(* IEC 61131-3 sources: ml2plc/benchmarks/st (part 13) *)

    weights_7 : ARRAY[0..191] OF REAL := [0.888088644, -0.123913772, -0.846282899, 1.17783785, -0.767203927, -0.449209094, -0.772179544, -0.308529139, 1.4158355, 1.31052208, -0.610198379, -0.72990191, -1.32865715, 0.598848462, 0.529765189, 0.906202614, 0.0025848723, -0.916793466, 1.49462843, -0.405332565, -0.581331134, -1.24053252, 0.719219387, 0.456818759, 1.07239103, -0.71875602, -0.512277603, -0.771926701, -0.468680173, 1.47650003, 1.16464531, -0.211401775, -0.830097437, -0.592156947, -0.122473739, 1.40973353, -0.256034911, -0.522334278, 1.13457429, -1.07700145, 0.666598201, 0.474731237, -1.27282381, 0.632757485, 0.708201051, -1.10329938, 0.727127552, 0.492805749, -1.15903831, 0.78498143, 0.360979617, -0.812300086, 0.210701555, 0.955269992, 1.52882719, -0.381138951, -0.742695808, -0.274786711, -0.196780428, 1.68793082, 1.54681039, -0.22795254, -0.553849936, -1.26980937, 0.545592904, 0.425203025, 1.34888792, -0.62540859, -0.476311505, 0.380844444, 0.586091816, -1.1150496, -1.01592028, -0.0146602849, 0.895467341, -0.456928283, -0.584338427, 1.16077256, 0.413884312, -0.21048446, -1.16396976, 0.751783848, 0.324061215, -1.49614906, -0.575325549, -0.530140579, 1.41179919, -1.35693932, 0.686669171, 0.656322777, 1.22251678, -0.695291579, -0.740689158, -0.676817656, -0.355217397, 1.59177208, 0.207133874, 0.497951657, -0.983146548, 0.469873518, 0.117614292, -1.43506837, 0.132174373, 0.389537215, -1.14951098, 0.820351005, 0.0726073906, -0.653037608, 1.48673153, -0.487765312, -0.680322826, 0.0507701635, 0.432502806, -0.945631862, -0.42844075, -0.336914688, 1.56399095, 0.778971314, 0.452257246, -1.42628229, -0.471889734, -0.441351414, 1.41961205, 0.00993562955, -0.574463367, 0.549236596, 1.21431422, -0.684745908, -0.146852493, -0.852580428, -0.388104379, 1.43994546, -0.78573972, -0.31785956, 1.49420559, 1.35582078, -0.0897780806, -0.4087421, 0.695370257, 0.364000231, -1.27974713, 0.373800397, 0.482034594, -1.2333101, 1.32530713, -0.490792662, -0.321068794, 0.503972769, 0.0731279776, -1.43025231, -0.400622934, -0.543340862, 1.15907669, 0.280509353, 0.306184769, -1.45866597, 1.17186499, -0.665238976, -0.192673638, -1.03320301, -0.00132938253, 0.908325374, 1.0105319, 0.0897968858, -0.713194191, 0.359024227, 0.363719821, -1.40014493, -0.18309705, -0.547121286, 0.972757518, 0.502420723, -0.138461307, -1.05406582, 1.36639011, -0.532719135, -0.751533031, 0.933193147, -0.895748973, -0.461577773, -0.881112456, -0.282391846, 0.816898346, 1.63772881, -0.375343144, -0.522669077, -0.108508743, -0.35503307, 1.0366466, -0.95520407, -0.139931589, 0.780282736];
    bias_7 : ARRAY[0..2] OF REAL := [0.0118476562, 0.164545983, -0.221493304];

END_VAR

VAR
    (* Merged variables from all regions *)
    buffer_0 : ARRAY[0..63] OF REAL;
    buffer_1 : ARRAY[0..63] OF REAL;
    c_state_0 : ARRAY[0..63] OF REAL;
    c_state_3 : ARRAY[0..63] OF REAL;
    f_gate_0 : ARRAY[0..63] OF REAL;
    f_gate_3 : ARRAY[0..63] OF REAL;
    g_gate_0 : ARRAY[0..63] OF REAL;
    g_gate_3 : ARRAY[0..63] OF REAL;
    h_state_0 : ARRAY[0..63] OF REAL;
    h_state_3 : ARRAY[0..63] OF REAL;
    i_gate_0 : ARRAY[0..63] OF REAL;
    i_gate_3 : ARRAY[0..63] OF REAL;
    o_gate_0 : ARRAY[0..63] OF REAL;
    o_gate_3 : ARRAY[0..63] OF REAL;

    (* Temporary computation variables *)
    i : DINT;
    j : DINT;
    t : DINT;
    sum : REAL;
    (* Computation helpers *)
    max_val : REAL;
    exp_val : REAL;
    exp_sum : REAL;
    (* Spatial loop variables *)
    oc : DINT;
    oh : DINT;
    ow : DINT;
    ic : DINT;
    kh : DINT;
    kw : DINT;
    ih : DINT;
    iw : DINT;
    (* Transpose loop variables *)
    t2_d0 : DINT;
    t2_d1 : DINT;
    t2_d2 : DINT;
END_VAR

(* Forward pass execution *)

(* Region: r0 [ACYCLIC] *)
(* Acyclic Region r0 *)
(* Layer 0: LSTM (hidden_size=64, input_size=1, seq_len=1) *)
(* Generating output: Y *)

(* Initialize states to zero *)
FOR j := 0 TO 63 DO
    h_state_0[j] := 0.0;
    c_state_0[j] := 0.0;
END_FOR;

(* Process 1 timesteps *)
FOR t := 0 TO 0 DO

    (* Input Gate *)
    FOR j := 0 TO 63 DO
        sum := 0.0;
        FOR i := 0 TO 0 DO
            sum := sum + input_data * weights_0_i[j * 1 + i] ;
        END_FOR;
        FOR i := 0 TO 63 DO
            sum := sum + h_state_0[i] * recurrent_0_i[j * 64 + i] ;
        END_FOR;
    sum := sum + bias_0_i[j];
    i_gate_0[j] := 1.0 / (1.0 + EXP(-sum));
    END_FOR;

    (* Forget Gate *)
    FOR j := 0 TO 63 DO
        sum := 0.0;
        FOR i := 0 TO 0 DO
            sum := sum + input_data * weights_0_f[j * 1 + i] ;
        END_FOR;
        FOR i := 0 TO 63 DO
            sum := sum + h_state_0[i] * recurrent_0_f[j * 64 + i] ;
        END_FOR;
    sum := sum + bias_0_f[j];
    f_gate_0[j] := 1.0 / (1.0 + EXP(-sum));
    END_FOR;

    (* Cell Gate *)
    FOR j := 0 TO 63 DO
        sum := 0.0;
        FOR i := 0 TO 0 DO
            sum := sum + input_data * weights_0_g[j * 1 + i] ;
        END_FOR;
        FOR i := 0 TO 63 DO
            sum := sum + h_state_0[i] * recurrent_0_g[j * 64 + i] ;
        END_FOR;
    sum := sum + bias_0_g[j];
    exp_val := EXP(2.0 * sum);
    g_gate_0[j] := (exp_val - 1.0) / (exp_val + 1.0);
    END_FOR;

    (* Output Gate *)
    FOR j := 0 TO 63 DO
        sum := 0.0;
        FOR i := 0 TO 0 DO
            sum := sum + input_data * weights_0_o[j * 1 + i] ;
        END_FOR;
        FOR i := 0 TO 63 DO
            sum := sum + h_state_0[i] * recurrent_0_o[j * 64 + i] ;
        END_FOR;
    sum := sum + bias_0_o[j];
    o_gate_0[j] := 1.0 / (1.0 + EXP(-sum));
    END_FOR;

    (* Cell state: c_t = f_t * c_{t-1} + i_t * g_t *)
    FOR j := 0 TO 63 DO
        c_state_0[j] := f_gate_0[j] * c_state_0[j] + i_gate_0[j] * g_gate_0[j];
    END_FOR;

    (* Hidden state: h_t = o_t * tanh(c_t) *)
    FOR j := 0 TO 63 DO
        exp_val := EXP(2.0 * c_state_0[j]);
        h_state_0[j] := o_gate_0[j] * ((exp_val - 1.0) / (exp_val + 1.0));
    END_FOR;

    (* Y output: Full sequence *)
    FOR j := 0 TO 63 DO
        buffer_0[t * 64 + j] := h_state_0[j];
    END_FOR;
END_FOR;

(* Layer 1: Squeeze *)
FOR i := 0 TO 63 DO
    buffer_1[i] := buffer_0[i];
END_FOR;

(* Layer 2: Transpose perm=(1, 0, 2)  (1, 1, 64) -> (1, 1, 64) *)
FOR t2_d0 := 0 TO 0 DO
    FOR t2_d1 := 0 TO 0 DO
        FOR t2_d2 := 0 TO 63 DO
            buffer_0[t2_d0 * 64 + t2_d1 * 64 + t2_d2] := buffer_1[t2_d1 * 64 + t2_d0 * 64 + t2_d2];
        END_FOR;
    END_FOR;
END_FOR;

(* Layer 3: LSTM (hidden_size=64, input_size=64, seq_len=1) *)
(* Generating output: Y *)

(* Initialize states to zero *)
FOR j := 0 TO 63 DO
    h_state_3[j] := 0.0;
    c_state_3[j] := 0.0;
END_FOR;

(* Process 1 timesteps *)
FOR t := 0 TO 0 DO

    (* Input Gate *)
    FOR j := 0 TO 63 DO
        sum := 0.0;
        FOR i := 0 TO 63 DO
            sum := sum + buffer_0[t * 64 + i] * weights_3_i[j * 64 + i] ;
        END_FOR;
        FOR i := 0 TO 63 DO
            sum := sum + h_state_3[i] * recurrent_3_i[j * 64 + i] ;
        END_FOR;
    sum := sum + bias_3_i[j];
    i_gate_3[j] := 1.0 / (1.0 + EXP(-sum));
    END_FOR;

    (* Forget Gate *)
    FOR j := 0 TO 63 DO
        sum := 0.0;
        FOR i := 0 TO 63 DO
            sum := sum + buffer_0[t * 64 + i] * weights_3_f[j * 64 + i] ;
        END_FOR;
        FOR i := 0 TO 63 DO
            sum := sum + h_state_3[i] * recurrent_3_f[j * 64 + i] ;
        END_FOR;
    sum := sum + bias_3_f[j];
    f_gate_3[j] := 1.0 / (1.0 + EXP(-sum));
    END_FOR;

    (* Cell Gate *)
    FOR j := 0 TO 63 DO
        sum := 0.0;
        FOR i := 0 TO 63 DO
            sum := sum + buffer_0[t * 64 + i] * weights_3_g[j * 64 + i] ;
        END_FOR;
        FOR i := 0 TO 63 DO
            sum := sum + h_state_3[i] * recurrent_3_g[j * 64 + i] ;
        END_FOR;
    sum := sum + bias_3_g[j];
    exp_val := EXP(2.0 * sum);
    g_gate_3[j] := (exp_val - 1.0) / (exp_val + 1.0);
    END_FOR;

    (* Output Gate *)
    FOR j := 0 TO 63 DO
        sum := 0.0;
        FOR i := 0 TO 63 DO
            sum := sum + buffer_0[t * 64 + i] * weights_3_o[j * 64 + i] ;
        END_FOR;
        FOR i := 0 TO 63 DO
            sum := sum + h_state_3[i] * recurrent_3_o[j * 64 + i] ;
        END_FOR;
    sum := sum + bias_3_o[j];
    o_gate_3[j] := 1.0 / (1.0 + EXP(-sum));
    END_FOR;

    (* Cell state: c_t = f_t * c_{t-1} + i_t * g_t *)
    FOR j := 0 TO 63 DO
        c_state_3[j] := f_gate_3[j] * c_state_3[j] + i_gate_3[j] * g_gate_3[j];
    END_FOR;

    (* Hidden state: h_t = o_t * tanh(c_t) *)
    FOR j := 0 TO 63 DO
        exp_val := EXP(2.0 * c_state_3[j]);
        h_state_3[j] := o_gate_3[j] * ((exp_val - 1.0) / (exp_val + 1.0));
    END_FOR;

    (* Y output: Full sequence *)
    FOR j := 0 TO 63 DO
        buffer_1[t * 64 + j] := h_state_3[j];
    END_FOR;
END_FOR;

(* Layer 4: Squeeze *)
FOR i := 0 TO 63 DO
    buffer_0[i] := buffer_1[i];
END_FOR;

(* Layer 5: Slice starts=[0] ends=[1] axes=[0] steps=[1] *)
FOR i := 0 TO 63 DO
    buffer_1[i] := buffer_0[i];
END_FOR;

(* Layer 6: Squeeze *)
FOR i := 0 TO 63 DO
    buffer_0[i] := buffer_1[i];
END_FOR;

(* Layer 7: Fused Linear + SOFTMAX *)
FOR j := 0 TO 2 DO
    sum := 0.0;
    FOR i := 0 TO 63 DO
        sum := sum + buffer_0[i] * weights_7[i * 3 + j];
    END_FOR;
output_data[j] := sum + bias_7[j];
END_FOR;

(* Softmax: find max *)
max_val := output_data[0];
FOR i := 1 TO 2 DO
    IF output_data[i] > max_val THEN
        max_val := output_data[i];
    END_IF;
END_FOR;

(* Softmax: compute exponentials and sum *)
exp_sum := 0.0;
FOR i := 0 TO 2 DO
    output_data[i] := EXP(output_data[i] - max_val);
    exp_sum := exp_sum + output_data[i];
END_FOR;

(* Softmax: normalize *)
FOR i := 0 TO 2 DO
    output_data[i] := output_data[i] / exp_sum;
END_FOR;

END_FUNCTION_BLOCK

(* ---- LSTM3_straton.st ---- *)
FUNCTION_BLOCK LSTM3_FB

    (* Model Inputs/Outputs *)
VAR_INPUT
    input_data : REAL;
END_VAR

VAR_OUTPUT
    output_data : ARRAY[0..2] OF REAL;
END_VAR

VAR
    CONSTANT weights_0_i : ARRAY[0..63] OF REAL := [0.702140272, 0.550907314, 0.840128601, 0.811903298, 0.307846963, 1.12213707, 0.702723861, 0.78549248, 1.03316271, 0.728771746, 0.658028424, 0.580750406, 0.615542233, 0.771269143, 0.595596969, 0.611394525, 0.644692361, 0.114490122, 0.525960624, 0.181024775, 0.43071872, 0.665743828, 0.662614048, 0.347228467, 0.769034982, 0.228199184, 0.700795293, 0.569566727, 0.677138209, 0.73381424, 0.549547136, 0.302287668, 0.169487387, 0.974528968, 0.748925805, 0.776894212, 0.810905218, 0.427933753, 0.884441376, 0.829136014, 0.288695246, 0.795262098, 0.532379746, 0.22446543, 0.771800041, 0.653539002, 0.731219053, 0.170757174, 0.902539074, 0.538231611, 0.51912272, 0.955829144, 0.832288802, 0.900867701, 0.702928185, 0.872188985, 0.894331634, 0.607017815, 0.705278337, 0.333420843, 0.529384255, 0.336027026, 0.648417652, 0.559612393];
    CONSTANT recurrent_0_i : ARRAY[0..4095] OF REAL := [0.0727516413, 0.0621806681, 0.0826341808, -0.0324631631, 0.0780053213, -0.130033791, -0.0319923647, 0.0896927789, 0.130534112, -0.0421945676, -0.0756037533, -0.0922252685, 0.00545726344, 0.0880259946, -0.0772752613, 0.0512711406, 0.0296145584, 0.0135381324, -0.0145865045, 0.0353048369, -0.0163449794, -0.0219417289, 0.00759037118, -0.0415089913, -0.0641311258, 0.0446674526, 0.0170345269, 0.114942849, 0.0462704226, 0.0438979566, 0.130931437, -0.0146956779, -0.0373039432, 0.160181582, 0.0509333275, -0.0090306839, 0.00299992273, -0.010383524, 0.031728372, -0.00710704457, -0.00758532062, -0.0451442599, 0.0935175195, -0.0125704622, 0.0317067243, 0.0606242865, -0.0168152805, 0.00345395319, -0.0898493975, 0.0553060398, -0.0737185553, -0.0635084957, -0.00217968249, -0.0560640506, 0.0309809372, -0.0389013216, -0.0571859553, -0.00478457334, -0.137683779, -0.0206679888, -0.0514972247, 0.0388438366, 0.0153822303, -0.0171498396, 0.00600126432, -0.0851558447, 0.133651495, -0.0185905043, -0.0246904604, 0.0102146799, 0.0566058196, 4.23480524e-05, -0.0203502793, 0.0520644151, -0.0723077804, 0.0706539601, 0.023620028, -0.114415541, -0.077967003, 0.0202202648, -0.0342062041, -0.0991770253, 0.0620289519, -0.039034795, -0.11893864, 0.0454845876, -0.00476856716, -0.124633782, 0.0523016639, -0.0491373278, -0.0463687293, -0.0284624062, -0.0796379447, 0.0411196351, 0.0183950588, -0.0835485458, -0.0130095724, 0.0761168301, 0.110718943, -0.0617460273, -0.105785653, 0.0356864445, 0.0494417138, 0.020865988, -0.0829355121, 0.000668380701, 0.00423853425, -0.117335983, -0.112802789, -0.0873446092, -0.0655066594, -0.0423219949, -0.0786840543, 0.00250472827, -0.110003382, -0.045915883, -0.0603204183, 0.0303344596, 0.0707006305, 0.0354735367, -0.0640057474, 0.0473994985, -0.0212647375, 0.0411032513, -0.0771477968, -0.0166638345, 0.00337213092, -0.0226932354, 0.0456429943, -0.0196843427, 0.0404657125, 0.0254306849, -0.0168858916, -0.100593567, -0.116192296, 0.0310631618, 0.0672013462, 0.114804812, -0.0465652943, -0.00154955732, -0.036767751, -0.0378884897, -0.0250008237, 0.0466526635, -0.0191811118, -0.000101840356, -0.0592753589, 0.172661081, -0.0531607121, 0.00527921086, -0.0125218285, 0.0705138072, 0.020655388, 0.100712925, 0.0040708594, 0.0298366249, -0.00289789634, -0.105439723, -0.00869502686, 0.0765521899, -0.0580295846, 0.0956573263, -0.0131847216, -0.0422052965, -0.00297464058, 0.0503321402, -0.0478489585, 0.0335775577, -0.0301637445, 0.00344321551, 0.0895170718, 0.0310253073, 0.00502613885, 0.0457690544, -0.0207835399, 0.000252262573, -0.00835427362, -0.133433089, -0.0304905064, 0.092546992, 0.0331540592, 0.000841447385, -0.0252766088, -0.0414331928, 0.0101674721, -0.0159507189, 0.00302448263, -0.00964387413, 0.0656525418, -0.157459468, 0.0171210915, 0.10000737, -0.0236126985, 0.0170642994, -0.0294568427, 0.0334513187, -0.0220087394, -0.0428130999, -0.0756321475, 0.0157396775, -0.0132302316, -0.0658647045, 0.0589430034, 0.00988156162, -0.0849569365, 0.121961564, 0.00635574851, -0.0347112417, 0.00926421676, 0.0173401404, -0.151415199, 0.041484613, 0.00184322847, 0.0359681174, 0.0752471238, 0.0984926, -0.0999504551, 0.0267645456, 0.0486583449, 0.0590231977, 0.00425340515, 0.0750458241, -0.00415878836, -0.0125731686, 0.0978570655, -0.0809679553, 0.00953727774, 0.0290226694, 0.0406909958, -0.122906491, 0.0246698428, 0.0127425753, 0.0167440623, 0.0282128006, 0.0204523206, -0.0491225682, -0.00133290479, -0.0879503638, -0.0175075829, -0.0297206547, -0.0100959539, 0.0516403019, -0.052208595, -0.0526957437, -0.142511413, 0.0631481856, 0.0082924366, 0.0142942322, 0.0194399487, 0.082317315, 0.182806715, -0.0128400987, 0.0133524388, -0.0546476245, 0.0249223039, -0.0169815794, 0.00866021402, -0.0423310734, 0.0564726405, -0.102079518, -0.00930380821, 0.0186641105, 0.0262102578, -0.0276058502, 0.00666292477, -0.0416896977, 0.0912574828, 0.0394550152, 0.0131434798, -0.0107459817, 0.0220733341, 0.101379797, 0.069571726, -0.00961366575, -0.0787620544, 0.0116914697, -0.10854429, -0.0954701975, 0.0340769216, 0.00364211295, -0.0838557333, 0.11981912, -0.00016324129, -0.0325293913, -0.0776118413, 0.0159091651, -0.0477694646, 0.117520049, 0.0343630239, 0.0626410767, 0.0725534111, 0.0137511753, 0.0102761351, 0.0384476483, -0.025758734, -0.0109584201, -0.115339629, -0.0080120489, 0.00114537869, 0.120408282, 0.0536845811, -0.0320632346, -0.0182842221, 0.0136444457, -0.0913924277, 0.0926747099, -0.0925770104, -0.0231577531, 0.0205560066, -0.00191105367, -0.0321596973, -0.12859036, -0.0584978908, -0.0560642928, 0.113133483, -0.027025789, -0.0500422195, -0.046241872, 0.00904796738, -0.142783582, 0.0597391538, -0.0933348238, -0.091109097, -0.0664444864, 0.0786642209, 0.0643827915, -0.00446130894, -0.0406435616, 0.0581320375, -0.0465331115, 0.0364481136, 0.0176456738, 0.0979348645, 0.0894413367, -0.0545003824, -0.0495841168, 0.00888519082, 0.0636737645, 0.05193891, -0.0283721257, -0.0566147231, 0.183045834, -0.118062697, -0.0693358406, 0.0176241342, -0.00353063643, -0.0731030107, -0.0132001694, -0.0521529317, 0.125817999, 0.0695978999, -0.124826491, -0.0061951708, 0.0417266451, 0.0583891943, 0.0235025808, -0.0648017526, 0.0367687866, -0.0333195329, -0.0380349644, -0.0129484069, -0.130066216, 0.0361705013, 0.00339826383, 0.0437863097, -0.0165002644, 0.0261191688, -0.0423497558, -0.125128835, -0.0824990794, -0.158404469, 0.0239589661, 0.000989105785, 0.0705716163, 0.000514748506, 0.0106146075, 0.018335579, -0.0927568302, 0.0252951495, -0.0790490359, -0.000428203493, -0.00807804428, 0.0282302741, 0.0416536778, -0.0353906341, -0.125360742, -0.0164563227, -0.0400473513, -0.0475901105, -0.0188975669, 0.0190299749, -0.035292007, 0.0398504995, 0.0578784384, -0.00539165642, 0.0377021693, -0.00657368964, -0.00917698257, -0.0644009337, -0.00816033222, -0.0400245786, 0.0934461951, -0.0305664521, -0.0227205046, -0.0205899216, -0.0152598266, 0.0277052615, 0.0136568416, -0.0807154402, -0.0698791817, -0.0617102832, -0.0738777146, -0.0762551874, 0.0600783564, 0.0449102037, -0.0579390265, 0.144962117, 0.194548294, -0.0171745792, -0.0391854942, 0.0970190018, -0.0735182762, -0.00443866057, 0.0561750755, -0.00835239142, 0.103401393, 0.0354097895, 0.0144966841, 0.0718112886, 0.0228926204, 0.0372653194, -0.0687554851, 0.10727971, -0.037785314, 0.0797682926, -0.00646833796, 0.00971507467, 0.0386701822, 0.118912876, -0.032234598, 0.0318986624, 0.0539872497, -0.011686909, 0.145176083, 0.0255599786, -0.039034158, 0.0321393982, -0.0146574825, 0.160541251, -0.0973295048, 0.0362529159, 0.025079282, 0.119155452, -0.0793333724, -0.0652497858, 0.0338132381, 0.0546442941, -0.0188240651, 0.00941769406, -0.104044199, -0.0805709586, -0.0476697013, 0.0640894994, 0.07038939, -0.000911274925, -0.0129568689, 0.00333408732, -0.0201132633, 0.00736489007, 0.0114483982, 0.103261217, -0.0535993725, -0.0637782216, 0.0585075244, -0.00838142354, -0.0303359125, -0.0881697759, 0.0637675673, 0.0675119534, -0.0465907231, 0.0223106146, 0.0744051114, -0.00451694895, 0.0699620992, -0.0100199496, -0.0766999424, -0.111208931, -0.00734356884, -0.0439275131, -0.0797161311, -0.0652370676, 0.00365057588, -0.0114077562, -0.00976049341, -0.00207494851, -0.0548781082, 0.00935276877, 0.0451770723, 0.0154793952, -0.0134702399, -0.0304076131, 0.0523790345, 0.0507434718, 0.0699445009, 0.0361545049, -0.0232983083, 0.014487464, -0.100811966, -0.0416969284, 0.0327967592, -0.0249530524, -0.0339162126, -0.017976515, -0.0419778116, 0.0222332217, 0.0152361365, -0.0173479971, 0.0431629382, 0.0682366565, 0.0238082893, -0.0795904398, 0.0329069197, 0.0875642598, 0.0079081133, -0.0893924832, -0.0986220166, -0.0576440096, 0.0620961636, -0.0173755735, 0.0642281398, 0.0128179947, 0.00068197638, 0.0281319804, -0.0740936846, 0.0206660945, 0.0549913384, -0.0514548644, 0.106060728, 0.0215401538, 0.00298270863, -0.0353878029, 0.0589390211, 0.0957489237, -0.0261493661, -0.116729505, 0.0467135832, -0.0562625453, 0.0103190532, 0.000896572019, 0.00233004056, -0.0809285343, 0.022660207, 0.110791236, 0.12861453, 0.0517879203, 0.0163614936, -0.0594949387, -0.0264125317, 0.0178101491, 0.0121639995, -0.103968374, -0.00524417032, 0.0263312124, 0.0630289018, -0.0221815184, 0.0465865284, 0.0157697946, 0.00964579266, 0.0674970746, -0.009665424, 0.00193209574, -0.0533254594, -0.167867079, -0.014877351, 0.0151824076, 0.0264426656, -0.125007585, -0.0209615547, 0.0590866096, -0.0137481289, 0.0121204332, -0.0151834041, -0.0251058768, -0.0110409586, -0.00677108858, 0.0129520297, -0.0732064545, -0.0273697656, 0.091351226, -0.0557100922, 0.0296072997, 0.00988943037, -0.0364736542, 0.065504536, -0.00958945323, 0.116355866, 0.0455187596, 0.0358052738, 0.0423866361, 0.126706302, -0.016172383, 0.00576764019, -0.0433344729, 0.0248547792, -0.0734665766, 0.0619035512, -0.00564275496, -0.0161651708, -0.0448754504, -0.0378655344, -0.0100620128, 0.00184470601, 0.0365175456, 0.0127978846, -0.0136364019, 0.043987263, -0.0878729597, -0.0277508721, -0.0749285445, 0.0541052632, 0.0489377081, 0.0708028525, -0.0602139272, -0.0754432306, 0.00850299187, -0.0961926952, 0.132325843, -0.116709456, 0.108343646, -0.0597229786, 0.0569296554, -0.00331771234, -0.0273206718, -0.0314441323, -0.000921917148, -0.157476932, -0.0827142447, 0.00737003703, 0.052945137, 0.0687581971, -0.000348506495, 0.0343997292, -0.0195971914, 0.125520691, 0.00101949577, -0.0154516073, 0.0158582088, 0.00286582764, -0.0688755289, 0.0439975187, -0.0276184082, 0.00204778835, -0.00275259465, -0.0708792955, -0.0564192757, -0.0506432205, 0.00576888025, -0.0713198557, 0.0567040592, 0.0332127437, 0.0334661454, -0.00076312013, -0.0548750758, -0.0580983646, 0.107379794, -0.0128812864, 0.118800402, -0.0523375235, 0.00846277364, -0.0320085548, 0.115329124, -0.0270583499, -0.0132279834, 0.0107595138, -0.0375581123, -0.0365415849, 0.00050151255, 0.082369104, -0.00622165669, 7.82900024e-05, -0.0483080707, -0.0812478885, 0.0232834574, -0.0151235107, -0.0244658086, -0.000501235016, 0.00333951134, 0.0400660373, -0.0880180597, 0.00398900174, 0.0124121793, 0.00375011051, -0.144496277, 0.034541361, 0.0617251918, 0.00635286514, 0.0420818478, -0.0161394067, -0.0328651518, 0.0820424035, 0.0222173464, 0.0229891762, 0.0139844613, -0.0297264177, 0.00847776048, 0.070485957, -0.058027342, 0.0854259282, 0.0362042785, 0.185735196, 0.0904341638, 0.0116911372, 0.0929991826, -0.0522834435, -0.145003289, 0.123330593, 0.0321200006, -0.137998715, 0.0165430456, -0.0304837991, -0.0096137803, -0.000575108454, 0.00894964393, -0.0625963882, 0.0877403393, -0.00540286303, 0.05565162, 0.117289849, 0.0030141864, -0.0417421907, -0.0236499757, 0.0914468393, 0.0819795579, -0.0468929261, -0.00116663426, 0.106944904, -0.00840409659, 0.0906113163, 0.035827592, 0.0802839696, 0.0457703471, -0.0492791533, -0.00685054809, 0.0727560148, -0.0435580648, -0.0374004319, -0.0588955544, 0.0217557084, 0.0269399136, -0.032965567, -0.156689122, 0.0972655118, -0.00287246145, -0.0220363066, -0.127908081, 0.0366795324, -0.00863787718, 0.00523071457, -0.0202574283, -0.0320058577, 0.101983219, -0.0471758954, 0.0736685321, -0.0319768637, 0.00369445607, 0.0711755827, 0.0862062871, -0.0234699268, -0.0473918878, -0.0423197597, -0.0217249542, -0.0155853694, -0.00140371313, -0.031561885, -0.012095931, 0.0411939137, -0.0171032492, 0.0350121111, -0.0700786561, 0.106874585, 0.0229188204, -0.0267229974, 0.0272093657, 0.0680414885, -0.182497233, 0.0379727185, -0.0413211621, -0.0382319614, 0.0367683172, -0.0470161811, 0.00117427809, 0.00355215091, -0.0241580792, -0.0915986449, 0.0951508805, -0.0273425989, -0.0247635655, -0.028161943, -0.0521801747, 0.117773622, 0.0734785274, 0.0860297233, -0.0260464326, -0.0355322622, -0.01959222, 0.0503423698, -0.0901166201, -0.0438693576, 0.0379061773, -0.0948499218, -0.0787415132, 0.0232516527, 0.0124969175, 0.18771562, 0.0921514928, 0.114925891, -0.0707947537, -0.000519088004, -0.0291188639, -0.0735063776, -0.0492690504, -0.0123775937, -0.0174803324, -0.0451487228, 0.0361573286, -0.00940452237, 0.033992283, 0.12313839, 0.0281803943, -0.0914258882, 0.0704093054, -0.039767459, 0.0598411039, -0.0283360202, 0.0249229707, -0.0383545458, -0.0305118412, -0.0356102437, 0.0561388247, -0.0697289929, 0.0612826683, 0.0374586843, 0.0655589849, -0.116294079, -0.0103302505, 0.0277131796, 0.0115445564, 0.00331265386, -0.0399645157, 0.00636392739, 0.0776276737, -0.0297414139, 0.0986465439, -0.101880111, -0.0839399397, -0.0568840578, 0.0191173181, -0.00985985994, -0.104261704, 0.0210980549, 0.0850705653, -0.0701188445, 0.0957206786, 0.0592016242, 0.108822487, -0.040555045, 0.0594565906, -0.0398680121, -0.0324985757, 0.0258895662, -0.0341325998, -0.0698637366, -0.1593602, 0.0453048572, -0.0243716724, 0.0558315925, -0.034077201, 0.139877036, -0.0237494931, -0.0362580866, -0.117848903, -0.0071857064, 0.038842354, 0.0734850243, -0.0919130966, 0.0219057612, 0.0234997906, 0.0286933333, 0.0519893244, 0.0763522089, 0.0483730026, 0.00100774318, 0.0531575605, -0.114286371, 0.0754203722, 0.0068904506, -0.0706003681, 0.0933185518, 0.0208554231, 0.0278633069, -0.0351458043, 0.0296566151, -0.06653402, 0.142907277, -0.0489391983, -0.0250295922, -0.0132226385, -0.036999926, 0.040843077, 0.158806115, -0.0184686184, 0.0620175451, -0.0525245406, 0.0129820816, -0.017142212, -0.0203886367, 0.0641498417, -0.03602634, -0.116563454, -0.0340168513, -0.00379975047, -0.00621868297, 0.0650157779, 0.0434404761, 0.0860811099, 0.063751176, -0.0145058017, -0.0197795611, 0.0182513129, -0.0370967872, 0.0123619623, 0.168666184, -0.0660671145, 0.0630441532, -0.0105630495, 0.0486272424, -0.0341909528, -0.0626777411, 0.0853702128, -0.022746291, -0.0413650274, 0.0112732453, 0.0499815829, -0.0165389869, 0.0203687884, -0.134544104, -0.0570603237, -0.0830415115, -0.00185097475, -0.030207064, -0.0200033523, -0.0974278226, -0.0238209311, -0.0631394014, -0.0549098514, -0.021339165, 0.020896947, 0.0140093444, 0.0288279913, -0.112859555, 0.150645897, -0.0089820018, -0.0444067419, 0.117183514, 0.116750821, -0.0631431118, -0.102793284, 0.0324017406, -0.0411568135, 0.0485532843, -0.026592534, 0.00423682667, 0.00513659976, -0.0274688713, -0.0157996807, -0.0854125023, -0.0108604785, -0.0931327194, -0.0067656883, -0.0331029296, 0.0856935978, -0.0143788885, -0.0392643176, -0.0604175478, 0.0404099748, -0.0238179155, -0.0178244021, 0.0153439678, -0.017928306, 0.0430681035, -0.0137550738, -0.117914356, -0.180906773, 0.0190907903, -0.0141145401, 0.053051848, 0.0289822202, -0.0848073289, 0.0269892141, 0.0303875655, 0.129724652, -0.0496526621, 0.0462062024, 0.0123959333, -0.0982962996, 0.0873335674, -0.113902688, -0.0148382001, -0.022349732, -0.0339166969, 0.108045816, 0.0368998051, -0.00215027854, 0.0359801911, -0.144334018, -0.0358332358, -0.0789693668, -0.000820970163, -0.0163820796, 0.0386639088, 0.110587113, -0.0314619169, -0.0274926089, 0.0944872648, -0.0798697397, -0.0451008752, 0.0266324598, -0.0654547438, 0.0199776348, -0.0124631887, -0.0389405303, -0.115865506, 0.107397661, -0.0170727521, -0.0208050422, -0.00403178856, 0.00181274489, -0.00149073335, 0.0569269955, 0.041924037, -0.0816717148, -0.00521243177, 0.00550422817, -0.0980434865, 0.0538859181, 0.0559096783, -0.00900849234, -0.0368861221, 0.0361628868, 0.0323648937, 0.0103506837, -0.0963612944, 0.128723457, 0.0365089402, -0.074579142, -0.081020236, -0.0360122994, -0.0592223667, 0.025372399, 0.088464506, 0.0271437094, -0.00152724795, -0.0353991948, 0.0527125001, 0.0137757715, 0.0114214001, 0.0405929014, -0.045993641, 0.0397221372, -0.059202753, 0.0435205773, 0.0180647969, 0.0445329957, 0.0311286338, 0.027261693, 0.0964478627, -0.00864790939, 0.132875443, -0.122668698, 0.0541860238, -0.0594329834, -0.0597948171, 0.0602433383, -0.0598982051, 0.152696952, 0.0508942716, -0.0447879098, 0.00811342895, -0.0245362502, -0.0291209966, -0.111188218, -0.0189557653, -0.145642966, -0.0732516944, -0.0738148466, -0.118594654, -0.00454571471, -0.0263547897, 0.017749887, -0.0820513368, 0.045788575, -0.0222869627, -0.0300645363, -0.0252726525, -0.123603433, -0.131661654, -0.0112165175, -0.0932581425, 0.00205570646, 0.0549669564, -0.0469899066, 0.0217208564, -0.174646497, -0.00242389715, -0.107725173, -0.039760232, 0.0438962542, 0.033221893, 0.0147209018, 0.114341497, -0.0104052667, -0.0847626626, 0.0683764517, 0.0144604817, -0.0515585765, -0.098916471, 0.00632204534, -0.0274075232, 0.0172482189, 0.0059097223, 0.000274197169, -0.0818955898, -0.00595346792, -0.0431167409, 0.0141846109, 0.0928108841, 0.0493697897, 0.0435281098, -0.00430369563, 0.0135970106, -0.0395035334, 0.0674678236, -0.0146978237, 0.01993981, 0.0717856139, -0.031349659, -0.0583848506, -0.0348999314, 0.0329215974, 0.00442747911, -0.0990120173, 0.0400124006, 0.0276716035, -0.00465472275, -0.0150943138, -0.0192471016, -0.00484694075, -0.0523224995, 0.023458479, -0.00613671122, 0.0824287683, -0.0669285506, -0.0130545525, 0.0678386837, -0.00856799539, -0.0425645411, 0.0343296602, -0.0361192375, -0.0378568284, 0.014862569, -0.0314017534, -0.0411946177, 0.0120962616, 0.0196509883, 0.0427911654, 0.0498198867, -0.0778862238, 0.0327159427, 0.08899685, 0.0718479902, 0.0423694775, 0.183253869, -0.0344530828, 0.0173815228, 0.00139276613, -0.00928234309, -0.0237438045, -0.0176289156, 0.0112874117, 0.0254508853, 0.0431757793, 0.0421911255, 0.036971435, -0.044771906, -0.0510402024, -0.0814980045, 0.0274636727, 0.0850320756, 0.0578455478, -0.0132112103, -0.0176027454, 0.00123652956, -0.0166772436, 0.0431952141, 0.0171799026, 0.0560129546, 0.0319918357, -0.0152601199, 0.00947227236, -0.043590717, -0.100858159, -0.0813885257, -0.00108298101, 0.0166240092, 0.118451767, -0.0627318546, 0.0100360308, -0.0795926377, 0.00262210146, -0.0433140695, 0.0305809751, 0.0439304747, 0.0272573233, 0.0373259112, -0.0514604449, 0.0383335948, 0.118634515, -0.186732113, -0.0432817824, -0.0429025069, -0.0772498772, -0.0196676329, 0.0119493557, 0.00927572045, -0.0202227216, -0.0596379042, 0.0605967566, -0.0875917971, 0.185680345, 0.063830778, -0.00155046163, -0.0119067458, -0.0070124995, -0.0461906269, 0.0614498556, -0.0131631885, 0.0642673522, 0.0830220282, -0.0180631597, -0.0748554394, 0.0787710473, 0.0185747221, -0.0305529945, 0.0152649563, -0.0486347228, 0.0563763492, 0.0376386195, -0.0268003289, 0.0335318744, -0.049739819, 0.0335873589, 0.0703956187, 0.010409697, -0.0668904781, -0.0863810778, 0.0244773123, 0.0535634831, -0.107205607, 0.0584613085, -0.0289510079, 0.0200893488, 0.0202745795, 0.0243469607, 0.0493172482, -0.021541819, 0.103889599, -0.0712386742, -0.0244257711, 0.0457455218, 0.0429964997, 0.0528058149, -0.0266966205, -0.151898935, -0.109488726, 0.0190092269, -0.0586468764, 0.0530709401, -0.00976852234, -0.121571757, -0.147223294, -0.0732008293, -0.15228352, 0.027742086, -0.0800120756, 0.0127792284, -0.0280551668, -0.00709801493, 0.0505800731, -0.0410012715, -0.021963004, 0.0187113285, 0.0563162267, 0.00314888172, 0.0538862199, -0.00776094105, -0.0730628967, 0.0652259737, 9.0313144e-05, 0.049799405, 0.0011129044, 0.0627703369, 0.0576126613, -0.0112601072, 0.0204492416, -0.0470470861, 0.0231554154, 0.00090185937, 0.0342733338, 0.0573027842, -0.0909369215, 0.0860854238, -0.0645645931, 0.0191594623, -0.048717726, 0.0948970616, -0.161608219, 0.021575287, -0.0176735464, 0.00495251268, 0.00645933347, -0.0594614148, 0.0986488909, 0.0211776476, -0.0407326743, 0.0726084188, -0.0272595752, -0.0514314249, -0.0716841146, 0.0093075484, 0.0756390244, 0.0412543677, 0.0520931222, 0.014929113, 0.00981443562, -0.0579506569, -0.0570658967, -0.0349842906, -0.0503895544, -0.0168755352, 0.0952543616, -0.126057655, 0.110528342, 0.0116437469, 0.0419249982, 0.0819886625, 0.0351492167, 0.122139595, 0.00687739346, 0.0488508306, 0.0675945133, 0.0209267922, -0.00816457346, 0.0928310156, -0.149517417, -0.0232153945, -0.0803592205, -0.0455706343, -0.0210929383, -0.0287392419, 0.0303849056, 0.00988229923, -0.00971780345, -0.0233898312, -0.0303801131, 0.151730031, 0.00840327516, -0.0425428972, -0.0570457727, 0.0173914358, -0.0240011215, -0.117590509, 0.0454662926, 0.00826025754, 0.0363563746, 0.0257966779, 0.0170941353, 0.0247139968, -0.12864086, -0.0123515511, -0.0647207052, 0.0734354332, -0.0274030156, -0.0336046293, 0.0670940652, 0.0164395086, -0.0834478885, 0.0560125038, -0.0427170359, -0.0566519797, 0.139318958, 0.0429757386, -0.0839925855, 0.0480794087, 0.0248762108, 0.0673513561, -0.0282134004, -0.0173287746, -0.0836200193, 0.0181073323, 0.00905436277, 0.0655650869, 0.0429399349, -0.0493150763, -0.00416665617, -0.0409714803, 0.0160837937, -0.00081096869, 0.0746367052, 0.110396989, 0.0320068114, 0.0846839473, -0.0721276253, -0.0497060865, 0.0726049691, 0.0102233756, -0.0872215778, 0.0585351624, -0.00976938102, -0.108745299, -0.0238607768, 0.00281488895, 0.0076521039, -0.00486782938, -0.0293733981, -0.0337358937, 0.0234056674, 0.00852487423, -0.0432054102, -0.0344540328, -0.0296666399, 0.0277531613, 0.0199462101, -0.102572076, 0.0106342034, 0.05281749, -0.0665505379, -0.0519861989, -0.0374915525, 0.0708934441, -0.0883556455, 0.101648919, -0.0238500293, 0.0375800878, -0.0255494751, -0.0600025021, -0.135210901, 0.120428331, -0.0514075086, 0.0258166976, 0.0299084987, -0.0264056828, 0.00941147283, -0.0154201016, -0.0893158242, -0.00582207181, -0.0930329859, -0.115079045, 0.075967066, -0.0117950849, -0.0617161952, 0.0191614833, -0.0026583611, -0.0172695909, 0.119176403, -0.0679154769, -0.0667522773, -0.0174201056, -0.0326822847, -0.105945945, 0.0328570381, 0.0220449418, -0.0880559385, -0.0545761883, -0.0361280851, -0.012021604, -0.025812868, 0.0658306107, -0.0864854902, 0.0647357255, 0.10267137, -0.0218578987, 0.0141268671, 0.0220957547, -0.212104455, -0.00901220739, 0.16071105, -0.0934063792, -0.0720212758, -0.0446557663, 0.0176140051, 0.0952594727, -0.00304227509, -0.0690695494, -0.0238600653, -0.0255746562, 0.0576497503, -0.0560034513, 0.0122720469, -0.0633462593, -0.0590704642, 0.0126576088, -0.00174971018, -0.0405229926, 0.0861680433, 0.0286935773, -0.0633817092, 0.00103684911, -0.0464625135, -0.0823629797, -0.0593407042, 0.0141500868, -0.0870034397, 0.0107747614, 0.0338124819, -0.0400126353, -0.0309788585, 0.0903759748, -0.0465827882, -0.0373132229, -0.00478894822, -0.0181359425, -0.0330074392, 0.0316597819, -0.0632642061, 0.0039414512, -0.0657994002, 0.100820124, 0.00455378043, -0.0351329185, 0.0416226089, 0.0397600383, -0.0343750902, 0.0478181131, 0.00230326038, -0.0338188298, -0.0526410937, 0.0029062666, 0.0680800006, 0.0313956626, 0.0869969204, 0.185322434, 0.0294733327, 0.00611761399, -0.11583668, -0.0575742163, 0.0311859623, -0.0306454524, -0.0121416431, 0.0707837641, 0.00341178849, -0.0260182619, 0.0737865195, 0.0154152196, -0.0104229245, 0.0181757435, -0.0196045917, -0.0473442003, 0.0294725373, 0.0427677035, 0.0239165537, -0.0044421996, 0.0520130545, 0.0841308832, 0.0421810821, 0.0710302964, -0.0945989788, -0.00716768578, -0.0358735509, 0.0298710074, -0.0491323099, 0.0118293744, 0.0500267744, 0.0160761066, 0.0524036475, 0.0198267978, -0.0250373967, -0.00914585777, 0.0339306332, 0.0137209278, -0.0643130392, 0.00979318749, 0.0793425739, 0.0689684451, -0.0250177532, 0.0551168919, 0.0256160051, 0.0273303092, -0.0670256764, -0.0750374943, 0.0795707852, -0.149131224, -0.0760348514, -0.0122559853, -0.0169459917, -0.0410757847, 0.0581504926, -0.0047336081, 0.0228611827, 0.0522755384, 0.0210218765, 0.130921111, 0.0628677383, -0.131930873, 0.0899220556, -0.0114390031, -0.126428112, 0.103056937, -0.0100312615, -0.0211761855, -0.0581869632, 0.0452357233, 0.0786141232, 0.108842447, 0.00525219738, 0.151705295, 0.0287047625, -0.0105385892, -0.00289420038, 0.0196365751, -0.0490774959, 0.00883252919, -0.0558812656, 0.1248478, -0.0505073145, -0.0166304056, 0.0691084936, 0.0161006004, -0.108558089, 0.00557874423, 0.0714525729, 0.0428007431, 0.0442438126, 0.0734011084, -0.00227193651, -0.106657088, 0.121946499, -0.079083465, -0.111123294, -0.135465428, 0.0523883142, -0.0416224226, 0.122332789, 0.0137510989, 0.0460521244, 0.0347447172, 0.0517446101, -0.00939925015, -0.00611661375, 0.00419576373, 0.0141259655, 0.00198347867, -0.0340772681, 0.0768256932, -0.0326022133, 0.0080893226, -0.0214685723, 0.0543903932, -0.032371331, -0.149114579, 0.0665993467, -0.00778121129, 0.107546717, -0.0166073479, -0.0799072385, 0.000907103531, -0.0839266255, -0.0739985257, -0.0361200124, -0.0330467299, -0.0180994309, -0.0292499084, -0.0461748093, 0.0353545845, 0.0465622544, 0.0678990707, -0.0331273004, -0.0579735264, 0.0208636113, -0.0177743211, 0.0489512533, -0.0734027624, -0.00151019357, -0.12947005, 0.0357025824, 0.0196994711, -0.0611494929, -0.0372755639, 0.0206014905, -0.0361978114, 0.0658185631, 0.0406925529, 0.187332213, 0.0459053144, -0.0248670485, 0.0693691969, -0.0583218709, -0.105129458, 0.0166231748, -0.07091894, -0.0221844073, -0.0692817047, -0.0241019763, 0.0811090171, 0.03763365, -0.112892151, -0.0178294666, 0.0393745415, -0.0920515805, 0.146565199, -0.0321527347, 0.0294383653, -0.0377589911, 0.113711596, -0.133004487, 0.0418280326, -0.114919066, -0.0242213886, 0.0343061537, 0.133941308, -0.0155828111, -0.0562956408, 0.109785452, 0.00697870273, 0.0540946424, 0.00834291987, -0.0255597495, 0.0171979871, 0.0761614889, -0.0391737632, 0.0701430067, -0.0601058044, -0.0175495055, 0.0760216042, 0.0506174862, -0.0205917656, 0.0289436188, 0.0666499659, -0.0409701988, -0.156672731, -0.0787394047, -0.0552437231, -0.0510800742, 0.0127478391, 0.0926389992, -0.00213698111, 0.0271617174, -0.0390887074, -0.0193803068, -0.133023724, 0.11377947, 0.0444727913, 0.00336797303, 0.0324987024, -0.11659871, -0.0198515803, 0.0432685986, 0.00555972941, 0.0206918679, -0.0355419591, -0.0146086421, 0.0920803249, -0.0200472437, -0.0119470125, -0.114049166, -0.0326045938, 0.0129803326, -0.0938383639, 0.0484809503, -0.0520552471, -0.0278478377, -0.0647886544, 0.10094054, -0.0756840855, 0.0378818139, 0.0306564011, -0.023524778, -0.0370059013, -0.00153457746, 0.0631585792, -0.02214038, 0.0689642578, -0.00959259458, 0.0905371904, 0.115043916, 0.0556401312, -0.0928566903, -0.00954530109, -0.0412723832, 0.0275241286, 0.0978282318, 0.00937830471, 0.0416356474, 0.0231232904, -0.0485541224, -0.0819698349, 0.00830572657, 0.00316089275, -0.0281392001, 0.0119747501, -0.0367307439, -0.0492811091, 0.0378377922, 0.0271666422, -0.07177867, 0.125349924, -0.0641519874, 0.0372795388, -0.00964075327, 0.0251864884, -0.00229698629, -0.0943838358, 0.0211065542, -0.0256559029, -0.0412544161, -0.0498182401, 0.025202591, -0.0710987672, -0.0533324815, -0.0049189534, -0.0387485325, -0.00538361538, -0.0506801419, 0.0376440212, -0.0961788148, 0.108937971, -0.0510260239, 0.0695248097, -0.0258867964, -0.0137048652, -0.0807042569, -0.00806998089, 0.111984894, 0.0686698109, -0.037598379, 0.0770009458, 0.0240798444, 0.0628106818, 0.0249741171, -0.00499903271, 0.0582997426, 0.0292410515, -0.0940985829, -0.0318885148, -0.109319203, -0.0142780645, -0.170994744, -0.0829356536, -0.0222196039, -0.0485832542, -0.108767927, 0.00559173245, 0.0229634978, 0.0269906968, -0.063782841, -0.0400377847, 0.00832005683, -0.0465570986, -0.0016413359, 0.0304886736, -0.0518755242, -0.090841189, 0.0730084032, 0.0245121755, -0.0412723497, 0.0586892217, 0.0229290389, -0.0936156809, 0.0652381554, -0.00508300401, -0.00557444245, 0.134620011, 0.0528185219, 0.0587821119, -0.043236874, -0.044430159, -0.0209521055, -0.0354268327, -0.0152262049, -0.0638363957, 0.0539329238, -0.0372782573, 0.0488509908, -0.0958636254, 0.00639156625, -0.0278961621, -0.0129365083, -0.00149445049, -0.028228743, 0.0155989379, -0.0429436192, -0.0473704934, -0.101443902, -0.0692045689, 0.0299465936, 0.0147465998, 0.00661268644, -0.0534076989, 0.00924651697, 0.104975708, 0.0415304974, 0.000269727781, 0.118143529, -0.00158391614, 0.0203097221, 0.00303321518, 0.0397381261, 0.0855536237, 0.0145944133, 0.00353995408, -0.0892745554, 0.084861517, 0.114215717, 0.0029919669, 0.0427440852, 0.0766353905, -0.0687552691, 0.0503479019, -0.0323194116, 0.08432208, -0.0564777441, 0.0409436077, 0.0231873803, -0.131554455, 0.0374630615, 0.0325829387, -0.00295856968, -0.0405622087, 0.0496319979, 0.0289352965, 0.0101500908, 0.0344187357, 0.00112904015, 0.00722406432, 0.0788021982, 0.0775272027, -0.0154337361, 0.0112905027, 0.0215975642, -0.0536064059, -0.00693354383, 0.0608174801, 0.0374165773, 0.0518301651, 0.0764183924, -0.0809245631, -0.00811586063, 0.0179242715, -0.155901596, -0.160923168, -0.0566306114, -0.114005692, 0.00758205634, -0.0906549394, 0.0521262363, -0.100310244, 0.00282220356, 0.0523931533, 0.0630677193, -0.0438348725, 0.00722100586, 0.00640934333, 0.0628485233, -0.0130613558, 0.00371759757, -0.040091224, -0.0462202132, -0.00305903191, -0.0221964736, -0.00167389773, -0.0507050231, -0.0611347631, -0.0574724302, 0.00265610404, 0.0517526865, 0.0469581559, -0.178494588, 0.00220534205, -0.069582358, -0.0215090066, 0.0047822278, 0.0341559276, -0.0422869809, -0.0846082047, -0.0232734829, 0.0593397543, 0.0222365819, 0.0572210252, 0.107284784, 0.054990232, -0.0879809335, 0.0285727177, -0.115808859, 0.0385797359, -0.0159076098, 0.0171930008, 0.046151299, -0.0399743095, 0.0645119846, -0.0433629826, -0.149094194, -0.0738952011, 0.0313407592, -0.0747917891, -0.0496746413, -0.178521425, -0.00650399923, 0.00110328197, 0.121303357, -0.0988033488, -0.177440211, -0.0286801942, -0.109008461, 0.0846569389, 0.095020026, 0.022543462, -0.0474546477, 0.0799250156, 0.0704054832, -0.0316202044, -0.06459295, -0.0750078782, -0.0141381584, -0.11284893, 0.0183110926, 0.0425815843, 0.0698241591, -0.0358852558, -0.0305983536, 0.0119026452, 0.127399877, -0.0716647208, 0.0284642577, -0.120591611, -0.0404190756, -0.0446741134, -0.0555381402, 0.0868036449, 0.0527058467, -0.131675854, 0.0365113765, 0.0500864051, 0.00530374376, 0.029813502, -0.0196713023, 0.0534248762, -0.0326415487, -0.0134224789, 0.0568323955, -0.0491549075, 0.00126836449, -0.0966521651, -0.0532193147, 0.00860303733, 0.00863775611, 0.0421172231, -0.0119322408, 0.0597736686, 0.0440536737, 0.0538674891, -0.000704284292, 0.106371388, -0.0165641587, -0.0867572576, -0.106977202, -0.00550343189, 0.152145311, -0.0535458848, -0.0440272726, 0.098293677, 0.0515624061, 0.0106035564, 0.0395671166, 0.0519889258, -0.149089932, 0.0714540854, -0.100583941, 0.12224327, -0.0508232266, 0.0780539289, -0.0732419416, -0.00868538581, 0.0239342973, 0.0249469392, -0.0694821477, 0.000374149997, -0.0066033937, -0.00721557811, -0.00396225415, -0.0228633173, -0.0310496539, -0.025368074, -0.104311243, -0.0255405679, -0.0418488085, -0.0395715125, -0.052135855, -0.00500662252, 0.0922299773, 0.00395811582, 0.0639874041, 0.0024171425, 0.0462996587, 0.0398141816, -0.0777477771, -0.0104797883, -0.0236524884, 0.0114733949, 0.0602850802, -0.0150871556, 0.105572626, -0.0660246611, -0.0779621452, 0.0586055852, 0.087809965, -0.0615009405, -0.0205225367, 0.003089651, 0.0474609733, 0.062135037, 0.148257151, -0.0197101831, -0.0681717098, 0.076816991, 0.10367243, -0.0258536674, 0.0274908822, -0.100731112, -0.0156992134, -0.0453392193, -0.00266639143, -0.00309458375, 0.0588642582, -0.0211847164, 0.109054767, 0.0417248867, -0.132930219, -0.0127346143, -0.0302010905, 0.0462420955, 0.11357449, 0.00859607384, -0.000631738454, -0.135843575, -0.00648586359, 0.0378909223, 0.0156545788, -0.0915854424, 0.00357584213, 0.00172258168, -0.0420532376, 0.0355732217, -0.217089221, 0.1031342, 0.0202132203, -0.0946729109, 0.0244514309, -0.0219765771, 0.0248513035, -0.0385242328, -0.040843837, 0.0365453511, 0.00641883537, 0.0336989835, -0.0317242965, 0.0309240855, -0.0726778135, 0.00256187283, -0.0185524039, -0.121674128, -0.0455776006, 0.102158509, 0.119345464, -0.000964865088, -0.0373238847, -0.102336988, 0.0252578836, 0.0418426618, 0.0300444476, 0.0675104037, -0.0650050715, 0.0353247002, -0.0786041245, 0.0956212133, -0.0525997803, 0.0740968138, -0.0549821109, -0.0615683049, -0.0116764717, 0.0040182434, -0.0371107236, -0.0122259604, 0.0746070296, 0.11985483, -0.0396226496, -0.0364514105, 0.0902988464, 0.0492551476, 0.0384663865, 0.072580874, 0.169797242, -0.0421398431, 0.0873509794, -0.0159340352, -0.0942513496, -0.0369788222, 0.11160478, -0.0652674437, -0.0534480438, -0.0672385544, 0.00392479636, 0.0475984924, 0.0620817207, 0.0202614926, -0.0367005356, -0.000590074807, -0.0297204033, -0.0414684601, 0.043605946, -0.00721757766, -0.0416722447, 0.0246268213, -0.0773160011, -0.0387003273, 0.0556836352, 0.0622895509, -0.0211151838, 0.0683159977, -0.0330114439, 0.0155544393, 0.0691765025, -0.0717128962, 0.0456270911, -0.037818253, 0.0419966877, 0.104023539, 0.0631524324, 0.0298485234, 0.0548062846, 0.0320408419, 0.008525596, -0.0130907465, 0.0581992306, 0.0336639956, 0.00489646336, 0.0389721319, -0.00712263677, -0.040096283, -0.00816118997, 0.0561630316, 0.0564079359, 0.0977385491, -0.0557625517, 0.121285796, -0.00108744763, 0.0322886258, 0.0216934383, 0.0553678386, -0.0743190646, -0.00782365073, -0.00824525394, -0.0199274216, 0.0515763201, 0.152581915, -0.0655806959, -0.079457745, -0.0627498329, -0.0110104606, -0.0766746104, -0.00850693788, -0.0526255593, 0.0717280433, 0.0114595369, 0.0301140957, 0.0614899024, -0.0672836825, -0.0738866329, -0.0854860023, -0.0378107652, 0.023471145, 0.0728512704, -0.143453404, 0.010287473, 0.0609739125, -0.0562127195, 0.0317436606, 0.019507695, -0.0257064644, 0.0747466385, 0.107812166, 0.00315844268, -0.013035031, -0.0583956093, 0.0416430756, -0.000154026784, -0.00386437285, -0.0288870521, -0.0548927747, 0.00224980572, 0.0140787903, 0.0334683284, -0.0285946839, -0.0317473076, -0.0301351491, 0.131981239, -0.0969547853, 0.0351068303, -0.11974702, 0.0399604477, -0.013861116, 0.0650198609, 0.0588160492, -0.0407459363, -0.0999091193, 0.109229282, 0.0604393072, 0.0215812474, -0.0133415759, -0.0412526429, -0.0891536921, 0.0472001992, -0.0385942794, -0.0372761562, 0.0164892618, -0.0372883528, -0.0557279214, 0.0152035058, 0.0812813714, -0.0231321603, -0.0780240893, 0.0370430872, -0.0311998241, -0.0423431695, 0.0466758758, 0.0314119086, 0.0622362643, -0.0562412627, -0.0344490111, -0.0442969017, -0.049304191, 0.00683883019, -0.020892404, -0.063206479, 0.0327898227, 0.0409695655, -0.0873368531, -0.0458602645, 0.0283657871, -0.0296935737, 0.0476444587, -0.0509530678, 0.117646679, -0.00621824618, 0.0277476795, -0.0555988513, -0.109740973, 0.0105130114, 0.0297524091, 0.184631735, 0.0790119618, -0.0460422598, 0.0910316855, 0.0578990951, 0.0182315111, -0.0127917863, -0.017960079, 0.0287283696, -0.0742677674, 0.044918377, -0.0483011827, 0.0250649806, 0.00678098574, -0.044269342, -0.0663781613, -0.000347543508, -0.0100505101, -0.0246662144, -0.057002686, -0.0568975918, 0.0301912036, -0.0200350732, -0.0188767109, 0.0522012115, 0.0463892408, 0.043591924, -0.152667135, 0.0824710801, 0.134318724, 0.0269743279, 0.151039392, 0.0226901323, -0.0730345622, -0.0330967121, -0.0516898558, -0.174812317, -0.0257074293, 0.0621301122, -0.0281107314, 0.0220478661, 0.0866282731, -0.027407404, -0.0878577456, 0.0419084169, -0.0111707188, -0.00934631936, -0.0522210747, 0.0537884869, 0.127143726, 0.0147805922, -0.00654637814, 0.0387307778, 0.10801103, 0.0300165135, 0.0864315182, 0.0728754625, 0.0718772709, -0.0364412367, -0.0547518767, 0.143709421, -0.0218934584, -0.133334041, 0.0624611191, 0.0578976758, -0.0396091118, 0.00708054099, 0.0405613296, 0.0726592913, 0.0309684258, -0.083744131, -0.0548501201, -0.0494272448, 0.101675875, -0.0215642154, 0.123375393, -0.0718978345, 0.165513113, 0.0417141467, -0.0385921896, 0.0647833198, 0.0625313818, -0.0273620039, 0.113160901, 0.0124858376, 0.0844068676, -0.00592989661, -0.125264242, 0.0214062557, 0.00101898704, -0.0866645724, 0.074369356, 0.0353511684, -0.00341259036, 0.0402248167, 0.103089698, 0.0241240896, 0.0281016678, 0.0647317246, 0.0484072156, 0.00260333717, 0.0806719288, 0.0556133464, 0.0305167902, -0.130550414, 0.0499900691, -0.0442105159, -0.0194056518, 0.0183764473, -0.0511059687, -0.130070806, -0.0861144736, -0.00400169939, 0.0577306412, 0.0422600433, -0.0579869635, -0.0578300878, -0.0537304431, -0.0602031723, -0.066088818, 0.040910773, -0.0332243033, 0.0792824775, 0.0043681711, 0.00194717385, 0.0401844606, -0.016646564, 0.117509194, -0.00988304988, -0.0904306918, 0.0285768807, -0.151715368, 0.0195446908, -0.00713053904, 0.0684813485, -0.0694144517, 0.0639567599, -0.0141224228, -0.0207244568, -0.0296922717, -0.0194474719, -0.0350046568, -0.0731175765, 0.168188646, -0.0249032006, 0.0842974335, -0.0823265016, -0.112943903, -0.00855501555, -0.0600771196, -0.0475757346, 0.0236428473, -0.0537813269, 0.146287277, -0.0509384796, -0.0470417179, -0.0222033858, -0.0364901014, 0.0707078725, 0.0310483929, -0.0450474359, -0.0181935355, -0.0425695963, -0.0426797159, -0.0115664834, 0.0199962053, -0.0284783319, 0.0902431235, -0.100104012, 0.0212346949, 0.0198086612, -0.0146595091, 0.0760433674, 0.0716702789, 0.00554377399, -0.0230141133, -0.050588496, 0.0202339869, -0.0210531391, 0.136061847, 0.0470025055, -0.10470514, -0.00303026522, -0.113174602, -0.0267245173, 0.132816851, 0.0213535279, 0.0259472076, 0.132329449, -0.0173266474, -0.0811171085, -0.0184324402, -0.0813559815, 0.0657531172, 0.046624817, 0.00359552959, 0.0575605258, -0.0541601181, 0.0254118703, -0.137719303, -0.0417364947, 0.0423041619, 0.0202506185, -0.0195877571, -0.023350738, 0.0826441273, 0.110886008, 0.0687579885, -0.0463316776, -0.134521782, 0.100194745, 0.0410161205, -0.00395131297, 0.00482333731, -0.00644457527, 0.0183433518, 0.0206830464, -0.0286361426, -0.00480449479, -0.126060754, -0.177004084, -0.0608632937, -0.0139637049, 0.0203376394, -0.0749329627, -0.0407788306, 0.0204052217, -0.0662969947, 0.078606464, -0.0162995551, -0.0446676165, 0.126014769, -0.0192059055, -0.0495526344, -0.102695242, -0.0839841068, 0.118974932, -0.0160563327, -0.0456284434, -0.0693094134, 0.0633227155, -0.0573969819, 0.0543826148, 0.0586393923, 0.00261447206, -0.0125287855, -0.00625405833, -0.00850772113, -0.0398782492, -0.118451536, 0.0265236162, 0.0489762612, 0.0341009386, -0.135604545, 0.020351816, 0.0166754648, -0.0374540947, 0.053348802, -0.0471646935, 0.0322194993, 0.0764915422, 0.0575322248, 0.0555176884, 0.0738041922, 0.0196397863, -0.0199799687, -0.0167425089, -0.0813268274, 0.0436506718, 0.0957128257, 0.00954717584, 0.0955782607, -0.0245291926, -0.0802243352, 0.0244744271, -0.0365811288, 0.0109992363, -0.016655989, -0.0683113039, 0.03798512, 0.000307982787, -0.0178943016, 0.0966184512, -0.023319792, 0.041559726, -0.0101287384, 0.0463580526, -0.00365750492, -0.0358866826, -0.0700493157, 0.0663632378, 0.011852961, 0.0954577252, 0.0503681414, -0.0189930126, 0.0833584666, -0.00434620492, 0.0278614219, 0.0824855343, -0.0362288356, 0.0619418994, -0.012426367, 0.0177298374, -0.0858480558, -0.0425604358, -0.00187760405, -0.0801159814, -0.0747970194, -0.0605991669, -0.054938674, -0.160571754, -0.10273765, -0.064515166, 0.0506173894, 0.172788367, -0.112273581, 0.10875617, 0.105825163, -0.0419232398, 0.00939384848, -0.0853435025, 0.150468662, -0.097040385, -0.0455691889, 0.0122150015, 0.0413690917, 0.0682350248, -0.0273765586, -0.0179612003, 0.0421005338, 0.156339943, -0.0342764854, -0.0325632803, 0.0643644631, 0.0477475636, 0.0803897455, 0.0825190842, 0.0547175817, 0.0173911434, -0.0715173557, -0.00152230356, 0.0400967933, -0.0453807414, -0.0151761044, -0.0338224657, 0.0100010531, -0.00146011403, -0.0140550099, -0.0557222106, -0.0344187729, 0.0561566874, 0.0133771412, -0.0760608837, 0.0155389486, -0.112964481, 0.0914521813, 0.0426513255, 0.0366894528, -0.0473994911, 0.0761143565, 0.0824425146, 0.0274065454, 0.0152111407, -0.0503255092, 0.0172616839, -0.0593324602, -0.0172303263, 0.00308240019, -0.0577234626, 0.0263771545, -0.0507110953, -0.0281999558, -0.090995945, 0.0636361092, 0.0812521353, 0.116399832, -0.178540945, -0.0231116042, -0.00664621592, -0.00276392698, 0.0626842231, -0.00238338951, -0.11642497, 0.132260993, -0.0321269259, 0.0353224277, 0.0228020456, -0.0109135956, -0.176569864, 0.115213133, 0.0010151458, 0.0676492006, 0.101031266, 0.143366262, 0.0417161956, -0.00427427515, 0.0658375919, -0.0152567644, 0.00748937763, 0.0704953149, 0.13803634, 0.0183069855, 0.162487373, 0.00474989414, -0.0824215859, -0.0786737055, 0.0798738673, -0.00576939806, -0.0380873792, 0.0382369757, -0.0899851173, 0.0582171828, 0.0747998357, -0.00938384421, 0.0178993065, -0.101265922, -0.0767208487, -0.0334910974, -0.0122476164, -0.108730927, 0.0226861201, 0.0451159962, 0.0346092135, 0.0383441411, 0.0947932526, 0.0272382237, -0.0212542247, -0.0790283605, -0.0552407913, -0.0681997985, 0.0571708828, -0.0888224468, 0.171371549, 0.115902402, 0.085053876, 0.0852688029, -0.0622111969, -0.0810289681, 0.0628453046, 0.0909025818, 0.0766188204, 0.015920477, 0.0323929489, -0.0491212904, 0.00635633245, 0.139184266, -0.0772110596, -0.00271943398, 0.0171520598, -0.0577545837, -0.0147244949, -0.130892605, 0.0210893378, -0.0356468558, -0.0687654093, -0.0233412031, -0.0378773734, -0.0688846037, 0.0723050535, 0.0304395817, 0.154884219, -0.0249646585, 0.0978060961, 0.00456910022, 0.170681819, 0.0672572032, 0.0128455516, 0.0483344123, -0.0275884941, 0.018953776, -0.0247757919, 0.024620343, 0.0379876159, -0.0161838569, 0.00522168819, 0.0413740091, 0.0556953102, 0.0979369208, 0.000465229154, -0.00256701373, -0.0528493561, 0.0299092606, 0.103071868, -0.021854179, 0.0181949586, -0.0524465144, 0.0198814608, -0.0476320088, -0.1071162, 0.013264575, 0.0278748982, 0.0314943418, 0.00166141428, 0.0398771614, -0.0338519588, -0.0514496826, 0.0188677199, -0.0722236931, 0.0850957707, 0.019859042, 0.0605553389, -0.0276205912, -0.0624502301, 0.0885268971, 0.0611201599, 0.0937642455, 0.0316938236, -0.0124673555, -0.0105345063, -0.115935177, -0.075589627, -0.0874573737, 0.0451529883, -0.0241872575, -0.107217774, 0.0114910956, 0.00739411917, 0.0635644943, 0.00718290592, -0.017211061, 0.0649744049, 0.144540027, 0.0213773698, 0.0330918059, 0.126072571, -0.0628160164, -0.0302060433, 0.0473956987, -0.0750607178, 0.0923222229, 0.0203207023, -0.0576080494, -0.0571265295, 0.0295807943, 0.0476654023, -0.0424895845, 0.00272396463, -0.00376596488, -0.05612389, -0.0827507675, -0.017534446, 0.0130465236, -0.0112675847, 0.0387097821, -0.0923534781, 0.0232520513, 0.104455814, -0.0591111444, -0.0408475026, -0.00170109258, 0.0355550572, -0.0936222076, -0.0633827522, -0.0336418115, -0.0283110663, 0.119734377, 0.0362372808, -0.0178521443, -0.0347434059, 0.0371553525, 0.0428178571, -0.0470798984, -0.014435729, -0.164340824, -0.0677405745, 0.0374167711, -0.0154086668, 0.0678320229, -0.0432913862, 0.00887353532, 0.0130027086, 0.00821114145, 0.095090799, 0.0587699004, 0.0332566127, -0.0636463091, 0.032122653, -0.0219024513, -0.0652124733, 0.0691806525, -0.0505850688, -0.0104172789, 0.223210961, -0.044111412, -0.0190373994, 0.0624974184, 0.00483464496, -0.0819261223, -0.0178205371, 0.0510521121, -0.00159915769, -0.0210735798, -0.0275107585, -0.0553292409, -0.0577378422, 0.0563777611, 0.039552357, -0.0373257883, 0.0426951572, 0.0649646223, -0.142188519, -0.0296199471, -0.141941428, 0.0800876543, 0.0174598247, 0.0182163995, -0.0711499974, -0.116931707, 0.0124670956, 0.0647682622, -0.0088250367, -0.0828026161, -0.0716979653, 0.0993459746, 0.0244998578, -0.0833762959, 0.0699710697, -0.0722075403, 0.0184278078, 0.0220115297, 0.035694994, 0.0999014378, 0.0220938455, -0.0733663961, -0.0680553392, -0.0286444314, -0.0238020867, 0.0613737963, -0.0661988258, 0.0434220359, -0.0388579257, -0.059150286, -0.0738395602, 0.0442918018, -0.00199081749, 0.0343519561, -0.048179362, -0.101486929, 0.0947650671, 0.00531408843, 0.00581371225, 0.0459128916, -0.104510233, -0.105772093, 0.0460408218, -0.0952528715, 0.00215967512, 0.037196029, -0.135131702, 0.0147949029, -0.140816733, -0.155108348, -0.0137244007, -0.100251906, 0.0525934808, 0.0418335721, 0.0528184474, 0.0185612068, -0.066091381, 0.0581442602, 0.0264060237, 0.0249687135, 0.0126784164, -0.0213382002, 0.14356859, -0.025588043, 0.0251991991, 0.0487632602, 0.051497601, -0.0186653063, 0.0307775959, 0.0873808786, -0.0129293213, -0.0343670473, -0.041797813, 0.00551332533, -0.0338438563, -0.0834582895, -0.00171607733, -0.136069417, 0.0233047828, 0.00045992434, 0.000560967252, -0.031112045, 0.0420279168, 0.0651004314, -0.0240920987, 0.0504302941, -0.0523189232, 0.00748384744, -0.0347873829, 0.0270464271, -0.0563101545, 0.00681879558, 0.0897459239, 0.0443956032, 0.0180710144, 0.0505091958, 0.0695903599, 0.125732213, -0.0377849378, 0.0318544284, -0.041692093, 0.00449652085, -0.0733940601, -0.0236523841, -0.0389677659, 0.0682021901, 0.0653477833, 0.0218751039, 0.0799584314, -0.044718679, -0.0546429828, -0.0343285501, -0.0238201618, 0.0650375411, 0.160124987, 0.00323855784, -0.0918040425, 0.0571831428, 0.0855839923, 0.0936674178, 0.0197503641, -0.0325945877, -0.0496607497, 0.0404912718, 0.011434311, -0.206179321, 0.0190077089, 0.0104357395, -0.0826573297, 0.0913137496, 0.0486619771, -0.052196864, -0.025139289, -0.0211637858, 0.0446099713, 0.0498885997, -0.00635213032, -0.0430392586, -0.12492241, -0.0517646745, -0.0389231369, -0.0605589636, -0.112328216, -0.0165648572, -0.0221584495, 0.0800962895, -0.165377423, 0.0768084005, -0.0111929718, 0.0502661578, 0.0293068029, 0.086451605, -0.0690438226, -0.0168637726, -0.113575645, 0.0728008151, -0.0284033678, 0.00199810136, -0.0326466598, 0.00110884011, 0.0239199251, -0.0273516327, -0.0887762457, -0.057633508, -0.0376840234, -0.0635560304, -0.0157976262, -0.0463864133, -0.0310379677, 0.000594924844, 0.0676720068, -0.0762467384, 0.0637137145, -0.0541101992, 0.0848938227, 0.0722700953, -0.00970964879, -0.0968726426, -0.0156627987, -0.082167469, -0.085821256, -0.00286627561, 0.0510836616, -0.0271748845, 0.0199986864, -0.120882206, -0.0941845253, 0.0714968219, -0.0353137963, -0.0155235436, -0.11322768, 0.0300724767, 0.02503125, -0.0805938989, -0.0422333963, 0.000452307984, 0.0826343447, 0.0291987602, -0.117046736, 0.146781072, 0.0266276747, 0.0717612505, 0.0328361355, -0.0160855427, 0.0627054721, -0.00673240144, -0.0527958274, 0.0986901745, 0.130189121, 0.0257242434, -0.0119243208, -0.0644691959, -0.0569007397, -0.0197811108, 0.0376521535, -0.0145491818, -0.0203202888, 0.0552487969, 0.0469736829, 0.0532319397, -0.0220983177, -0.109317824, 0.0277715139, -0.0971366167, 0.11868684, -0.0519852042, -0.0462112874, 0.110858575, -0.00812960044, 0.07215783, 0.0420408919, 0.0272742826, 0.0513974205, -0.0118993046, 0.000521635753, 0.0774578229, 0.137766019, 0.00389761105, -0.0847367123, 0.124371111, -0.0781337768, 0.0236005578, -0.0448037386, -0.0195980482, 0.064603053, 0.0510761738, 0.0787157565, 0.0232228003, -0.178466871, -0.0180326495, -0.00609694142, 0.0539999232, 0.127497181, -0.163495481, 0.0055763945, 0.021452615, 0.0167651288, -0.0564832278, -0.0881112367, 0.0691584572, 0.00940729119, -0.0354472846, 0.0706351697, -0.0157173183, 0.0690189824, -0.0348912403, -0.172110319, -0.00943912566, 0.037896499, 0.0879924074, -0.0132095292, 0.0273147691, 0.0782328248, -0.0353201181, -0.0368057862, 0.0926254913, 0.0984198749, 0.0888203457, 0.0110497028, -0.0468932949, 0.0700697228, 0.0721681267, -0.0407189876, -0.0508127771, 0.00764561631, 0.0620290115, -0.018086303, 0.0721296072, -0.0532863215, 0.0285714287, 0.0565509051, -0.0246238019, -0.0535491854, 0.00527651608, 0.0480368733, -0.0522501208, -0.0694386736, 0.0114324987, -0.0569064915, -0.00525434176, -0.086925745, -0.00653358176, -0.0407739989, -0.0666615441, -0.013990188, 0.0202354565, 0.0117556173, 0.0172367785, 0.0228445139, 0.0163306054, 0.171092138, -0.000374388881, -0.0166255478, -0.0411830619, -0.054597754, 0.00360160507, -0.00733478786, -0.0771324262, 0.00589535013, 0.0139383953, -0.0553720295, -0.0029944079, 0.0624362491, 0.0426834784, -0.0417445153, -0.0688990876, -0.14986451, 0.0661635771, 0.102298096, -0.0286631137, -0.00590039417, 0.0234006699, -0.0607436597, 0.0334910899, -0.0732105374, 0.0726313069, 0.103060856, 0.059321247, 0.117203362, -0.00131064467, 0.010926961, 0.00992588699, 0.0934898481, 0.0287312325, 0.0179790948, -0.0190981403, -0.0463288128, 0.0243524648, 0.0986140445, 0.0259257164, 0.0221054554, 0.0201974791, -0.101369828, 0.0743303299, -0.0123497397, -0.0316775106, 0.0110243559, -0.0451925546, -0.0274194404, 0.0198468529, -0.063109301, 0.0784273893, -0.079125829, -0.0810243487, 0.00667224312, 0.0253600981, -0.00810301397, -0.0233241413, -0.0154799037, -0.0222160909, 0.0666123331, 0.0847653896, -0.0614793934, 0.101951972, 0.0692358017, -0.129346803, -0.0389242321, -0.0615266636, 0.0449628793, 0.0873149037, -0.0889803916, 0.0828250796, -0.0695593879, -0.00529191643, 0.0390869677, 0.0497748591, -0.0497797728, -0.0923573971, 0.0842193663, 0.0490318798, 0.0939242989, 0.0431354567, 0.0075036101, -0.0502004996, 0.0051574707, 0.104648948, 0.00652322173, 0.0311393365, -0.0889016911, 0.046053566, -0.077221781, -0.0539447963, 0.0284959376, -0.0782696754, 0.0726768821, 0.0369494893, 0.0109350355, 0.0849522352, -0.0148188025, -0.00333061721, -0.0220909752, 0.0817275271, -0.000128056854, 0.0143208802, 0.0698198825, 0.118775882, -0.0905991495, -0.0931259245, -0.0306694824, -0.0226295888, -0.0445462242, -0.02356942, 0.0209103636, 0.0200701039, -0.0976861268, 0.0168927442, -0.0741260946, -0.0285322461, 0.121816196, -0.0573611073, 0.0380295366, -0.0369049162, 0.100978494, -0.0513944328, 0.0728330538, -0.0434479676, 0.0569366477, 0.039275758, 0.00326382788, 0.00178216584, -0.0554266125, 0.0447509438, 0.0463842712, -0.00143668056, -0.0497579575, -0.0403893478, 0.00282532722, -0.021620594, -0.0561324209, 0.0627597421, 0.0772250146, 0.0611826219, -0.101728, 0.0425148942, 0.0411761068, -0.108952448, -0.0502944626, 0.000726735219, -0.0114530418, -0.217278063, -0.00120753399, -0.134166822, -0.0578782335, 0.0359523296, -0.00815599784, -0.0596450344, 0.0944110006, -0.0364188068, -0.0051490441, 0.00569918659, 0.0921898484, 0.0650417656, 0.00425115088, 0.143778682, -0.053511072, -0.0609003678, 0.0591868237, 0.0643764287, -0.0527997017, -0.00172682526, 0.0506346524, 0.00102965347, 0.102674454, 0.0281052012, 0.0704697296, -0.061931923, -0.0409564339, 0.034145046, -0.147151709, -0.043701373, 0.117814213, 0.00428507011, 0.0280635897, 0.0622178502, 0.0829013065, 0.0693673119, -0.0946927667, -0.106617078, -0.000915246375, -0.0758073702, 0.0673018843, 0.0832968578, -0.0876506045, -0.0684491694, 0.011782553, 0.0124366907, -0.0322360061, 0.0601471327, -0.0132275485, -0.00912743434, -0.0743104294, -0.0523917526, -0.0177966133, 0.0322803557, -0.12027818, -0.179780707, 0.0397666655, 0.0871073157, 0.0361456871, 0.0192496721, 0.0740107521, -0.0601837412, 0.00571251102, 0.048491329, 0.0490451455, 0.0143180341, 0.0589662269, -0.0321560577, -0.00506042317, 0.113666214, -0.00667214021, 0.047034964, 0.116589114, -0.00167111773, 0.0323045552, 0.082508415, 0.207803503, -0.0146126729, -0.068054013, -0.0145918261, -0.0141749717, -0.0789187774, -0.0144576468, -0.0139304902, 0.0157333538, 0.0893411785, -0.032695841, 0.0383776724, -0.0559048019, -0.0227198377, -0.0431284308, 0.115025818, -0.0656343773, 0.0579454601, -0.00356069184, -0.0369944833, 0.155177191, -0.0208048802, 0.02005562, 0.0832887143, -0.114914574, -0.0887392536, -0.0147787016, 0.0706412643, 0.0913077369, -0.144511506, -0.0877337456, -0.0451671295, 0.0256611761, 0.0988015458, 0.0451758653, 0.0310547724, -0.00588363595, 0.0488314852, 0.0772113204, 0.0739604384, -0.0632761493, -0.080322504, -0.0433514975, 0.0508803353, 0.00592380576, -0.0488886088, -0.0323207751, -0.0969795883, -0.0664113164, 0.0180361234, 0.142998949, 0.01674206, -0.0285663232, 0.0650697947, 0.0355888791, 0.0443377793, 0.103645802, 0.0734687224, -0.0599622317, -0.00753226224, 0.0170119163, 0.047288429, 0.120533921, -0.00502235303, 0.0266937762, -0.0339505374, 0.0209436454, -0.0600645356, 0.0243292581, 0.0910030305, 0.0375225767, -0.0125856623, 0.0423483588, 0.0493672714, -0.012294271, -0.0531083457, 0.10499195, 0.0168936998, 0.0884558409, -0.120901324, -0.0413734056, -0.032425005, 0.0257995129, -0.0491530783, 0.0316093862, 0.0229974203, -0.0243101493, 0.111842476, 0.0420154482, 0.038370844, -0.0425583646, 0.0349923484, -0.0169296768, -0.0846606344, -0.00560978567, -0.104491726, 0.0748140067, 0.0776159838, 0.10322924, 0.0315449275, -0.00243660808, -0.0387761593, -0.0396274887, -0.00475567207, 0.076740995, 0.059409298, 0.0456399024, -0.0138041256, 0.0166268982, -0.0361152515, -0.00875334442, 0.0298692957, -0.00163854565, -0.020314699, 0.0837704986, -0.0538312718, -0.0692103952, 0.107342288, -0.070803389, 0.0353907496, -0.0458231717, -0.142203629, 0.0130435675, 0.00728995726, -0.010904571, 0.0181974322, -0.0177388601, 0.0646408871, -0.0300395433, -0.0032200797, 0.0791164115, -0.0304487329, -0.0339283869, -0.0499682464, 0.00879298896, 0.0932347029, 0.0261517558, 0.121718884, 0.0708100796, 0.10898643, -0.0353405066, 0.000164954923, 0.0522483625, -0.0247272216, 0.033231236, -0.116206191, -0.00151216215, -0.024410788, -0.0165810678, 0.0444157943, 0.0302606802, -0.1038495, 0.0615112334, -0.00725403056, 0.119801059, -0.0251923427, -0.0582809336, -0.00923966989, 0.0668835565, -0.0560684465, -0.0180041213, 0.0253624022, 0.0424987227, -0.0759863555, -0.024532754, -0.00648979703, 0.118599974, -0.118901506, 0.0166608915, 0.0860791132, -0.115887888, -0.0413733348, 0.0430880785, 0.0469225943, -0.0201336052, 0.105008431, 0.011856419, -0.00948309526, 0.0378922671, -0.00603734329, 0.0647123754, -0.00429551955, -0.0816417858, -0.0272960998, 0.00608416088, -0.021304803, -0.0373854339, -0.0505375117, 0.121371053, -0.103410885, -0.00353913195, 0.00895364303, -0.0192505382, -0.0020865649, 0.0507494956, -0.00524902064, -0.0161629748, -0.0223817211, 0.0313353986, -0.124332212, -0.012889999, 0.0343106166, -0.027769275, 0.0182169117, -0.050058566, -0.0499154627, 0.00406805426, -0.00722800661, 0.00199822336, 0.0155832153, -0.0795259476, 0.0235153642, -0.0279665086, -0.0735083967, -0.0395488329, 0.0996877775, -0.100186974, 0.0335906446, 0.0726341605, 0.000761864707, 0.0465911552, 0.00783610996, -0.0558331423, -0.0300832018, 0.0426513255, 0.0209049527, 0.085289903, 0.0327272676, 0.0397153758, 0.0511196963, 0.0783239976, -0.0824877843, 0.0640061796, 0.0145687666, 0.0530257113, 0.0180169754, -0.0332160816, 0.0940923691, 0.0237015449, -0.13688682, 0.0209730752, -0.134351626, -0.0243419074, -0.133830249, 0.0331348106, -0.0154519267, -0.0396372229, 0.0504556112, 0.137901902, 0.0451988354, 0.0245524999, -0.0222883336, 0.116566993, -0.113128595, -0.0366410725, 0.0129554765, 0.0713988543, 0.0670085475, -0.0591761358, 0.0672670603, -0.0779664814, -0.0297863353, -0.133227706, 0.0908347815, 0.0168455578, 0.0329658985, -0.0233854614, 0.0169380866, 0.043512933, -0.0264570527, -0.0739393756, 0.00335022272, -0.0392536484, 0.0944359601, -0.0087780077, 0.0620283, -0.015076464, -0.19268696, 0.0398401581, 0.0429010764, -0.0572125651, -0.0206910521, 0.0677373782, 0.00495192595, 0.0617411099, -0.0203344077, 0.0340360068, -0.0623074509, 0.0366723724, 0.0575639419, -0.119209975, -0.0425331816, -0.0308947489, 0.0385033973, 0.102489576, 0.0565514974, 0.113505311, -0.0691952333, -0.0244075805, -0.0288813524, -0.0458136871, -0.0475862063, -0.0580462515, 0.0812397227, -0.118253723, 0.0729867071, 0.0104914941, 0.0816968381, 0.0620579906, -0.0106690116, 0.0762378946, -0.0197269283, -0.119938746, -0.0373863801, -0.0765926242, 0.0684237555, -0.0109639838, 0.00195817649, -0.0115007246, -0.102584273, -0.0426782891, -0.0247023106, 0.0726862177, -0.0135520324, 0.0266301036, -0.00465337466, -0.0629284978, 0.0171643253, 0.106216289, 0.0259720795, 0.134041995, 0.0131572997, 0.00893884338, -0.0128664393, 0.0191027932, -0.0298050549, 0.0507684313, 0.00955994334, 0.0203105602, 0.0271586105, 0.0634404421, 0.0331248082, -0.027467303, -0.0337019563, 0.00549930613, 0.0485441014, -0.0820040479, 0.0647023842, -0.03118404, 0.0381694324, -0.120596409, 0.00405105762, 0.0470582843, 0.0421390235, 0.0558481403, 0.0227792244, 0.00232546171, 0.0203727763, 0.0329870246, -0.00913679507, 0.00542233791, 0.0326804668, 0.0516836643, -0.00668152329, -0.113703594, 0.00792934932, -0.100547522, -0.0116469357, 0.0608402602, 0.00933902618, -0.072523728, 0.0825108439, 0.047987543, -0.135880008, 0.043875061, 0.087684691, 0.0541803055, -0.0520437099, -0.0432396866, -0.0770369321, -0.0167596415, -0.00916953757, 0.081689477, -0.0433455035, -0.0237326846, 0.0506320521, 0.125054032, -0.0777374059, -0.0284106452, 0.0599854216, -0.0668424815, -0.0930463746, -0.065400809, -0.0269185267, 0.0197632089, -0.0743044019, -0.0126272477, 0.0349280275, 0.0065385066, -0.104033835, -0.0158705916, 0.00572146149, 0.00123008108, -0.159773067, -0.114516899, -0.0284334235, 0.0300769694, 0.0377564207, 0.0364852473, -0.0538404211, -0.0390040651, -0.0112615097, -0.0241562724, 0.0871999562, 0.00464407634, 0.193107814, 0.0650430322, -0.088600114, 0.0486501157, -0.0416172706, 0.0675915778, -0.00498365983, 0.0602493808, 0.103646383, -0.0680672824, -0.0779883489, -0.0584908947, 0.0545057505, -0.0315716453, 0.0738639385, 0.0397104882, 0.167447194, 0.0838308409, -0.052024927, 0.0177263226, -0.0255030468, -0.0349459276, -0.072929211, -0.00671998784, -0.0894785151, -0.0437568724, -0.023049105, 0.0537241362, -0.00767988339, 0.00176991429, 0.0666914433, 0.00931717269, 0.0666778162, 0.0762925893, -0.0518660471, 0.00794638693, -0.0555208288, -0.0398611315, -0.00251298398, -0.0451297425, -0.00623324607, -0.0251096673, -0.0302794259, -0.0156251527, 0.0431078598, 0.0426377766, 0.00500511983, 0.119465999, 0.104776397, -0.0642026886, 0.0366924293, -0.0462633707, -0.0613944419, -0.0197751187, -0.00981658045, 0.04499631, -0.0370547399, -0.0232003555, 0.0686958581, -0.00233231857, -0.033743687, 0.0270552188, -0.128848284, 0.0207115673, -0.00663662702, -0.00459149433, -0.00697533041, -0.0319461077, -0.00151833612, -0.0933296084, 0.0241516493, 0.0613977239, -0.118570551, -0.0593892448, 0.024415018, -0.0609763637, 0.0811836869, 0.0377169028, 0.10369055, 0.0938747674, 0.109625481, 0.0649345145, -0.0242359042, -0.0572986007, 0.0685245693, 0.0325403586, 0.020280784, 0.00820967183, -0.0120230569, 0.127929434, -0.0542152748, -0.0573881865, -0.00447639357, 0.059505593, -0.0602974854, 0.0548756048, -0.0291398391, -0.0537097082, 0.0525500402, 0.0445300043, 0.00536491163, 0.0559389144, -0.00901229959, 0.0128884437, -0.0156487767, 0.0291651003, 0.013363149, 0.0379870422, 0.0190792084, 0.110151999, -0.0426378958, 0.156422675, -0.0527738668, -0.0848110318, -0.0275939796, 0.0424579717, -0.0407079197, -0.140546858, 0.0778859258, 0.0212555937, 0.100470148, 0.0252361521, -0.0235062782, 0.0775677487, -0.0235892367, 0.120493814, -0.0489098355, -0.0885234177, -0.0448108353, 0.122688122, -0.0353725478, -0.085962005, 0.0489472337, 0.0243719667, -0.0112771727, -0.112333745, -0.0173595846, -0.042562075, -0.0155199543, 0.142047748, -0.00654774718, -0.0707080811, -0.0704635605, 0.0160170756, 0.048383642, -0.0910952389, -0.0596754327, -0.0163724814, 0.0133493058, 0.0612010285, 0.0724545643, -0.0881462842, 0.135168493, -0.0387480035, -0.0339688249, 0.161951616, 0.132496089, 0.0611590296, 0.0292575881, 0.0203857347, 0.0642239079, -0.0570195206, 0.00449317321, 0.00462812185, -0.0301356353, -0.0331426486, -0.0413808227, 0.0761849508, -0.0526299253, 0.00907731801, -0.0337697864, -0.0904527903, -0.0811025202, 0.094873786, 0.0643247515, 0.043566335];
    CONSTANT bias_0_i : ARRAY[0..63] OF REAL := [0.557149589, 0.620696902, 0.895506322, 0.549719632, 0.672894001, 1.15932477, 0.544620633, 0.552206576, 1.08217514, 0.525080025, 0.589199841, 0.580554187, 0.594992697, 0.567867696, 0.549335718, 0.686280966, 0.786747336, 0.633696258, 0.757360458, 0.655798256, 0.70659709, 0.787525356, 0.616207957, 0.667597473, 0.548698783, 0.629144371, 0.811792314, 0.57614702, 0.601757526, 0.548455477, 0.640272677, 0.651031792, 0.651111484, 0.967581689, 0.564899862, 0.591845453, 0.73757869, 0.794382334, 0.926623523, 0.543820262, 0.648953378, 0.599694192, 0.546814561, 0.620168686, 1.07619512, 0.540103734, 0.519084692, 0.646295607, 1.13459384, 0.819661498, 0.79537499, 1.14667702, 1.06166852, 1.07402825, 0.542853296, 0.743338704, 1.18120193, 0.829793751, 0.544563711, 0.654161394, 0.562430322, 0.633703232, 0.609814882, 0.683588922];
    CONSTANT weights_0_f : ARRAY[0..63] OF REAL := [-0.0972258896, 0.050810039, 0.103591904, -0.151559591, -0.12631993, -0.0278594568, 0.0511496663, -0.0248928815, -0.0107669681, 0.0179153532, -0.00145217776, 0.0987181515, -0.0138257742, -0.0954465121, -0.0270122588, 0.046705246, 0.0429453552, -0.00344921649, -0.0856930092, -0.0354830921, 0.128278121, -0.00401186943, -0.148586124, -0.109839961, -0.14002116, 0.0943036228, 0.0928951651, -0.0137155801, 0.150729075, 0.00850623846, 0.143254027, 0.107316509, -0.0664839447, 0.0822855383, 0.0174088329, -0.0571946576, -0.0489450172, 0.0903148055, 0.055499211, -0.0399800166, -0.0752305835, -0.0558629856, -0.107780077, 0.0128436536, 0.0913120955, -0.0740158558, 0.0231325477, 0.0374446213, 0.0614935905, -0.0222444087, 0.15084587, -0.0129477233, -0.133767843, 0.0278934091, -0.0156487226, -0.0476486161, 0.00977171957, 0.0435241759, 0.120144472, 0.0274345428, 0.1381201, -0.00205555558, 0.0619449466, 0.0855321288];
    CONSTANT recurrent_0_f : ARRAY[0..4095] OF REAL := [0.0300157573, -0.107296921, 0.0577121899, 0.105559483, 0.0968114436, 0.0540135652, -0.16776602, 0.00489261188, 0.00876335707, -0.0560048781, 0.00808845647, 0.0350553691, 0.00702001154, -0.0585917719, 0.00585619546, 0.00908345543, -0.00727013359, -0.0709282309, 0.0392159522, 0.0374129489, 0.0811483786, 0.00797758065, 0.157243893, 0.0251566432, -0.0373158418, 0.049337849, -0.0145778172, -0.050251171, 0.0534369424, -0.0187977664, -0.0288828406, 0.0362210721, -0.0544360355, 0.106145248, 0.00803098734, 0.0568142347, -0.0750947297, -0.0875710994, -0.00890454557, -0.128214076, -0.0628437325, -0.00575138442, 0.0420288593, -0.0228305589, -0.0761641264, 0.014828057, 0.0304486379, 0.0380928591, 0.0477362424, -0.107235461, -0.0554246083, 0.0914537236, -0.144681022, 0.0244761687, 0.0109966258, 0.0931695104, 0.0262197107, -0.073358357, -0.0192161556, 0.0533077121, 0.121210866, -0.0218135007, -0.0247535203, -0.0305508971, -0.00396067835, -0.082525678, 0.0340822525, 0.0110075753, 0.0258307457, -0.0863573402, 0.0158065259, 0.0099548921, 0.164907068, 0.0200332776, -0.0531619489, 0.052447442, 0.0376975313, 0.0247805864, -0.0540729389, 0.0550032444, 0.124538578, -0.0314540714, -0.0518662483, 0.0452731736, 0.0532553047, 0.0706339926, -0.039131023, 0.0481084473, 0.0495813116, 0.00543319434, -0.072397992, 0.0215297993, -0.00718787778, 0.0377878249, 0.0161217861, 0.0528881736, 0.0244731586, -0.0130320787, 0.0786133185, 0.0653051287, -0.102847569, -0.0340424329, 0.0618168116, 7.66108278e-05, 0.0987020805, 0.00815586001, -0.0390097164, -0.0837471038, 0.131946817, 0.0269339792, -0.0420012623, 0.0653122067, -0.0287024807, 0.0874734819, 0.0999993384, 0.0786093101, -0.048870936, -0.047350578, 0.0356673785, -0.105057344, -0.0582771972, -0.0241910089, -0.0163621847, 0.0106756343, 0.0598100014, -0.0566131659, -0.0904669538, 0.0410108939, -0.0327403322, -0.00844661146, 0.0155591443, -0.0690867603, 0.0335778557, 0.0117144659, -0.0685847402, -0.156900227, -0.14021191, -0.0627200902, -0.00635191938, 0.00835708622, -0.0173370969, 0.0135392789, -0.000423413701, 0.0749883279, 0.0320111997, -0.0404338203, -0.00162578188, 0.0477140881, 0.0769734234, 0.0448120795, -0.0917899907, -0.15990217, -0.0353840329, 0.0825516433, -0.038971778, -0.0699695125, -0.0724905059, -0.169047311, -0.00978161395, 0.0599830784, -0.0719687566, -0.0387360007, 0.0646608472, 0.00624832138, 0.0111842062, -0.113380417, -0.0616687164, -0.0287733041, -0.0666333735, 0.00454676896, 0.0551150814, 0.0658587217, 0.0388762951, 0.0565043017, -0.137978807, 0.0592838749, 0.0543245226, -0.00752030872, -0.0374696553, -0.0551998578, -0.149481416, -0.045555979, 0.0746385604, -0.0107241916, 0.106372446, -0.0165081695, -0.048127573, -0.035963688, 0.0233876929, -0.0560876392, -0.0281021409, 0.0426667072, -0.0399390087, -0.0614325814, 0.0169947892, 0.0532067381, -0.12927492, 0.0189563688, 0.0966870189, 0.0529292226, -0.0225986615, 0.092780441, 0.0348804146, -0.0135886325, 0.00089642033, 0.0731530935, 0.137950227, -0.0180324651, 0.0859919563, -0.0463475846, 0.1633448, 0.0413299873, 0.024440024, 0.0487221852, 0.0410910994, -0.0340180844, -0.00988311786, 0.0776593834, -0.0416503921, -0.0127016902, 0.07471136, 0.122479618, -0.024158163, 0.0390037745, -0.0847889632, -0.0399800502, -0.0483349934, 0.058813069, 0.0505923182, -0.0144980345, -0.0228271559, -0.0313460752, -0.0968465656, 0.117606729, -0.0667021573, 0.00384232774, -0.000127766281, -0.0428667888, 0.0689500272, 0.095163852, -0.08197999, 0.0210441761, 0.02325904, -0.0105144884, -0.0580793098, -0.0906413347, -0.0582061149, -0.0288412273, -0.0632094219, 0.0455037057, 0.00596623309, -0.0303176232, -0.0214533545, -0.0345825441, -0.0750864446, -0.033472456, -0.134758562, 0.010237705, -0.0136257289, 0.0738518611, -0.0405869447, 0.0506134406, -0.0324666202, 0.0226186737, 0.00947999489, 0.00477958797, -0.0586758852, 0.0553540699, 0.0358029902, 0.0130361225, -0.0763754174, -0.0570643246, -0.0065658493, -0.0137131577, -0.0680585355, -0.0225489214, -0.0337488241, -0.060984157, -0.0606652945, 0.0599233136, 0.0670647994, -0.0640354082, -0.0724011883, 0.0454865322, -0.0205971804, 0.103284724, -0.0468193628, 0.0912635773, 0.011042811, -0.0336309336, 0.0799990892, -0.124603756, 0.0209672339, -0.103411168, -0.082585901, 0.102924213, -0.0518376902, 0.00844401494, -0.0200045854, 0.0489162579, 0.0277457964, -0.0381961875, 0.0780443996, -0.0527090169, -0.107666291, 0.0454847813, 0.0171944462, -0.0260603949, -0.0668711662, 0.0269614719, 0.0766852051, -0.0282195285, -0.0632535219, 0.00401621126, 0.0280937403, 0.0668497905, -0.0103374571, -0.0465457663, -0.0886795148, 0.0730986595, -0.00652642827, 0.00411921926, 0.0804560408, 0.00585519522, -0.0295318626, 0.00653597014, -0.117826082, 0.0224966276, -0.0548547767, -0.0237554908, -0.116732739, -0.078685686, -0.0182806049, -0.0258663185, -0.0448314622, 0.00296929502, -0.0174326487, 0.0123361563, 0.115678288, 0.0170686021, 0.000709696906, 0.008760361, 0.0223996714, -0.00904988311, 0.113368645, 0.0460165888, -0.00989809353, 0.0597530231, 0.0311281141, -0.0211067125, -0.0570268147, -0.085159108, 0.0670105293, 0.0310663804, -0.113299958, 0.00302693248, 0.043690294, -0.0186505914, 0.0275345128, 0.0376328826, 0.024277024, 0.0375690684, -0.136905819, -0.0424578339, 0.016883824, 0.126654163, 0.0156297982, 0.0037272023, -0.0293239541, 0.0188393947, -0.0974337608, 0.0242494568, 0.13715142, -0.0868369639, -0.0535554253, -0.0241719708, 0.0743580312, -0.131574586, -0.0544683971, 0.0757071599, -0.00118608773, 0.049573902, -0.0789082944, -0.109159254, 0.111150555, 0.0896267518, -0.0142246876, 0.0146565801, -0.0129523175, -0.0396546461, 0.0315510593, -0.0262436382, -0.0816748738, 0.0140542705, 0.000450707506, 0.102194883, -0.00306949858, 0.0619575381, 0.00415146723, 0.106028907, 0.0566340312, 0.06110017, -0.0118694296, 0.0370037146, 0.0784573033, 0.0166829154, 0.000742133707, 0.00824813545, 0.0526863299, 0.0685219839, -0.0598439872, -0.0869649798, 0.0630509257, 0.0370814875, 0.0166548714, -0.0629559755, 0.0496402197, -0.0112267174, -0.00971570425, -0.0353600942, -0.0609243214, -0.0848553926, -0.0169025995, 0.0187554099, 0.0603696033, -0.064923048, -0.063279599, 0.0475542843, 0.0805823728, 0.0169862397, 0.0462651923, 0.157721177, 0.000756570138, -0.0523853749, 0.046252165, -0.00386148551, 0.0224416535, 0.0239563063, -0.0321284756, 0.00585745461, 0.00876095891, -0.0366843566, -0.0793705136, 0.0741518587, -0.0546076894, 0.0954839215, 0.0708603039, 0.0679697022, -0.0339210033, -0.0515459552, -0.0378705487, 0.150107846, 0.126022175, -0.0676481277, -0.0398717113, -0.0422539152, -0.00127757434, 0.0248618983, -0.0570580214, 0.0462330058, 0.00609673746, 0.137676865, 0.0166428797, -0.0292401295, 0.00300678937, 0.00606477633, -0.10857936, -0.0740942359, -0.0516215116, -0.0230301395, 0.00412933528, 0.0229637623, -0.0125627089, -0.015044773, -0.0759615302, -0.0942339301, 0.0611146986, -0.0233977698, 0.0531103685, -0.0210845899, -0.0150890173, -0.10126923, 0.0471062958, -0.0209739208, 0.0235699471, 0.115066424, -0.0744652152, 0.0154174948, -0.108182766, 0.0875094458, 0.0582373701, -0.0244229827, 0.0107523333, -0.0703744739, -0.0150046265, 0.0136150364, 0.0866806209, 0.12061213, -0.11909014, 0.114309385, 0.0500720516, 0.00634593517, -0.0430119559, -0.0514486097, 0.0398652405, 0.0551493317, -0.0993671119, 0.00719310902, -0.047901541, -0.0508369058, -0.0309242606, -0.013848301, -0.023289321, -0.0446673855, 0.064715378, 0.0638258532, 0.0198455267, 0.090196006, 0.156398654, 0.0234048031, 0.0152038177, -0.00111340173, 0.0572613962, 0.00924503896, 0.0184654947, 0.0100080296, -0.0453504585, 0.04000137, -0.0207371768, -0.0381314158, -0.0529899225, 0.0080802897, 0.0100207627, -0.124000855, 0.161762699, 0.0167510733, 0.00431261212, -0.095543161, -0.0612663478, -0.0459377989, -0.0071751792, -0.0178307109, 0.0883974135, -0.0141734937, -0.0300204903, 0.0190088414, -0.0101148617, -0.0286343805, 0.105847232, -0.0920557827, -0.0758810788, -0.0451645702, 0.0132741099, -4.77768481e-07, -0.17043224, 0.0218138378, -0.0782996938, 0.0390630476, -0.104807951, 0.0525238179, -0.0892623961, -0.0573253706, -0.0605598614, -0.0807707608, -0.00543115009, 0.0154707022, -0.0947566777, 0.00108426716, -0.0436592326, -0.125980109, 0.000533373095, -0.0281456113, 0.0337875783, -0.0501380377, 0.103047363, -0.0963550508, 0.0534056947, -0.03477896, 0.00157832401, -0.00905328989, 0.0942664444, -0.0532143936, 0.124488257, -0.0211327989, -0.0355936587, -0.0517729372, -0.0313892774, -0.0338115282, 0.0462723188, 0.0271287803, 0.0703095943, -0.123422019, 0.106645875, 0.00953736529, -0.0284832586, 0.0174854808, -0.0391965099, -0.0674657971, 0.0257983748, -0.0608835518, -0.0568342879, -0.0842557698, -0.0432316214, 0.0472160168, 0.0617087558, -0.0475719571, -0.132592425, -0.0148834372, 0.0646051541, -0.0638714507, 0.117436953, 0.0114657842, -0.0409544706, -0.00761602446, -0.0380030833, -0.141652435, -0.0373622663, -0.0416792296, 0.0538599044, -0.0852228105, 0.0240976773, -0.0186880771, -0.0207654685, 0.00741029717, 0.0343466252, 0.0271975119, -0.00911446661, 0.0659701973, 0.18114318, -0.0341234803, -0.0835203901, -0.00271802954, -0.0826100558, -0.0774667412, -0.0370144583, 0.0870874673, -0.0742704421, -0.0575494841, 0.0078181047, -0.0408584401, 0.018003514, 0.0536768101, -0.0443420634, 0.0129242837, -0.0655382499, -0.0244756844, -0.0738591999, -0.069828026, -0.0348306969, 0.0188186318, 0.086288169, -0.0024923922, -0.0955157652, 0.0610312819, 0.0031343305, 0.0491240025, 0.0391001776, -0.0323164761, 0.126216397, -0.0513802953, 0.0317445472, 0.114380985, 0.0458053052, 0.0489692725, -0.00333530991, -0.0775371343, -0.00248528831, -0.0141479364, 0.0427913144, 0.131443486, 0.0205759369, -0.00734642707, -0.0217872784, -0.0553966351, -0.0452353396, -0.0428337678, 0.0225552116, -0.0252576731, 0.0469143577, 0.0702069923, -0.0293021239, 0.0238809809, 0.0554527156, 0.00405825861, -0.0510712899, 0.0522107519, -0.0105979033, 0.0920042992, 0.0443653315, -0.0928714648, -0.149346665, -0.141751111, 0.0259605683, -0.0129188504, 0.0907077491, -0.0236674957, -0.0809622332, 0.0505908467, -0.0218496453, 0.0495832078, -0.00846260227, 0.0718351901, -0.057102304, 0.0426336229, -0.0337992273, -0.0598484576, 0.117320947, -0.0752067268, 0.0144730173, 0.0100675169, 0.00259863771, 0.0309539642, 0.0136928679, 0.0466301404, -0.00197487045, 0.0182793867, 0.116525896, -0.0388804078, -0.0222464819, -0.0369414613, 0.071102187, -0.0302814133, -0.0440358929, -0.0263258927, 0.0202665031, 0.132969484, -0.0388124287, -0.0266971104, -0.048445873, -0.00834849197, -0.107946344, -0.0641651675, -7.19409436e-05, -0.0740435123, 0.0832368731, 0.00473503396, 0.00838960055, 0.0228951089, -0.0460565761, 0.0217994265, -0.0177010968, 0.0127926543, -0.0418456383, -0.0244947132, 0.0483016036, 0.0715101287, -0.042323906, -0.0616275743, -0.00429606065, -0.0329274461, -0.0246998817, 0.0421429537, 0.0619165152, 0.0294495858, -0.0732646883, -0.0532499962, -0.0646737143, -0.0286637843, -0.0769366995, -0.0831085443, -0.130764842, -0.139869228, -0.0202841852, 0.000687207095, -0.0906598642, -0.0296818297, 0.00713240262, -0.0127066262, -0.0465552732, -0.0952125713, -0.0339140631, 0.0349725448, 0.0211253129, 0.0198765993, -0.0359740742, -0.0352531113, -0.000742357224, -0.0289845653, -0.0763724446, -0.0921858028, 0.081972748, 0.0510017127, -0.0569426231, 0.0582687855, -0.0320537314, -0.0790166333, -0.0513422005, -0.00978533272, 0.0181314293, 0.0569599867, 0.102170706, -0.0381839499, -0.00386366202, 0.0599790588, 0.0444344729, -0.0521000698, -0.0625491738, 0.0398212373, -0.135570988, 0.0469256528, -0.0768292472, -0.126335174, -0.00219687261, 0.00219954923, -0.0717327148, 0.0364705846, -0.037130978, 0.0685085356, 0.0250764824, 0.108345382, 0.0570757613, -0.00320311636, 0.0413179547, 0.120515242, -0.0378896408, -0.0113706701, 0.000555124134, -0.0137712061, -0.0437348783, 0.0242755823, -0.0850516409, 0.0546437614, -0.0123460442, -0.0342373475, -0.0166758616, 0.0336131155, -0.0818632841, 0.00588049134, 0.0270376056, -0.0321143158, 0.107972741, 0.0639909878, -0.0605289228, -0.129043028, -0.196594536, 0.0127318371, -0.00260038069, 0.0148955993, 0.0519536249, 0.0274236873, -0.0405782275, -0.0486324951, -0.0612642206, -0.0596810356, -0.0317957476, 0.071118705, 0.0336470529, -0.00383951515, 0.0473859198, 0.0705588982, 0.0880139992, -0.0736380816, 0.0134094683, -0.203612849, 0.0478955694, -0.0322210379, 0.0234853271, -0.00329319201, -0.0609398857, 0.0519850254, -0.0112326592, -0.0371385291, 0.00545526482, -0.0417935252, -0.0235753935, 0.0153615568, 0.0117863519, -0.125851348, -0.071494475, 0.0101061538, 0.0543513671, -0.109989181, -0.031799119, -0.05039474, 0.174945265, 0.00244279206, -0.038289763, 0.0148941912, -0.0979054943, 0.0468814857, 0.00293183746, -0.184212461, 0.0126420148, -0.0509346947, 0.000762090087, -0.0274722427, 0.00877875462, -0.0205828883, 0.0026405314, -0.0501936711, -0.0116727501, 0.0605931804, 0.0181433, 0.0809305757, -0.0609121397, -0.0220409408, -0.0525621399, -0.0140582491, 0.0238242038, 0.00380199985, -0.0105551984, -0.0807524025, 0.0312406681, -0.0689856857, -0.0503122024, 0.107463822, 0.105646774, 0.0307489894, 0.0566367805, 0.00213884097, 0.022006616, -0.0114289206, 0.0962001234, -0.0263432097, -0.00195169449, -0.0731972829, -0.107580319, 0.0711313859, 0.0181213524, 0.00312610716, -0.0304220095, -0.0469525009, -0.0531173944, -0.0234208144, 0.000626548193, 0.0384521149, -0.0825555325, -0.0298601352, -0.117202811, -0.154552102, 0.0194538906, 0.0108771585, 0.0112806028, -0.0147998147, 0.0256627239, -0.0636195615, 0.0203298926, 0.000429701991, -0.0896791816, 0.0164592527, -0.0710541159, 0.0371221118, 0.0780697688, 0.0575666353, 0.00764066912, 0.0059041502, -0.0134018231, 0.0116832303, 0.0577438325, -0.0706727877, 0.151920915, -0.0287999269, 0.0493378974, 0.0481058359, 0.0311756749, 0.059492927, -0.0964401141, -0.0468929484, 0.00606832001, -0.0781605691, -0.0636321455, 0.115212642, 0.125354901, 0.0813867152, 0.07418897, 0.0592895001, 0.11521548, 0.00933777168, -0.0316360407, -0.0665410385, -0.095013909, 0.065659374, -0.016752772, 0.056795679, -0.168719336, -0.0343472511, 0.00340427831, 0.0479519591, -0.0511112735, -0.103744403, -0.0616893731, 0.0578040406, -0.0548961312, 0.0190597288, -0.00635266583, -0.0434646457, -0.014270667, -0.031191783, -0.0188119151, -0.00411997736, -0.0306532402, 0.00313681457, 0.0159047227, 0.0555365682, -0.0177582894, 0.0581847504, -0.0469771922, -0.0725724474, -0.0209033731, 0.129915252, -0.0683327094, -0.0711028203, 0.0495454296, 0.0346807986, -0.118461847, 0.0177230835, -0.0507178567, 0.0497463495, 0.124651693, -0.0584628545, 0.0581578724, -0.0386074558, 0.0155322477, -0.0071358243, 0.0284308009, 0.0585779399, -0.0156616047, 0.112183586, 0.0188615564, 0.0879934207, -0.00844823197, -0.0314642303, -0.144461453, -0.0476539135, -0.00798191782, 0.0415343605, 0.0175704733, -0.021485528, 0.0324046127, -0.0104173888, -0.0383688584, 0.0294174012, -0.0187220704, -0.017875582, -0.0362265222, 0.00190203823, 0.0287796874, -0.0209825523, -0.116158538, 0.0385428406, 0.0510926731, 0.0366497934, -0.0726718232, 0.0318535417, -0.00530965813, 0.0421004817, 0.0166246276, 0.0426737405, 0.0370895341, -0.0235159174, 0.00781212375, -0.0987262577, 0.0173497312, 0.063046746, -0.0252205618, -0.0975227505, -0.141204387, -0.0738607943, -0.0302525591, -0.146124572, 0.0729016736, 0.0490379594, 0.0766173452, -0.0944663212, 0.0569506772, 0.0215772502, -0.0979636461, -0.0609431788, 0.0937463567, 0.0794628561, 0.0135755651, 0.069560267, 0.0786357224, -0.0372091159, -0.0124980779, -0.0461122096, -0.000945813023, -0.0767264143, 0.0724421144, -0.00539458916, 0.0449222326, 0.111242414, -0.00288730115, -0.12592648, -0.0393019989, -0.0149923405, 0.0307417959, -0.0694728345, -0.016268203, -0.0652458593, 0.0505090617, -0.030680785, -0.0939506441, 0.0603994876, 0.0292880721, -0.102742732, -0.0629078001, -0.00609797426, -0.0880881697, 0.0653271303, -0.045205798, 0.00520604104, 0.0185705535, -0.01783254, 0.0255823992, -0.150696874, 0.0518658422, -0.131320894, 0.0341961309, -0.0201621018, -0.037930239, -0.0239071157, -0.0374914072, -0.0203422178, 0.0398034751, 0.0651344806, -0.0719605833, 0.0307432972, -0.0404192433, 0.0816474184, -0.0618630424, 0.0836635157, -0.0971608609, 0.145391867, 0.014767563, 0.0389636569, 0.0471174754, -0.016892869, 0.0172007363, 0.0124081224, 0.00728872046, -0.0272685643, 0.0272303447, -0.0686877668, -0.0235823914, -0.00710995588, -0.15847455, 0.0094242543, -0.00601251004, -0.123179108, -0.031815283, 0.0743712634, 0.0150883691, 0.0975313336, -0.0283058025, -0.0166965295, -0.117393054, 0.0396461301, -0.102597401, -0.106020734, -0.0214482173, 0.12707451, -0.0556858778, -0.0374464989, -0.0737756193, -0.0332069397, 0.0431115925, 0.0722956508, 0.0732016265, -0.0260919966, 0.050417725, 0.0808667392, -0.0863302201, 0.0221759044, -0.0456107371, -0.105728447, -0.0600369275, 0.0824415162, 0.0136104412, -0.0794505551, 0.0507579036, 0.00501812622, 0.135426968, 0.0552411899, -0.0668459386, -0.0326608196, -0.0572552681, -0.092473425, -0.00125965476, 0.0450726375, 0.0269976519, 0.0337952897, 0.0659958571, -0.13193664, -0.058439225, -0.0766070038, -1.44280493e-05, 0.10533163, 0.142132089, -0.00944938697, -0.0129964361, 0.00211798307, -0.00728274882, 0.0072149504, -0.0161147229, 0.00529440306, -0.0709677339, -0.0200598631, 0.0278503057, 0.0179317817, -0.0857382119, 0.159815744, 0.109231807, 0.0831665471, -0.0327979699, -0.0526622906, 0.0464353375, 0.0284734741, -0.0427694358, -0.0711058974, -0.0839088038, 0.0195920877, 0.0139979618, 0.00333881564, 0.0512295291, 0.0437079668, -0.00752245123, 0.0317304954, -0.0401867963, 0.0284368582, 0.0770598873, -0.0266718697, 0.113287754, 0.000354602002, 0.0552334003, 0.137481332, 0.0774497315, -0.00843666773, 0.0198671743, 0.0210164897, -0.0412956476, 0.0675320998, 0.0112238843, -0.0750028864, 0.0582809262, -0.0143759772, -0.012905905, -0.150767058, -0.0505688526, -0.00693381345, -0.0182181746, 0.0696848109, 0.0140968878, 0.0918711945, -0.00677535404, 0.0585777462, -0.0434732512, 0.0411020294, 0.0542318076, 0.00982689951, -0.02255507, 0.0229797587, 0.111543067, -0.0112353787, -0.022189483, 0.0283819735, 0.0342839547, 0.0815160125, 0.138156563, -0.0550806895, 0.170456052, -0.0200003814, 0.0905138105, -0.0295825023, 0.135435194, -0.0674221814, -0.0493251458, 0.00595238851, -0.179528683, 0.0782173797, 0.0113523165, -0.0198757425, 0.0710524917, -0.0804977566, 0.0171708986, -0.0115417354, -0.0199554339, -0.0237090029, 0.11330723, 0.00954803266, 0.0262243375, 0.0715917051, 0.101236075, -0.0485668778, -0.0343779698, -0.0158949755, -0.0443178862, 0.0815009847, -0.0435290039, 0.0599850491, -0.00203195028, 0.0303352531, 0.116828352, 0.101558164, -0.0289837997, 0.0128748678, 0.0664595515, 0.0724234059, 0.0962413698, -0.0882667825, -0.0259502642, -0.0251223966, 0.0745185316, 0.0716595575, 0.0186935943, 0.0882871822, -0.0175877213, 0.0178745687, -0.0414037518, -0.111047722, 0.080509007, -0.0477794558, 0.0185205843, 0.0177610256, -0.0840014815, -0.0153660495, 0.0576493107, -0.0411044545, 0.0305890888, -0.0222739577, -0.00175685808, -0.00374436658, 0.0276121683, -0.0746644139, 0.0713727772, -0.138044238, 0.0156429484, -0.0435051546, -0.0174354445, 0.0596997961, -0.0227762219, 0.0275202971, -0.131491795, 0.0293372404, -0.0175958108, -0.037708126, 0.160618708, 0.0584641099, -0.126507178, -0.022465799, -0.0318544023, 0.00500431284, 0.0659823418, -0.0671814159, -0.0262736399, 0.0940687507, -0.00817685947, -0.0687940568, -0.00376525265, 0.0811941251, 0.0593241118, -0.00122466264, -0.0553934872, -0.0442702658, -0.0742721558, -0.0608431697, -0.0130608073, 0.0213107429, -0.0223005917, 0.0162595548, 0.0470586233, 0.0263670199, 0.0137835341, -0.0276703667, 0.045861315, -0.0423991494, 0.0548932776, -0.175383106, 0.0634888932, 0.0540193915, -0.0790458992, 0.0196334384, -0.00465807691, 0.0266548842, -0.0368627794, 0.0578659698, 0.00344062317, 0.0396462567, -0.0491361842, -0.0551700145, -0.0568456277, 0.0657523572, 0.0205887072, -0.111551419, 0.0452845432, -0.0192324258, 0.0698562115, -0.0474697426, -0.0361267589, -0.0285734776, -0.0897198766, -0.0758599639, -0.00738490093, 0.0257108826, 0.0372551531, -0.0686983913, 0.0113472436, 0.102236107, 0.00290569384, 0.0061129909, -0.0311949328, 0.113335073, 0.0380158424, 0.0155398687, 0.0312801749, 0.140485883, 0.0517903492, -0.0631593689, 0.052538231, -0.00393506698, -0.115367033, 0.0821724609, 0.00941016432, -0.0208612513, -0.0854508206, -0.0317099541, 0.0331769735, 0.0491336584, -0.000963477883, 0.0402674899, -0.0122544682, -0.0112764183, -0.0259621963, -0.0710512027, 0.0941303223, -0.0520865172, -0.0108082639, 0.120718181, 0.071119681, -0.0460885502, 0.0829018056, 0.00449483469, 0.0729888603, -0.0469497591, 0.0724814534, -0.180181056, 0.00309667923, 0.0897707492, -0.0610198379, -0.0766315609, 0.049891673, 0.11916092, -0.0543759391, 0.0534043536, 0.0337224454, 0.0504887849, -0.0129272975, -0.0697007552, -0.116602771, 0.108816735, -0.00892505888, -0.0880535245, 0.0587470308, -0.0186763145, 0.024901282, 0.0436722077, -0.000474594533, -0.0680011362, 0.0406705886, 0.093441315, 0.072278738, 0.0779481828, 0.0417279154, 0.0148036722, 0.0158227887, 0.0815258473, -0.0338716209, 0.0568503886, 0.0870490149, 0.118014261, 0.0279028304, -0.127121836, -0.00928720273, 0.00227311021, -0.0958245322, 0.0164720155, 0.0553140268, -0.0165274087, 0.00276194699, 0.0226365793, 0.0486386605, 0.0600383841, -0.0897603035, -0.00248141447, 0.0421509743, 0.0641591549, -0.093434833, 0.0514228828, 0.0813401192, -0.0186321884, 0.084352836, -0.110522412, 0.0110403849, -0.101047009, -0.0320625342, -0.0150115676, -0.0187792554, 0.0369519778, 0.0513808988, 0.15571554, -0.0890792906, 0.0299205109, -0.0106817111, -0.00820039585, 0.0726606101, -0.00610040408, 0.0680249035, -0.0590909794, 0.0168055221, -0.0538729206, -0.0597762577, -0.0244927071, -0.0475040749, -0.0671022311, -0.0265631769, -0.024594916, -0.0190176852, 0.0616992861, 0.059548974, 0.0446457379, -0.0300932303, -0.0819071159, -0.0148397181, 0.0510867611, 0.0136436932, 0.00267535471, 0.021764908, -0.0606418811, 0.0534243733, 0.0684300661, -0.095559895, 0.0286345817, -0.00460017892, 0.137911603, 0.0709685162, -0.0244417228, -0.0736082271, -0.00772494171, -0.000423151068, 0.0590124615, -0.0231226627, 0.0147387069, 0.0654460564, 0.100305125, 0.0292335823, -0.000347823283, 0.00400845055, 0.0379685163, 0.012252002, 0.00349133648, 0.0260682143, -0.059414614, 0.0927681625, 0.0475824177, 0.163947627, -0.0395782515, 0.0985130891, -0.0209101159, -0.0734324828, -0.106071897, 0.0295046382, 0.045582816, -0.00657141209, 0.0545752048, -2.92211771e-05, -0.0505888052, 0.00175773224, 0.018442221, -0.00747473352, 0.00795825571, -0.0159421675, 0.0164856426, 0.0743281245, 0.0307121426, -0.0596217886, 0.0863663554, 0.0323865525, 0.038819924, 0.000710537657, -0.0370529555, 0.0420183763, 0.0643882975, 0.0770071, -0.0172498468, 0.0497667491, 0.0720921159, -0.0163541045, -8.86656344e-05, 0.0375771597, -0.000295935897, 0.0374080688, 0.136759758, -0.0592932552, -0.00905792788, 0.0909006968, 0.046994701, 0.0290816184, -0.0521103106, 0.0580660366, 0.0635811388, 0.0122698592, 0.0555296056, -0.0228268653, 0.0349534154, -0.00424944051, 0.0304875188, 0.128829405, -0.0168012958, -0.055431854, 0.0274568256, -0.0444900654, -0.0890202224, -0.0030472111, 0.147902966, -0.0497640446, 0.0882239863, -0.0453582928, 0.017187532, -0.0182270277, 0.00447232788, 0.0568287857, 0.023605071, 0.0876043215, 0.0749583617, -0.0553779751, -0.0186833981, 0.0612326041, 0.0289207641, -0.126845181, 0.0502403118, -0.0478155948, 0.0812591612, -0.0952136591, -0.0721295998, 0.0450125337, -0.095405519, -0.0470645018, 0.00452820584, 0.0103754066, 0.0322743282, 0.0183758624, 0.0272299983, 0.0136208832, -0.011821527, 0.0360416323, -0.126070812, -0.0182594527, 0.00666202605, -0.0751212835, 0.0516611524, -0.0155047271, 0.0869452059, -0.0505760759, -0.0954601392, -0.0752341151, 0.0599434562, 0.0859812647, -0.0764811561, -0.010005191, -0.000140191521, 0.139839351, -0.00855318271, 0.0115316417, -0.0532930158, -0.0776077956, -0.0302928165, -0.0492541716, -0.0478124917, 0.0778949857, -0.0244202539, 0.0435359702, 0.0697957799, 0.072151199, 0.0978388563, 0.0594229177, -0.0954355747, -0.0867710859, -0.00336071663, -0.0154293245, -0.0472878143, -0.124766864, -0.00481133442, -0.0384963751, -0.0452389866, -0.00163068436, -0.0617119223, -0.106980875, 0.09947142, 0.063511543, 0.040238902, 0.0837928504, -0.0395397767, 0.0741849989, 0.0453262106, 0.00407153927, 0.0815881491, -0.0770316496, 0.00234743021, 0.0425972939, -0.00379472785, -0.0330946781, -0.00304131582, 0.0459878296, -0.0580381937, 0.064416416, 0.0110614914, -0.0338125825, 0.0360614099, 0.0164295975, 0.0215409324, 0.0470439233, -0.0520781204, -0.0707670525, -0.0355552472, -0.0162347835, -0.0916745216, -0.147062033, -0.00794365257, -0.0634822249, 0.0187621154, -0.0072186403, 0.00693030097, -0.0833823383, -0.0685342401, 0.0410865396, 0.021156393, 0.0674097687, -0.0460976474, 0.0254148897, -0.0693674535, 0.0247437414, -0.00030358287, -0.021148121, -0.0254203063, -0.0437479727, 0.0475757346, -0.00368373049, 0.0455008075, -0.105302155, -0.100783736, -0.059329249, 0.0415895879, -0.00438736612, 0.0716163069, -0.0396604091, 0.0736739263, 0.0511809029, 0.114312403, -0.0357594937, 0.0979067385, -0.00336160231, -0.0470240712, -0.0963593125, 0.0237926617, -0.000601712614, 0.0308345947, 0.102995485, 0.022467887, -0.0151176509, 0.0146277957, -0.000870541669, -0.0091063194, -0.0339862816, 0.0114137009, 0.0443384573, -0.00991028827, -0.0973331034, 0.0441233441, -0.0963969305, -0.0254261754, 0.0785122812, 0.0440628305, 0.0624476597, -0.00908709317, -0.0702229664, -0.0262233913, -0.0242057703, -0.000536231324, -0.00409665704, 0.0342630595, -0.00961654447, 0.034133181, -0.111113235, 0.0299617983, 0.0335191116, 0.0769206733, -0.00602729432, 0.0350972451, -0.0763334259, -0.0651243031, 0.111685283, 0.0664815754, -0.0429194309, -0.0353906117, 0.0155405067, 0.0296241622, -0.00895168353, 0.0666698515, 0.0739005953, -0.0650133193, -0.135277018, 0.102647275, -0.0674302429, 0.0470988452, 0.0264908224, 0.0061578583, 0.0977551341, 0.0961238667, -0.100649089, 0.0406196192, -0.000916211284, 0.0013770964, -0.0373530686, 0.090361774, -0.000571231358, 0.0353590809, 0.0556531027, -0.0360044017, -0.118675537, 0.00773452781, -0.00821574964, -0.129309908, 0.117962629, -0.0146916155, -0.0182366762, 0.0218699127, 0.0899865031, 0.0169488266, -0.0661243945, -0.107516676, 0.0349629819, -0.0594974831, -0.0737116337, 0.0514822379, 0.0119839944, -0.051653184, -0.0178696197, 0.0362947211, 0.000236622989, -0.202823579, 0.100061789, 0.114121303, 0.0156493895, 0.0361946151, 0.0113394931, 0.0550334752, 0.0142558776, -0.0146049634, -0.07990174, 0.03813003, 0.0430245437, -0.0124333035, 0.0938652903, 0.0728699565, 0.0459039956, -0.08093822, -0.0301704109, -0.0382108912, 0.0266480483, -0.0564455651, 0.0536727607, -0.0157301072, 0.00682708481, 0.0117938016, -0.0324358121, -0.0542678386, 0.0319058858, -0.0588584021, 0.0561320893, 0.130907536, 0.0366793722, 0.0508610979, 0.00354824495, 0.138257027, -0.0656450167, 0.0424082279, -0.0186371766, -0.00111340825, -0.0589470565, -0.0481215194, -0.0182844214, -0.058582291, -0.0512895659, 0.00234188838, -0.0661974847, 0.0830206573, 0.0266912356, -0.0416301414, 0.0208151732, -0.00435829163, 0.00619913451, -0.00665958133, -0.0683136731, 0.0261326246, -0.0603247583, -0.030451864, -0.134579107, 0.0856557786, -0.134901494, -0.0624972656, 0.0233187079, -0.00918305572, 0.0356052592, 0.0254772697, -0.0202677064, -0.063587375, -0.0745346323, -0.0152491368, 0.0108408406, 0.00164440647, 0.0100206565, 0.0697661564, -0.0512892157, 0.0540677607, -0.110494338, 0.136273861, 0.0119559281, -0.000351485796, 0.076251559, 0.00177314342, -0.0185832996, -0.014385283, 0.00929901376, 0.030984886, 0.0752916634, 0.00357770897, -0.133668244, -0.0806700215, -0.0632615462, 0.0514740124, -0.0126636904, -0.0114159919, 0.00991117768, -0.0765579343, -0.158915341, -0.0233150646, 0.0208109356, -0.0294479989, -0.122707568, 0.0248023123, 0.0353147574, 0.0768506601, -0.0213364009, -0.0176323038, -0.0668524802, 0.0420197994, 0.113398165, 0.0289836079, -0.0703490078, 0.0113566248, 0.0657502413, -0.064447552, -0.0568786189, 0.00577317551, -0.075506933, 0.0105375554, -0.0884989202, 0.0531153008, 0.0199516378, 0.00714925397, -0.196908295, 0.062297143, -0.0470579229, 0.00535312481, 0.0761762485, -0.165942758, -0.021334609, -0.00209301617, 0.0436096974, -0.0656614602, 0.0381878689, -0.0271022506, -0.0629928708, -0.0724918991, 0.00151832961, -0.00492772274, -0.0169231016, 0.00294148549, 0.0630060211, -0.00702680834, 0.103614599, -0.0277113169, 0.0686661154, -0.0492463782, -0.0575140379, -0.0664964989, 0.121500842, 0.0416047648, -0.0559566319, 0.02674428, -0.0769223198, 0.075026691, 0.00284983567, -0.115497753, -0.0541323759, 0.0418400168, -0.0283171535, -0.0536403432, -0.0472886004, -0.0325779989, 0.0034962506, -0.025822578, 0.0249830037, -0.00433831103, -0.0697114393, -0.122336604, -0.0307708252, -0.0594526231, 0.000370936468, -0.00850662589, 0.0746043921, 0.000625038403, 0.0480554402, 0.0194305293, 0.102841884, -0.000957332551, 0.0079627391, -0.0536535196, 0.0252215136, 0.00617412478, 0.0656590983, -0.0165666584, 0.0520427004, -0.0932068378, 0.0629480183, 0.137324661, -0.0883045048, -0.0535468683, 0.04913361, -0.0449029468, 0.0526470132, -0.0837362707, -0.0731720403, -0.0245988425, -0.0183166042, -0.08067213, -0.00450671557, -0.131562054, -0.0607740879, -0.0500571318, -0.0688363612, -0.0545937829, 0.0541550145, 0.0478787571, -0.100023203, -0.0562713929, -0.0598613508, 0.0882329792, -0.0711460561, 0.00229808548, -0.0771372393, 0.0790798143, 0.0134686232, -0.0108972043, 0.101201199, 0.0381906331, -0.0236407705, 0.0456900597, 0.0683217496, -0.0181267913, -0.142836317, 0.0499501452, -0.00357577298, 0.0818683654, -0.0516990945, 0.112652406, -0.0879362822, -0.0412990525, -0.0435129516, 0.0530302078, 0.00753782317, -0.0103394203, -0.113468543, 0.00393888401, 0.0430542305, -0.0991563946, -0.0656711832, 0.163774505, 0.0531020835, -0.0592267737, -0.0073725814, -0.0321563631, -0.0142563935, -0.105408728, -0.0280363113, -7.33286142e-05, -0.0258809663, -0.0473232828, 0.0032044882, -0.0450153537, -0.0532960445, -0.0615855753, 0.00778417429, 0.0041831471, -0.00524075702, 0.0228698738, 0.0614221543, 0.00402660668, -0.0238150302, 0.0738576651, 0.0269466322, -0.0133383647, 0.0311506707, -0.0712363273, -0.0779514238, -0.114374563, 0.04239434, -0.00277828798, -0.0402479433, -0.079252474, 0.0231916178, -0.00225579366, -0.0618388616, -0.0110141272, 0.0391204767, -0.0469195843, -0.0638582185, 0.071978949, -0.011590559, -0.00427569589, -0.0532582439, 0.0585490949, -0.0511503294, 0.00598193984, 0.123238713, 0.0346515216, -0.0520669706, 0.113400199, 0.0907458216, -0.0702292845, 0.0389042534, -0.00404449832, 0.0736160874, 0.0388934165, 0.0466618165, 0.108994663, 0.09106832, 0.0300671905, 0.0388143584, 0.0434229262, 0.0723200142, 0.115112618, 0.00486603007, -0.0254915692, -0.0196508542, -0.0855910331, 0.00867968146, -0.0102319364, -0.00442096032, 0.051562503, -0.0257901531, -0.0958380923, 0.0316315554, -0.154216707, -0.0674449056, 0.0272293575, 0.0838137716, 0.0966868401, -0.0600471497, -0.0515384749, -0.0039906376, -0.00892661884, -0.13223879, 0.0174390785, -0.138658226, 0.0107445074, -0.0626263842, -0.0127585046, -0.0576431155, 0.0479596183, 0.109288901, -0.0342611261, 0.159175709, -0.0373381041, -0.0919338167, 0.0636126027, 0.0714582503, -0.0594209135, -0.0358245447, -0.00872441754, -0.0724314973, 0.0365815945, 0.019486405, 0.0668292865, -0.0412320197, -0.0135822697, 0.0507908612, -0.0292699169, -0.0338540822, -0.0239487719, 0.00985379145, 0.0247995164, 0.0167899299, -0.0126943421, -0.0424789675, -0.0692631006, -0.0625886396, 0.0332871377, 0.0392154977, 0.046094019, 0.0354588963, 0.140024304, -0.139790013, 0.0670035481, -0.064532347, 0.100462317, -0.0957116634, 0.0602088384, -0.0855569616, 0.101311266, 0.0897070393, -0.00622749981, -0.00115730427, -0.0711332634, 0.0710380971, -0.018597085, -0.0571301654, 0.051692389, -0.0386115946, -0.0739023089, -0.0584098026, -0.0994265303, 0.0800986812, -0.0226804502, 0.0287728608, -0.0223561227, -0.113707162, -0.0412001014, 0.00798535813, -0.0368543565, 0.0626538843, 0.0209903289, -0.0211640075, -0.082355909, -0.0256390776, -0.0487164333, -0.0463558882, -0.047578048, -0.0852676779, -0.0254986323, -0.00152657472, -0.092315957, -0.123599537, -0.0112181921, -0.0046400195, 0.121392928, 0.025643941, 0.122754768, 0.0185011737, -0.0831996053, 0.0621068254, -0.0494964086, 0.111018084, 0.0297669042, -0.0155222639, -0.0119001176, -0.00128799491, -0.00557321869, -0.0162937157, 0.0770080388, -0.0285283923, -0.104027048, -0.0982666612, 0.0225247666, 0.00802648813, 0.00118900184, -0.109698035, 0.067589052, -0.0469475277, 0.0203107893, 0.0234843325, -0.0313501433, -0.000745411962, -0.0368155017, 0.00568490103, -0.0261498019, -0.0389427394, -0.0794990435, -0.0296408292, 0.109177478, 0.0325602777, -0.0334580168, -0.170560166, 0.00342586637, -0.0559075326, 0.0171828158, -0.0703995079, -0.0374180675, 0.0109978039, -0.00167782884, 0.043880403, -0.0217684656, -0.0462836325, -0.0469024219, 0.0823281184, 0.0374536961, 0.0292149168, 0.0223761108, -0.106840752, 0.000103849918, -0.0354231596, 0.0182724558, -0.13642019, -0.0856509879, -0.014119301, 0.0462180302, -0.0491417013, -0.0104149841, 0.0491163582, 0.0205129106, 0.0649414361, 0.037804395, 0.040461421, -0.0495519564, 0.0283405147, 0.0624213889, 0.0398034118, -0.0410586894, -0.0815684348, 0.0512367897, 0.0223541129, -0.00989829376, -0.0130436886, 0.0757523924, -0.00515081361, -0.0730558932, 0.0320465267, -0.00857695937, -0.0806317925, 0.0279297102, -0.0246432945, -0.0483816788, 0.00798191782, -0.0589826256, -0.0563129932, -0.0364476889, 0.0567692816, -0.00600192044, -0.0459529385, -0.139255688, -0.0303245261, 0.0186996274, 0.0734643713, -0.0368433781, -0.110486992, -0.0339182727, 0.0288793221, 0.0765346363, -0.128872678, 0.0284972172, 0.0712290257, 0.0292674564, -0.0923582017, 0.122514822, -0.0141425449, -0.023105029, 0.053995382, -0.0536839105, 0.0222591516, 0.067343615, -0.0495528281, 0.107660443, 0.00114707462, 0.0166068859, -0.0164854825, 0.0783448443, -0.0427716002, -0.00397504866, 0.073449105, 0.149562895, -0.00719949929, -0.0207619313, -0.00146194082, 0.126207888, 0.0411823094, 0.0814019814, 0.0927758515, 0.0431634486, 0.089347519, 0.0507778302, -0.0231358539, 0.0442269146, 0.0974288583, 0.0643353835, 0.104393393, -0.0288960095, 0.0763740912, 0.0251511447, 0.0115142595, 0.0491543822, 0.00783968717, 0.0298399106, 0.0130653959, 0.00786384754, 0.0648100972, -0.0536608472, 0.000275403436, 0.0412608869, -0.0442459658, -0.0178164579, 0.0147872102, -0.0659606606, 0.0125337383, -0.0969907343, 0.0340121202, -0.147724167, 0.0794025511, -0.0151667744, -0.00873299036, 0.112291977, -0.014848101, 0.191120476, 0.00163297355, 0.00122271827, -0.140272528, -0.0523022264, -0.0467030481, -0.0318848863, -0.0832360238, 0.100232348, -0.00624156184, -0.0245157126, 0.0351526178, -0.0345866531, -0.0476002693, -0.0539702103, 0.0531913713, 0.0726050511, 0.158330321, -0.00117380172, -0.0488243438, 0.0151165035, -0.0884667411, 0.0150398053, 0.100097612, -0.00501692481, -0.0556602664, 0.0396614522, 0.00732987933, 0.00400307681, -0.0153083447, -0.0630880222, -0.0466349907, 0.00711335428, -0.0679616705, 0.0131458361, -0.0808020607, 0.104224131, 0.0602303408, 0.0901438892, 0.00158551312, -0.0639543533, -0.116641514, 0.0262246542, -0.0232329443, -0.109544262, 0.174844474, 0.050198812, 0.0641451776, -0.0448447913, 0.10102357, -0.0260062311, -0.0358123332, -0.0168521404, -0.0565307364, 0.0429335982, 0.141919643, -0.00534844398, -0.0150071457, 0.0357227474, 0.0479923822, -0.0432240739, 0.0455152467, -0.0403398387, -0.0252203122, -0.0141034257, 0.0424684063, 0.0184082203, -0.00933267921, -0.00230838591, -0.0446829386, -0.105363771, -0.0196014158, 0.0738840923, -0.082031399, -0.190825433, 0.0496896543, -0.0732061341, 0.0125593534, -0.0271144565, -0.0377364829, -0.113841057, -0.00843485631, -0.0024445327, 0.0729354694, 0.0562470928, 0.0476794988, 0.0482817441, 0.0115363076, 0.0726508424, -0.0758034214, 0.0502102152, -0.0035237628, 0.00509096403, -0.000869088806, -0.11856851, -0.0172609035, 0.0536386818, 0.0396515839, 0.122773603, -0.0308346134, -0.0880051553, -0.0806351602, -0.0727893487, 0.0208604895, 0.0370517485, -0.0853930265, -0.03130465, -0.0879868045, -0.0281146877, -0.0867229775, -0.0284860618, 0.0269446224, -0.0510630682, -0.0405789614, -0.0577245504, 0.0179252699, -0.0473303571, 0.0624001101, -0.0510875136, -0.0296407547, 0.0335749611, -0.04302999, -0.0523483157, 0.0663412437, -0.00900157169, -0.0296637807, -0.0837188736, -0.0525992066, 0.0536954999, -0.0186074823, 0.0867669359, -0.0474121757, -0.0703267902, -0.0122002857, 0.0150674805, -0.13100715, 0.0233776923, -0.0451542288, 0.0217646472, 0.100174919, 0.0426718369, -0.0138558736, -0.0477688685, -0.112276495, 0.00485369191, 0.00660805125, 0.0429948904, 0.0537965186, -0.0807079151, 0.0131279994, -0.0701279044, 0.122121394, -0.128034905, 0.0439936072, -0.141157091, 0.121826403, -0.08293318, 0.0684459955, 0.0310336687, -0.0681967884, -0.017216742, -0.0997434705, -0.0478654765, -0.0235749185, 0.0831564069, 0.0268044341, 0.0130881127, 0.0428807959, 0.0727542639, 0.0279251859, 0.011901971, 0.00996486843, 0.0600239187, 0.0219573006, -0.136379257, -0.0298984088, 0.043327041, -0.0986257941, 0.0249502286, 4.05553728e-05, -0.0814153925, 0.0216127373, -0.0241992325, 0.0232727043, 0.0298146009, 0.0414998978, -0.0725062937, 0.0859083608, 0.0421535224, -0.0404414497, 0.0181416478, 0.0107587101, -0.00611246936, 0.00402363297, 0.0922489837, -0.0164177027, 0.0260459781, 0.0817983449, 0.0217644833, -0.0167400651, -0.0685246512, -0.149026424, 0.0713879913, -0.0388812385, 0.0400551818, 0.0419062302, -0.0224685557, -0.0413398966, -0.027663609, 0.0331780091, -0.0177993327, -0.124532469, -0.095648624, -0.0418065004, -0.0819868743, 0.122692823, -0.0442254171, 0.0463492982, -0.030052403, -0.0929630324, -0.0243065339, 0.0923779309, 0.0408683196, 0.0820688009, 0.0882338956, -0.0251470413, -0.00624269526, 0.126063228, -0.029209543, 0.0355586521, -0.0653761253, -0.0197694451, -0.00596020464, 0.0587397702, -0.115629293, -0.0752471983, -0.0162388161, 0.0350908823, -0.0141521497, 0.00708530284, -0.0907153487, -0.0908495858, 0.0507154539, 0.0201784577, 0.0690165907, -0.0779961869, -0.0317785591, 0.00336016063, 0.0711848289, 0.0369975269, 0.0309573486, -0.109106801, -0.00914905407, 0.0876875147, -0.0711093023, -0.0414840281, -0.0196994953, -0.0420634151, -0.0886219218, -0.0991885513, 0.0369526818, -0.00856760424, 0.0270003583, -0.00322042266, 0.104991138, 0.0362386256, -0.108001046, 0.0299428124, -0.0856452882, -0.047418341, 0.0115645491, 0.0850456432, 0.136194035, -0.0316643342, 0.0383179039, 0.052085638, -0.0634030774, -0.00373797049, -0.062366832, -0.0839076862, -0.00321283448, -0.127361536, -0.117611811, 0.0649010986, 0.0250289943, 0.0747210309, -0.0635356456, 0.0666100457, 0.0524176918, 0.0827337056, -0.0031545735, -0.030966891, -0.025643453, 0.00783623941, -0.0498177074, 0.0101410206, 0.0465142019, 0.104158878, 0.0538403876, 0.105358213, 0.10463158, 0.0728892237, -0.0659171343, -0.0071498286, 0.0409778878, -0.0533908643, -0.0269968528, 0.00537291914, -0.0167357028, -0.0542261004, -0.0264697708, 0.0649209321, 0.00562486425, -0.078290455, -0.0301799402, -0.0396311358, 0.0498488806, -0.0608386993, -0.121679798, -0.0424144566, -0.101940505, 0.138346016, -0.0247701369, -0.0585908741, -0.0631965995, -0.0478361361, -0.0914618671, 0.0260726195, -0.120376013, 0.0118363611, -0.00604729913, -0.0168034807, 0.0506373197, -0.0345347784, -0.0832358599, -0.0361929014, 0.0114472592, 0.081957534, 0.0523104854, -0.0217854492, -0.033708185, -0.0472963527, -0.0628994033, -0.0480692387, 0.001929141, -0.0209593922, 0.101744853, 0.01414611, -0.0366679169, 0.0593956076, 0.00308167096, 0.0110140909, 0.101774275, 0.00835005287, 0.0232221708, -0.0656514019, 0.0431903675, 0.0923357308, 0.0676914304, -0.0187924132, -0.00379694602, 0.11188484, -0.115201734, -0.0403196067, -0.0632556155, 0.0217211135, 0.0387047082, -0.0244503077, -0.0215889253, -0.0384796336, -0.00307661295, -0.0718727857, 0.0133105125, -0.0491234437, 0.0376469418, 0.0118808523, 0.0203267261, -0.109959148, -0.0282824505, -0.0202198699, 0.0226617269, 0.0633247197, 0.0118141593, -0.0101759331, 0.0381266624, 0.106288128, 0.0304039326, -0.0695357248, 0.0328905433, 0.075065434, -0.0510398448, 0.0110777989, 0.0278759226, 0.0927972496, 0.0358517468, -0.210644707, 0.0215705633, -0.0170749202, -0.0503018647, 0.0153489299, -0.0752708092, -0.054475233, 0.0507027954, 0.00628920272, -0.0201173648, -0.00399248069, 0.0252465066, 0.0999787003, 0.13058953, -0.062581256, 0.0148989912, 0.0864780918, 0.0105943158, 0.118947454, 0.0233809762, 0.0450160056, 0.0172462538, -0.0144504737, -0.0310064666, -0.0137993451, -0.0318533778, 0.146467894, -0.0273016356, -0.102862895, -0.0613403954, 0.041406706, -0.0256335996, 0.0421037748, 0.0375077613, -0.11444512, -0.0507230237, 0.0455504395, 0.00221366715, 0.229563221, -0.0949061364, 0.0851142928, -0.00966047868, -0.0264595449, 0.0601200014, 0.0777863637, -0.0105279032, -0.116519243, -0.0223890375, 0.0628159493, 0.152149305, -0.0975992456, -0.0235308036, -0.0772626549, -0.0298480783, -0.0712135285, 0.0226339232, -0.0215983242, -0.0421964601, 0.0922935084, 0.0635753572, 0.00575707667, -0.0868083388, -0.037115369, 0.0801732317, -0.0492756367, -0.0262582209, 0.0257645715, 0.052389659, -0.0251567736, -0.0943191797, 0.0489675961, -0.0232405737, 0.0430886522, -0.0816913247, 0.102276124, 0.0163074248, -0.0582618788, 0.0787617862, 0.0102452869, -0.0496148616, 0.0192592684, 0.123371288, -0.0271462258, 0.06752716, 0.0795108899, 0.0624162331, -0.0759384632, -0.0248846896, 0.0234479494, -0.0482824184, -0.00685673207, 0.0855260938, 0.0107843969, -0.0113728102, -0.0373565592, 0.00753186457, 0.0250684135, 0.0551184453, 0.0383309349, -0.0971988663, 0.124966308, 0.0615704358, -0.0953281894, -0.0284687858, -0.0505576953, -0.0602671728, -0.200355232, 0.0468630567, 0.0746757239, 0.13662222, -0.0628385693, 0.0152048916, -0.0210232195, -0.00131607242, -0.0558450446, 0.0213233121, -0.00659259781, 0.00367828552, 0.0871913657, 0.00931879506, 0.0897677392, -0.0236726739, 0.0279342402, -0.0175310932, -0.0787250102, -0.0196127351, -0.0334822536, -0.0333999768, -0.0249295197, 0.059769839, 0.042923905, 0.162160173, -0.0505244061, 0.00797021016, -0.092655845, 0.0421476103, -0.0489855893, 0.0708907023, 0.0748008937, -0.0966250747, 0.0810881853, 0.0188420899, -0.0255011339, 0.0772066936, 0.0266787168, -0.0594868585, -0.0456732586, 0.0951411352, -0.0154170543, 0.0691231638, -0.00984910596, -0.0413136296, 0.0706344321, -0.0266577266, -0.0868716761, 0.0830847397, -0.0107623497, -0.0221581906, -0.0837728232, -0.000261315145, -0.117857374, 0.0513177775, -0.0411504656, -0.0618194565, 0.0791345462, 0.0165001098, -0.0308103748, 0.00686467858, 0.103483453, -0.00371338427, 0.0774708092, -0.0746427625, -0.0162100494, 0.0275091548, 0.0138276611, 0.0286125224, 0.0219381656, 0.0426561646, 0.0794264972, 0.00133450888, 0.0737243667, -0.0169447064, 0.0433264002, -0.0012736097, -0.0249856152, -0.030008316, 0.157068267, -0.00769524276, -0.0462254323, 0.0222761016, 0.007889539, -0.0693490282, -0.0983556286, 0.150570318, -0.134598985, 0.0639032945, 0.00854932889, 0.051869899, 0.00420638826, 0.0676100627, -0.130077541, -0.0402148962, 0.0332589447, 0.0396894701, 0.0653833821, -0.00954185426, -0.0416257605, 0.0263223909, -0.0214542486, -0.00996944308, 0.0822702497, -0.0215292387, 0.086395368, 0.0478596874, -0.101059303, 0.0468727462, 0.0736261457, -0.0030699675, 0.0646912232, -0.0455570593, 0.0221026298, 0.0592654124, -0.0269551463, -0.0400718972, 0.0179079622, 0.0622584969, 0.0227873195, -0.0636694804, 0.00989277661, -0.114476956, 0.0762022883, -0.062514171, 0.0227152295, 0.0925726369, 0.00170127861, -0.0646214038, 0.043654602, -0.0173907503, -0.00643299334, 0.0975144953, 0.0822733864, 0.022763215, -0.00732895825, -0.0809313953, -0.0711122379, -0.111108579, 0.00472774729, -0.155565694, -0.0858013406, 0.00700040208, -0.0396955088, -0.0909059793, 0.0507231094, -0.0647651255, -0.00767456181, 0.16497691, -0.149384141, -0.0411503166, -0.0122785531, -0.00280779228, -0.0336751826, -0.0886300057, -0.0845317021, -0.036026977, -0.0573642999, 0.0547272265, 0.0129092075, 0.0210604407, 0.0727588311, 0.0579680316, 0.0292192027, 0.0662830621, 0.0749937817, 0.000851269811, 0.00157426763, 0.0532496721, -0.00610272493, -0.0174139775, 0.0294752326, 0.0900547877, -0.0292545669, -0.0537517071, 0.0680302233, 0.0255860277, 0.00676572323, 0.0767123699, 0.0680063069, -0.0438368767, 0.00264221616, -0.0727874264, -0.166978449, 0.0613660961, 0.114054509, 0.149120882, 0.077867195, 0.020376835, 0.0373401754, -0.0480047762, 0.169552654, -0.0576319993, 0.145785511, -0.0389896929, -0.0401603766, 0.0229748152, 0.110711455, 0.0116823204, 0.0388501622, -0.00470389612, -0.0190922655, 0.0177334137, -0.0398545489, -0.00175582059, 0.069974035, 0.0147722131, 0.00534011703, -0.0796792582, -0.0275453366, 0.0785744861, 0.0450469777, 0.00944564119, 0.0907722339, -0.0159705002, -0.012611798, -0.0306889545, 0.0320927761, -0.0188522171, 0.0547658503, -0.0955944732, 0.00123614445, 0.0869101733, 0.0627448782, -0.079220064, 0.0522994213, 0.00224558031, -0.0162150152, -0.0259681381, -0.0626722872, -0.130126655, 0.0856325328, 0.00620901957, 0.0151104387, 0.0416606627, 0.0155630587, -0.0896422863, 0.00188501552, 0.00841740426, -0.0521952137, -0.0216675363, 0.02849265, -0.0610549785, 0.0459467396, -0.0848054364, 0.0867174193, -0.0654042214, 0.0110846488, -0.066037491, -0.0076175062, 0.00418529194, -0.01894347, -0.0207504369, -0.0331593975, 0.00153754279, -0.0587283634, -0.0177199971, -0.104922697, -0.0841468126, -0.0131656919, -0.014361525, 0.0460430197, 0.0203863829, 0.00274782255, -0.16865401, -0.0016321037, 0.106147997, -0.0195879396, -0.0185016356, 0.154084757, 0.0054557668, 0.00630028266, -0.0200805031, -0.110674784, 0.113205783, 0.0313374288, -0.0442044251, -0.13534075, -0.0351653695, 0.0659490377, 0.0599162281, -0.0930598751, -0.0088927215, 0.0369860157, 0.044912219, -0.0438780002, 0.012475878, -0.00858119037, -0.0496248528, 0.0516645648, -0.0095990533, -0.0841310397, 0.0511544272, 0.106277607, 0.0374979749, -0.0185278319, -0.085943684, 0.00602632016, -0.0893028826, -0.0434319079, 0.0539812036, -0.0510410927, 0.183443248, 0.0494461358, 0.128872976, -0.0150585882, 0.0300107189, 0.0950379968, 0.0403474495, 0.0512554944, -0.00949157681, -0.0852464512, 0.00995048508, 0.0322411805, -0.105127797, -0.114629336, -0.0600172542, 0.0529371127, 0.0992998779, -0.0201824084, 0.0151111186, -0.0725996941, -0.0565026142, -0.0304286163, 0.0209496003, -0.00247463211, 0.0789061487, -0.0161107779, -0.0700700954, 0.0681259781, -0.0760259032, 0.00105957314, -0.105654038, 0.0477458537, -0.0323687717, -0.0496293493, -0.00972076599, 0.128960192, 0.0870439187, -0.00614603423, -0.00333144981, -0.0563246757, -0.0690083504, 0.0195674896, 0.0084388759, 0.0502358042, 0.149670064, 0.0840686709, 0.0315471068, 0.020206403, 0.0690457895, -0.0741327181, -0.0267885476, -0.090405874, 0.0553143844, -0.0698693246, -0.108412452, 0.00959519297, 0.0957986191, 0.0938214511, -0.0723310262, -0.0402347036, 0.0983432531, -0.0367692374, -0.0770791695, 0.0390468761, -0.0179023165, 0.0456901975, -0.0114207296, 0.109032594, 0.129397228, -0.06511949, 0.0657798201, -0.125876442, 0.101577789, -0.00751718972, 0.05052571, -0.138598636, 0.0872033164, -0.0756148398, 0.0100236349, 0.0612523891, -0.0617438406, 0.0384409912, -0.128118366, 0.025034897, 0.0635608807, -0.0484598763, -0.0328407064, 0.0170689039, -0.0560454838, -0.0182302892, -0.0041722618, 0.0531054065, 0.0157475565, -0.0191789363, 0.0275798514, 0.0253439024, 0.0384207368, -0.107161373, -0.00644496456, 0.104860663, -0.00406992156, 0.00712282769, -0.0273554437, -0.0118243508, 0.0248243269, 0.0183168985, -0.012124151, 0.0140287578, -0.078517884, -0.0103985276, 0.063864246, 0.106309205, 0.0390842184, -0.0690605566, 0.00937034003, -0.0635004118, -0.0857211575, -0.00190764014, 0.0157235973, -0.0992204547, 0.0519966967, -0.17544426, -0.0508512706, 0.0322943032, -0.0287256874, -0.0272098202, -0.0265219491, 0.0572342388, 0.0329430476, -0.0339044966, -0.075075224, -0.0859181881, 0.00145858899, 0.0841681212, 0.0173426513, 0.0547166504, -0.0303188656, 0.0787743628, 0.0457511246, 0.010878535, 0.0255478919, 0.0900510773, 0.0215361975, -0.0322675146, -0.0418702699, 0.0299271457, 0.0546380281, 0.0538790114, -0.0100034699, -0.0224084128, -0.00508561172, 0.0152663626, 0.055271104, 0.0182426535, -0.0622355044, 0.0545172356, -0.0944176242, -0.0133834789, -0.0213274527, -0.0769234151, -0.0411180034, -0.0157406516, 0.0800870955, 0.057321392, -0.0215420369, -0.129882321, 0.0440563336, -0.0226000603, 0.00509729609, -0.0234147515, -0.0101710707, -0.0305681545, -0.0256329477, 0.00180998817, -0.0122924522, 0.017725233, -0.0441546813, 0.103631072, 0.0675418898, -0.0632346869, 0.0353666618, 0.0676773489, -0.00349519262, -0.0168017447, -0.0845970362, 0.0094102351, -0.000715238042, -0.0910702571, 0.0277075302, 0.00221918058, -0.0422398448, -0.040655937, -0.0297275335, 0.0104903504, -0.0015773084, 0.00691782217, 0.0379387289, 0.0448956788, -0.0694757253, 0.0144133717, -0.0391342565, 0.0815122724, 0.0139185283, 0.014715245, 0.147531897, 0.0297246762, 0.140969202, -0.0280634928, -0.131946936, -0.025080869, -0.0812521428, 0.0197385289, -0.0548864938, -0.0596676618, 0.0526864417, -0.0422517173, -0.0329750478, -0.151260406, 0.0342650712, -0.0493682809, -0.0138619337, 0.000737296417, -0.00650860183, 0.00592454057, -0.0644744784, -0.00937987119, 0.0966760889, -0.0368182547, -0.0561390854, -0.0122595802, -0.044610627, -0.0427267253, 0.0261523519, 0.0552324802, -0.133556947, -0.0793345571, 0.0906136781, -0.0395403691, -0.01307307, 0.0391273573, 0.0634972751, -0.0430783108, 0.043919865, -0.0543998405, 0.050850708, 0.0411434621, -0.0256112292, -0.0887005776, 0.109898433, -0.058176104, 0.0435316004, -0.000602371991, 0.0314278938, 0.00066623278, -0.00263828924, -0.0102431364, 0.0146305514, 0.0207039136, -0.0112496857, 0.13573727, -0.0275485106, -0.0482266657, -0.0370065644, 0.151276827, 0.0435078293, 0.00135911768, -0.0430634394, -0.00319447718, 0.00565682026, -0.070520483, 0.024573788, -0.0046765483, -0.0286862142, 0.0772430599, -0.110488892, 0.00214591064, -0.0017450694, -0.020990368, 0.0463565663, 0.066084981, -0.0593725517, 0.00982001889, -0.0451216996, -0.0172102861, -0.0513852686, -0.00727432733, 0.0123199485, 0.00668398477, 0.0216202606, -0.00748495013, 0.0354989059, 0.0922414362, 0.0157978497, -0.0361201465, 0.082894139, -0.0646007732, -0.00972089171, 0.0107940985, -0.225798666, 0.0363088511, -0.0300963763, -0.0521194376, -0.0939533114, -0.0595852397, -0.0703465194, 0.116963029, -0.0248812176, 0.0248628408, 0.021702107, -0.0480697788, -0.0397238173, -0.03429088, 0.0719931722, -0.0394061543, 0.0114826765, -0.0571210496, 0.0680134445, 0.0292406529, 0.0281575359, 0.00717210444, -0.0369810015, -0.0190533549, 0.0150481015, -0.0117387054, 0.0639001429, 0.0372794308, 0.00371855218, -0.0193396136, -0.117099866, -0.0828941464, 0.0121081341, -0.0244761799, -0.0255028158, -0.0318410657, -0.0286944397, 0.0493089631, -0.0324905142, -0.0341451988, -0.0127818771, 0.0452495143, -0.126098096, -0.0315716863, -0.0482584275, 0.005084306, 0.00973041356, 0.0948285013, 0.0901907608, 0.00151643902, -0.11976669, 0.0879791602, -0.0443039536, -0.0906420052, 0.0617935322, -0.0349473841, -0.0822580308, -0.0823693946, -0.0114820674, 0.0753556788, 0.0444406644, 0.0306949131, -0.0323597714, 0.132427111, 0.00939624943, 0.104174532, -0.0243637897, 0.00233740732, 0.0739128292, -0.0666283518, -0.0130364271, -0.00263343519, 0.00153722963, 0.0646293908, 0.00971084647, 0.0207044836, 0.0430175811, 0.0261249654, 0.129058644, 0.0656372085, 0.0572115034, -0.112717815, -0.0525403433, 0.0804309249, -0.00388916722, 0.0535279177, 0.0211513042, 0.0874609798, -0.0127248913, 0.00927163195, -0.00117566064, 0.0187003948, 0.0746483952, -0.0280186813, 0.0547470301, -0.110899061, -0.114001378, 0.0433497205, 0.00770346262, 0.0581384376, 0.000574407401, 0.0648812428, -0.00253759138, -0.0626765341, 0.0191185959, 0.00825243723, 0.0263058022, 0.0298263058, -0.0831383839, -0.0146999806, -0.0658679679, 0.0386553146, -0.0657345504, -0.0205592699, -0.0268240143, 0.0221242774, -0.0175097957, -0.059482675, -0.0105682146, -0.0872407034, 0.0940551534, -0.00376821286, 0.0103017371, 0.0266460516, 0.180327952, -0.0186312832, -0.0744505897, 0.0627357364, -0.00251487596, -0.0410550237, -0.012822194, -0.0356829949, 0.0976379737, 0.000514240237, 0.04100696, 0.106039599, 0.0152142178, 0.0467813723, -0.150179595, -0.0155127589, -0.00957605429, -0.0193987582, 0.0763824433, -0.0770917684, 0.081620343, -0.0322763063, 0.104996897, 0.00758426543, 0.170526117, -0.0542769656, -0.0716079846, 0.0647917166, -0.0429567508, -0.0623636916, -0.0489886291, 0.020243451, 0.0706255063, 0.0238528475, 0.047688581, 0.0733051002, -0.0554361679, 0.232940093, -0.0695162565, -0.0590134859, -0.0550089926, 0.0196601395, 0.0243985951, 0.0517330393, -0.0531237759, 0.0619931184, 0.0281106867, -0.0551919043, 0.0146903247, -0.0580469519, -0.0795866475, 0.0108202919, 0.0867381468, 0.109796897, 0.00811877381, -0.0400859267, 0.0645622164, 0.00928810611, 0.0342610329, 0.0315460078, -0.0817455798, 0.123105973, 0.0668828562, 0.0465821251, 0.0134259639, 0.0615614802, 0.0227601342, 0.0585081652, -0.0611969382, 0.0172028914, -0.0358809158, -0.0128495879, -0.0821195841, 0.00618747249, -0.0454788469, 0.105804324, -0.0176044255, 0.0405101702, -0.0292864256, 0.0233910494, -0.025192827, -0.0312486663, 0.0180517733, -0.016661806, 0.0777479261, -0.129380882, -0.0451043062, -0.0319344848, 0.0416108221, 0.0815054178, -0.0920516849, -0.0100542856, -0.111545153, -0.0561509654, 0.0313889608, -0.0773571655, 0.046628017, 0.00535817491, 0.0487535596, 0.0216938015, -0.0557895154, 0.104152054, 0.0699986219, -0.00808387809, 0.00408079941, -0.029250063, 0.0708507523, 0.0687088817, -0.0214304477, -0.00520200748, 0.00976883247, 0.0657177046, 0.0562655292, 0.0538188145, -0.0165550318, -0.0289269984, 0.0731174573, -0.0277810134, -0.0105520301, -0.0446213447, -0.0131835025, 0.059898641, 0.0204441324, -0.00773157738, -0.00405251142, 0.015112265, -0.000342171639, 0.00478193164, 0.0253996439, -0.0484651253, -0.0315660872, -0.0107570905, -0.133314699, 0.0612211302, 0.0747045949, -0.0177192204, 0.0402086414, -0.0312886648, -0.0193530731, -0.0946298838, 0.0752811134, 0.0341706686, -0.0564576685, 0.0196592771, -0.0641864613, 0.126299188, -0.0236910637, 0.0560906753, -0.0083694458, 0.111020304, 0.0529743358, 0.0875263736, 0.0167604834, -0.0896236822, -0.025494663, 0.0463420078, -0.103654683, -0.0210032966, 0.00552533008, 0.00688660517, 0.0591736771, 0.0759595856, 0.0404704511, 0.0487403162, 0.0691098869, 0.00912425853, -0.0180258006, -0.0106740231, 0.00178129598, 0.0216437392, 0.00244355761, -0.0975364298, 0.0147012826, -0.0495922416, -0.02287931, 0.10947419, 0.050613679, 0.0894236714, 0.0623275787, -0.00320071541, -0.033641234, 0.131710827, -0.125496715, -0.0462804809, -0.0460643694, -0.0953746811, -0.00889004022, 0.118052706, -0.0667778999, -0.0133435521, -0.030920662, 0.0498138182, -0.0386170074, -0.0142802922, 0.0688701272, -0.0266187936, 0.00762451254, -0.0605605282, 0.0103181377, -0.00750357844, 0.00569614395, 0.0543710068, 0.0661029965, -0.081736058, -0.0244649462, 0.00796968769, 0.0216992628, 0.0720511675, 0.0205531269, -0.114837237, 0.0401188731, -0.10663683, 0.139999405, 0.0874945223, 0.0693346038, -0.077024743, 0.0343449935, -0.0758866668, -0.00565212686, -0.0300139375, 0.0720785111, 0.0280683637, -0.0016435422, 0.113789186, -0.0616969988, 0.0708234981, -0.0232442897, -0.1073566, 0.00374428299, 0.00734259654, -0.0940107927, -0.00127174146, -0.145696223, 0.0194209628, -0.0300043058, -0.0243853759, -0.0499064028, 0.129020929, 0.0394175351, 0.0395161584, -0.0553765558, -0.0789635032, -0.0456503741, -0.0388430059, -0.0205404088, 0.00434309244, -0.0111577008, 0.0887822807, -0.0246210508, -0.128890976, 0.0691070482, -0.0654581413, 0.101507232, -0.0100079384, 0.00432548393, 0.0620917976, -0.00314891525, 0.00771834701, 0.041378133, -0.0246183276, -0.0999459252, -0.0505741984, -0.0998098925, 0.0442011468, -0.00178184919, -0.131378531, 0.102398507, -0.0420437083, -0.0415701009, 0.1121848, 0.162975714, 0.0312584788, -0.052917175, -0.00630946271, -0.0122770071, 0.058539249, 0.0603848547, 0.0622089505, -0.136828452, 0.0944014043, 0.0796410739, 0.00162931776, -0.0472676754, 0.0761734769, -0.0606164038, -0.0248263106, -0.0524409004, 0.0366512351, 0.00172413373, -0.128477365, -0.00964768324, 0.037448369, -0.00916153565, 0.0782021582, 0.0525283478, -0.13682586, 0.0260457881, -0.0689895079, 0.107476562, 0.000512594357, -0.0255439896, 0.0253176652, 0.0466695204, 0.0254534315, 0.00695104152, -0.0137286065, -0.0362772569, -0.0312191471, 0.0037508402, -0.074491553, -0.0252933614, 0.0345676392, -0.0229077395, 0.00814678892, -0.00895130821, -0.0134142041, 0.0863745362, 0.0984717458, 0.0407752208, 0.061877884, -0.0152371787, 0.0340818018, -0.0530208908, -0.000142361503, 0.00749082118, 0.0228016227, -0.0516728237, 0.0243119262, 0.049913682, 0.00730761839, -0.0513710901, 0.107980385, 0.0701932013, 0.0351378322, 0.0649125725, -0.0676849335, 0.0182300694, 0.130661428, -0.107070848, -0.155545861, 0.0495502241, -0.0824099779, 0.134152278, -0.00340128597, -0.0195551105, -0.0323081203, -0.0359198116, 0.0382399149, 0.0449491367, 0.0474850647, 0.000331875868, -0.0191117451, 0.047182586, 0.0440613963, -0.021301711, -0.0278403945, 0.0186600443, -0.0355576873, -0.00705558807, 0.0601502359, 0.193301961, -0.0209947303, 0.0815899447, 0.0201693606, 0.00183786452, 0.0123391729, 0.0369979292, -0.06023781, -0.0408579409, -0.0491956472, -0.0842604786, 0.115169995, -0.0211197529, 0.0968379155, -0.0253970623, -0.0397769324, -0.0227480512, -0.0505167507, -0.073838897, -0.0568714291, 0.0501287989, 0.119802952, -0.0451339222, -0.004891105, 0.0589094609, 0.0234993063, 0.0152090145, -0.00864690728, -0.00884205196, -0.0196170323, 0.154187307, 0.0880857706, 0.0791010931, -0.0840472952, 0.0691868439, 0.019202508, 0.0612286814, -0.0106645636, -0.0559821799, 0.0584457964, -0.0925194025, 0.0446734577, 0.125199825, 0.00832133554, -0.112132341, -0.00512407999, -0.0764019117, 0.0189055335, 0.103203505, 0.117475532, 0.034303166, -0.0261024777, -0.0315298066, -0.0613420531, 0.0545644648, -0.0385459587, -0.044767797, -0.0984572023, -0.0740322843, -0.0442995131, 0.106362291, 0.0777801871, 0.00996433012, 0.104895405, 0.0288609788, -0.0533554256, -0.0310401358, -0.0207837969, -0.00572202122, 0.0423340164, -0.115558937, -0.0174778774, -0.0496467724, -0.0862012953, 0.0145331295, 0.0801969245, 0.0162990317, 0.0271583125, -0.0411906913, -0.068494752, -0.0318453908, -0.0188762657, 0.143572226, 0.00964309927, -0.037913084, 0.0497611761, -0.0457598045, -0.074146539, -0.011894796, -0.135687903, 0.0597968884, -0.0878565237, 0.0783867538, 0.0686763078, 0.013648239, 0.0111385323, 0.0889137536, -0.0170432758, 0.0535282753];
    CONSTANT bias_0_f : ARRAY[0..63] OF REAL := [1, 1, 1, 1, 1, 1, 1, 1, 1, 1, 1, 1, 1, 1, 1, 1, 1, 1, 1, 1, 1, 1, 1, 1, 1, 1, 1, 1, 1, 1, 1, 1, 1, 1, 1, 1, 1, 1, 1, 1, 1, 1, 1, 1, 1, 1, 1, 1, 1, 1, 1, 1, 1, 1, 1, 1, 1, 1, 1, 1, 1, 1, 1, 1];
    CONSTANT weights_0_g : ARRAY[0..63] OF REAL := [-0.59718734, -0.654758811, -0.532963514, -0.596531868, 0.481612563, 0.543547213, 0.627410829, 0.598454714, -0.516591609, -0.647696674, 0.579932809, -0.656442165, 0.614671767, -0.659679055, 0.640318751, -0.615781784, 0.547570586, 0.308117598, 0.46901831, -0.391173273, -0.424857318, -0.467698723, -0.651260734, -0.456590921, -0.641651571, 0.354110599, 0.464462638, -0.60339886, 0.615200937, -0.664138854, 0.648917615, 0.424222559, -0.396425158, 0.567390382, 0.583124459, -0.601320446, -0.563392878, 0.509967506, -0.540180624, -0.552794456, 0.397468328, -0.571196795, 0.673171759, 0.33233586, 0.616161585, -0.630228579, 0.665058136, -0.375944227, -0.611979842, 0.566402078, -0.539952815, 0.553126574, -0.572719336, 0.593717635, 0.669392467, -0.536695957, -0.561653733, 0.498186916, -0.628992558, 0.379528999, 0.629658639, 0.379309207, 0.593511701, -0.648261726];
    CONSTANT recurrent_0_g : ARRAY[0..4095] OF REAL := [0.0481209122, -0.0318202786, -0.00970466435, -0.00290437834, -0.00275036343, 0.0990201086, -0.0936367735, 0.0976686925, -0.0418446027, -0.0556133538, -0.0564777665, 0.0787887424, -0.0114290044, 0.0218893196, -0.205614388, 0.0152208209, 0.0181199498, -0.0284064934, -0.0342439152, -0.137017965, 0.0287700593, -0.005193057, -0.0650635883, 0.0365564413, -0.0217278358, -0.037748199, -0.0658341497, -0.0255905949, 0.038009502, -0.0546126626, -0.0460595936, 0.0218206272, 0.00399468094, 0.017680075, -0.0763128102, 0.033127699, -0.0077143684, 0.0247347672, -0.0203642212, -0.0115557015, -0.0358676016, -0.0744479746, -0.0645529106, -0.0100551089, -0.0719601512, -0.0227489267, -0.0323692374, 0.0465080179, 0.0370282643, -0.00665151142, 0.0832517296, 0.031519033, -0.0226245075, 0.0370324701, -0.0916333497, 0.0264598839, -0.0413973629, -0.0424684957, -0.0249657538, 0.0204738416, -0.0227105767, -0.0446569808, 0.162603825, -0.0907681957, 0.0164916813, 0.0177964829, -0.0274613909, 0.0213896874, 0.0284074415, 0.0556536093, 0.0117608476, -0.0119014224, -0.0100097964, 0.00712328544, 0.0960042924, -0.0221355092, -0.012341205, -0.0822810605, 0.00621075649, 0.0158543587, -0.039224375, 0.0956175774, 0.00211340189, -0.0302987769, 0.12488319, 0.00465582032, 0.0415266529, -0.0592013597, -0.0298871212, 0.016132934, -0.0860709399, -0.0107791489, 0.0462909974, 0.0498189665, -0.074474223, -0.0412580259, 0.0958068594, -0.154954642, -0.0296173394, -0.0703037158, -0.124084823, -0.0115249828, -0.0230197664, 0.0145090697, 0.112648077, 0.0573431365, 0.0689995661, 0.00494860392, -0.106822893, -0.0473375469, 0.0597126819, 0.0464154631, -0.0783604831, 0.0411163755, -0.042815987, -0.144586474, 0.0362219065, 0.0469412208, -0.0197538324, -0.0835709572, -0.0351632386, -0.0158051811, -0.0422700793, -0.0241524391, 0.100690037, 0.0244359579, 0.0488995612, 0.00180372223, 0.0105709136, -0.00768259261, 0.0435547382, -0.00588419288, -0.0233278256, 0.0167928301, 0.0635891631, -0.0251090061, 0.0264639761, 0.0245278087, -0.0183625892, 0.0156504158, -0.133418605, -0.0845454261, 0.0411974192, -0.0011469014, -0.108427346, 0.0473438799, -0.0647937134, 0.0844287574, 0.0139159337, -0.00464433711, -0.0027067028, 0.0205416046, 0.014629676, -0.0079770796, -0.0146780107, -0.0633884817, -0.0847715065, 0.0574441627, -0.105344526, -0.0986291617, -0.00424446538, 0.11857038, 0.0929525048, -0.0331288353, 0.0511972271, -0.0552587993, 0.0188592188, 0.0982365981, 0.0103346799, -0.11088606, -0.0574182793, -0.176203132, 0.0718074515, -0.0143269673, 0.0819053799, 0.0379631668, -0.0151833482, -0.0886700973, 0.077685751, 0.0705799013, -0.0297324546, -0.0491581336, 0.0320661142, 0.0583819747, -0.0129403826, 0.000415268354, -0.118025079, 0.0136062186, 0.0317530483, -0.0342542715, -0.0568282753, 0.0458773263, 0.0344045423, 0.030919224, -0.0318309776, -0.0827476084, 0.0554043949, -0.0085471943, -0.0501176566, -0.0169954561, 0.0408830978, 0.0345368758, -0.0808091015, 0.0242243763, 0.0804605633, 0.0474758744, -0.143990472, -0.00798570178, -0.0439949185, 0.0783360153, 0.00613855012, 0.152479038, 0.0479704067, 0.103156649, -0.0484668873, -0.0600567758, 0.0747681037, -0.0369002745, -0.0376364291, 0.00931490492, -0.0468802452, 0.0452210717, 0.00375288352, 0.223672509, 0.137855217, 0.0708141923, 0.0284974016, 0.0316613838, 0.00279800408, 0.0199050196, 0.12772654, -0.0388306119, -0.0690812916, 0.0302683115, -0.0769119114, -0.041855935, -0.0184757449, -0.0478848442, -0.0423739105, 0.0511118919, -0.0660206825, 0.0214776322, -0.00486254599, 0.00831041113, -0.0175945442, 0.0189309586, -0.0749505684, 0.0745484382, 0.0784307197, 0.0503095761, 0.0636417791, 0.115242943, -0.0942134261, -0.000691486523, -0.0126986243, -0.102407835, -0.00622267881, 0.0795919672, 0.121291116, 0.0149243735, -0.00184394466, 0.0745658278, -0.029508058, 0.0160574839, -0.00490237307, -0.0382324681, 0.121351637, -0.0154690221, -0.0327811427, 0.0973794535, 0.0707743093, -0.0297274534, -0.0442907587, 0.0230267383, -0.0672419667, -0.0936394632, -0.0378915146, 0.010241054, -0.0626864731, -0.0348511972, -0.0236552395, -0.0291376412, -0.0406767838, -0.103340656, 0.0272771958, 0.0680017024, 0.0294110794, -0.0185967591, 0.0548906513, 0.0235778578, 0.0202316325, 0.0469122306, 0.0539038628, -0.0166766569, -0.00477358513, -0.137759894, 0.0127764996, -0.0961342454, -0.0594221987, 0.0728827417, -0.0164189395, -0.00518658012, -0.0957915857, 0.00829045102, 0.0060982313, -0.108702123, -0.00571756996, 0.011730358, -0.109703034, 0.013793895, -0.01103439, -0.00292722974, 0.119150594, -0.0654953867, -0.131435096, -0.0615822636, 0.0777779296, 0.077475585, -0.0213961024, 0.0456323996, 0.0151772602, -0.0128919464, -0.00187631208, -0.0770529062, -0.0266140085, -0.135572195, 0.0990621373, -0.0836972222, 0.00765161868, 0.0372014344, -0.0157342777, 0.046461232, 0.0439010821, -0.11344932, 0.0120108882, -0.079943575, 0.0361242145, 0.059530139, 0.1079956, -0.0724539235, 0.0395812504, -0.118950441, 0.0581818745, 0.00589985959, 0.00956692733, 0.119364187, -0.0501967296, -0.0618815012, 0.0700081289, -0.00458050519, -0.0538546704, 0.026847139, 0.015209035, 0.0251028202, 0.0991470516, 0.0500489101, -0.015465362, -0.0499136411, -0.0779527053, -0.0647690147, 0.00187926646, 0.000785894692, -0.0298743118, -0.079399772, 0.00420416519, 0.00767213851, 0.0429056548, 0.069042176, -0.0115484241, -0.100130901, -0.0152462944, -0.141715929, -0.06294927, 0.00300536305, -0.00711894408, 0.0651451647, 0.0162868313, 0.0156217925, 0.087315619, -0.0116047934, -0.0446378961, 0.0188532714, -0.0363255925, -0.0206964687, 0.0638260022, 0.0427516736, 0.0962982848, -0.000738136703, -0.100229278, 0.0488995053, 0.03522937, 0.0224751662, 0.0014051646, -0.0589457527, 0.0064151939, -0.0551948473, -0.0919054002, -0.122769751, 0.0627653897, 0.0240616575, -0.0568497702, 0.0125247864, 0.0841191709, -0.0876669362, 0.0636893734, 0.0542640686, 0.0451811217, -0.0322294272, 0.00800275244, -0.0454603657, 0.0555975735, 0.018392466, 0.0210544299, 0.0131536471, -0.0680367053, 0.00835058279, 0.051352419, 0.0290030446, 0.223232776, -0.0436089598, -0.0516412109, 0.0185786393, 0.00577225722, 0.0267854705, -0.0379125513, -0.0165023953, 0.0399743877, -0.013742689, 0.0576421283, 0.0605019405, -0.0926445574, 0.0552524626, 0.038678471, 0.0476564392, 0.069373332, 0.0356642194, 0.049644962, -0.18419756, 0.061424315, -0.00396628678, 0.173152342, -0.0782242119, -0.00853672251, 0.0579292998, 0.0296671931, 0.0431504995, 0.00694876024, -0.00365337171, 0.00795618631, 0.036209058, 0.0228915084, 0.0393313058, -0.115138032, 0.0527001247, 0.00259985588, -0.140608296, 0.0402385257, 0.0532492884, 0.00673503103, -0.0785810426, 0.0723578632, 0.133191809, -0.0573731363, 0.00135149504, 0.0363229215, 0.169861257, -0.032099396, -0.00696232356, 0.0118630938, -0.067776747, -0.0342655331, 0.118268475, 0.0883374289, 0.0637449771, -0.0541283078, -0.0899446458, 0.0376625471, 0.0942173004, -0.0317836255, -0.00520051457, -0.0337636024, 0.0278342813, -0.0441194773, -0.0208879635, -0.0166095793, -0.136137962, 0.0225438811, 0.028527312, -0.0204672888, -0.111636817, 0.0609205514, -0.0297671221, 0.0422912873, 0.0566930138, -0.0438183621, -0.0542889014, -0.0104457084, 0.0645867288, -0.00627774, 0.0382623039, 0.0610745773, 0.00748553127, -0.0615660101, -0.0687104315, 0.0212151445, -0.137569904, -0.130664855, 0.0052475594, 0.0478997082, -0.0951935798, -0.129320979, 0.0327419378, 0.0141034257, 0.0599292889, -0.023001885, 0.112600863, -0.180389807, -0.0478617251, -0.108216099, -0.00132560916, 0.0768594742, 0.025723394, 0.0230658501, 0.0124216359, 0.112398446, -0.0201180503, 0.00827030931, -0.0433050543, -0.0133112697, -0.0448576361, -0.00985031389, -0.0463208407, -0.108422384, 0.0818410814, 0.014295781, 0.0476117656, -0.080968082, 0.0702591613, -0.037799105, 0.0174957048, 0.00386841036, -0.0508742332, 0.0835343897, -0.0123609006, 0.00578187406, -0.0170176364, 0.0335893482, -0.161683038, -0.0468972176, 0.00365513656, -0.0580082387, 0.00578364357, -0.0271733981, -0.0293255299, -0.015630452, 0.036914099, 0.0184712932, 0.017311858, -0.0375006273, 0.0248549618, 0.0181586277, 0.0372040607, 0.122081101, 0.0129180709, -0.069092229, 4.61568125e-05, 0.0141924052, 0.0245402232, 0.0328482389, 0.0326962508, -0.00475404412, 0.126613453, -0.0365736336, 0.0202107634, 0.00670441799, -0.0342802107, -0.0309105664, -0.117560178, 0.00874035433, -0.0867343992, -0.0489641055, -0.0621264018, -0.0782420784, 0.0110636912, 0.0189643651, 0.0254211426, 0.0323629826, 0.0175361186, 0.00821964629, -0.0352783836, -0.026747942, -0.0338488594, -0.0480204672, 0.178073749, 0.0150867915, -0.0393434726, 0.119698055, 0.0209258795, -0.034920793, 0.0432537459, 0.0193708185, -0.0156848282, 0.0321556851, 0.0506595224, -0.0899810866, 0.11158587, 0.0048500672, 0.0901765525, -0.0639372915, -0.128660902, 0.0620967709, 0.00270261988, 0.0502362065, -0.0321554467, -0.144941673, 0.00120547414, -0.0796487033, -0.0480318367, 0.140227005, -0.0196647234, -0.178954765, 0.0206949543, -0.07161735, -0.0766613334, -0.0471355617, 0.125506446, 0.0201372728, 0.057826899, 0.0323966891, -0.0778779611, 0.00571985915, -0.0521460772, 0.0584396943, 0.017673837, 0.0298046097, -0.0585550144, 0.00364940055, 0.0553209931, 0.00706443936, -0.0350266472, 0.106554076, -0.0728589073, -0.015205238, 0.108272955, 0.0273931529, -0.0182952788, 0.0927042291, 0.1110285, 0.0235592145, 0.0894330814, 0.0167295616, -0.00135597819, -0.0577400625, -0.000300495885, -0.117229655, -0.0391341709, -0.00462239562, -0.104280978, -0.0822803676, 0.0824518204, 0.0501513109, 0.127776951, 0.0266683772, -0.0333210044, 0.0495061539, -0.0195217375, -0.0020740442, -0.0615060478, -0.077499263, -0.0539976731, -0.00234729145, 0.0269302428, 0.0488361865, -0.0136367977, 0.106795713, 0.00983078778, 0.0404809564, -0.0170145817, -0.0510442406, 0.0200570561, -0.0909764245, -0.0110744797, 0.0307489485, -0.0250330158, 0.0187591948, 0.0241823718, 0.0275000576, 0.0774741769, -0.0884157717, -0.0736636966, -0.0650302395, -0.037942525, -0.0280007608, -0.046552524, 0.0456949584, 0.0517659038, -0.0650030226, -0.170385316, 0.0340338983, -0.0241850466, -0.0224057902, 0.11006891, -0.0337545238, -0.0527094305, -0.0553541705, -0.0439890511, 0.0177379418, 0.0458082706, -0.0723290518, -0.0321814567, 0.025533095, 0.0281248074, 0.0878937691, 0.0336395875, 0.0259274412, -0.125957265, 0.0391919501, -0.0251755603, 0.0211277232, -0.0278907381, 0.0222725831, -0.00522296038, 0.0184913874, 0.114900775, -0.139606744, -0.0102660134, -0.0418461263, -0.0440084971, -0.0724901706, -0.0273834858, -0.066111438, 0.0256347246, 0.0197810046, -0.0506107286, 0.0275419205, 0.0963028595, 0.0410624444, -0.0184595585, -0.11321824, 0.013122756, 0.0534582585, 0.0112230945, -0.123381555, -0.0182994064, -0.0118550183, 0.0601564497, 0.0450157933, 0.000831920654, 0.0489078164, -0.0160342883, 0.00291860476, -0.0700190961, -0.021231601, -0.0476933345, -0.0166842993, 0.00678215921, 0.0171712432, 0.0231642704, 0.06855838, 0.0576967895, 0.00613667071, -0.0384696573, -0.15129137, 0.038532909, 0.13642779, -0.0366146453, -0.0880282149, 0.000459298957, 0.0403979793, -0.0466576666, 0.0962288752, 0.0426511876, 0.0612617284, 0.0403866768, 0.0632477552, -0.0450474471, 0.00374693144, -0.0240001492, -0.00581013225, -0.0600609444, -0.0843619481, 0.113087408, -0.00712958723, 0.0238859244, 0.0449041799, -0.0338831842, -0.0562099293, -0.0229946077, -0.0107966587, -0.0429909937, -0.0180925671, 0.0642202646, 0.0231274776, 0.0782754943, -0.0284954421, 0.0365221612, -0.0310026966, -0.0401229523, 0.00871577766, -0.0359195769, -0.0456489697, -0.00756221544, -0.107447088, -0.0312013887, 0.0863746852, 0.052147083, 0.0308211409, -0.00791497342, -0.0170036554, 0.0204932727, -0.0273714438, 0.00312257558, 0.0411597528, -0.0490261801, -0.00702317245, -0.0436934456, 0.00491887098, -0.0183614958, 0.00572536513, 0.0202722792, -0.0191663131, 0.0718074962, -0.0192947239, -0.0795083642, -0.0438840538, -0.0110500725, 0.0777254701, 0.0627994984, -0.00645396765, 0.0945438668, -0.066645287, -0.0140715651, -0.0130456872, -0.0747533068, -0.0513444953, 0.0044493638, 0.0323071256, -0.0745799541, -0.00599613879, -0.121034116, 0.0455755889, -0.096720174, -0.0297351964, 0.0622085109, 0.0443798527, -0.0134973312, 0.0455619283, 0.057053756, 0.0374863707, 0.0315487757, -0.0963983759, -0.0530716814, 0.0119701754, -0.0350041129, 0.0811880305, 0.107285455, 0.157880977, -0.00360907614, 0.13897568, 0.00456034206, -0.0327878632, -0.0863745734, 0.00712788105, -0.0183715019, 0.0741946772, -0.0889983699, -0.115648195, -0.055796802, -0.0787045807, 0.0941687897, -0.0179556571, 0.132844016, 0.0386615954, 0.0620229617, 0.0198719017, 0.0204281956, -0.0220341291, -0.0495671928, -0.0185134746, 0.0279251672, -0.106061883, 0.0109254159, -0.0280910153, -0.0658846572, -0.0472168177, -0.108801812, 0.00997927599, -0.00405341247, 0.083818756, -0.112704068, -0.10473299, 0.0724331066, -0.102572724, 0.0289460868, 0.0815427005, -0.0263789799, 0.0103766369, 0.0396544486, -0.0248612817, 0.0700480193, -0.00640966743, 0.02097876, 0.0185124483, 0.0580330007, 0.0572261736, -0.0207672901, 0.0909210965, 0.00181337446, 0.0867288262, -0.0432980172, -0.0198968742, 0.073626332, 0.0299158916, 0.0450405627, -0.031508252, 0.104846664, -0.11461927, -0.00100136083, 0.00705582462, -0.0166247822, -0.0530819371, 0.0750560388, 0.0281708203, -0.0790766552, -0.151709929, -0.0869254097, -0.121713176, -0.106249183, 0.0423684977, -0.0515973233, 0.025914995, -0.0347193368, -0.0648983195, -0.0121801095, -0.104125112, -0.0125135016, 0.0369128287, 0.0256222486, -0.112580098, 0.0390904918, -0.0488199405, 0.0313525088, 0.124518193, -0.0721309856, 0.0227762647, 0.0360551029, 0.016752487, -0.0343185365, 0.0238141567, 0.0821570605, 0.00898459926, 0.16732052, 0.0623603836, 7.33090565e-05, -0.0469410568, 0.100447275, -0.00677802227, -0.0621812493, -0.0202499852, 0.00267476588, -0.0853958428, 0.00704954891, -0.0110385669, -0.0519299619, -0.0122630307, -0.0541042536, -0.00767853204, 0.0619523376, 0.0162527915, -0.0525096431, 0.0088917315, -0.0308911689, -0.0330346264, 0.0748803392, -0.0928550661, 0.0775584802, 0.0113597028, -0.0360381715, -0.0221998356, 0.0145231094, 0.0499595031, 0.0438217111, 0.0493916869, 0.0987473205, 0.0548540652, -0.109685831, -0.0464524962, -0.0478717871, 0.105852693, -0.0407229438, -0.00312836468, -0.0293584224, -0.0373990871, 0.0746089295, 0.0177721344, 0.051328972, 0.156803042, 0.00370166078, -0.0567074902, -0.0473086834, 0.0427102149, -0.00934480503, 0.0413946509, 0.113321967, 0.0857391134, 0.0380230434, 0.0648645833, -0.0120184785, 0.0535119697, -0.0385288782, -0.0135407634, -0.0964917094, 0.0874497965, 0.00108434074, -0.144482508, 0.0785604417, -0.0629226491, 0.0786609575, -0.0747968405, 0.0427639708, 0.015671391, -0.0752736405, 0.00807333179, -0.0236102194, 0.137812942, 0.0693999678, -0.0383155867, 0.0189865436, -0.0680732355, -0.0268307887, 0.0781384483, 0.0677730739, -0.0124174301, 0.0905554518, 0.00874091871, 0.0110436436, 0.080707863, -0.0232983772, -0.117284365, -0.0258648247, 0.00250049494, 0.16272372, -0.0679185838, -0.0224808753, -0.0650340095, -0.0163707584, -0.00510245655, -0.0911356658, -0.0405044816, -0.0403025113, -0.0591014363, 0.0208199918, -0.00787425041, 0.070880726, 0.0509448647, 0.00232681073, -0.0459237248, -0.0840739608, -0.0128986835, 0.0156580452, 0.0746299177, -0.0362110548, -0.0935138389, -0.0977835953, 0.0449482128, 0.0919752643, 0.0343250558, 0.0393615663, 0.0337222815, -0.00249612331, -0.104778022, 0.0307323113, -0.0637253001, -0.0532381609, -0.00681231543, -0.0515490845, -0.0476092659, -0.138044789, 0.0233308692, 0.0432448648, 0.09477029, -0.0449744575, -0.0258047823, 0.0199477226, 0.110396601, -0.0461071171, -0.0765727833, -0.100457534, 0.00327436067, -0.0350628719, -0.0664845929, 0.145648047, 0.0549397953, -0.0286890082, -0.0137136104, 0.0720597729, -0.0895970911, -0.141181692, 0.0554166697, 0.00294139329, -0.0716697425, -0.0761943161, -0.0842018127, -0.0368512794, 0.0226985905, 0.0280064791, -0.0433114879, 0.0182159357, -0.00750421919, 0.0796084031, 0.0343470238, 0.0502757952, -0.00197853521, 0.0140378019, -0.024121806, 0.0345112011, 0.0225584842, -0.0380386673, -0.0472035706, -0.0391502231, -0.00918582827, 0.0454934612, 0.00277288631, -0.0189364627, 0.088180013, 0.0653253943, -0.0102603706, 0.0055696941, 0.0671821088, -0.0022907462, 0.0808660462, -0.0267980788, 0.025423795, 0.0490402654, 0.0702161267, -0.0383854136, -0.00789637212, -0.0306695029, 0.0450484604, -0.0388167091, -0.10609749, -0.0277900603, 0.0719657987, -0.165123627, 0.000689312466, 0.0703398436, 0.0711275414, 0.0693190992, 0.0494399481, -0.0426387601, 0.013213479, 0.00340628065, 0.0935201645, 0.000743723474, -0.0921040997, 0.125364736, -0.0963561609, 0.054403089, 0.0337063596, -0.0468962938, 0.0211268198, 0.108646907, -0.0155733861, -0.105246648, -0.039495822, 0.0604975484, 0.0136065856, -0.0467163324, 0.00234889425, 0.0171512365, 0.0447443351, -0.041860383, 0.133673549, 0.0533847958, -0.0932198837, -0.00490728766, 0.0326834098, -0.00924667157, -0.0203219987, -0.00111838058, 0.0897222608, -0.16880703, -0.0764932483, -0.0934206098, -0.0321779363, 0.00244071521, -0.066392906, 0.0457569174, -0.00558981672, 0.122725204, -0.123424225, -0.112033449, -0.0371551625, -0.0124348812, 0.0834423229, -0.0046160277, -0.0259561874, 0.0431323275, 0.0343380384, -0.0749207512, 0.0373918861, 0.03548605, -0.00775843952, 0.0114278831, -0.044160407, -0.0630012304, 0.00885489956, -0.0644601583, 0.0514997691, -0.0674148351, -0.000801049173, -0.0248331372, -0.0273230411, 0.00697711296, -0.153315246, -0.101669349, 0.0117361899, 0.0785069317, 0.0701476038, 0.00413423777, 0.100262329, -0.0700106919, 0.0447569974, 0.0454962067, -0.0349731036, -0.125184476, -0.0526507832, 0.0559355766, 0.0843899921, -0.0531100109, -0.0739149749, 0.0177767407, 0.0624389611, -0.00888402387, -0.0174835678, 0.00704896264, 0.00679837167, -0.0573560409, 0.0343110412, -0.0745702982, 0.100997314, -0.0872376785, -0.066832006, -0.0915832445, 0.0491389297, 0.0449462384, 0.0670973435, 0.0158868078, -0.0123562841, -0.151852489, 0.00113863684, -0.0875073746, 0.00578712299, -0.0520261414, -0.0425501168, 0.0312268976, -0.0676039755, -0.0329743996, 0.115326986, 0.00371781271, 0.0700134039, 0.13351433, 0.109993905, -0.0490467101, -0.00116261095, 0.103204951, -0.0233638883, 0.0579097569, -0.00423125923, 0.0394633114, -0.00179227069, -0.0272249039, 0.016013518, 0.0664092451, 0.021862261, -0.0098572392, -0.0411397554, -0.0164106991, -0.00709867291, 0.0678975731, -0.0157848224, 0.0440931395, -0.0509038605, -0.132192969, -0.134671226, 0.018839173, 0.123835646, 0.00620973483, 0.0375349373, 0.0937119052, -0.110467553, 0.0718783066, 0.0321933925, -0.0216813739, -0.0765284598, -0.0729833394, 0.110161297, -0.0496276319, -0.10669595, 0.0610559359, 0.0266519599, 0.024480233, 0.0131997876, 0.0788992569, -0.0837132484, 0.0524157807, 0.0891485587, -0.0495346896, 0.0113467937, 0.0430697314, -0.00399557827, -0.0888357237, -0.04823488, 0.0428044833, -0.0218219571, -0.049988009, -0.0297640171, 0.0641734079, -0.00857078563, -0.0439059734, -0.0172368158, 0.00380734494, 0.0124965943, 0.0195954219, -0.121491201, -0.00273006782, -0.0584536269, 0.0717246681, -0.0633384287, 0.00393397175, -0.0967641994, 0.0857604146, -0.0169189703, -0.0077670794, -0.0925148129, 0.00356252119, 0.0541334078, 0.0407074094, 0.0570226908, 0.0423023589, -0.0421995409, 0.0668428242, 0.0828292966, -0.0388631001, 0.044825118, -0.0113215446, -0.00229228614, 0.0638577193, -0.0541986525, 0.0392766818, 0.0207372513, 0.122101203, -0.0374232531, 0.0343491621, -0.12858279, -0.0398529209, -0.0189455971, -0.0161126144, -0.0269678123, 0.143331021, -0.0516516827, 0.00435102684, 0.0862914473, -0.00858026277, 0.0291463248, -0.016167976, 0.0814914033, 0.0335224867, 0.0722127035, 0.0362363309, 0.0352626853, -0.0310319923, -0.0513597652, -0.0654821992, -0.0167266447, -0.00566356257, 0.00895902514, -0.0931169391, -0.0171670727, -0.0258844364, -0.0279674605, -0.0934784189, -0.0405637287, 0.0395140424, -0.00940208696, -0.0371163934, -0.0512821227, -0.0617666207, 0.00312861241, -0.0396652743, -0.0330410376, -0.0350976661, 0.0592487454, 0.0168273486, 0.0460043922, -0.068073079, -0.0354389511, -0.0070019234, -0.0201342925, -0.0740064383, -0.0985625535, 0.109604456, 0.00744982809, 0.0499990582, -0.0913917571, -0.0760618821, -0.00663454551, 0.095058769, 0.0984187648, 0.086010322, 0.00255531631, -0.0553069189, 0.0326800868, 0.118444778, -0.00917500444, -0.0529425405, -0.0467088483, -0.057951156, 0.0604806431, 0.037785124, -0.0233308673, -0.0214508213, 0.0160038956, 0.0201747715, 0.093188554, -0.0278952122, 0.0407564975, 0.0290678702, -0.0616962761, 0.109116971, 0.0545500442, 0.0562264249, 0.0204357766, -0.0588595085, -0.0797440335, 0.104199581, -0.0113319103, 0.0202118214, -0.0470490791, -0.0503209159, -0.00406551547, -0.148654908, 0.0157267656, 0.0869958401, 0.131356552, 0.0617513843, -0.137257427, -0.0557870641, 0.0204233006, 0.0164770335, -0.0680170506, 0.055826664, 0.0141050098, -0.000411175191, -0.0126514919, -0.0469707698, 0.0356213972, -0.00365147367, -0.0831606239, -0.0333047397, -0.0315936208, 0.0866669863, -0.00560810324, 0.0486792885, 0.0163613725, 0.0672739893, -0.0312143788, 0.035975907, 0.0887759328, -0.0322332159, 0.0700955912, 0.067183584, 0.0560502186, -0.145593554, -0.0201487988, -0.17184335, -0.175876051, -0.0536855161, 0.0437362455, -0.0762054473, 0.020145813, 0.0859210193, -0.0183991119, 0.082898289, -0.0865213871, 0.0455945395, -0.0923885703, 0.0201766863, 0.0235567391, 0.00166189671, -0.126334324, 0.0104457736, -0.0839416385, -0.145371616, -0.0621561036, -0.0389697924, -0.0357878767, -0.000569142401, 0.088126041, -0.012336798, 0.132560045, -0.0168081969, 0.0210299399, -0.114906453, -0.0487332717, -0.0576963723, 0.08126764, -0.0170844682, 0.15879257, 0.0390506163, 0.0271640867, 0.032145083, -0.118259393, -0.026053451, 0.0304594599, 0.0193315297, 0.00426006224, 0.0487677045, -0.127483457, -0.0247131083, 0.00520783011, 0.0422325246, 0.0628959686, -0.00937768072, -0.0798375756, 0.00526973139, -0.0230605975, 0.0278230458, -0.015190633, -0.0390762016, 0.0378631502, 0.0325350948, 0.00402753334, -0.0154148303, 0.0552802756, -0.00210960582, 0.00410776678, 0.0478105396, 0.147735938, -0.0677689165, -0.0523314662, -0.0148229077, -0.0358465463, -0.0562868752, 0.0687464103, 0.0209784731, -0.0728497356, -0.0830795914, -0.0207745656, -0.0896096528, 0.0604444854, -0.051528167, 0.117564246, 0.0540245064, 0.0122621823, 0.0533122085, -0.0745593458, -0.0536674857, -0.0729632825, -0.00508011458, 0.032732591, 0.174379155, -0.0351487659, -0.0432448797, -0.0770454705, -0.0280206744, -0.0112591609, -0.0604792088, 0.0313924029, -0.010354016, 0.165250868, -0.0119367782, 0.0626074076, 0.00134766847, -0.0565094762, -0.097651422, -0.0535871722, -0.0217829123, 0.0847785324, 0.0888899118, -0.0187548269, -0.00319143012, -0.031487897, 0.0128169376, -0.0119436681, 0.039205391, 0.0817883611, 0.0454290509, -0.0981512666, 0.0798369944, 0.0262276698, 0.0339503624, -0.0393401906, -0.0285993144, -0.0246126465, 0.0251000859, -0.0793290883, 0.0479018465, 0.0538914651, -0.0681251809, 0.00710714422, 0.112784632, 0.0473594442, -0.108741477, -0.143058866, -0.021414388, -0.0754344463, -0.0993086845, -0.0213276427, 0.0124653531, 0.0831999481, -0.138760224, 0.0565210134, -0.0562419891, 0.0452317521, 0.071887888, -0.0181150213, -0.0408135653, -0.128034428, -0.0674634352, -0.0137788486, -0.0589382574, -0.021415988, -0.0480030216, 0.00845495611, -0.23522377, 0.0711150765, 0.0391303822, -0.0317100994, 0.0424706191, -0.0137902126, -0.0833254084, 0.00742999464, -0.0294535942, -0.0192015357, 0.0305824056, 0.00186828431, -0.0791531727, -0.0463692918, 0.0958603621, -0.0250745974, 0.0704268962, 0.0976651981, -0.00902186055, 0.00842957944, 0.00719482172, -0.00222524256, -0.0258013234, -0.126656577, -0.0502824448, -0.0517087393, 0.033074785, -0.0130861662, -0.056914445, 0.00920967758, -0.0662592053, 0.0150485635, 0.0195489917, 0.109873742, -0.00402418105, 0.0425244533, 0.123894185, -0.00381089188, 0.0175240878, -0.0642656311, 0.00325660803, 0.0580130145, 0.00884908251, -0.0451986901, 0.0102753434, -0.0434884056, 0.0693225414, -0.0231948923, 0.0263490211, 0.0259765089, -0.0155510735, -0.0913651809, 0.000178758986, -0.0589917824, 0.0832998008, -0.061676763, 0.032646507, -0.0242344383, -0.00502131088, 0.0320100263, -0.140749574, 0.0082251234, 0.0054948125, -0.0383517258, -0.031341929, -0.0776535049, 0.0673101693, -0.0471187867, 0.0038197306, -0.0748489872, -0.0125974556, 0.0261118878, -0.030079525, 0.0568254404, -0.070515871, 0.0653721541, 0.0256158337, 0.0375468805, 0.060077861, -0.0122621469, 0.0280455388, -0.0174301565, -0.0258607063, 0.0277182981, -0.0530786812, 0.0413826033, -0.00954391435, 0.0798512474, 0.0131942499, -0.0647169203, 0.0883338973, -0.0757359117, 0.0651931316, -0.08559338, -0.00492510293, 0.0671376586, -0.00483021885, 0.019877255, 0.0292623006, -0.0245957244, 0.0511968136, -0.0557926744, 0.0767183304, 0.0403989851, -0.0530728698, 0.00403285911, 0.0265462939, 0.0372774825, 0.0331319869, 0.0317157283, -0.000328839524, 0.0696135238, 0.22497198, 0.029403165, -0.063406907, 0.0596498474, -0.00453359634, -0.00460745068, 0.0388002172, 0.0470163822, -0.0924427807, -0.0776350275, -0.122637093, 0.00585639477, 0.0648606643, 0.0527789295, 0.0966849029, 0.0227448158, 0.0196636021, -0.0914843827, 0.0110604446, -0.0222737417, 0.0194348935, 0.0205718502, -0.158367962, 0.0795231685, -0.0509676076, 0.0412261672, 0.0339675099, -0.0411967114, -0.0345254727, 0.0379131548, -0.0458045155, 0.0795515478, 0.028041102, 0.0457426161, -0.0328665227, -0.0100045754, 0.00767892785, 0.0601071939, 0.00571505167, -0.0360711403, -0.0598788038, 0.0955239385, 0.0540545508, 0.054462783, -0.158046633, -0.00715309381, 0.0511963628, 0.0795604736, 0.0340496339, 0.0699889585, -0.0264358073, -0.107294738, 0.0785360411, -0.0395349786, 0.0183147267, 0.084531866, -0.0178029481, -0.0461838581, 0.0304375887, -0.027625313, -0.0240503773, -0.076764904, -0.061923746, -0.0269242655, -0.108283713, 0.0242877342, -0.0158310607, -0.104776725, 0.0842112005, -0.128649354, -0.160961986, 0.0475827307, -0.00771825574, -0.0361148268, -0.0477065854, -0.0282700732, 0.0345622152, 0.0850288644, -0.0528912544, 0.0417205244, 0.0404912196, 0.0291186757, 0.0695577636, -0.100897305, -0.0494647659, 0.0219904445, 0.0232919939, -0.0412437133, -0.057831604, 0.0384221934, 0.0113774389, 0.0155264148, 0.00825793296, -0.100460932, -0.056418784, -0.00504833274, -0.0381764695, -0.123155445, 0.0394152813, 0.0292115584, 0.0252512004, -0.0778217688, 0.0401267111, 0.0833734348, -0.0448985957, -0.0260450877, -0.00156772323, -0.015842773, 0.0405933596, 0.0414074324, -0.0164530557, 0.0241394192, -0.108059987, 0.0151647851, 0.0686879233, -0.0308864638, 0.00535558909, 0.0499273576, 0.0604701415, -0.0535615087, 0.0751591772, -0.0335483626, 0.123964965, 0.0308629498, -0.0801210552, -0.00535691436, -0.0834186748, -0.018937042, 0.0462034829, -0.0951785892, -0.00635819929, -0.0276774466, -0.00173071027, 0.0538236387, 0.0478764512, -0.0341162905, -0.0230466239, 0.0638933331, 0.00398610625, 0.042982433, -0.0650900602, -0.0902234688, -0.00778864603, 0.0307439361, -0.0614889525, 0.0939205587, -0.0740359575, 0.0395269692, 0.0186250117, 0.112409011, 0.0178404991, -0.0579250343, -0.0965748206, -0.0242376234, -0.0314598419, 0.022085024, -0.0130205359, 0.0420831852, 0.0939634517, -0.0138993179, 0.171575099, -0.0730244219, -0.130276218, -0.112991668, 0.159022763, -0.0297501404, -0.166945696, -0.0118776429, 0.0283993762, -0.107067414, -0.0101310238, -0.081896767, -0.0201093145, -0.00360797904, 0.107232116, 0.014786086, -0.0684963912, -0.100018784, 0.0396719277, 0.0329135545, -0.00335169677, 0.0525870621, 0.0352525152, 0.0304436609, 0.0136254113, 0.0571700633, -0.017121572, -0.0459432155, -0.0535720363, -0.0370734558, -0.0255964324, 0.00722439308, 0.0100322692, 0.0936748385, 0.0392240658, -0.0450329445, -0.102835342, -0.01803305, -0.0027119536, 0.000686083455, -0.0262447912, -0.0244153645, 0.0996294245, 0.160265952, 0.0174035244, -0.0181496907, -0.0874229074, -0.0340590551, 0.0494551286, -0.0896435305, 0.0090267593, -0.011298812, -0.0349937044, -0.0563521162, -0.020006869, -0.00306661916, -0.0467281044, -0.0959168822, -0.000710475491, 0.0160875991, 0.0613734052, 0.00380967022, -0.00285200775, 0.0998165384, -0.0835248679, -0.0224947855, -0.00109235756, -0.123580478, 0.0138304345, 0.0292002633, 0.0619599894, -0.024383232, -0.0890621021, -0.0477156676, -0.00767880492, -0.07755211, 0.0379336365, 0.0282836836, 0.0121202217, 0.0700273812, 0.077599436, -0.0282810107, 0.0873090699, 0.0170445964, 0.0217204187, 0.0357856713, -0.124284752, -0.0176754631, 0.0292597283, -0.0277153738, 0.0340308547, -0.0351814777, -0.0185415074, 0.0657032058, -0.070098199, 0.0163267124, -0.0359653756, 0.0431222655, -0.0805179477, 0.0551398806, -0.0429115556, 0.039605882, 0.125053793, 0.0103085376, 0.016506806, -0.0767327547, -0.0145367458, -0.00527186738, -0.109325774, 0.00158104394, -0.0645579472, 0.0414604209, 0.0704116151, -0.0550332256, -0.079351984, -0.0402190648, -0.0678713173, -0.00361617655, 0.00728332764, -0.0924493521, -0.0715293139, -0.0627117902, 0.138858184, -0.0787227899, 0.0878711119, 0.0903199762, -0.0314689875, -0.101632565, -0.0277199894, 0.0456825122, 0.0400777832, 0.0206087139, 0.00740317628, 0.0462091863, -0.0205879845, 0.00412323372, -0.0854965746, -0.0270496532, 0.0537586994, 0.0209500827, -0.00426409394, 0.0223928615, -4.31127846e-05, -0.123981491, 0.0320555232, -0.000461637974, 0.0719709396, -0.0821013078, 0.0520155355, -0.0581474714, 0.043170061, 0.0477350801, -0.0482107103, 0.0453792661, -0.0878505558, 0.0651191846, -0.0550199747, 0.0114516839, -0.0134740882, 0.019735653, -0.00105285458, -0.0154596092, 0.0565496385, 0.131995961, 0.0106603578, 0.0428187959, 0.0278355088, -0.04933827, -0.0904063508, -0.0304906089, -0.13550666, 0.0764463022, -0.00670049433, 0.020669749, 0.0304554198, 0.00477591436, 0.0705404133, 0.0484770127, -0.0078827301, 0.0109620914, -0.0700891167, -0.102043234, -0.00599737279, 0.0399149507, 0.0239164066, 0.0184967127, -0.034097746, 0.106267288, -0.0741966218, -0.094293043, 0.0152545823, 0.039439626, 0.00443127472, -0.126506031, 0.0146793108, -0.00417120196, -0.152482659, 0.0430405028, -0.0735604465, 0.00370641239, -0.0684757754, 0.135406911, 0.0257249549, -0.0108325416, -0.0201357678, 0.0574883036, 0.0695692152, 0.0266307369, 0.141420886, 0.0824303776, -0.084047012, 0.0514349453, 0.0188176166, -0.00754374824, -0.0172986593, 0.0694952235, 0.0892180577, -0.0456226654, 0.014485009, -0.0377262458, -0.0674300194, 0.0369834974, -0.0324523523, 0.0640139952, -0.0502232984, -0.0138668008, -0.0174614154, 0.0846967846, -0.117430434, 0.00789684057, 0.0359769762, -0.0229859129, 0.0274296813, -0.0409591384, -0.0772005469, 0.0136770494, 0.0680422038, 0.021900624, -0.0571149364, -0.00919441693, -0.0769463107, -0.0379129797, -0.0244451091, -0.00108371116, -0.134768829, -0.0302732959, -0.0192979164, 0.0894578919, -0.042584978, 0.0138898045, 0.0229867212, 0.0396369509, -0.00647289678, -0.058911074, -0.00774299912, -0.0241449736, -0.0155218299, 0.0452623069, -0.0422731116, 0.124407053, -0.101004273, -0.109089985, 0.0241209343, -0.0319802389, 0.0618858412, -0.104659766, -0.0236198213, -0.0525226332, -0.0204020422, 0.0444595031, -0.0484412126, 0.00843760185, 0.0739820227, 0.0294990018, -0.0333282128, 0.0785892531, -0.205169261, 0.146262214, -0.0366105214, 0.0265037641, -0.0547129326, 0.0283375494, -0.00136286567, -0.101287931, -0.0229337569, -0.0427873954, 0.0548651852, -0.00641091028, 0.0818172842, -0.0336215198, -0.120600149, -0.0876964852, -0.00719404873, 0.043784555, 0.0818615258, 0.0160490647, -0.00279035978, -0.00169721525, 0.0297120623, 0.0481560379, -0.00340225501, 0.0897073969, -0.018950453, -0.0165265184, -0.0431759544, -0.0669650882, 0.12288031, -0.0137352683, -0.0687472746, -0.0284581166, -0.0267633256, 0.00139244506, 0.0258420948, 0.0411406532, 0.0287138373, -0.0488306545, 0.00070649758, 0.13510251, 0.0621741079, 0.000955080613, 0.0634306595, 0.0369181111, 0.0277759265, 0.0670921057, 0.0985985398, -0.137788251, 0.0575925261, -0.0786205754, -0.118083365, -0.0208788253, 0.039425727, 0.0306449607, 0.0296049956, 0.0243346523, 0.0358010419, -0.0267876927, 0.0848198682, -0.039069593, 0.0176634844, -0.00116391666, -0.0144650191, 0.0339574739, -0.0374406874, -0.0428140163, -0.0710135773, 0.0283427089, 0.0835082531, -0.00906604249, -0.0411554985, 0.0739738047, -0.0189926662, -0.0252566449, -0.0116466815, 0.0340939611, 0.113228142, 0.0806068033, 0.0643591732, 0.0140811261, 0.042673789, -0.191585913, 0.0494581833, -0.030789692, 0.0597962923, -0.0125313029, 0.0817469284, 0.168146908, -0.0528120548, 0.00892654061, -0.0317977481, -0.0724169388, 0.0255409386, -0.0364715829, -0.0301792603, 0.0195860378, -0.0338978507, -0.0801440477, -0.0120657105, 0.0596922264, -0.00874493457, 0.121094428, 0.0708883181, -0.0149152083, 0.014944056, -0.0213558134, 0.0833455995, 0.0197257046, -0.0397833399, 0.0338381976, 0.00830554217, 0.0368271209, -0.0645696893, -0.101337522, 0.0923627317, 0.0610283427, -0.0257757399, -0.103941455, 0.0605494305, -0.0309514273, -0.0055113472, -0.0272281468, 0.0351940207, -0.00256633386, 0.0295238253, 0.0661296919, 0.068804726, -0.0388357118, -0.0532150567, 0.039346125, 0.0340142064, 0.0550237782, 0.0415559821, -0.0522850864, -0.105249263, 0.0124835959, -0.149731562, -0.0593612902, 0.0822790861, -0.00512557989, 0.03279626, 0.0674115345, 0.0259852875, -0.0777577981, -0.0727019012, 0.07311216, 0.0607876554, 0.029598169, -0.000872975215, 0.048749797, -0.0189535096, -0.0636676028, 0.0206812583, -0.149629742, 0.0257316083, 0.105723716, -0.0360996872, 0.0338115022, -0.0360098034, -0.150207654, -0.0113919582, -0.0497757755, -0.0376224257, 0.010868337, -0.0651779771, 0.000354363583, 0.0765347034, 0.00184120052, 0.0805332065, -0.0169758648, -0.0782428607, -0.0974958912, -0.116587415, -0.0211042687, 0.0526664257, -0.0128923822, -0.0608641915, -0.0232686047, -0.00864091702, -0.0134981433, 0.0171436779, 0.0173625126, 0.0547433458, -0.00981733575, 0.0505603403, 0.0299072489, 0.0209988356, 0.0734175816, -0.0199452303, 0.0516468212, -0.0163122434, -0.0143064726, 0.000568790361, -0.0805694535, 0.0614973009, 0.0719416589, 0.052525606, 0.115427695, -0.0925088376, -0.00752420817, 0.0467291698, -0.0388741791, 0.0419192985, 0.0359211974, 0.0629161596, -0.0352669246, 0.0362250581, -0.0923455358, -0.0280749276, -0.0626645982, -0.005751363, -0.022441756, 0.0223358795, 0.043843165, -0.0708922818, -0.0274405628, -0.0362168215, 0.114612833, 0.0180925261, 0.00879310537, 0.0876049474, 0.0473484583, 0.132705808, -0.106990419, -0.00035004667, 0.0237937458, -0.0216909889, -0.109508529, 0.100424141, -0.0414635427, -0.0958008021, -0.0667974949, 0.0679017454, -0.120272838, 0.102716468, 0.00915881991, 0.0977998972, 0.0425018296, -0.160360903, -0.064005211, 0.00124069396, -0.00363787636, -0.00426357426, -0.0214137193, -0.0104995091, 0.0480857007, 0.161474854, 0.0341324918, -0.0272884779, 0.0479773656, -0.0246429555, 0.0198291838, -0.0326992348, -0.069773823, -0.00768797239, -0.0472273752, -0.000691863243, -0.0756409317, -0.0700881779, 0.000398247153, 0.0808655918, 0.0512093976, -0.0463012159, -0.0348239616, 0.0418741331, -0.0345728621, -0.0323799811, -0.0494922586, -0.0705569014, 0.0630198568, 0.0776791871, 0.0139671341, -0.0635786131, -0.0494511276, -0.07453309, -0.00169473421, -0.0472554937, -0.111381955, 0.0366191939, 0.0675320178, 0.0231734607, -0.0630619824, 0.0791029483, -0.0195170939, 0.0553529412, 0.0782957524, -0.0206020568, 0.0127631333, -0.0143370237, 0.0718804896, 0.0197598338, 0.027839547, -0.00322605995, 0.0468392149, 0.0643025786, 0.125367671, 0.00281882752, -0.0283946618, 0.0239227228, 0.0611252487, 0.0226834156, -0.08678554, 0.00260752439, -0.056965325, 0.0965060592, -0.0359185264, 0.0653933287, 0.0124843251, -0.0117376018, 0.106193826, 0.0554171503, -0.0193779022, 0.141835064, 0.00335691683, 0.0138336811, 0.0364889018, -0.015252417, -0.0240376648, -0.0502208993, -0.0984525532, 0.0377380922, 0.0700503662, 0.00973891746, -0.108584166, -0.0191087052, -0.064934127, 0.0390886664, -0.0633433759, -0.0236953385, 0.0651853606, -0.0308972616, 0.0145662688, 0.0389599428, -0.123911798, 0.0314725414, -0.0665021017, 0.0181828942, 0.100704998, 0.0947147161, 0.121352561, 0.0914779529, -0.0123241842, 0.00159506244, -0.0166297033, 0.111245692, 0.0306047089, 0.0483554304, 0.0815960765, 0.0939605683, -0.144702062, -0.026737269, 0.0687930584, 0.099370569, -0.00924576819, -0.0111892018, -0.00826215558, 0.0518443026, 0.0611222833, -0.0611283407, 0.0774296969, -0.0617843568, 0.0744241849, -0.0446566902, 0.0439996086, -0.0497374237, -0.023755705, -0.00537319481, -0.0613298565, -0.0202764831, 0.105274282, 0.0538301915, -0.0278049428, -0.0214678161, 0.0338929296, 0.153826043, 0.0531112589, -0.0624416731, -0.00406610966, 0.0771012008, -0.0810915232, -0.00404860079, -0.0070518814, -0.0274198186, -0.0243172832, -0.00354258716, 0.0509218909, -0.01358038, -0.0742220804, -0.104827151, -0.0613276735, -0.128273591, -0.00304749794, 0.0820524991, 0.102520354, -0.0437029675, 0.00253154337, 0.00355464965, 0.0338010676, -0.00310611166, -0.0497729778, 0.0204216428, -0.0426606275, -0.0259824973, 0.103215985, -0.0622049198, 0.0177591778, 0.00805706903, 0.0654050261, -0.0413892865, 0.0424751863, 0.0389198624, 0.129071906, -0.0924053043, -0.00951092131, -0.0995962545, -0.0196446758, -0.0411661193, 0.0303242616, 0.0544071347, -0.0165973473, -0.0190687887, 0.0460706539, 0.0481170937, 0.00521525461, 0.0615332201, -0.0138894878, 0.0629429221, 0.0188272148, 0.0645333529, -0.112449788, -0.0796088576, 0.0595843494, -0.0757595971, 0.0233897734, 0.0538358651, -0.0479861349, 0.0390440784, -0.118164249, -0.0228865556, -0.0125200767, -0.0924512967, 0.0292225555, -0.123107538, -0.0517924577, -0.042208828, -0.00905832835, 0.0264931507, -0.114739299, 0.0022890456, 0.0705937296, 0.0230474472, 0.0445196964, -0.0252405554, -0.0574160293, -0.00563791115, -0.0591321215, 0.105041645, 0.0162827242, -0.0159014985, 0.0198964141, -0.0534997284, 0.0333555192, 0.0352296121, 0.0559886172, 0.025293462, -0.0884019285, -0.0302855242, 0.102193311, -0.154002801, -0.000932867173, 0.00626800489, 0.0131553337, 0.0937674865, 0.0429573096, -0.119402193, 0.0191562697, 0.0293847565, 0.0485196374, 0.134859204, -0.0864450708, -0.0480053797, 0.0538776852, 0.0346692652, 0.0741332322, 0.0328877792, -0.030711595, -0.0129628722, -0.078539826, -0.0995112211, 0.0568457581, 0.0431236997, 0.0640261024, -0.0128824571, 0.0589009821, 0.0684028566, -0.0567931943, -0.0752976686, 0.0807084665, 0.0214182511, -0.040305879, -0.0120218173, 0.0354591012, 0.00710163219, -0.0271234177, 0.0349637978, 0.0301369913, 0.0289370157, 0.0570953712, 0.0647136867, -0.0894503593, -0.120303392, 0.0157001317, 0.0127883786, 0.0261324402, 0.0461795069, 0.0575956367, 0.0509790294, -0.019913977, 0.0808205009, -0.0281112455, 0.0316304415, 0.0314365365, 0.0944491178, 0.0665691942, -0.0301116239, 0.115353502, -0.0664916337, 0.0734346658, -0.0777676329, -0.0429663248, 0.161868215, -0.10320656, 0.112261094, 0.117354162, 0.0197173785, 0.00444236584, -0.0464475378, 0.09225896, 0.020424461, 0.00536470767, 0.0234805197, 0.0751858503, 0.0640073866, -0.0476553999, 0.0765952468, -0.0601787046, 0.0799819976, -0.0693865865, -0.0414067805, -0.0199543163, -0.0474591479, 0.00405289978, -0.0921546072, -0.00920628197, 0.0468858406, 0.104200438, -0.0764785334, 0.0627960861, -0.0501770973, -0.0596859157, 0.00824402086, -0.0656843707, 0.0273697786, 0.0630233884, -0.126935452, -0.0146518387, 0.0579690114, 0.0838320926, 0.122515112, -0.0182949863, -0.0914339796, 0.00154069811, -0.0247800127, -0.102166817, -0.0945275426, 0.122807965, 0.131390989, -0.00587345567, -0.0786869228, 0.0212463923, -0.0395794287, -0.0131474677, -0.0381132923, 0.0263320245, 0.0894348398, -0.154338613, 0.0110530499, -0.0922434777, -0.00759971188, -0.160012305, 0.0738580674, -0.0513093844, 0.0270811357, 0.063596189, -0.0848937333, -0.0214031246, 0.052909907, -0.0697827041, -0.0753467679, -0.0854087621, -0.00488964515, 0.0621982478, -0.0150694996, -0.170356378, 0.0560002103, 0.0331740938, -0.0252884384, -0.017979769, -0.00263714883, -0.00330292061, -0.00365110394, -0.0507900454, 0.0196132362, -0.0549773537, -0.0324734673, -0.0871634781, 0.0995452404, 0.017264016, -0.00888042618, -0.0175289214, -0.040420182, 0.0419059135, -0.0964919478, 0.0502507612, 0.0567813665, 0.00474262796, 0.0458938219, -0.109633453, 0.0998094454, 0.00364132668, -0.0911779553, 0.0331636071, 0.0855786577, -0.107374929, -0.0224664994, -0.000765305012, -0.0714482814, 0.103808306, -0.0731329024, 0.0835931972, -0.0471782722, 0.105101429, -0.0689914897, 0.0758177042, -0.0657361075, -0.00453515165, 0.0859735385, 0.140476763, 0.0535909422, -0.0119659174, -0.039860554, 0.0254895017, -0.0844546556, 0.0366881192, 0.047922466, 0.0036543645, -0.0358057581, 0.0647788793, 0.027530266, -0.0146779083, 0.0190014765, 0.102737941, 0.0260957927, 0.0133577744, 0.090441525, -0.0800664574, 0.0402105637, 0.00637933612, -0.0870320573, 0.0416977033, -0.0724343061, -0.0724514127, -0.0756017268, 0.0449556597, -0.0770365447, -0.094012633, 0.0169666484, -0.0604530834, -0.0119794961, -0.0296169464, -0.0182167497, 0.00311820139, 0.0188847445, -0.0615576729, 0.081466876, 0.03135176, -0.064924337, 0.0165789854, -0.0213897806, -0.0832084939, 0.0138829947, -0.0481648222, -0.068301402, -0.105001867, 0.0202965103, -0.0275194831, 0.0461513996, -0.00282274326, -0.0420830175, -0.00901214033, 0.104135387, -0.026667513, -0.0501220822, -0.0211645328, 0.0260755643, 0.0366583802, 0.0379104242, 0.0428654142, 0.00207943236, -0.0272428263, 0.0508336425, 0.0345884636, 0.030708028, 0.0927383527, -0.0506587364, -0.0474001542, 0.0975712612, -0.0461767912, 0.0785885528, -0.00822654739, -0.0764655992, -0.0412812978, -0.0233451203, -0.0492914915, 0.0196376704, 0.00331841595, -0.155132622, -0.0511276312, 0.0456443541, 0.0518271178, 0.0220165923, 0.028902486, 0.0874899328, -0.109388873, -0.0217077136, 0.124211319, -0.137767449, 0.0378271677, 0.0107774027, -0.0208922699, -0.0363437943, -0.0730300918, 0.0636523962, 0.021817226, -0.0805155858, -0.0151718901, -0.000913062133, 0.0732663572, -0.0859595984, 0.00871815905, 0.0488275811, 0.0290048681, -0.0100099035, -0.048069112, -0.00914128125, 0.0286560543, 0.0647854805, 0.0454113707, 0.0901111513, -0.0271694791, -0.0388707183, 0.0126525927, 0.0517581105, -0.0812128335, -0.0296413638, 0.0886463895, -0.0482202955, 0.0609410703, -0.0118579054, -0.042096179, -0.0287402868, -0.036506176, -0.0558843017, 0.0764846876, 0.0297001153, 0.117473118, 0.0221678987, 0.140879154, 0.0125083141, -0.0423781201, -0.0285840984, 0.0400817469, -0.013714483, 0.00734990602, -0.0954379439, -0.0371691026, -0.0712833628, -0.00684283022, 0.0395526737, -0.0154475356, -0.048626896, 0.0332213119, -0.0258385297, -0.00113342039, 0.0387322679, 0.0294040497, -0.0428540222, 0.0243901554, 0.0338843428, -0.0673692748, -0.0165437981, -0.0238987692, -0.0630893484, -0.0089747142, -0.0822747499, -0.0521690547, -0.0512124561, -0.177520901, -0.0344200954, 0.0814849958, -0.000873167068, -0.0574686974, -0.0415621027, 0.0236720163, 0.00065103732, -0.0884868875, 0.0770121515, 0.120225757, 0.0519356579, -0.0197645947, 0.0821143389, -0.119676083, -0.0385078005, -0.00692158472, 0.0158718061, -0.0339390524, -0.0775201917, -0.0383195058, 0.0507715866, -0.0184547789, 0.0238665901, -0.014214796, 0.0209062509, 0.0242193062, -0.00141819497, 0.00692214351, 0.0374578685, -0.0173916519, 0.0625144541, -0.0313805379, -0.118092038, -0.0013872229, -0.0306943599, 0.035175886, -0.106766209, -0.0444181859, -0.000435531139, 0.0271715578, -0.0614502616, 0.083078742, 0.125069976, -0.0187428892, 0.0118645411, 0.0150925284, -0.112407535, 0.101660348, -0.0412534997, 0.12648873, -0.0888188183, -0.00799131021, 0.00716023287, 0.0294510331, 0.0610299185, 0.0376382619, -0.0032101199, 0.0695243403, 0.00305525865, -0.00300749578, -0.0317306593, -0.0440058932, 0.0746480078, -0.0228453763, -0.0933810994, -0.109526873, 0.00298138894, -0.110289164, -0.0178135727, 0.0166152269, -0.0675438717, 0.0303429626, 0.111184388, 0.0643074885, 0.0398091711, 0.0890834928, 0.0130663086, -0.115961395, -0.0627881587, 0.00760303997, 0.182588398, -0.0104363523, 0.0734993368, 0.0184030998, -0.114456728, 0.038190715, -0.0541619882, -0.0242964402, 0.0394015461, 0.0477589183, -0.00264003128, -0.0493176579, -0.0128857121, -0.0414938368, 0.108017333, -0.0944479927, 0.0359684266, 0.056056276, 0.0276363213, -0.124510586, -0.0117321275, -0.0544987023, -0.0241859294, -0.00926302094, 0.0522548929, 0.0626090467, 0.0387314036, -0.0622218475, -0.0100225778, -0.0615585335, 0.0938540697, -0.059868928, 0.0660054237, -0.0213241931, 0.00500091631, 0.0162497777, -0.081181936, -0.00911408849, 0.00272774138, -0.0281694401, -0.0126839522, 0.0954968333, 0.0848784074, 0.0969819948, 0.0117116123, 0.0704694986, 0.0726951063, -0.0480228141, -0.0442797132, 0.0604094565, 0.00725152344, -0.0223079976, 0.021759402, -0.125143394, -0.131980091, 0.0427825227, 0.0298181102, -0.0591773763, 0.0159153156, -0.00683892518, -0.130983442, 0.0175854117, -0.0604125261, -0.0670502558, -0.0174585823, 0.075420469, -0.0090696644, -0.158749849, -0.0345814712, 0.100698307, -0.00131180137, -0.0727219954, 0.0901203007, 0.0487782918, -0.0365524814, 0.0508513041, -0.0356357507, -0.026303906, -0.0503677055, -0.00311584352, 0.026720779, -0.0545347445, -0.0972394794, -0.127279475, 0.0424370393, 0.0411688909, 0.108897105, 0.111440197, 0.0727081299, 0.0386688001, -0.0574060455, -0.0480149426, 0.0587941855, -0.0315570571, 0.0149631556, 0.0608740896, -0.00282233022, 0.0588156916, 0.0550168753, -0.00352934562, -0.00595449563, 0.0362947248, -0.00425619073, 0.0214026123, 0.0861438438, 0.016392624, -0.0481089093, 0.0629308298, 0.0187059622, -0.00877061114, -0.0102445884, -0.0555398688, -0.0202465095, -0.00316029973, -0.0736439675, -0.0833783075, -0.0193466172, 0.0141924946, 0.0416547693, -0.0147441458, -0.064637199, -0.00535998773, -0.0525402203, 0.0476203375, 0.0963367596, 0.0137013644, 0.00772009045, 0.07207378, -0.0335871428, -0.00214026356, -0.0041450467, -0.0382905491, -0.029754689, -0.00746493787, 0.00490388181, 0.0492588133, 0.0540007502, 0.0863560736, 0.00244447216, -0.0311946329, 0.0792047158, 0.00161223812, 0.0527098663, -0.0458053686, -0.169502273, -0.00125134503, -0.133062884, 0.0552582815, 0.0536512211, 0.024506554, -0.0158500653, -0.0882110298, 0.0739501193, 0.0192317571, -0.0201549679, -0.0592633821, 0.03385894, -0.102220789, -0.0156797878, 0.0962860137, 0.00793076307, -0.0206457097, -0.0368536636, 0.0329591855, 0.119305857, -0.0199357327, 0.0112215523, 0.0406704508, -0.00535112433, -0.00419330131, -0.0565921143, 0.00923812855, 0.00506248511, 0.0802902803, -0.0690763369, -0.00641982071, -0.0504676811, 0.0534303375, 0.0185494926, 0.112645112, 0.114990473, -0.108184911, -0.118708849, 0.0205293465, 0.0799019337, 0.0527776219, 0.0562684014, 0.00158056244, -0.0319742113, -0.0329294726, -0.0514441878, -0.0824511573, 0.0129657052, -0.0552038215, -0.0339935869, -0.0118879359, -0.0628834814, 0.0313808024, 0.0234189089, 0.0413986817, 0.122857526, 0.07108666, 0.0850967169, -0.0232612919, 0.0413610898, -0.103143692, -0.0849683657, 0.0547915734, 0.0728617236, -0.00469026156, 0.0268891864, 0.00526945945, -0.0898173451, 0.0448876359, -0.0462168604, -0.0161455087, -0.0305345096, 0.0170825832, -0.0591151863, 0.0808007792, -0.0346651524, 0.0201067217, 0.0485038757, -0.0382999629, -0.00971189793, 0.0532421544, 0.066681467, -0.0196481552, 0.0112449778, -0.10701029, 0.0253744181, 0.00411620783, 0.0408724174, -0.105399154, 0.0540573299, -0.0137080066, -0.0767449513, 0.0335149318, -0.0276999753, 0.0461446494, 0.0686794892, -0.0970996618, 0.0948420167, 0.0292930454, -0.00235683098, -0.0422637425, -0.00771948323, 0.0473752245, 0.12806493, 0.0797860622, 0.0526821576, 0.0275474563, 0.00680147205, 0.00534571521, -0.00609148946, -0.0469631962, -0.109895684, -0.0489392504, 0.0118197631, -0.0245287493, 0.0783787072, 0.0512709543, -0.0866212994, -0.0208278876, 0.0346602872, -0.0721480921, 0.0291726012, -0.0341879614, -0.121030957, 0.0489149615, 0.0460931957, -0.0652834028, 0.0706439838, 0.00154211326, 0.0886257887, -0.0143617941, -0.0464408956, 0.0509227552, 0.0692922696, -0.036983151, -0.047252886, -0.0377750657, 0.0251179338, -0.040810965, 0.0308794938, 0.0634416267, 0.0280654058, -0.00847002678, -0.00948635116, -0.0756070465, -0.167530015, -0.0451081842, 0.0682652071, -0.0970221311, 0.112296745, 0.039185863, 0.0178513806, 0.0411128178, 0.00404301658, -0.0386188515, -0.0945572108, -0.129466668, -0.0732636377, -0.0445229784, 0.0360318124, -0.129789457, -0.0505905524, 0.0172151458, 0.00125723984, -0.0734494627, -0.0551522449, 0.0664369017, -0.050375361, 0.0738972053, -0.095365718, -0.0311549269, 0.0148815559, -0.0639430135, -0.000410469249, -0.0740771741, 0.00665809074, -0.0168390423, -0.0652531087, 0.0188372992, -0.0410046875, 0.0307904445, 0.029824581, -0.0674064308, 0.0444030836, -0.00864167511, 0.025579311, -0.0564590245, -0.0318515711, -0.118101709, 0.0296132248, -0.0154637303, 0.0195945017, 0.0539270788, 0.00230327435, -0.107506797, 0.047890313, 0.104820907, 0.00317370426, 0.056395188, -0.0386147611, 0.00254535186, 0.132224351, -0.131078675, -0.0229842179, -0.0498849079, -0.036458768, 0.0912048817, 0.0577849299, 0.0563270375, 0.0386679135, 0.0207617283, 0.0282165948, 0.022253111, 0.0162841864, 0.0609981604, -0.0535034984, -0.00639118999, 0.0175048709, -5.16884029e-05, -0.0496583395, 0.0420942381, -0.00711002946, 0.0533797741, 0.0754599348, 0.0450676493, -0.0988175124, -0.0117549403, 0.0397280343, -0.0656344146, -0.0690754279, 0.00671907514, -0.0357163586, 0.0704929158, -0.0104445647, -0.031824138, 0.0632856339, -0.161348209, 0.0730081424, 0.0338676609, 0.0422311872, -0.0428464711, -0.0331770591, 0.0502553098, -0.0321431831, -0.173599273, 0.0672221407, -0.134899676, 0.0315435417, -0.0236472562, 0.109340206, 0.0198541153, -0.00735092442, -0.0903198123, -0.0266532432, -0.0513025485, 0.00721043674, 0.071140334, 0.079477936, 0.0349715501, 0.00725980056, -0.0391205661, -0.00306599308, -0.0327405334, -0.0486809984, 0.0492282584, -0.0904380158, -0.075029321, -0.0714832842, 0.00332455663, 0.0284815412, 0.0440489016, 0.0446873829, -0.026955219, 0.00358369038, -0.0196625702, 0.124643825, -0.127783328, -0.00134702632, -0.0584786907, 0.0593934767, 0.0422235765, 0.0127851395, -0.0459921472, 0.0656854659, -0.0386239924, 0.146688282, 0.00100399076, -0.034374468, 0.109392554, 0.0923388749, -0.0546806306, -0.00773739396, -0.0400057919, 0.00593503425, 0.0323669463, -0.153363675, -0.0233262014, 0.000179575756, -0.0146199949, -0.0022193559, -0.113891542, 0.0625784472, 0.00597323198, 0.0225357246, -0.090168193, 0.00866935961, 0.0341421142, 0.0408706442, 0.0155995823, 0.130314946, -0.0341695324, 0.059675999, -0.0914648771, 0.0415834077, 0.107751623, -0.0561147109, 0.0860907659, 0.0813505352, 0.0876493827, -0.0822477043, 0.0635892674, -0.0679197013, -0.0907210261, -0.0291095674, -0.0881702974, 0.0369192995, -0.0670497566, -0.0129519645, 0.0381920002, 0.0378953293, 0.0725994259, -0.113148898, -0.0569427311, -0.0372201502, 0.0286789481, -0.0310309846, -0.0636191219, -0.0256764609, 0.0669033006, -0.0567787401, -0.0482122675, 0.00114958361, -0.11021357, 0.0051893089, 0.00271702185, 0.0142258443, 0.0357285775, 0.0446433574, -0.0247358754, -0.0635410994, 0.0193568245, -0.0775561482, 0.0203439202, 0.0762478411, -0.0149462633, -0.108457632, -0.0279274881, 0.0374750644, 0.0117988223, 0.0121162571, -0.0320138372, 0.0168421566, -0.0261973664, 0.0337602198, -0.0159253664, 0.0284005143, 0.0759739131, -0.0799477026, 0.0859935135, 0.0497951061, -0.0269434694, 0.0195953101, -0.0687096864, -0.0860879496, -0.0250251368, -0.0095516229, -0.0168621205, 0.0408060104, -0.135441706, 0.00510279089, -0.0503132716, 0.0770833269, -0.000826317817, 0.0140401246, 0.0687637851, 0.0842372924, 0.121560618, 0.0179199502, -0.0422263332, -0.0214175247, 0.00272018462, -0.0335430577, 0.00117124617, -0.0579549558, -0.199777588, 0.0642453954, -0.0254165158, -0.0149962958, -0.0111465156, -0.104544483, 0.0647178218, -0.0770204961, -0.0407639816, 0.062060453, 0.0558163077, -0.0440091416, -0.0594021194, 0.200664967, -0.0584888831, 0.00234861672, 0.0138185192, 0.0135267861, -0.0327968858, 0.0377394482, 0.0850461125, 0.0219436623, 0.0265891105, -0.0510989316, -0.00208813953, -0.00678487681, -0.0396078601, -0.000987812877, 0.0239344053, -0.0372508988, 0.0748797655, 0.0297940243, -0.0017893184, 0.0170243997, 0.0995491296, 0.0162544418, 0.0433318987, -0.0467717573, 0.0378603712, -0.0230618529, -0.073737286, -0.0342540666, 0.0815814361, -0.0365770012, 0.012538448, -0.0577073283, -0.0641034096, 0.0255438257, 0.0682753772, -0.0223117881, -0.0653793886, -0.0944478959, -0.00180123886, -0.0551710464, 0.0525893942, -0.0324791297, -0.046548564, 0.0998585597, -0.0556193143, -0.0447430015, 0.0557243079, -0.121187761, -0.0431325361, 0.0779469386, 0.0228930581, 0.0202800035, 0.0659439564, 0.0775793418, -0.0461503975, -0.00362607371, -0.01950147, 0.0482348539, -0.00718002534, 0.0396164469, -0.00538680237, 0.0288968012, -0.0650010556, 0.0818163753, -0.0484575331, -0.0266407616, 0.129377127, -0.00811688602, 0.042746067, -0.0013094563, -0.0285873413, 0.000206872821, 0.0562502071, -0.144764781, 0.0402151421, 0.119644538, 0.0391079187, 0.0697217509, 0.0204200484, -0.0743757784, -0.151584938, -0.0535127148, -0.118473932, 0.00919396244, 0.0561908111, 0.0231487975, -0.0392600931, 0.125568688, -0.0326452516, 0.0317110866, 0.0393072478, 0.0323630348, 0.0547082461, -0.078403458, -0.0415681899, -0.0610673018, -0.00704309018, 0.102814399, -0.0250502452, -0.0377188735, -0.0293809194, -0.0874250159, -0.0764820278, 0.0942795202, -0.00932341814, 0.0207654443, 0.0527497716, 0.0023898948, 0.100227103, -0.0881473869, -0.0752742887, -0.024146799, 0.0114771556, -0.0607805662, -0.0811965689, 0.0646127611, 0.0470304862, -0.0186578501, -0.0583441183, -0.014339719, -0.070796147, 0.0362280682, -0.0201590341, -0.112398393, -0.0751717761, 0.0189484451, -0.00200688094, 0.0613171607, 0.0848162398, -0.000150227919, -0.0381221622, 0.0770019591, -0.06227725, -0.0613719746, -0.000652793795, 0.0467086844, 0.0977834091, -0.0114194788, 0.0521992408, 0.0102171414, 0.000946729444, 0.0403355584, 0.0259718113, 0.0267805047, -0.055299297, 0.00198041089, 0.0394504145, 0.0790686682, -0.0540598072, -0.0283055827, -0.0507030264, 0.00996241905, 0.0685543865, 0.0494354889, -0.0635630488, 0.0830745474, -0.0405947864, 0.0234066024, 0.0562989414, 0.110519238, -0.0531953871, 0.212189823, 0.0286800582, -0.032331489, -0.0397319831, -0.0383385569, -0.0514768958, 0.0158981495, 0.0262787007, -0.0396511555, -0.145273358, -0.0895341486, 0.0293900706, 0.00152272498, 0.0301828049, 0.0914210528, 0.0124843568, 0.0206753816, -0.00602560956, -0.0494831018, 0.0677944273, -0.0172597207, 0.0425618924, 0.0792742148, -0.039050594, -0.0174557902, -0.0205573794, -0.0393580347, -0.0211485699, -0.0886224508, -0.00134828826, 0.0773447454, 0.0430288017, -0.00456147641, 0.0368180126, 0.0646788031, -0.0476199202, 0.0174671747, -0.0636112019, -0.0288969185, -0.0225829519, 0.0485399179, 0.00591194443, 0.116158247, -0.00657456741, 0.0595768094, 0.0390549824, -0.0105256485, 0.0730780512, 0.0236759596, 0.0280053206, -0.0820956156, 0.0680081919, -0.0438183621, 0.0410097949, 0.112720445, 0.0168523714, -0.0743870586, 0.0337031595, 0.0962074548, 0.0636099055, 0.0476261228, -0.0367568806, 0.0368436202, 0.0300498009, 0.0421456285, -0.00217331806, -0.127972439, 0.143809721, -0.024754161, 0.034049727, 0.0408620462, -0.0469989665, -0.0703472272, -0.0068266606, 0.0225884914, -0.00917713158, -0.0338857919, 0.00352562917, -0.104598217, -0.00930152833, -0.00950537063, 0.00212710351, -0.0998543203, 0.0684099197, 0.0832060724, 0.0283557586, -0.0746253431, -0.0420238189, 0.0369771197, -0.0640626103, -0.0084672505, 0.0122978734, 0.0447237641, 0.114800915, 0.0556197502, 0.0262267888, -0.000956702977, 0.0156191103, 0.00397255551, -0.0692345351, -0.0339734107, 0.0737388879, 0.0444058217, 0.00664451532, 0.0339780599, -0.0116809411, 0.00553921238, 0.0288744401, 0.0158728324, 0.0758246854, -0.139482543, 0.021029491, -0.00922196545, 0.0330005959, 0.06800735, -0.097424522, 0.00916396081, -0.111921705, -0.0794535726, 0.0220277905, -0.098205559, -0.00732165575, -0.01040617, -0.0619256571, 0.0068370644, -0.0208522324, -0.0311741456, 0.100607485, 0.0333196148, -0.0188607108, -0.0892812908, -0.0663246512, 0.0541642159, 0.0279562753, -0.00575182959, -0.0391349569, 0.0124036651, 0.00331590977, -0.00905902497, 0.0484393574, 0.0184538718, -0.0334754884, -0.105743185, 0.0182477627, -0.00290905451, 0.0273549408, 0.0186522622, 0.0815647468, -0.0573766343, -0.0490213037, 0.0934362113, -0.0702387914, -0.0122584254, -0.152391717, 0.0848972648, -0.0581107512, -0.0854292437, -0.159846291, 0.0377594233, 0.0396380201, -0.016254507, 0.0344747156, 0.00536912307, 0.0253601857, 0.051652126, 0.100804061, -0.0102779176, -0.100455418, 0.0800712928, -0.0492326953, -0.103087597, -0.0147352451, 0.0342755243, 0.0326107219, -0.00316662341, 0.173796818, 0.116489306, -0.0710143521, 0.0404003188, -0.00651132083, -0.0655920804, -0.164468363, -0.0128657799, 0.120914921, -0.00825567544, -0.00865926594, -0.00851593912, -0.0223424938, -0.0115752667, 0.0103667788, 0.0461478345, -0.0199756473, 0.0036690752, 3.55497468e-05, 0.037134286, 0.0516283214, -0.0206424147, -0.0600434802, -0.010141043, -0.0576493442, 0.136944488, -0.105680771, -0.0280563906, 0.0748131797, -0.0856805071, 0.0665436834, 0.0968690813, -0.0191562772, -0.0130782751, 0.0405418538, -0.0347978771, 0.0297841933, -0.00603448786, -0.0430874638, 0.12894392, 0.0160344839, 0.00919822883, -0.0431805477, -0.00821978506, -0.0168002676, 0.0708543807, 0.0416652188, -0.0116853677, -0.0176087171, -0.00768917054, 0.0805195495, -0.0587298945, 0.00707336515, 0.0385528728, 0.0373706669, 0.0135366116, -0.0758024007, -0.108873144, 0.0516984984, 0.0643637776, -0.0451599658, -0.0254372619, -0.00107329618, 0.0579927377, 0.0716033429, -0.0768122301, -0.0629114956, 0.0321965851, -0.0547396615, 0.0390078388, 0.0210687034, -0.0474462658, -0.0226366092, -0.0402391255, 0.0872484893, 0.0502401143, -0.0582539812, -0.0195663758, 0.138116255, -0.0303044226, -0.0330397747, -0.0313093923, -0.0501377583, -0.0790042654, 0.0241870265, -0.0270849038, -0.0648228601, 0.0633109361, 0.01771814, -0.0488246642, 0.0115915686, 0.0108992849, -0.0553428866, -0.0925596654, 0.0755458102, -0.0308532827, 0.013367597, 0.0728941485, 0.0977265537, -0.0291156732, 0.0332275629, -0.0194436498, -0.0348986983, 0.00186088495, 0.0373687558, 0.0456007347, -0.0279398356, -0.0490836315, 0.021963913, 0.0483690128, -0.0278167874, -0.0138684539, -0.00244236179, 0.0089628417, 0.142583564, -0.149847493, 0.030828137, 0.0715482086, 0.0975498706, 0.14701134, 0.0516622439, 0.008002555, 0.000751985237, 0.12546967, 0.00772314519, -0.0371123813, -0.0205380507, 0.0231281184, 0.105787843, 0.0989311039, -0.0378679708, -0.0843519196, -0.0257754382, 0.165929005, 0.0952999592, 0.0245888643, 0.0641800165, -0.0947913826, -0.0203602482, 0.00208738539, 0.0134785697, 0.0635763034, 0.0639363676, -0.030568352];
    CONSTANT bias_0_g : ARRAY[0..63] OF REAL := [-0.0225758869, 0.0595553853, 0.185007155, -0.0504416823, -0.275670499, -0.149840713, 0.0620010719, 0.0258966275, 0.157322526, -0.0664864928, -0.0155564565, 0.0228382032, -0.0366479158, 0.00698181195, 0.0336448178, 0.0918879211, -0.214506492, -0.386997402, -0.205793798, 0.303307623, 0.223864034, 0.187949032, 0.0650451854, 0.261836261, -0.0115475887, -0.345695168, -0.18322891, 0.014604792, -0.0443478301, -0.00914174598, -0.0661112294, -0.316377968, 0.299803227, -0.130490348, 0.00724883843, 0.0396462865, 0.0943433568, -0.196832821, 0.120711617, -0.0831028894, -0.311803371, 0.052451957, 0.0236868374, -0.382010788, -0.181389451, -0.044888895, 0.071627304, 0.354185909, 0.162193984, -0.208105564, 0.19731006, -0.151724979, 0.134141475, -0.141540319, 0.0184668638, 0.0866918266, 0.149765149, -0.182034194, -0.0206596591, -0.327164948, -0.0388776623, -0.338875651, -0.0334542282, 0.0930260718];
    CONSTANT weights_0_o : ARRAY[0..63] OF REAL := [0.7519629, 0.708712757, 0.561989963, 0.744129241, 0.274747133, 0.91726774, 0.711698532, 0.616924286, 0.925325692, 0.741589785, 0.752218366, 0.588025391, 0.790107727, 0.644657731, 0.790763199, 0.697027624, 0.414068162, 0.122064807, 0.568506837, 0.222044766, 0.477075577, 0.569981694, 0.6902439, 0.47118932, 0.688800156, 0.28779614, 0.677336633, 0.71704638, 0.747944415, 0.654153645, 0.746845126, 0.173875913, 0.413205981, 0.757462323, 0.713766336, 0.528290153, 0.616287291, 0.454509318, 0.921783805, 0.857708097, 0.196458578, 0.542137325, 0.71070528, 0.30841586, 0.880288243, 0.750655532, 0.710614026, 0.268657416, 0.882015169, 0.557459533, 0.519826412, 0.955013812, 0.942320228, 0.949047506, 0.691468298, 0.67184782, 0.948599577, 0.510954976, 0.702806115, 0.193465561, 0.738945425, 0.187323287, 0.707145572, 0.81588316];
    CONSTANT recurrent_0_o : ARRAY[0..4095] OF REAL := [0.0489207432, -0.0996182486, -0.104952954, 0.00388177671, 0.021840632, 0.0544938184, 0.0236378573, 0.0598623306, 0.0851075426, -0.0246005319, 0.0860376954, -0.000180922216, 0.0331445001, 0.011467196, -0.0227980614, 0.042894423, -0.0262304321, 0.0191361643, -0.0633681118, 0.0112459511, -0.0892005414, 0.121077031, 0.0339767486, -0.030193042, 0.0434504747, 0.150327444, 0.0579681136, -0.0189039689, 0.026478529, -0.00685659423, 0.0355070867, 0.0199786332, 0.00773932412, -0.0649817809, 0.0828063935, -0.0336835571, -0.0438758358, 0.00632085279, 0.0383913741, 0.00901141949, -0.0399221405, 0.0662798509, 0.0331747755, -0.00287792739, 0.141503349, -0.0263352338, -0.0782542154, -0.046877414, 0.101755798, 0.00568526238, -0.0709223524, 0.0412884764, 0.0350211412, -0.0791817531, -0.0914061144, 0.0534140095, 0.0561926737, 0.0518550947, -0.0177766569, -0.0303250775, -0.0381444991, 0.0670959577, 0.0441615842, 0.0667975992, -0.0334072895, -0.0952907205, 0.0204527453, 0.00243228138, 0.0546310395, -0.00253700931, 0.0200143605, -0.0463880375, -0.134058684, 0.0243678316, 0.0259992667, -0.117743298, 0.00188423041, -0.0291984603, 0.00225576386, -0.000799461268, 0.087586388, -0.053850662, 0.0840993449, 0.128663719, 0.0394558161, -0.0375596918, -0.047042951, -0.0289745852, 0.0154407574, 0.00378552475, 0.12023589, -0.0332220122, -0.0186153837, 0.0792418867, 0.0811079368, -0.0112350788, 0.107358396, -0.0099527007, 0.0334596932, 0.0842557326, 0.0644082278, -0.0883702934, 0.107007898, 0.00425976515, -0.0622161441, -0.0996078253, 0.0798855498, 0.109726965, 0.0548738316, 0.00314371358, 0.0353557095, 0.100286506, 0.0659422353, 0.0348635465, 0.0483465269, -0.0262031034, -0.012874647, 0.026808152, -0.0494508594, 0.00823145732, 0.0794796795, 0.0306071863, -0.0931525007, 0.0051366603, -0.0548378602, 0.0426580422, -0.00976184942, -0.0510310344, -0.0525079295, 0.0100662336, 0.0215323046, -0.0578476116, -0.0182377081, 0.0384202562, 0.0508384742, -0.0525421016, -0.0344453603, -0.0508078709, -0.0209409464, -0.0700552091, -0.024914261, -0.010203436, -0.0634157285, -0.0102344155, 0.0333143324, 0.0302098133, -0.0648940951, -0.0381746143, -0.0407165661, 0.0300954543, 0.0125519764, 0.0033537196, -0.0749643296, 0.145514891, 0.0966463163, 0.0585655421, 0.0153121194, -0.0122141093, 0.00737738609, -0.0677625909, 0.0187220629, 0.0186869912, -0.0329783559, 0.0093861036, -0.0496005341, -0.105336338, 0.0635403767, 0.0047832597, -0.0296360962, 0.0113514373, 0.000254392624, 0.129150346, 0.0441638716, 0.00908795185, 0.0554776639, -0.128619611, -0.0407441631, -0.000351348892, -0.094847396, -0.0346427225, 0.0258873664, -0.107073918, -0.00240627257, 0.0207787864, -0.0526111759, -0.0598161221, 0.00602654368, 0.0610072687, -0.0157896914, -0.0216664188, 0.0268461481, -0.00204994809, -0.110921569, 0.0971338227, -0.0146537162, 0.0778791755, -0.0412621908, 0.00361991394, -0.110252127, -0.0033848756, 0.0867285058, 0.0141183594, -0.0978397354, 0.0522605851, -0.0525847338, 0.0836603642, 0.0202452261, -0.0469065756, -0.102603473, -0.0771438777, 0.0289257839, 0.0463489406, -0.0505081043, 0.0348018669, 0.0617071688, -0.159421399, -0.0302333608, -0.0385930389, 0.0640206635, 0.00792024471, 0.038648732, 0.0785473138, -0.0572423488, 0.00947043858, 0.0591879003, -0.00161777809, 0.0749231651, -0.0633680522, 0.0451328829, -0.038916681, -0.145598412, 0.112259418, 0.053966105, 0.0418384373, 0.00967805646, 0.0496267676, -0.0296346992, -0.133916289, -0.0691784173, -0.0439499803, 0.0579275116, -0.0996822789, 0.0281891078, 0.073532261, 0.0688669756, -0.0406364016, 0.0768532455, 0.0179092437, 0.0529112741, 0.0144107379, -0.114816226, -0.0623274557, -0.0479176603, -0.0144851506, -0.058670491, -0.0442495793, 0.054937724, 0.0156568736, -0.0352829769, -0.100619279, 0.134879008, 0.0855379254, 0.029024601, -0.0141360732, 0.100755319, -0.0447310768, 0.0507849678, -0.0375701562, -0.00166633911, -0.0834201872, 0.114714235, -0.0145840663, -0.0207685344, -0.0139047205, -0.0192832462, -0.0400657952, -0.0534725152, 0.0237659141, -0.0178591851, 0.116257131, -0.0880570039, 0.00214307383, -0.0132516474, -0.00516001042, -0.0118059777, -0.0453950129, 0.0624831207, -0.0362048671, 0.00762055162, -0.117592126, -0.0827926472, -0.0113356728, 0.0179843996, 0.0416827723, -0.0066757109, -0.0111289378, -0.0797280595, -0.0314054377, 0.139076173, -0.0836744234, -0.0491223931, 0.128351122, 0.00208370923, -0.0129573504, -0.0885379538, -0.146524936, -0.0277015008, -0.00209120288, -0.00652960781, 0.00505205011, -0.0133063626, 0.0364567749, 0.0575172156, 0.0264859516, -0.0899147838, -0.032427758, -0.0541715473, -0.0374686345, -0.0586880073, 0.137751982, -0.112302154, 0.022068521, 0.0780058652, -0.0158320758, -0.017865397, 0.0873443037, -0.00508407364, -0.0493847728, -0.0659772158, -0.026107721, 0.0310844183, 0.0581566952, 0.00584043702, 0.0190598071, -0.0467157587, 0.0410924256, 0.0961778611, -0.0697619542, -0.0667384341, 0.128524363, 0.0502807833, 0.0252052005, 0.0165828019, -0.0808899924, -0.0300327409, 0.116285764, -0.09241651, 0.133292034, -0.0573155321, 0.0841670111, 0.0525554046, -0.109709807, 0.116765074, 0.0644502416, 0.0134185292, 0.0644217208, -0.0203446243, 0.147896603, -0.0543538108, 0.0391157269, -0.0126085617, 0.0338744633, 0.0281186886, -0.0381015316, -0.0106114317, 0.0680520311, -0.0848235935, 0.0242021158, 0.00979540497, 0.0464764647, 0.0881815404, -0.0430723205, -0.0319354534, -0.0228650868, -0.0948898718, -0.00922867563, 0.116969928, 0.0277317725, 0.00446022768, -0.0212527383, -0.0177736469, 0.00632203743, -0.00843990687, 0.0479193889, -0.0688794032, 0.0344369486, 0.00186440814, -0.0496517792, 0.0500193574, -0.0043256795, -0.117115222, -0.00074189232, 0.0432040617, 0.0184376184, -0.150119394, 0.0195795111, -0.00528148469, 0.0230835229, 0.00746740494, 0.066319935, 0.0064150379, 0.0911360234, 0.0473778695, -0.0833897442, 0.0687825978, -0.00921613071, -0.0491583534, 0.0229335409, -0.0298461467, 0.00212302152, 0.0247548632, -0.0182353668, -0.104718596, -0.146888539, -0.0704599842, -0.0783024803, -0.0885671824, 0.0341995284, -0.0400329754, -0.00656351354, -0.0633721873, -0.0515429005, 0.0711144805, -0.068589516, -0.0160931628, 0.104965404, -0.0117810238, -0.0409668796, -0.00488566514, -0.0227422006, 0.0419279523, -0.0520865694, -0.0656612217, -0.0426112413, -0.00441919547, 0.0476857796, 0.0140198432, -0.00667859148, 0.0763169527, 0.0818673745, -0.0470707454, -0.097009331, 0.0552561507, -0.0280755553, 0.0423200577, -0.022111509, 0.0968581736, 0.11471574, 0.0640713051, 0.0451810248, -0.0385862552, 0.0270083584, -0.0543174148, -0.0208577029, -0.020620726, -0.0398950838, 0.0152758397, -0.090677999, 0.0320581496, -0.0673296601, -0.000710567459, -0.0154965222, -0.0431158468, 0.0209875815, 0.0784731209, -0.0476803146, -0.0100085372, -0.0812713057, 0.0453999788, -0.0521486737, -0.0189935155, -0.0294351634, -0.00196124427, -0.012928036, 0.0546167158, 0.0553783886, -0.0129677178, 0.017909212, 0.0794564486, -0.01138537, -0.0246365443, 0.0876680911, 0.000540263951, -0.0138177788, 0.122772291, -0.020761691, -0.0816517398, 0.0175698511, -0.0253941584, 0.0789160579, -0.105710104, -0.0394714028, 0.0524880812, 0.0339578167, -0.120478876, 0.0550823137, -0.0714456439, -0.0677922517, -0.0546886772, -0.0500687584, 0.0311231911, 0.0508797243, -0.0460948981, 0.0502713509, -0.0489882156, 0.0300840586, 0.03536826, 0.00476030586, 0.0053704232, -0.017719958, -0.105078049, -0.0424538292, 0.046875257, 0.0187156145, 0.0639873818, -0.0473330729, 0.0368481241, -0.0581644364, -0.0711598843, -0.00126787089, -0.0701822042, 0.0290794671, -0.013930453, 0.0194939096, -0.0527851507, 0.0821156427, -0.0325515568, -0.0769806877, 0.0531322844, 0.0016006846, 0.0810368359, -0.0310466532, -0.023639258, -0.0366886593, 0.0241841152, 0.0298246816, 0.0233992971, -0.0594913624, -0.0847461522, -0.061545074, -0.0621985607, 0.116194651, -0.0260647479, 0.0540968031, -0.0511154495, 0.0550713539, -0.0892230272, -0.0528794602, 0.00364543125, -0.0186723545, -0.0356975906, -0.0369166881, 0.0136959553, 0.0315532647, -0.0064436812, 0.0674879104, -0.055009678, -0.0343020298, 0.0636775345, -0.000251784455, -0.0207594782, 0.0749258697, 0.00340543012, 0.0666735917, -0.100481763, -0.152589396, -0.069031626, 0.0819491893, 0.0939499587, 0.0557769313, 0.0161313359, -0.108943455, 0.0908565223, -0.0671487898, 0.0621765628, 0.0654389337, 0.0872035325, 0.0182403885, -0.0150894392, -0.0879181623, -0.00392939709, 0.0551660284, 0.0450397991, -0.054049965, 0.0760113522, 0.050063841, -0.0363876261, -0.00715898164, -0.0444022194, 0.0836029872, -0.0952367187, 0.00753673213, -0.158136144, -0.0912612453, 0.00735832006, -0.0216287766, 0.0325958692, 0.0132113742, -0.0142756552, 0.0120593831, 0.0562750027, 0.0234061852, -0.0839226991, 0.0700246543, 0.0402348526, 0.110188901, 0.085305959, 0.00799281895, -0.0743744522, 0.0908793509, -0.00794482604, -0.0544873402, -0.0905054659, 0.0456978381, -0.0538770892, -0.0151171926, 0.037486922, -0.0569863729, 0.0680634975, 0.13338469, -0.00119119138, -0.0225900747, 0.0600275733, -0.0138948644, 0.0124960383, 0.021723263, 0.0248966422, 0.0271963626, 0.0119008077, -0.0603619888, 0.0416958928, 0.0278034266, 0.0686454624, 0.0536708087, 0.0818630755, -0.0275984481, -0.0433301628, -0.0637640059, -0.00770678464, -0.00815215986, -0.0346980654, 0.030484736, 0.0257449858, 0.0445872545, 0.0296262037, -0.0346277989, 0.0564447083, -0.0311599001, 0.0469898507, -0.0604605637, 0.06379655, 0.0875809789, -0.0610883273, 0.126367703, 0.0589446649, 0.164977521, -0.122112222, -0.067499131, -0.00448070653, -0.0220134929, 0.0842579156, 0.0240859464, -0.0724281296, 0.0321303047, 0.0400830582, 0.070545271, -0.0862180963, 0.0694640204, -0.037666671, -0.0310527571, 0.0380247086, 0.0247088317, 0.0110623837, -0.0539379604, -0.0361893699, -0.00644869916, 0.0814822614, 0.0202466715, -0.020760756, -0.0120847132, -0.115228362, 0.0451136641, 0.0246617123, -0.0152040953, -0.128099978, -0.0654590428, -0.0394524336, 0.0680671409, -0.0805750638, -0.0446120501, 0.0163637046, -0.0618752725, -0.0222185738, -0.102858141, 0.0209314339, -0.0308102742, 0.032563448, -0.0130797923, -0.0644943789, -0.0484713987, -0.0274234302, 0.0600465089, -0.0579487942, -0.0579860061, 0.0319475383, -0.0305550955, 0.0833145678, -0.0316383801, 0.0411320664, 0.0158117954, -0.0620448217, 0.0754485503, 0.036890246, -0.081994012, -0.0268892907, 0.0210090503, 0.0746083111, -0.105157807, -0.0317369811, -0.0927379131, 0.010111697, -0.0158461016, 0.00684279064, -0.00164840091, -0.059134692, 0.0141944662, 0.0717771277, -0.0831093267, -0.0153469667, -0.0618811473, -0.0154191293, 0.0634172782, -0.0280117113, -0.00517418701, 0.0872334614, 0.0210242514, 0.0486453138, -0.0260084812, 0.018292807, 0.0112259686, -0.0690205991, 0.0132348277, 0.0228861701, 0.0113966595, -0.0583233088, 0.0468286537, 0.00132655725, -0.0314484723, 0.0385567807, -0.014038017, 0.00117720105, -0.00338249188, 0.016154319, -0.0676974058, 0.0803395808, 0.0321162865, -0.0845740139, 0.00873133633, 0.151597798, 0.0835854113, -0.0115977675, -0.00496777333, -0.00635943841, -0.0132669751, 0.0799859613, 0.0594360456, -0.0173449777, 0.0663833246, -0.0652325973, -0.0173939019, 0.0760888457, -0.00244770013, -0.0287574176, 0.0504974164, -0.0142380521, 0.0239177831, 0.0793199912, -0.00932121743, 0.0204264596, 0.100783631, -0.0805539414, -0.0484617539, -0.0231467169, -0.034118548, -0.0387519002, -0.0325032696, -0.0276750978, 0.0349069238, -0.0406788737, -0.0257365257, 0.11205709, -0.0466008522, -0.0318287387, 0.0113046058, 0.00733099878, 0.0814749748, 0.0224900357, 0.0373800956, -0.0217409208, -0.053523846, -0.0157984216, -0.147161633, -0.0260422714, 0.0787447244, -0.0475726761, -0.141773179, 0.0638272315, -0.130933046, -0.128154144, -0.0617523119, -0.0220184028, 0.0180003513, 0.0693545341, -0.03799529, 0.0413703248, 0.0531932414, 0.0380416363, 0.0915600955, 0.0570532754, -0.129434153, -0.056219697, -0.00800924748, 0.0478676371, -0.135996714, 0.00758393109, 0.00669563562, -0.0482816882, 0.0444399714, 0.0518862009, -0.000936537515, 0.00148539664, 0.00924326107, 0.075868845, -0.0573241934, -0.0326449201, -0.0305022746, -0.0152279697, -0.0661599785, 0.024448961, 0.0236885697, -0.0373446271, 0.00430306373, -0.0362367518, -0.0120894061, 0.0536467694, -0.00174810458, 0.0326837786, -0.0456118695, -0.026486624, -0.0719535649, 0.0245877411, 0.0183842015, 0.10165301, -0.0959579051, -0.0268683862, 0.00978240557, -0.0318669155, -0.0297890045, 0.018161118, 0.0121509014, -0.135054916, 0.0129512567, -0.0507491343, -0.0697966367, 0.103113525, -0.114300884, 0.0368019193, 0.026678212, 0.0380492061, 0.051856529, -0.0739401728, -0.0221610274, 0.00341419969, -0.0128066493, 0.027107764, 0.0186144058, 0.0217119176, -0.0765653253, 0.00514073297, 0.0647628158, 0.140952751, 0.0485100001, -0.0256131161, -0.117874078, -0.0608194247, -0.0790309161, 0.0506668091, -0.142421484, -0.0417591855, 0.0616610795, 0.00648172712, -0.0529969446, -0.00569268316, 0.0996995494, 0.0424410999, 0.126730099, -0.013253781, 0.0209860783, 0.117405422, 0.0410836749, -0.0331164263, 0.00302413944, 0.0737161934, 0.0350383744, -0.018053975, -0.087764442, -0.0159006305, 0.0909630358, -0.0370275192, 0.0584055781, 0.0243670754, -0.00560101867, -0.0474086218, -0.032188423, -0.0182326455, 0.0759636611, 0.0752968639, -0.0208698846, -0.0648351014, 0.0565419905, -0.0229970776, -0.0849007294, 0.0768636018, -0.0950835496, 0.0130023453, 0.0434273183, 0.0691810623, -0.0947320536, -0.0106760766, -0.0217655431, -0.0412964411, 0.0728489012, -0.0807142779, 0.0319461375, 0.0706743374, -0.0134156775, 0.0289668515, -0.076116018, 0.072122857, 0.0695477724, 0.0856732503, -0.0673222542, 0.114025913, 0.0213296637, -0.0133889616, 0.0425762199, 0.0246015061, 0.063953802, -0.0388719328, 0.0177426096, 0.0200623311, 0.0302252937, -0.0130109787, -0.025115665, -0.0832961947, 0.0544550195, 0.000935546122, -0.0936248302, 0.0173202902, 0.0153739639, -0.00111944508, 0.113897122, -0.100584231, 0.05236727, -0.0883226246, -0.0608032569, 0.0253955014, -0.0409346782, -0.0135400984, -0.0058462508, -0.0632548407, -0.000178921502, 0.0284727365, 0.00815154519, 0.00303628552, 0.00793007482, -0.0235454962, 0.0536862761, 0.0405858606, 0.0384193659, 0.046679318, -0.0106061809, 0.0399687737, -0.0257779229, -0.00785798579, 0.0185846966, 0.0762275457, -0.0257641058, 0.0433734506, -0.0457892381, 0.029625617, -0.0500297099, 0.0468119532, 0.00343723875, 0.0298494063, 0.0767991394, -0.0400525853, -0.0279743373, -0.0406299159, 0.0024908022, 0.0176862106, -0.0221953616, -0.0736412182, -0.0702325627, -0.101827465, -0.138535321, 0.0814120471, -0.0379535593, -0.035327252, 0.0273327455, -0.0256212205, -0.0922422037, 0.040183235, -0.0339703076, -0.0525668934, 0.0450968407, -0.0796107724, 0.0786161795, -0.0771979168, -0.0304565337, -0.0359584615, -0.00357550196, 0.0627327934, 0.0414175913, -0.01446083, -0.00106278807, 0.0145163611, 0.0389034636, 0.0741425306, 0.0560302585, -0.119377248, 0.0322585031, -0.0320047662, 0.019394042, 0.0857254639, -0.0924353749, -0.0109822042, 0.0433163121, -0.0774459392, 0.139330715, 0.0707374066, 0.0438952893, -0.0404270068, 0.0275607929, -0.0762103721, -0.0782006606, 0.114917167, -0.0340028182, -0.0129296863, -0.0617869161, 0.0172483958, 0.0551176704, -0.0158024374, -0.045908194, -0.0283399541, 0.00907150563, -0.0398350433, 0.115211241, 0.0512478873, 0.0419996977, 0.0328524634, 0.141346633, -0.0663913786, 0.0483483896, 0.10283906, -0.0951984897, -0.0351549797, 0.0163322166, -0.0874588266, 0.0969983563, 0.091551587, -0.0181501303, -0.0209838636, 0.128547817, -0.0783229098, -0.00559064932, -0.0947994366, 0.027296152, 0.00885994732, 0.0686174333, 0.0711648166, -0.0525312051, 0.00501684844, 0.0141710686, 0.00456897542, 0.075033091, -0.0800696909, -0.0323179029, 0.0296551511, -0.0436992049, 0.0391427204, 0.064627789, -0.0976679474, 0.0234005842, -0.0229313113, -0.00343156792, 0.0266880933, 0.00942680519, 0.00766727421, -0.00205071177, 0.014766315, -0.0161233135, -0.00476189004, 0.0345248133, -0.0960306823, 0.0651817992, 0.00452155713, -0.0180524085, -0.060987588, 0.0872602612, 0.0414179713, -0.0630545467, 0.0432770476, -0.0243404638, 0.0958171636, -0.0803921297, 0.0595680885, 0.0980401635, 0.00928722229, 0.0603970364, 0.0681929588, -0.0673865825, -0.0553686433, 0.0960672572, -0.0915255398, 0.0555837192, 0.0637090653, 0.0196703728, -0.0470352322, 0.066775471, -0.0179889165, 0.0113385301, 0.0130350608, 0.0128617063, -0.00894834474, 0.070101276, -0.0301503241, 0.00264464878, -0.058697544, -0.0986367464, -0.0238779038, 0.0334106013, 0.0760604367, 0.0159991384, 0.0872678161, -0.0150096379, -0.0280542951, -0.0323568657, -0.0350878648, -0.0385220647, -0.0243062228, 0.0350914076, -0.0392305218, -0.0754082575, 0.0344575234, 0.0724492148, 0.0894953832, -0.0726514235, 0.00558044901, -0.0508277416, 0.0329446346, 0.0396493822, -0.0849051923, 0.0335638523, 0.0249660015, 0.113666147, 0.038970165, 0.0250126459, 0.085332498, 0.0406925716, 0.02617497, 0.0285719987, 0.0303135496, 0.0126770847, 0.117714718, -0.109309614, 0.0360136852, -0.0615008548, -0.0216108635, -0.0449773259, -0.00208033249, -0.0187073015, -0.0242121927, 0.0675222948, -0.108681813, 0.047112681, -0.00553419068, -0.0535204336, -0.112703897, 0.013363421, 0.0513217673, -0.0439626984, 0.0142940907, 0.0232440736, -0.0690158233, -0.00557856727, -0.103870481, 0.035943646, 0.0265898239, -0.0906002074, 0.0705483034, -0.0709042847, 0.0337374806, -0.0447738431, -0.0962034762, 0.00710726157, -0.0309997629, -0.0488276258, 0.0350311622, 0.0439302102, 0.0111076906, -0.115815088, -0.0536187589, 0.0190750714, -0.0486599356, 0.106979027, -0.0380212516, -0.0335139148, -0.0768163651, 0.093032442, -0.117673367, -0.0476720259, 0.0661338717, 0.0441746116, -0.105016351, -0.154389054, -0.0481063165, 0.100755915, 0.0328793526, -0.109111562, -0.00951075833, 0.0346248597, 0.0915664658, -0.00690461416, -0.0579210706, -0.00736375246, 0.0243018102, -0.00797929242, -0.0270060711, 0.0498547256, 0.0430264473, -0.0813161805, -0.0394414552, -0.0436755978, -0.0480009019, 0.0101616196, -0.0567662567, 0.0228532907, 0.051887501, -0.0712503791, -0.0593095906, 0.0696244463, 0.0488236435, -0.0410599299, 0.0201899707, 0.0801115036, 0.00248872861, 0.0449310839, -0.0243616384, -0.0307227913, -0.0449212454, -0.00600031205, -0.0188684091, -0.023989683, 0.0105438568, 0.023723213, 0.0404933691, 0.0892639309, 0.0417711921, -0.0647321641, -0.0407553576, 0.0349460095, 0.144405276, -0.052420292, -0.0658970028, -0.111308843, -0.00734805688, 0.0438100062, 0.0354890041, -0.0790705532, 0.105788887, 0.144318178, 0.136512011, 0.0256172102, 0.0668599755, -0.0192053989, -0.02297079, 0.0160418674, -0.0569440313, 0.0897481069, 0.072089076, 0.0582722239, -0.0916632637, -0.0965394452, 0.0664415583, 0.00358017976, -0.0678060055, -0.00103117712, 0.0414431505, 0.0375579111, 0.128294021, 0.0416217707, 0.00301510235, 0.0684802234, 0.0540548675, 0.0545829274, -0.0368041545, -0.036121428, -0.00545704737, 0.0242428966, -0.0121388221, -0.05997812, 0.0442032441, 0.0111766756, -0.0412380248, -0.0500744507, -0.0697601363, 0.113554522, 0.0684996247, 0.0131196529, -0.120839655, 0.0428753681, 0.0123680085, 0.0641750917, 0.0748378336, -0.00879754312, -0.166479528, -0.130509436, 0.108633928, -0.00336496392, -0.0528886616, 0.0313835628, -0.0270992294, -0.0663156062, -0.0169528853, 0.0797479004, -0.0669530034, 0.00805508532, -0.040048521, -0.0020545423, -0.0625480413, 0.137955651, -0.0305294655, -0.0010163039, 0.0160851385, 0.00692472281, -0.0721204653, -0.200991914, -0.0526736751, -0.09982308, -0.0432392061, 0.00981911831, 0.0276473965, 0.0374192558, 0.0872737989, 0.0833740607, -0.0342625305, 0.170609295, 0.00635366468, -0.028008204, -0.0818210468, -0.00278044306, -0.00906104129, -0.060424149, 0.0740749389, -0.0130091598, 0.0536574312, -0.14790453, 0.0182392262, 0.112219386, -0.0389456525, 0.0479793027, 0.0490317307, -0.0467449166, 0.0584384874, -0.0414829589, 0.0531908721, 0.0218016692, -0.0489403754, 0.104162365, -0.00850681216, -0.0448522419, 0.0993189812, -0.00669082254, -0.125117525, 0.0287737306, -0.0543053187, -0.12294507, -0.0479411967, 0.0314116925, 0.0466014519, 0.0237070732, 0.0727744177, 0.0319961831, 0.013148427, -0.0154100163, -0.00147012621, -0.0314357765, 0.0496883467, 0.00143335387, -0.0299351625, -0.0187889766, -0.0344188958, 0.117686182, 0.064450413, -0.0749027431, 0.0367034003, 0.0483763553, 0.0487295538, 0.016247768, 0.047797136, 0.0326349102, 0.0242631249, 0.081236206, -0.034705393, -0.108959198, -0.0364753529, -0.0196703877, 0.0154500315, 0.066694811, 0.180976674, -0.0334356241, -0.0716987848, 0.0444132984, -0.0812027156, 0.0514127091, -0.0226110592, 0.0129635707, -0.114580669, -0.0920626521, -0.00405873172, 0.157762513, 0.0837559178, 0.008011356, -0.0768600702, 0.0618026853, -0.0241873562, 0.000971716829, -0.0575393476, -0.0212962925, 0.0996681601, 0.0722231716, 0.0396050848, -0.0386350937, 0.00968257058, -0.0101240501, 0.069004342, -0.0312676467, -0.0176417269, 0.0976688713, 0.0668433905, -0.00169128552, 0.0253218077, 0.113676004, 0.0209028609, 0.0784313157, -0.0778982192, 0.0544664934, 0.107612371, 0.00546895061, 0.028367212, -0.00280095264, -0.0146827623, -0.0581016988, -0.0385343917, -0.00925797876, 0.0567749478, -0.165961593, 0.120664716, -0.018851921, -0.0126736127, 0.0266426578, 0.0530390441, -0.141782403, 0.0322804004, 0.0629792884, -0.0442320742, -0.105256341, 0.0244656093, -0.0272188671, -0.0615175664, -0.0228276737, 0.118850753, -0.0460100621, -0.0201987512, -0.0146559067, -0.0225452222, -0.0194424316, 0.0164002292, 0.0749964043, -0.000333596021, 0.0209661163, -0.0603591502, -0.043878451, -0.0967830122, -0.0524108857, 0.152114764, -0.0824826881, 0.0309071504, -0.00603337772, -0.0418354273, -0.0832386464, 0.0171953663, 0.0335386284, 0.0798386484, -0.00994795747, -0.0189932436, 0.0152305467, -0.109571204, -0.00524315052, 0.0166361332, 0.0587245673, 0.117997125, -0.0128748603, -0.0502700731, 0.066460669, -0.0815355778, 0.0178302601, -0.123600617, -0.0636502057, 0.00701700896, 0.0128129022, -0.0633087978, -0.00695089623, 0.0019126659, 0.0515845865, 0.0205534119, -0.0487041511, 0.0405475944, 0.0876201838, 0.0838473216, 0.0168466177, 0.0434087142, -0.0166050456, -0.0191648006, 0.141568795, -0.150803402, -0.031563703, 0.0832959637, -0.0474180132, -0.0383364111, -0.0073572183, -0.0161246322, 0.149443477, -0.0989671499, -0.0233748462, 0.0317183658, 0.112239048, 0.179274201, 0.0203227252, 0.132903934, -0.0222158954, -0.0259621963, 0.0982027352, -0.0336368978, 0.0602178499, 0.0706666261, 0.105114922, 0.0289735589, -0.016035337, 0.00802578405, 0.0625568256, 0.0782575086, 0.188058838, 0.0144755915, -0.0692011267, 0.0176524222, -0.0484759957, -0.113558479, 0.0492948964, -0.0366999432, -0.0394458696, 0.0801637247, -0.00624522381, -0.0613866672, -0.0611268431, -0.0999632776, -0.00822096318, 0.00206070766, -0.0771138519, 0.0113010388, -0.0213001631, 0.0334789492, 0.0766096637, -0.0206592586, 0.0295011215, -0.0730838254, 0.0312298536, 0.0585869625, 0.0809112787, -0.0228695795, -0.0480644628, 0.053102605, -0.0268568806, -0.0091864299, 0.0854697376, 0.0751238316, -0.0384300761, -0.0706340596, 0.0591493398, 0.0800262615, 0.0151398182, 0.0725961998, -0.00620491616, -0.0267420374, 0.0277093314, 0.0799219012, 0.0814106315, 0.0381436571, -0.007295602, -0.0430039875, 0.0110437283, 0.0220797546, -0.021849582, -0.0399202146, 0.00327817909, -0.0146754691, -0.0690897033, 0.0567473061, 0.0405254848, 0.101513088, -0.0570031404, -0.0228256732, 0.0739719719, 0.12461336, 0.092683889, 0.0204576049, -0.0347290933, 0.0544375442, -0.0401212722, 0.0468926802, 0.0310485847, 0.0675424039, -0.0330932029, -0.00638925843, -0.00159768201, -0.0506717451, 0.0626053214, -0.0158194546, 0.0894839019, 0.0225493945, 0.0684331805, 0.0415887535, 0.105692424, 0.0383309647, -0.0720047951, 0.075071454, 0.0810718015, 0.0160716884, -0.0374981537, 0.0578320995, -0.0396482572, 0.0149666686, 0.0236607399, 0.138371214, -0.0359981656, -0.100909695, -0.0922122225, -0.0261964016, -0.12982592, 0.13219057, -0.0253417045, -0.0930862948, -0.0353386849, 0.0966111869, 0.0415017232, 0.0219236221, 0.0318210572, -0.00643536169, -0.043713592, -0.0296496637, -0.0714464337, -0.0794356093, -0.00768351089, 0.0502969921, 0.0367745906, 0.0189926978, 0.118370935, -0.0141379582, -0.00927751977, -0.029813299, 0.0526867434, -0.0165897515, -0.00956278853, -0.0342390463, -0.0130996983, 0.0729671046, -0.0431652814, 0.0472786203, 0.0262430962, 0.00580816902, -0.00184729882, -0.0328836739, -0.0326149426, -0.104502305, -0.000888961367, 0.0360196866, 0.0598701984, -0.0210313722, -0.0210123137, 0.00655640289, -0.00311486796, 0.0225449502, 0.0532348379, 0.0259421915, -0.0950381458, 0.0196599569, -0.0539802201, 0.0153882168, 0.0813516304, 0.0167507008, 0.073296167, -0.00551114697, 0.0813157409, 0.0671304613, -0.0562030226, 0.0118149733, -0.0890379697, 0.0721032917, -0.130086064, -0.186802149, -0.114462078, 0.00110373471, 0.000850011595, 0.166916355, 0.128142476, 0.0608409606, 0.0480179973, 0.0162943192, -0.112821512, 0.184779227, 0.0242991392, 0.0615214147, -0.0131022912, 0.0429481231, -0.0269970279, -0.0432117134, -0.048785504, 0.0433057845, 0.0295303948, -0.0111923218, -0.0404965803, -0.000669879839, -0.000912575983, -0.0588420406, 0.0269155279, -0.0799991563, 0.0291563906, 0.0973874629, -0.0216904432, -0.044387836, 0.126204967, 0.0621459037, -0.0056558419, 0.0412794948, -0.011912642, -0.0280526802, -0.0476566553, -0.0281894356, -0.0339744613, 0.0921439454, 0.00194188766, 0.0329542086, -0.0657317936, -0.102583244, -0.0177890323, 0.0525078475, -0.105440818, 0.0411671363, 0.119331479, 0.0105616301, -0.0188129358, -0.0240105372, -0.0544621758, 0.0422329456, -0.0967406258, 0.000552302226, -0.00502418354, -0.141634494, 0.0234485418, 0.0289576706, 0.0510377474, 0.0553935803, -0.0295651779, 0.0891121924, 0.022242697, -0.02962666, 0.0363544822, 0.0857499689, 0.082044065, -0.0519868918, 0.0249197837, -0.00205135834, -0.0865466297, 0.000350799412, -0.0184425153, 0.0670586824, -0.120342113, -0.0331440009, -0.0585890561, -0.00491240807, 0.0323148184, -0.012731798, 0.011709705, 0.0462337658, -0.00309255999, -0.0289770197, -0.00412789173, -0.0012231674, 0.00871458463, -0.0913771167, -0.0455166735, -0.028447751, -0.0203141458, -0.0444666818, 0.0489444397, 0.0867197439, 0.0982919857, 0.0443457291, 0.0843705535, 0.0100161824, 0.0484755039, 0.0264325961, 0.0556238145, 0.0782444552, 0.00826611556, -0.0815408751, -0.036863938, -0.0865916014, -0.11316032, -0.0116961729, 0.0299393348, 0.109950021, 0.0749869943, -0.0839978829, 0.0304061733, 0.0269843414, 0.0576304123, -0.0946580097, 0.026472168, 0.0122161172, 0.0286391731, -0.0212597363, -0.0961300954, -0.0800899714, -0.00713242311, -0.00140731409, 0.042431172, -0.108701371, -0.0192928333, -0.0283041913, 0.0511169806, -0.0140472827, 0.0130148241, -0.10639599, -0.1017038, 0.0796498954, 0.0251909904, -0.027459776, -0.00359712541, 0.0058404142, -0.00739690103, -0.0941277444, 0.00167841977, 0.037710648, 0.00931508467, -0.104109757, 0.0260281675, -0.0357531235, -0.0880550593, -0.0230396241, -0.0106818993, 0.0699100643, 0.0379487574, -0.111484647, -0.131087661, -0.0427435786, -0.037547864, -0.0549940728, -0.0935803652, 0.028666053, 0.0499371141, 0.0407195687, -0.00210960768, -0.0809178054, 0.000182838179, 0.0690048337, 0.032112997, -0.0756960884, -0.0438861772, -0.0421447903, 0.00260864035, -0.00814455003, -0.0648220703, 0.0338696986, -0.0405191779, -0.00729243364, -0.0279864408, 0.065960288, -0.00768788066, 0.0604736917, 0.0222599022, -0.0299177319, 0.0140532972, -0.10241323, 0.0647619516, -0.00380254537, -0.0916775391, -0.0223087743, -0.0252346061, -0.0969133973, -0.014513541, 0.0285261199, -0.00501779094, -0.000239043497, 0.020745201, 0.0363049582, -0.00750590302, -0.0941943377, 0.0805186033, 0.143347591, -0.0257309712, 0.0807706788, 0.0634687394, -0.151733994, 0.102499381, -0.107922532, 0.100087576, 0.0438607559, 0.0071092993, -0.0607305095, -0.0603791699, -0.0256896503, 0.0590706505, 0.0883758441, 0.0644083992, 0.0636949092, -0.00614757743, -0.108773403, 0.00294307061, 0.114896014, 0.0095947478, -0.0645734668, -0.071901761, 0.0504343808, 0.0358902141, 0.10865213, 0.0691803023, -0.0228052754, -0.040295057, -0.0483355522, -0.0328826681, -0.0142255109, -0.0669835806, -0.0960129648, -0.0829334036, 0.101534449, -0.201541901, 0.0250377413, 0.0183187202, -0.0452129021, -0.051333338, 0.0304997079, -0.0797326788, 0.00135975517, -0.0131384153, 0.0998899564, -0.0367455408, 0.00272747129, 0.00358362682, -0.029034378, -0.0493533984, 0.0212970916, -0.0195701811, -0.0140849873, 0.14900656, -0.041751191, 0.0477996394, 0.0153446719, -0.00231361017, -0.0418426953, 0.00141642964, 0.0181682277, -0.0624107271, 0.0338134691, -0.0571032763, 0.165114596, 0.0506624132, -0.0630114079, -0.0850313678, -0.0104804523, -0.0868232325, 0.0837274119, -0.0446486175, -0.0569588505, -0.0632043034, 0.00194896781, 0.0103039453, -0.0416809358, -0.0135880876, 0.0251447391, -0.0524212047, -0.0324766077, 0.0691483915, -0.0277678668, 0.0400982425, 0.136338085, 0.0119939838, 0.0332214423, -0.03274142, -0.0113746105, 0.00536523014, 0.0618670695, 0.0695354044, -0.019611543, -0.0395252556, 0.0689252391, 0.0380045474, 0.0109895635, -0.0262189992, -0.135897398, 0.0316147506, -0.111785449, -0.0371512324, 0.0407916009, -0.0671351478, 0.128250986, -0.0957079977, -0.193647698, 0.0105984602, 0.0845922902, -0.0335145369, 0.104173467, -0.0292843711, -0.0413455963, -0.0817551315, -0.00991834607, -0.0288008116, -0.0915459618, -0.000306397676, 0.0230409019, -0.0609088913, 0.0955903456, 0.000647189096, -0.0249774922, -0.114429437, 0.0608190112, -0.115648434, -0.0678047687, -0.0120425727, -0.0428964682, -0.00868016388, 0.0246779658, 0.0459028631, -0.000142196193, -0.0467417836, 0.103471473, -0.0328707695, 0.0220221151, 0.00916886609, -0.0122190677, 0.0218311343, 0.0335342512, -0.0146234371, 0.0438102633, -0.077614136, 0.0470140576, 0.049997624, 0.0259098671, -0.083344467, 0.00949325599, 0.0295782313, 0.004311678, -0.0654341727, -0.011575494, -0.0266373605, -0.0669188946, 0.0225583967, -0.0412625, -0.0288016349, 0.0348377898, 0.0220591351, 0.0417983122, -0.0160438605, -0.0384733155, -0.00264788326, 0.00121475756, 0.000582023524, -0.0186849032, -0.054115653, -0.00787138753, -0.174607947, -0.0349131525, 0.0395045802, -0.0366799459, -0.0455558449, -0.0416939817, -0.0877359286, 0.035285905, -0.0311112106, -0.0622054525, -0.112809017, -0.0541132465, -0.0406626798, -0.0284972787, 0.0569148771, 0.0218789093, 0.0210940968, -0.0058397036, -0.114482872, -0.0979745165, 0.030799035, -0.0713793039, 0.0471961796, 0.0554683469, -0.0128943883, 0.0308776908, 0.065305829, 0.0600022785, 0.0578908846, -0.0959817097, 0.0287072025, -0.0018175561, 0.0227530953, 0.0304102376, 0.114969306, 0.139094412, -0.0768289268, 0.118822396, 0.0398704968, -0.089787446, -0.0362221971, 0.0400245413, -0.0501707643, 0.0217582174, 0.106088743, -0.00965043716, -0.0552714169, -0.0358450301, -0.0532797575, -0.118430391, 0.0108947149, -0.00399960484, 0.130610287, -0.0910229534, 0.076496549, 0.192751497, 0.153142869, -0.078721121, 0.0974171236, -0.0637671575, 0.133412272, 0.054068774, 0.0659344643, 0.0738890544, 0.129213035, 0.0617097616, -0.00218380103, 0.0743098333, 0.088109754, 0.00424233824, 0.00474822661, -0.0533786342, -0.0542675555, -0.0530552007, -0.0147651928, 0.0204822794, 0.0055515375, 0.0824306905, 0.0630644038, -0.123938724, 0.0445184782, -0.0124926716, 0.0399354398, 0.0462415703, -0.00357718952, -0.0310765319, -0.0180594008, -0.0647205636, -0.0929303989, -0.0461111665, 0.0672799498, 0.0245015472, -0.0589751303, -0.00370876817, 0.125348523, 0.0173412561, 0.00147062447, 0.0107325977, 0.0203702617, 0.0249537919, -0.154006839, -0.0301519893, 0.0608085394, 0.0263827238, 0.029455971, -0.0220873933, -0.00259258039, 0.0024119243, -0.00270884484, 0.103533603, 0.0581201389, -0.000676386524, -0.0915270224, 0.0643412694, -0.0548654199, 0.112059109, -0.0694910213, 0.0078248689, 0.0504440106, -0.0054148878, -0.0970134139, 0.0345405787, -0.0322505422, -0.0876624286, 0.113000952, -0.00536632352, -0.0115357321, -0.0457229577, -0.0715270936, 0.0115144514, 0.0045977179, 0.0407942012, 0.0495418385, -0.00701943412, 0.0182470679, -0.0764279217, -0.0539766066, 0.00375521788, -0.0104515478, 0.0231417604, -0.121165156, 0.114111945, 0.126064762, -0.00388064608, -0.0940569341, 0.0338260531, 0.0326401293, -0.0471561998, 0.0579081513, -0.0229190495, 0.0184844956, -0.0135091394, -0.0416546166, 0.0318427682, 0.00775113609, -0.0370019525, 0.0524832718, 0.0156050082, -0.0353443697, 0.00207883306, 0.00526856538, -0.0722670928, -0.0175125673, 0.00250724517, -0.0678912252, 0.0274016261, -0.0103717912, -0.134072885, -0.00206018589, 0.0782609358, 0.000707497587, -0.0891390592, 0.0435113795, 0.156323299, 0.0321706012, 0.0317773744, 0.0236559734, 0.0203740932, 0.0369281024, -0.111315168, 0.00825900584, -0.00578446686, -0.0563890189, 0.0631061643, -0.0372106321, 0.0403984897, 0.0308041405, 0.0374712758, 0.0968400836, -0.118751407, -0.055689536, 0.00489810202, 0.0166433491, -0.113952667, 0.0398088172, -0.0872384384, 0.0256094169, -0.0208025426, 0.0503279343, -0.000680567697, -0.0218897313, -0.0121672219, -0.120445907, -0.0290362444, 0.0458957329, -0.0203261208, -0.00833878387, 0.114699118, 0.161920175, -0.0622126386, -0.0531367436, -0.13449356, 0.105220392, 0.0362993777, -0.129608437, -0.0238405224, 0.0240593851, 0.0851430371, 0.0542634204, -0.0814281031, -0.0046661892, -0.0636177808, 0.0421245061, -0.013777907, -0.0477692746, -0.0335178003, -0.0191314854, 0.0911717638, -0.0496318638, 0.0787354186, 0.0420840308, -0.0109629817, -0.0119278589, 0.0346168764, 0.139694706, 0.0746696517, 0.0735565349, -0.000398144126, 0.10765253, 0.0973338857, 0.0839474499, 0.0529223457, -0.0598912463, -0.0240280405, 0.0603810847, 0.062021669, 0.0403415672, 0.0777214617, -0.0505453795, 0.00169499218, -0.0807233974, 0.0275564678, -0.0800994933, 0.00755414926, -0.00802462548, -0.0184881929, 0.0277756825, -0.120351225, 0.0715057999, 0.0191288032, -0.0875440687, 0.041579783, 0.0396026149, 0.0641781166, -0.016230844, -0.0655719265, -0.122426778, 0.0120705441, 0.0442694761, -0.109588109, 0.0847536922, -0.191989169, -0.0943643898, 0.0422161222, 0.00967109203, 0.0594437197, -0.0525187366, -0.119888216, -0.0454047248, -0.0449278206, -0.00292979926, -0.0749732852, 0.0184259433, -0.044917129, -0.056080848, -0.00320152752, 0.0933674052, -0.131221339, -0.0771456808, -0.0841135234, 0.0220176056, 0.0196069814, -0.0715225711, -0.106456585, -0.00247021019, -0.100794949, 0.0340740941, 0.000489225611, -0.0045605395, 0.0626360327, 0.0680942833, 0.0400962122, -0.0290915836, -0.0799229592, -0.0815847367, -0.067881614, -0.0388026759, -0.0311572291, 0.0294365287, -0.0725417212, 0.010124512, -0.00307039917, -0.0668264925, 0.0872276425, -0.0413211808, -0.0094450824, -0.18829672, 0.0206325836, 0.143229589, -0.00178726763, -0.0195381213, -0.030122865, 0.0337282568, 0.0147296134, 0.0674443021, 0.0269484706, -0.0818429291, -0.103444442, -0.00453380123, -0.011223549, 0.12715055, 0.0188172814, -0.0135700395, -0.0304954834, -0.0450241454, -0.00558831636, 0.00901627727, 0.0103639551, 0.0834274888, 0.0984052718, 0.00306586549, -0.00368587533, 0.0187812671, -0.00268950011, -0.0886186585, -0.0258823447, 0.113775909, -0.0843832046, -0.157115117, 0.0873185322, 0.0322909057, -0.000849812757, 0.0580909327, -0.0271804854, 0.0336103626, -0.0132620633, -0.0427452177, -0.020930456, -0.0737413988, 0.0191306379, 0.0429741628, 0.0165928602, -0.11342749, 0.104298979, -8.81515443e-05, -0.0605594032, 0.114668787, -0.0729807019, 0.00987668801, -0.0355439112, 0.0099394368, 0.0560149178, -0.0637701973, -0.0337059349, -0.0380720422, 0.0153781716, 0.0746347308, 0.000765843317, 0.00429571932, -0.0602201037, 0.111807078, 0.00919496175, -0.0103673441, 0.0497356206, 0.0775526166, 0.0500015728, -0.0514182672, 0.162355468, -0.0642543882, 0.0335088596, -0.0879339129, 0.060004659, -0.0849946439, 0.099622868, -0.027500499, 0.0260770805, 0.0599495545, -0.00223706011, -0.0513610877, -0.0196459536, 0.0575621054, 0.0649092197, -0.0428130403, 0.00475160591, 0.0316760316, -0.0389932171, -0.0718734562, -0.0425538272, 0.0844969302, -0.0461762212, -0.0315701067, -0.00920138694, 0.0413366929, 0.0719121844, -0.091469422, 0.0181102734, -0.0468295068, 0.104960881, 0.0102319177, -0.0418468229, 0.0634507909, 0.0279579256, -0.093235068, -0.0226055048, -0.021448141, 0.176433355, 0.0110506285, 0.0214498751, 0.0419226103, 0.00179289654, 0.120292678, 0.00706778094, -0.0599086359, -0.0641222596, 0.0887141153, -0.0507612899, -0.0465898514, 0.0435211547, 0.111409873, 0.117250025, 0.0492768362, -0.00773958489, -0.114262708, -0.0873803347, -0.0210083034, 0.00988515466, 0.0237416793, 0.0657975301, -0.0509653911, -0.032384783, 0.0596269369, -0.0890459865, 0.00208871253, 0.0965588689, 0.0173936486, -0.0910615325, -0.0252134837, 0.0354683772, 0.0709091723, 0.00448856875, -0.00221450347, 0.0129852872, 0.00403427705, -0.0404043794, 0.0697907507, -0.022720024, 0.0418550074, -0.0277890302, 0.0558229201, -0.0567896888, -0.0148143359, 0.0827597231, -0.0282895435, -0.104259551, 0.00877619907, 0.0970312059, 0.0242693834, -0.0596213117, 0.0262636393, 0.0212463029, -0.00684286561, 0.0366535373, 0.0799304396, 0.0525771752, -0.0883747563, -0.179550573, -0.0952791944, 0.0235669762, -0.0118365213, -0.0891181231, -0.0680910796, 0.0355285704, 0.0676126629, 0.108318977, 0.017775286, 0.0988742113, 0.00480408221, -0.00208715117, -0.01695171, 0.11249584, 0.0339142717, -0.0248192232, -0.0316888392, 0.0249721035, -0.00418414082, 0.00789755117, -0.016163379, 0.0166317746, 0.00545700872, -0.0243010577, -0.0228729863, 0.0763797387, -0.0154581768, -0.100936271, -0.0781337693, -0.0480149686, 0.0530673973, 0.0738910362, -0.0447604209, -0.00449215993, 0.0136270933, 0.0087039005, -0.0784128234, 0.0166925862, -0.0337094143, 0.0675746948, 0.010148678, -0.0266291015, 0.0272338502, 0.0580152161, -0.0286588576, 0.114627868, 0.112889558, 0.032557331, -0.0456488468, -0.0246344134, -0.0374983773, 0.0440980941, -0.0243410245, 0.00580131961, 0.045960132, 0.064993836, 0.0417101234, -0.0652032495, 0.0332746096, 0.0467936769, 0.0448275656, -0.0423467606, 0.091368705, 0.0381434448, -0.012054557, 0.0838974565, 0.0626250952, -0.0887676477, -0.0852957964, -0.00335176848, -0.00846866984, -0.0274248458, -0.023089027, -0.0742072165, -0.0940124765, 0.0543522947, -0.0219289456, -0.0210896172, 0.0899827257, 0.0676006377, -0.0517056771, -0.0680012852, 0.119685143, -0.00181921851, -0.0629452914, -0.00572227314, 0.0686477944, 0.00747396704, -0.0128121451, 0.108327873, -0.012849059, 0.0109706242, 0.0120692514, -0.123631217, -0.0586675107, 0.0427028313, -0.0462197065, 0.0160779729, -0.0626947358, -0.0532093272, -0.145670623, 0.097358346, 0.111907288, 0.0236618631, -0.0300452318, 0.0135302339, -0.00335860997, -0.016559381, 0.0894594863, 0.0348632745, -0.078807801, -0.0467812419, 0.105145149, -0.00522746705, 0.0751669556, -0.0196651556, -0.0283020176, 0.0590309277, -0.0196496844, -0.132960245, 0.0437823609, 0.0259339083, -0.0946520641, -0.0230558645, 0.1160651, -0.0237118732, -0.0388044789, -0.0789281055, -0.0821341574, -0.0196833406, -0.150081486, 0.0627293587, 0.0813195556, -0.0418570004, 0.0435353629, 0.0677542537, 0.0628151894, -0.0508136936, 0.0217916202, -0.135659009, -0.0214436203, 0.0702478811, -0.0497100651, 0.156953782, 0.00712094456, -0.0251476616, -0.0929391757, 0.0134378737, -0.000400929712, -0.0136013785, 0.0110868756, 0.0228250697, -0.10061945, -0.0736554116, -0.0243354365, 0.0445340574, 0.0463513434, -0.0645009428, -0.008876862, -0.0910077468, -0.0769906715, 0.0626367331, -0.110591181, 0.0436903872, 0.0688429177, -0.042393215, 0.023736082, 0.113998309, 0.0303321369, -0.00861303508, -0.0868714675, -0.0202704184, 0.0172802582, 0.0427288786, -0.0326127335, -0.0489475168, 0.121791288, -0.0625449717, 0.0315280631, -0.0603316501, 0.0334082916, 0.11952731, -0.0394092128, 0.0875948742, -0.0371525809, -0.00417886302, 0.0788129419, -0.0289812647, 0.0653141961, 0.00378620811, 0.0679804534, -0.0401788838, -0.0462654307, -0.0567128733, 0.00389130041, 0.0341692902, 0.0724724233, -0.0267045088, -0.0827875286, 0.0932042301, -0.011805323, -0.0404965207, -0.00572291575, -0.041634243, -0.080533646, 0.0223352965, 0.00108978339, 0.00445140526, 0.0287799463, 0.0976763889, -0.00342730619, 0.0261146594, -0.0252177939, 0.0373998471, -0.10728351, 0.0487615466, -0.00232692622, 0.0352337733, -0.0344574973, 0.0313353688, -0.0535807125, 0.0313085727, -0.112473421, 0.0329722464, -0.042473603, 0.0439547338, 0.0288941432, -0.127786949, 0.0110157374, 0.0882805586, -0.00272948202, 0.0181754939, 0.0114538362, 0.0537753738, 0.0667803362, -0.0677053407, 0.00496108457, -0.0720811188, -0.0615162142, -0.020356467, -0.0175721757, -0.0520251393, 0.0469468869, 0.0427129269, -0.101062745, 0.0402955115, 0.0702897757, 0.107999116, 0.028353259, 0.000175202265, 0.0319545195, 0.0224591531, -0.0443576686, -0.0535160303, 0.083751604, 0.0535791516, -0.118515864, -0.0711420178, -0.135623768, 0.0382780172, -0.0780748576, 0.102795526, -0.00695921853, 0.0161857717, -0.0557194687, 0.0256048311, -0.0153498333, -0.0672700703, -0.0733335614, 0.0276577733, 0.0542402379, -0.0864430517, 0.0187365226, 0.0403345674, -0.0506104305, -0.0114181833, 0.0182452817, 0.0639782846, -0.041567646, -0.174882635, -0.0071022138, -0.0518129282, 0.156194434, -0.00319527555, -0.0252434034, -0.030735122, -0.0383832902, -0.00307705253, -0.0487023145, 0.032265991, -0.0466151014, 0.136572123, 0.0611563325, 0.0544733331, 0.0878918767, 0.0343078859, -0.0135430023, 0.02802811, -0.0182215385, 0.0810912475, -0.0444691777, 0.0105526354, 0.164107308, 0.0147133088, -0.116141923, -0.0226079356, -0.0330710933, -0.0843250155, 0.00712005189, -0.106961481, -0.0945995599, -0.0114363721, -0.14336966, 0.084244363, 0.0389979742, 0.0225144178, 0.0235317498, -0.0167024359, 0.0584151633, -0.0250904728, -0.0159091577, -0.000552236917, 0.0713454038, 0.137021065, 0.00234995922, -0.0463563055, 0.0270676129, -0.067719765, -0.0399121419, 0.104360074, -0.00893343985, 0.0551207215, 0.118400902, -0.0701415539, -0.0387297273, -0.0508602411, 0.0381536894, 0.118008196, -0.11745958, 0.011596337, 0.0465168841, 0.0252112132, -0.0205298029, -0.0324858725, 0.125305489, -0.0452805087, 0.081967622, 0.0505525693, -0.0537428595, -0.0221687071, -0.0494968593, -0.00660148449, 0.0776317939, 0.0704046488, 0.0601929054, 0.0276133455, -0.0149744693, 0.054941047, -0.0370928459, -0.059791483, 0.0346804298, -0.160057783, 0.0794646442, -0.0843058079, -0.0360735357, -0.00650537107, -0.104105644, -0.0440651588, -0.0623810887, -0.0210951213, -0.035369236, 0.00526613649, 0.0611581132, 0.00800221786, 0.0447306708, -0.0415446237, -0.050212007, 0.0888394117, -0.109994367, -0.0269243047, -0.0352931283, 0.0570776127, 0.0657386556, -0.0722398832, -0.0906543583, 0.0143183768, 0.151019558, -0.0690796748, -0.0234915912, 0.0268165916, 0.0328775421, 0.114779577, -0.0520847216, 0.0304257534, 0.0984320641, 0.0802848712, -0.00827683508, 0.00761024468, -0.0278177261, 0.0101151615, -0.0495297499, -0.0792890862, 0.0050776992, -0.101408519, -0.0517062917, -0.0263916589, -0.0267344564, -0.0629847497, -0.0775898993, 0.00773979258, -0.0915154815, 0.0596392043, 0.0280450843, 0.0234408304, 0.140804037, -0.047485169, 0.0262268595, -0.0946769714, 0.129156768, 0.00343287364, 0.063563548, 0.0135316625, 0.0591734685, 0.099732846, 0.0304324254, 0.0602355301, 0.00678694248, -0.00180233922, 0.102937885, -0.00805503316, 0.0104419887, 0.0551552139, 0.011435776, 0.0179958791, -0.104006931, 0.119327992, -0.0639179796, 0.005029005, -0.0661187321, -0.0270529706, -0.0167394392, -0.0237004366, -0.0422669798, 0.00553747825, 0.0286485385, 0.026242936, -0.0266333688, 0.079406105, 0.0706346855, 0.0409847647, 0.152258739, -0.00351316156, 0.0119571043, -0.0294431746, -0.0192513242, 0.157942057, -0.0410583988, 0.00437228847, -0.024731636, -0.105326973, -0.042579025, 0.135244086, -0.019126296, -0.0130200777, -0.101585604, 0.146087825, 0.0132060628, 0.0578999259, -0.0182653051, 0.0436916351, 0.0710629448, 0.125556126, 0.115638174, -0.052748166, 0.0165997688, -0.0602921434, -0.101736024, 0.00287885312, -0.0432907008, -0.0417793766, -0.0816098154, 0.0441878252, -0.0124421101, 0.129645571, 0.0637945682, -0.161455527, 0.0435950272, 0.0757146031, -0.0767993852, -0.0142434519, 0.0194436722, 0.0696630701, -0.0755678043, -0.0458197519, -0.0309413634, 0.0816416815, -0.00238332432, -0.00855722092, 0.0498217829, 0.0141457357, -0.0826084539, -0.0100752236, 0.0605480447, -0.0141655887, -0.0542897247, 0.0284324735, 0.0677687228, 0.0337968692, -0.0199569054, -0.0523342118, 0.101626344, 0.00714364462, -0.0136163607, 0.0880083144, 0.0456181504, 0.0847083926, -0.0485587753, 0.0128885945, -0.0608888045, -0.0855963305, -0.0591631792, -0.0486954637, 0.0229094196, 0.107164204, -0.0159299392, 0.00904549658, -0.011729775, -0.031865444, 0.0258475132, 0.100127511, -0.0262039211, -0.0664022416, -0.00470724469, 0.0137329018, 0.0313126333, 0.0355348326, 0.0117307901, -0.0188957192, 0.0566124171, -0.0282677375, -0.0594578981, 0.00672836509, -0.1033215, -0.027556913, -0.0512220748, -0.0300782528, 0.178176463, -0.0328881592, -0.0147119835, 0.0337706953, -0.0506363325, -0.00279865228, 0.0404461697, -0.0222785361, -0.049528636, -0.0502120517, -0.0519173816, -0.133914351, -0.0162610076, -0.128599644, -0.0782211721, 0.0178051163, 0.0826841071, 0.0437118746, -0.0206440911, -0.0561366975, -0.000832460588, -0.0528845377, -0.00570855197, -0.0470915996, -0.0587879047, 0.0092945192, -0.0215655863, -0.10565196, -0.197383344, 0.0572952554, 0.0231805742, -0.00923884287, -0.064807646, 0.0883572549, -0.0648361742, -0.0135531072, 0.0472305343, -0.0266639106, 0.062329188, 0.0269762725, -0.0928731263, 0.0704310834, -0.0198958367, -0.0149159636, 0.00686603785, 0.0269686077, -0.0873637795, -0.0286721215, -0.0215567499, 0.130196318, -0.0423342884, 0.194212511, -0.081414789, -0.0076991953, -0.0783355385, 0.0927469283, 0.00718300603, 0.0361262634, -0.0961883143, 0.0405300185, 0.0641446561, -0.0466955677, -0.00139584765, -0.00198541954, -0.0511209927, -0.0421742275, -0.00424954388, 0.129908264, 0.0717779696, 0.0956653804, 0.0375357829, -0.00401965296, 0.0184375029, 0.0662451535, -0.0168066621, -0.0567378663, -0.0829721168, -0.0760762691, 0.0368871428, 0.0185185932, 0.0986614674, 0.032808654, 0.0720618591, -0.130547792, -0.0912173092, 0.0793833584, 0.0626734868, 0.0696957856, 0.0524793118, -0.0546380728, 0.0786301345, -0.00327313878, -0.00244732574, 0.042441003, 0.0445609018, 0.130712867, 0.111797251, -0.0289119966, 0.0280290227, 0.0407425798, 0.0693059936, -0.0312035903, -0.00197154656, 0.0118433312, -0.0273596942, -0.0346964598, -0.0292564966, 0.0249565803, 0.0129551161, 0.0299617406, 0.000187253579, 0.00736359134, -0.0952908024, 0.00776585657, 0.0325814746, -0.0011729449, 0.146065399, 0.0799128786, 0.0176936984, 0.096888423, -0.0499947444, 0.132609472, 0.025535427, 0.0368944556, 0.103180341, 0.0279245451, -0.0523713529, -0.0207858272, -0.0649965629, -0.109815642, -0.133886978, -0.0656646788, 0.116181061, -0.0448692292, -0.0682580769, 0.0750780702, 0.0789603889, -0.0191625282, -0.0370198749, 0.0562203117, -0.089303799, -0.120916001, 0.0440229811, 0.017071113, 0.00819048472, 0.0358136892, -0.0303053651, 0.0487265848, -0.0692953542, -0.0274103396, -0.0482576378, -0.0872205496, -0.101346761, -0.00348056271, -0.0524663664, 0.0925177261, -0.0841329768, -0.0143443421, -0.0131710516, -0.0559271723, -0.0509468168, 0.0350430645, -0.0165694728, 0.0357682668, -0.0127721224, -0.084207423, 0.0555599667, 0.00161979324, 0.0112772826, -0.138291493, -0.0120617738, -0.0162966996, -0.102659881, 0.0489581376, -0.0340032019, -0.0954410508, -0.020711178, -0.103112854, 0.153401434, -0.0932793617, 0.0349052958, 0.0299746729, -0.0241311789, 0.0108946143, 0.0215884894, 0.125622466, 0.00799371302, -0.195095733, 0.023905009, 0.036067538, 0.0351097323, -0.0200363398, 0.0492321625, -0.0948540717, 0.0532651842, 0.0503873155, 0.0436795428, -0.0725123212, -0.000908751041, -0.118674353, -0.0630601272, 0.0237448011, -0.11190787, -0.115581997, 0.0427568741, 0.0191384964, 0.0489196479, -0.150875747, -0.135023072, 0.0364912562, 0.0928073674, -0.011888206, -0.0624923557, -0.0767630935, 0.0269377157, -0.0323881693, 0.0229685605, 0.036328841, -0.0204502065, -0.073223874, -0.0286484621, -0.042256888, -0.0104460148, -1.6849488e-05, -0.00619425625, 0.139555767, 0.0651475564, 0.0535817519, -0.0556522235, 0.0809327662, -0.0492313951, -0.0195028186, 0.0271754377, 0.0098871924, -0.11343652, 0.108601764, 0.0212724674, 0.132927358, -0.016385613, 0.0751721114, -0.0541994795, 0.0941608995, 0.0402350947, -0.0411919653, -0.00882468186, -0.0157360956, 0.0178215299, -0.00205023913, 0.0452934168, 0.0612306781, -0.00629303604, 0.0972539186, 0.00905103795, 0.0317829028, -0.0471964255, -0.0577480607, -0.0199942179, 0.0152428132, 0.0241903905, -0.0584285855, -0.0795418099, -0.113055572, 0.104456373, -0.109334648, 0.0227580853, -0.0778715611, -0.150127411, -0.142432541, -0.0423689522, 0.0305046812, -0.0299814418, 0.0384439975, 0.0699854195, -0.0252225082, -0.0170006454, 0.0358190499, -0.113607176, -0.0428070128, -0.0566250496, -0.0393508449, 0.0288561918, 0.00104911998, -0.0738223419, 0.106368646, 0.0238269866, 0.0330828764, 0.113931336, -0.0369522385, -0.081184186, 0.0646849498, 5.19249588e-05, -0.0116207115, -0.0554731637, -0.00514118932, 0.0757739246, -0.0411596559, 0.134028032, 0.0607964098, -0.0278406367, 0.0352571495, 0.109581649, 0.0125203719, 0.000600435771, -0.0962911993, 0.133485198, 0.0850446001, -0.0738526061, -0.0530114062, 0.113869861, -0.0147250518, 0.0589881614, 0.0164035652, -0.0655556321, -0.0828794092, 0.0308509953, 0.0514469855, 0.0379033573, 0.0268833041, -0.142309442, 0.0360097326, 0.0909472406, -0.047603406, 0.0208126921, -0.00891117379, -0.0457498506, 0.0185710695, -0.0432754308, 0.0400561243, 0.00278019346, -0.0769423395, -0.0224651936, 0.0154477358, -0.040421661, -0.0685800612, -0.0204324275, 0.055664178, -0.0309199207, -0.0138037521, 0.0513601191, 0.0086802505, 0.000328170136, 0.0482764989, -0.0449494906, -0.0518102422, -0.0789839774, 0.0388445444, 0.0390803218, -0.0430651978, 0.0575419664, 0.137506798, 0.0374329649, 0.0602476336, -0.036358919, 0.000168859959, 0.0304721482, 0.0338621587, -0.0483214594, 0.0318760835, 0.0811550543, 0.00569907157, -0.0646105856, -0.0354435071, 0.135020778, 0.0412066467, 0.133714512, -0.0288339183, -0.104476959, -0.123337314, -0.137497395, 0.151561648, 0.0509389825, -0.0501207858, -0.0602918044, -0.0250656512, 0.0055895485, 0.0689757019, -0.0308203734, -0.100049324, 0.0328471772, 0.00582807232, -0.00715701468, 0.0805223286, -0.0629422143, -0.00300725549, 0.101139702, 0.0708577335, 0.0402698517, 0.10742756, 0.0346029699, -0.0617076531, 0.0611690134, -0.0736576021, -0.0275723394, 0.0196858793, 0.0528421961, -0.0818997025, -0.00524347322, 0.0511385351, -0.136113361, -0.0185631718, 0.0657188147, -0.140423834, 0.0440328717, 0.072102353, 0.053271722, 0.00526520796, 0.022299353, 0.051257655, 0.0415132456, 0.104825124, -0.00929822028, -0.00303138467, -0.037035007, 0.0533859916, 0.0831701979, 0.0780397952, -0.0654217079, 0.0437477306, 0.00813025795, 0.0593174472, -0.0651469082, 0.115364529, -0.00285707228, 0.0519138724, -0.00148043036, 0.0106875747, 0.0956581607, -0.018087808, -0.00546352193, 0.0617973395, 0.0994482189, -0.0978432894, -0.0179051105, 0.0142586818, 0.134737208, -0.00662420318, -0.0112975892, -0.0516164303, 0.0183628481, -0.0142547842, 0.129786283, 0.0688032135, 0.000256869942, 0.0139758456, -0.100280538, 0.00106888637, -0.0435144976, 0.0470736697, 0.0716782063, -0.0380197018, 0.0265397467, -0.0455018766, 0.0143005624, -0.0217618458, -0.0830904692, 0.00432692468, -0.0199053437, -0.0289525799, -0.00746858865, 0.0156876408, 0.0489094853, 0.0620405562, 0.0504702218, -0.0594833121, 0.00575947482, 0.0388537534, 0.0612031706, -0.0562399775, -0.0941119939, 0.053586334, -0.0913747698, 0.0837126821, 0.019398775, 0.000907974318, 0.0714335963, -0.00580542721, 0.0159939378, -0.0638639331, 0.0735958815, -0.0223918464, 0.0367563888, 0.0683975071, -0.0444335863, -0.0298664439, 0.00724903448, 0.0606348328, -0.0906336531, -0.0319926068, 0.0185662583, -0.0239852071, -0.0339926705, 0.130873993, 0.0684631392, -0.0175832678, 0.0703755692, 0.0903693661, 0.054419525, 0.0450843684, -0.00594607973, -0.0352552533, -0.0565803275, 0.0623022988, -0.0245604701, 0.0182057917, -0.120825686, -0.0132247172, -0.0253527462, -0.0456854813, -0.027723629, 0.060072381, 0.0545640476, -0.0304024816, 0.0458347276, -0.0247822534, -0.0526043735, 0.126125365, 0.135813415, -0.0791728944, -0.066400148, 0.0696547851, 0.0493155271, -0.129303932, 0.0276266281, 0.0915443897, 0.0569891855, 0.0098314872, 0.0386766046, -0.0266428366, 0.016939234, -0.013839649, 0.106271133, -0.00699316338, -0.00174673297, -0.00109564513, 0.0482021645, 0.011738346, -0.0366197117, 0.171940655, -0.055389449, -0.100271314, 0.0365726203, -0.0936080068, 0.00547959469, -0.0907428786, 0.0875035822, 0.0542516261, -0.0588709041, -0.0327620544, 0.0060365852, 0.0490757674, -0.00671805069, 0.105863348, 0.0723394156, -0.0746447667, -0.0556726381, -0.0201146789, 0.0598063096, -0.0232595727, -0.0580297261, 0.0898887515, 0.0515060946, -0.000780483708, 0.0145142619, 0.0386898965, -0.0255828612, 0.0238320194, 0.00855911151, 0.0982022285, 0.0453072451, -0.119265392, 0.122585699, 0.0296006873, 0.112326294, -0.025307931, -0.01295113, -0.0417767167, 0.0959235504, -0.0914410949, 0.111983821, 0.0353446715, 0.00137972925, -0.149913996, 0.0460681692, -0.0517969541, -0.113715298, -0.112907112, -0.129507795, -0.0806752145, -0.0521873347, 0.0211963058, -0.0705100819, -0.0122897793, -0.0357527398, 0.0923158303, -0.0366787612, 0.0357766561, 0.0639059767, 0.0536018014, 0.0377076678, -0.0190985985, -0.0868470296, -0.0856646374, -0.0969800502, -0.155979827, 0.00997250155, -0.14321053, 0.0559573956, 0.00282313488, 0.0252706297, -0.0313694738, 0.0862585828, -0.0452943221, 0.098857373, 0.0293958858, 0.0521099977, 0.00256046327, -0.0223779399, 0.0623505637, -0.0765269697, -0.0851114169, 0.0880696699, 0.0554719083, -0.050662946, -0.0783270746, 0.0493648425, -0.0126534328, -0.0391949676, -0.0316629596, -0.0476705953, 0.046895206, -0.0173123255, 0.00136741996, -0.00448701531, 0.0327305496, -0.105013773, -0.0459271707, -0.0276662391, -0.0261136312, -0.0576968193, 0.0525827594, 0.00364556536, -0.0115968287, -0.0617727935, -0.0365634561, -0.0567271002, 0.0217187107, 0.0492976084, -0.0280287527, 0.0216550119, -0.0330982283, -0.0974075198, -0.0765775889, -0.0173772238, 0.0687277094, 0.0537037291, 0.0358378664, -0.0642583594, -0.0882536843, -0.0219793171, -0.0944289416, -0.00437883381, 0.0234113354, 0.0826886892, -0.04128832, 0.0831653476, -0.02940703, -0.0337581187, 0.0619091392, 0.0441856906, 0.0693871528, -0.0688716099, -0.0191987529, -0.0617373697, 0.0497171283, 0.00187313184, 0.145926401, -0.0416486412, -0.0219981596, 0.0138280541, -0.0567112975, 0.0154636679, -0.0561905019, 0.0506791323, 0.101463027, 0.151062578, 0.0687830523, -0.101705603, -0.0523636118, -0.030089058, -0.0690361634, 0.0160269402, 0.0308208354, 0.0291081071, 0.0732349604, 0.0382921807, -0.034624815, -0.0483729914, 0.14700301, 0.0436632857, 0.0287404694, 0.132106334, -0.0992597714, 0.0430740751, -0.167150855, 0.134502336, -0.00803485513, -0.0402739234, 0.0139839482, 0.0192187689, -0.15193595, 0.112887859, -0.0808533728, -0.093750976, -0.00189099275, -0.0131205078, -0.0387071297, -0.107041217, -0.0545439757, 0.00303797773, 0.0670112893, -0.023910353, -0.0125194713, 0.0438937359, 0.0349927992, -0.0327213556, 0.091033496, 0.0239645913, 0.0976982862, -0.0428775176, -0.138354793, -0.0702264085, -0.0800770819, 0.0101706767, -0.0692842156, 0.00787558593, 0.0842271596, -0.118677564, -0.0310803242, 0.0218988862, 0.0045571099, 0.0930025131, 0.0476951711, 0.0667954907, 0.0518937893, 0.0696247295, -0.00674023852, 0.00389996357, -0.0416572466, 0.0901752189, 0.0582431778, -0.0179458931, 0.0181185212, 0.0227411687, -0.08677838, 0.0375101604, -0.0477446057, -0.0864975154, -0.0721852407, -0.00117101334, -0.0698436275, -0.0452621244, 0.0144802826, -0.0268776435, -0.047778815, 0.0611376092, 0.0360228419, 0.0702620074, 0.0462913141, 0.0817417055, 0.0942117348, 0.0347194336, -0.0515818372, -0.0356176645, -0.106147617, 0.0378560498, -0.170979455, 0.103543155, -0.0348379351, 0.0938812643, 0.0529162623, 0.0120922439, -0.00355465943, 0.0324143507, 0.0486200638, -0.0678899288, -0.0984239355, 0.0160683487, -0.0246096496, 0.115997225, -0.110947073, -0.0867623761, 0.0626195446, 0.11056228, -0.0638028979, -0.0485575534, -0.0868593082, -0.0715334415, -0.0182123706, -0.105600968, 0.0384222232, 0.0276586562, -0.0497897118, -0.0403108634, -0.106564187, -0.00672912411, 0.0264774021, 0.0640708804, 0.00270042382, -0.128070235, -0.0106159896, -0.0350066312, -0.024903249, 0.0278657433, -0.0662305728, -0.0241936184, 0.0483643524, -0.116221316, 0.00459046802, -0.156511158, -0.0918338895, -0.0996401012, -0.0410874002, 0.0768202469, -0.00780009432, 0.011227943, 0.0283633303, 0.14154765, 0.101129919, -0.0947135016, 0.0782444105, 0.000163465738, -0.038605053, -0.0639200509, -0.048382923, 0.0231307372, -0.112709269, 0.0501804464, -0.0729039758, -0.000406133011, -0.0160389319, -0.0762058198, -0.0176509749, 0.066750288, 0.0918518826, 0.0236206073, -0.0323796868, -0.0168142878, -0.0459107161, -0.0576644503, -0.00522529008, -0.103753723, -0.0241519678, 0.047558967, -0.0335726738, 0.0163476821, -0.0271658655, 0.0451743826, 0.0304347649, 0.0549066514, 0.0261297598, -0.0171702001, 0.0206196401, -0.0230964907, 0.134645104, 0.132786676, -0.0353303552, -0.031571649, 0.0190999582, -0.0112066101, 0.0473771319, -0.0704853609, -0.0708022788, -0.0275107771, 0.00979784317, 0.0687821805, -0.152077913, 0.0279169884, 0.0548784062, 0.0107158367, 0.000214008614, -0.0331896581, -0.0150913605, 0.15168643, 0.0216256399, -0.055669684, -0.00985519774, 0.020958934, 0.00189213408, -0.0134218149, -0.0512841642, -0.0230130032, -0.049885489, -0.0768733323, -0.0800726861, -0.054872904, 0.00264478941, -0.13091433, -0.0282860696, 0.0217010733, 0.00567382295, -0.156414047, -0.0398377068, 0.00270777941, -0.0499432012, 0.0166897718, 0.0101039689, -0.0477613509, 0.00888098031, 0.0662591681, -0.0554639399, 0.0187477749, 0.0336377323, 0.0251136031, -0.133064821, -0.0126457484, -0.0105030155, -0.0140854307, 0.019213723, -0.0805561692, 0.0802005604, -0.0540246107, -0.0146111576, -0.025273703, 0.00897808932, -0.031222662, 0.0524445958, 0.0310434848, 0.121040016, -0.0810230523, -0.0358245857, 0.124070935, 0.0767713934, -0.0886022747, 0.00355428737, -0.0584391654, 0.0438103937, 0.00287393946, -0.122106925, -0.0568982512, 0.0117828399, -0.0986436158, -0.017583048, -0.0102847051, 0.0432225987, -0.0276271347, -0.156640813, -0.123027079, 0.0882055461, 0.0390510596, 0.00933926739, 0.105590925, 0.0418130159, 0.0904245228, -0.0657639876, 0.00261240453, -0.0126623744, 0.210236236, 0.0594069995, -0.099819459, 0.00615834258, 0.0488923155, -0.021860756, 0.0369348451, -0.110402897, -0.0597476214, 0.0170283243, 0.00256883167, 0.0209132899, 0.000933450647, -0.0592737123, -0.15596965, 0.0413424373, -0.00346540287];
    CONSTANT bias_0_o : ARRAY[0..63] OF REAL := [0.558418989, 0.619741023, 0.888044596, 0.554675877, 0.672804177, 1.15733361, 0.547720611, 0.559062123, 1.08087564, 0.5283131, 0.58876282, 0.58257848, 0.593611479, 0.573188305, 0.547690094, 0.68624264, 0.779895008, 0.636355102, 0.759450912, 0.658933282, 0.709287882, 0.784237385, 0.617185712, 0.673908889, 0.553099871, 0.633745313, 0.811307073, 0.575079858, 0.601960182, 0.552821636, 0.638540089, 0.647475541, 0.663177431, 0.964920223, 0.568021059, 0.59758383, 0.740071595, 0.795531034, 0.926966667, 0.545593619, 0.646610439, 0.60432446, 0.546364844, 0.626123905, 1.07764459, 0.540417314, 0.523464262, 0.652773023, 1.13402641, 0.820446372, 0.79551357, 1.14666879, 1.06271923, 1.07444584, 0.545953751, 0.746542752, 1.18182158, 0.826829255, 0.547304332, 0.650002182, 0.561002016, 0.629313529, 0.610247195, 0.681436837];
    CONSTANT weights_3_i : ARRAY[0..4095] OF REAL := [-0.755418241, -0.608314455, 0.360285342, -0.978372037, -0.73372668, 0.0433106236, 0.822168231, 0.994398952, 0.25576961, -0.897847056, 0.964666605, -0.67579025, 0.684332669, -0.809585214, 0.803079665, -0.566751003, -0.408394217, -0.656475842, -0.573797286, 0.747748673, 0.673770845, 0.494365126, -0.699537992, 0.490632325, -0.776397467, -0.676654398, -0.511669755, -0.888815522, 0.76610291, -0.882459223, 0.662760258, -0.724328101, 0.691716373, 0.15585357, 0.931201696, -0.696478367, -0.448318452, -0.338864177, -0.335456759, -0.962986171, -0.592431247, -0.779655039, 0.954741716, -0.817907333, -0.192427114, -0.807255626, 0.855172753, 0.651954412, -0.136959985, -0.420822144, 0.212966338, 0.0445446782, -0.199813604, 0.248965874, 0.838989556, -0.666503072, 0.0486680828, -0.293471068, -0.931513965, -0.615072489, 0.794350803, -0.767282784, 0.800647199, -0.493104696, -1.04894054, -0.839424491, 0.412440658, -1.0782311, -0.610590279, -0.224400103, 0.914384246, 1.09467459, 0.400612175, -0.913536131, 0.880798876, -0.830022335, 0.92901969, -0.925858378, 0.89776057, -0.89756012, -0.580115438, -0.734643281, -0.744657338, 0.821060002, 0.721544206, 0.541094124, -1.03695524, 0.84263134, -1.04971743, -0.930462301, -0.712232709, -0.888018429, 0.880688429, -0.845546246, 1.02739179, -0.692478418, 0.718065321, 0.435147166, 0.961075187, -1.06043577, -0.756034374, -0.573500693, -0.538568377, -0.953424215, -0.810650885, -0.987207532, 1.03647971, -1.00058937, -0.177239105, -1.03699946, 0.988714695, 0.85310322, 0.00717389304, -0.556754231, 0.507442653, -0.0378301032, -0.5122298, 0.447235465, 0.929611444, -0.663908243, -0.0585526079, -0.597246766, -1.02065659, -0.686075151, 0.851084769, -0.72992599, 1.05275869, -0.917103529, -0.811452985, -0.826563954, 0.179984301, -0.835142732, -0.659547448, 0.0863112807, 0.886351824, 0.986944258, 0.135068983, -0.902180672, 0.906524837, -0.855773032, 0.879188478, -0.831542015, 1.05893993, -0.684074581, -0.332585782, -0.95702374, -0.37826848, 0.763411939, 0.510935485, 0.350773633, -0.693967283, 0.556139767, -0.845410943, -0.825000584, -0.515352011, -0.92987591, 1.00201797, -0.865815759, 0.830607235, -0.826742411, 0.697724342, 0.417915851, 1.0467155, -0.983205199, -0.84478277, -0.321441144, -0.468818843, -1.02750862, -0.712836921, -0.86461699, 0.983835578, -0.8388744, 0.0762428418, -1.09817517, 0.828923643, 0.793307722, -0.144390121, -0.211029708, 0.395367414, 0.285318285, -0.472778082, 0.456979275, 0.940658331, -0.763034642, -0.381549388, -0.177495673, -0.90530616, -0.753831744, 0.832921624, -0.774398565, 0.829895437, -0.799162805, -1.21820855, -1.06696033, 0.835389137, -1.26682889, -0.971710622, -0.315437734, 1.23276997, 1.17181158, 0.632770717, -1.20906186, 1.19340575, -1.00084484, 1.0859555, -1.01537168, 1.13232636, -1.02199805, -0.834645152, -1.13640141, -0.815388441, 1.07765841, 0.891493738, 0.978649795, -0.936340988, 0.979935467, -1.06374216, -1.15059888, -0.748942852, -1.1597482, 0.973263681, -1.20231974, 0.933190823, -1.07081246, 0.847544432, 0.364830196, 1.18962157, -0.963554561, -0.808535457, -0.784963489, -0.234990507, -1.13459432, -0.984087408, -0.955592215, 1.10403454, -0.945870757, -0.478384674, -1.300861, 1.14212894, 0.987192571, 0.187816009, -0.865885556, 0.823636711, -0.232717544, -0.0860770419, 0.194109485, 0.987924933, -0.769749939, 0.309627205, -0.921204448, -1.20993173, -0.932157576, 1.02401316, -1.02380764, 1.10313702, -0.987564266, -0.935450852, -0.861052155, 0.385243714, -1.02241755, -0.624481618, -0.0734320283, 1.08894765, 1.13742781, 0.431176722, -1.01322722, 0.922006667, -1.00998127, 0.889069557, -1.04747951, 1.01184118, -0.793883562, -0.560060322, -0.940799952, -0.584474564, 0.723362207, 0.875515103, 0.720968366, -0.911121428, 0.727347374, -1.01887119, -0.835917115, -0.646595657, -1.01109087, 0.976727664, -1.11480069, 0.928580701, -0.732790411, 0.783455253, 0.3726089, 1.02210438, -1.08693635, -0.840154052, -0.561535776, -0.370871723, -1.16396987, -0.911427081, -0.889419734, 0.99090308, -0.945265174, -0.207709432, -1.06947768, 1.11887705, 0.939141095, 0.0903663933, -0.52419728, 0.454987019, -0.0681321621, -0.422043651, 0.423526645, 0.912625194, -0.80558151, -0.0357627831, -0.431746542, -0.890021265, -0.730353892, 0.89218235, -0.759410143, 1.06895053, -0.926181376, -0.741033196, -0.726513982, 0.322699696, -0.972041905, -0.655323505, -0.0292269848, 0.952426255, 0.866428375, 0.11949563, -0.757095098, 0.942866147, -0.796896994, 0.654191136, -0.645846605, 0.824801743, -0.611181915, -0.335965067, -0.810628414, -0.466565788, 0.80544591, 0.691729486, 0.480921775, -0.511504292, 0.702025712, -0.86025691, -0.776957631, -0.29298532, -0.687556684, 0.643776953, -0.739982367, 0.726881027, -0.640373349, 0.57354337, 0.242517203, 0.994883716, -0.606989563, -0.609171987, -0.233668387, -0.257614791, -0.828473866, -0.774299979, -0.623594999, 0.742574334, -0.704159379, 0.0296151433, -0.955602169, 0.968825579, 0.601331949, -0.0735772476, -0.287132144, 0.151510775, -0.0786359683, -0.34978804, 0.133115217, 0.822498322, -0.692448258, -0.215515405, -0.396737725, -0.794197142, -0.61843133, 0.780855775, -0.798789084, 0.636612952, -0.596487164, -1.02452493, -0.733386755, 0.353141606, -0.952989697, -0.727705657, -0.0627208352, 1.21137989, 1.08253932, 0.228804052, -0.90075475, 0.982092619, -0.998478949, 0.896557331, -0.98023051, 1.0387373, -0.700028658, -0.67096138, -0.968751729, -0.84728229, 0.789013982, 0.836730242, 0.688243866, -0.731738687, 0.969447136, -1.06666744, -0.995709002, -0.664720893, -1.05856693, 1.07691407, -1.02315605, 0.728992403, -0.76652348, 0.844830453, 0.179572225, 1.22721124, -0.94140029, -0.715959311, -0.724516153, -0.228294402, -1.1530093, -0.956407428, -0.899410546, 1.09126186, -0.873448253, -0.168818444, -1.22987664, 0.95296061, 1.00769937, -0.0702653304, -0.381446481, 0.512703001, -0.0435364284, -0.11453981, 0.199777916, 1.06700945, -0.684714496, -0.112935178, -0.602526605, -1.02280688, -0.943379998, 0.718487859, -0.927234292, 0.962290883, -0.675989389, -1.04286563, -0.876557887, 0.462482393, -1.0861553, -0.654765189, -0.159290239, 1.07852364, 0.884891152, 0.140386865, -0.963511288, 0.946421504, -1.04198098, 0.839310706, -0.855860889, 0.870488524, -0.702690423, -0.439044088, -0.933871686, -0.589861751, 0.68892163, 0.597560287, 0.425204217, -0.761139214, 0.624503672, -1.02760601, -0.710986853, -0.510669291, -0.832123697, 0.788684607, -1.05656803, 0.902100027, -0.718313038, 0.701382101, 0.336199254, 0.926524699, -0.974620879, -0.690556526, -0.451145768, -0.556159139, -0.986128032, -0.619695544, -0.912777424, 0.842693388, -0.935300767, -0.196174338, -1.05631256, 0.853555441, 0.757244647, -0.184759662, -0.334762543, 0.513675153, -0.0197210051, -0.422626376, 0.306616992, 0.808679283, -0.666823506, -0.0260220375, -0.534840167, -1.05868638, -0.803471029, 1.01640034, -0.656452358, 0.937075615, -0.736741483, -0.969046772, -1.02430713, 0.475471109, -1.01880741, -0.75838691, -0.216517732, 1.14114225, 1.03535259, 0.448151171, -1.05993211, 0.987955809, -0.877148211, 0.88578999, -1.0774231, 1.1040051, -0.910460174, -0.731224537, -0.890228271, -0.725291908, 0.832292557, 0.822500288, 0.545910835, -1.05995345, 0.645671725, -1.10371053, -0.76795429, -0.622391164, -1.10858274, 0.959112167, -1.00889635, 0.884062827, -0.833665311, 0.735249817, 0.367521971, 1.13251293, -0.887471735, -0.932527363, -0.492527246, -0.614649892, -1.0094378, -0.774402618, -1.00567007, 1.00681162, -1.0051012, -0.196057275, -0.977808416, 0.948892236, 0.812963963, -0.00821041875, -0.638639331, 0.399548352, -0.122351654, -0.428168148, 0.473601997, 1.1022259, -0.944955647, 0.0435571112, -0.59750545, -1.01166987, -0.901804149, 0.864712179, -0.801286817, 1.12397861, -0.907543123, -0.968958914, -0.976406515, 0.252034068, -0.996525466, -0.691133738, 0.385438502, 1.00782788, 1.03370297, -0.205928698, -0.884970367, 0.929853916, -0.834381342, 0.924174666, -1.03883147, 1.00104129, -0.721402526, -0.389019519, -0.985671699, -0.479267389, 0.820142806, 0.544877887, 0.263722688, -0.816414952, 0.742167115, -0.977280498, -0.892438114, -0.266501427, -1.07392192, 0.829976678, -0.806288183, 0.836611867, -0.78686285, 0.632151425, 0.518191278, 1.08450913, -0.888277173, -0.780584574, -0.232404694, -0.511793911, -0.958422065, -0.690973699, -0.888970733, 0.83754319, -0.908099651, 0.106050521, -0.930795074, 1.08223093, 0.926879644, -0.449428767, -0.245660082, 0.120277353, 0.183214977, -0.581604123, 0.423586756, 1.03415048, -0.713971019, -0.32305634, -0.0967770889, -0.897503495, -0.723082781, 0.830310166, -0.742337167, 1.02575874, -0.733720362, -0.907611549, -0.854992867, 0.505329072, -0.944037795, -0.70937115, 0.0261288676, 1.01350021, 1.02204335, 0.252643436, -0.978096724, 0.862670481, -0.808062732, 0.896382809, -0.813757539, 0.814833641, -0.642812908, -0.639273047, -0.728571594, -0.703681052, 0.663110316, 0.717055142, 0.489002317, -0.705394208, 0.834371388, -0.781721294, -0.752015114, -0.457937121, -0.792781293, 0.914688826, -0.795861661, 0.595086515, -0.710880637, 0.675870419, 0.406664968, 0.96637696, -0.754895449, -0.686368406, -0.552339971, -0.444466829, -0.997712076, -0.626592398, -0.661046863, 0.88097173, -0.889222741, -0.146164373, -1.08511758, 0.943219721, 0.812917054, 0.0503441095, -0.434279114, 0.274424821, -0.0832945555, -0.193505302, 0.222719252, 0.873863757, -0.539601743, -0.0734653994, -0.442973316, -0.834634125, -0.730556786, 0.631379664, -0.775440812, 0.95656389, -0.50474453, -0.931799293, -0.82169944, 0.194752201, -0.989303291, -0.519775212, 0.112227432, 0.991141856, 1.01745415, -0.0274739582, -0.793622792, 1.06043375, -0.888234019, 0.880099654, -0.893237174, 0.881158412, -0.823377252, -0.437752366, -0.797185361, -0.37659806, 0.858986139, 0.569999754, 0.340523064, -0.836035669, 0.670638025, -0.794342041, -0.702752113, -0.431304663, -0.928568959, 0.926226974, -0.848105371, 0.720710158, -0.622902155, 0.705539167, 0.549153447, 0.870801866, -0.725703001, -0.770241082, -0.183786377, -0.615487993, -0.998608351, -0.745964348, -0.855395079, 0.966465652, -0.77130127, 0.0715011135, -0.96620065, 1.05865717, 0.790433645, -0.268629074, -0.174874589, 0.14475368, 0.0939831361, -0.337278485, 0.395812422, 0.894006252, -0.766367733, -0.176003799, -0.224346429, -0.793370366, -0.638615549, 0.867665052, -0.81962198, 0.82810998, -0.582147717, -0.842648268, -0.783048689, -0.235769719, -0.998877823, -0.327204019, 0.566020548, 0.916653872, 0.854219079, -0.460341662, -0.77112639, 0.933426797, -0.836915135, 0.874533951, -0.83277452, 0.746362567, -0.628461123, -0.084711656, -0.582916021, -0.243317723, 0.525368094, 0.259333014, 0.0327389203, -0.729031205, 0.317607105, -0.839289486, -0.4789671, -0.0461727753, -0.787092328, 0.83384794, -0.75443393, 0.908382654, -0.363875389, 0.546058953, 0.507456422, 0.980222464, -0.675206363, -0.637511611, -0.0142121417, -0.64180088, -0.892539263, -0.407804877, -0.669094205, 0.856718063, -0.493220001, 0.303538859, -0.858540893, 0.940325439, 0.49160096, -0.469009638, 0.17257607, -0.0190391336, 0.469112605, -0.543920636, 0.637618363, 0.764873981, -0.86711055, -0.494828016, 0.157218501, -0.862574041, -0.368994653, 0.676885366, -0.610570908, 0.725115955, -0.861623049, -1.07505918, -0.965862215, 0.60238415, -1.16023743, -0.840752125, -0.105824895, 0.948305309, 0.953172028, 0.288685203, -1.11643279, 1.03585219, -0.971423209, 0.863259971, -1.14757454, 0.967280209, -0.897893667, -0.533795834, -0.847732723, -0.714499772, 0.851787329, 0.7199862, 0.513467252, -0.877711296, 0.906861722, -1.14302409, -0.950012863, -0.768051147, -1.0575242, 0.983039558, -0.990966916, 0.832446694, -0.754112124, 0.893297434, 0.629224181, 0.992561221, -1.00884116, -0.913590014, -0.671533048, -0.474662781, -1.20630717, -0.696899891, -1.07192814, 1.13243151, -0.784192502, -0.15621908, -1.12142682, 1.06379509, 0.912983716, 0.025483191, -0.665657282, 0.413258642, -0.0918736681, -0.556712985, 0.362460822, 1.10431266, -0.784294367, -0.0139337517, -0.611807585, -1.0611099, -0.826119184, 0.902756155, -0.86417675, 1.1229434, -0.856812537, -1.27942991, -0.90530479, 0.625030518, -1.15539479, -0.873494685, -0.260905921, 1.24086809, 1.25946474, 0.39319101, -1.0907501, 1.2032733, -1.08172178, 1.06699085, -1.20631349, 1.22948694, -0.834533453, -0.750264943, -0.992371202, -0.807569206, 0.856315017, 1.08617556, 0.892702281, -1.01682568, 0.886915743, -1.23190653, -1.06336915, -0.932261586, -1.07520664, 1.07185602, -1.12734389, 0.907818377, -0.820663929, 1.01829791, 0.166351378, 1.20455956, -1.17253053, -0.824744999, -0.65868187, -0.317878783, -1.15693378, -0.843500435, -0.920814574, 1.09634209, -0.871699572, -0.450535893, -1.1738621, 1.13490057, 0.895801008, 0.131369889, -0.693567574, 0.74108988, -0.10059008, -0.126341328, 0.0593591593, 1.12989569, -0.740600109, 0.221153483, -0.637960136, -1.14117575, -1.0811311, 1.03810823, -0.89616704, 1.20454895, -0.886058986, -0.818703711, -0.964950979, 0.3011401, -1.05881941, -0.722192585, 0.00358383521, 0.935663342, 0.809548557, 0.160762921, -0.876804471, 0.833429694, -0.830048382, 0.89588958, -0.958845794, 0.874411643, -0.660538614, -0.362247705, -0.670403838, -0.563105106, 0.636587739, 0.495884269, 0.332683057, -0.74164784, 0.724646091, -0.972233713, -0.764483392, -0.447217792, -0.837968588, 0.850412071, -0.983349562, 0.785379887, -0.654432178, 0.724678636, 0.41592297, 0.989545166, -0.950459421, -0.639414907, -0.337752908, -0.484309226, -0.905988812, -0.595648468, -0.844717622, 0.827573478, -0.838856101, 0.0187437031, -0.849463165, 0.889378548, 0.561864376, -0.29927808, -0.392451555, 0.388448268, 0.198650107, -0.559829533, 0.414166063, 0.893056631, -0.908913195, -0.0640959814, -0.374392003, -0.958116055, -0.677774489, 0.828592062, -0.582134187, 0.876991391, -0.876230657, -0.908975899, -0.721173704, 0.494917125, -0.823946416, -0.64437598, -0.217759445, 0.913173795, 0.996590257, 0.367991656, -0.879616201, 0.771492779, -0.98472321, 0.963087082, -0.95259285, 0.839489877, -0.713660777, -0.755366445, -0.73727572, -0.641714454, 0.926426113, 0.728988111, 0.707814932, -0.803486705, 0.719608545, -0.83762908, -0.814273715, -0.611875772, -0.942105889, 0.880182147, -0.971608341, 0.790809631, -0.911215127, 0.898607135, 0.352806628, 0.81870687, -0.761086822, -0.796402991, -0.50277096, -0.537348866, -1.07715547, -0.857042789, -0.950789869, 0.867072821, -0.848236322, -0.411746114, -0.88702327, 1.00351846, 0.825973809, 0.0270913597, -0.71621424, 0.615491807, -0.173585027, -0.227682218, 0.179880247, 0.919904411, -0.736029685, 0.193204731, -0.500456929, -0.822526693, -0.700240195, 0.966011167, -0.801102698, 1.00703526, -0.885540664, -0.713978291, -0.611588717, 0.260023504, -0.922345757, -0.705840707, -0.0141039658, 0.976248503, 0.964204967, 0.26765269, -0.956324041, 0.796898186, -0.789989054, 0.782559752, -0.77758646, 0.867500961, -0.549102545, -0.493753225, -0.801779151, -0.454341143, 0.621101618, 0.647966027, 0.436664164, -0.748553097, 0.54489243, -0.788911521, -0.871274948, -0.460166365, -0.842250288, 0.652063608, -0.863243103, 0.620145023, -0.706633389, 0.78117007, 0.261015654, 0.84503752, -0.820280135, -0.517355144, -0.459893852, -0.314167231, -1.01927006, -0.700387955, -0.742943883, 0.900053501, -0.856171072, -0.0286465324, -0.895612955, 0.856761158, 0.584023952, -0.0770339519, -0.429291189, 0.261452138, 0.0627180338, -0.181542769, 0.112061031, 0.788401484, -0.513115346, 0.077620104, -0.450713575, -0.737526596, -0.571692765, 0.607120872, -0.79032129, 0.799625099, -0.475847691, -1.09786475, -0.772961438, 0.495320827, -1.1611439, -0.766513824, -0.143397436, 0.962765157, 1.06331944, 0.313598633, -1.01686382, 1.1133368, -1.08287513, 0.804114819, -0.856840074, 0.993985593, -0.812854052, -0.610591054, -0.851494789, -0.838413715, 0.978924334, 0.82232976, 0.771277666, -0.730287552, 0.951943219, -0.973897278, -0.990049124, -0.570291817, -0.936770022, 0.858006418, -0.819337249, 0.831573308, -0.891148806, 0.78176415, 0.188151807, 1.05254877, -1.00523531, -0.750526607, -0.642461479, -0.223760605, -1.2113694, -0.936775982, -0.840746224, 1.07401752, -0.79121995, -0.265156776, -1.12808418, 1.07336295, 0.848082721, -0.0801268965, -0.639466107, 0.423318893, -0.197285667, -0.299851, 0.153514013, 0.886098623, -0.601903439, 0.022839861, -0.633413076, -0.839836955, -0.761352301, 0.943436801, -0.842834294, 0.856992543, -0.752803981, -0.976946771, -0.860103667, 0.148241594, -1.17027724, -0.680404603, 0.260861218, 1.1012404, 1.09432316, -0.084494032, -0.919311583, 1.13092101, -1.07132185, 0.954994619, -1.13993835, 1.00824094, -0.845583439, -0.461782247, -0.95956552, -0.488822222, 1.02185178, 0.83047843, 0.552198887, -1.01375663, 0.755363405, -1.0269655, -0.961519718, -0.430978894, -0.921435118, 1.03942025, -1.01963305, 0.888223827, -0.95802629, 0.907438338, 0.721813977, 1.08516002, -1.1015048, -0.968381882, -0.325145304, -0.652126908, -1.28460324, -0.947565973, -0.874286115, 1.05251586, -0.949869156, 0.153231531, -1.18712854, 1.00515926, 0.865185499, -0.298296869, -0.212462679, 0.421099901, 0.405747652, -0.775304854, 0.56657511, 1.02249587, -0.934783936, -0.514021575, -0.20079039, -1.01075089, -0.857002079, 0.987509191, -0.929678917, 0.932180822, -0.886357069, -0.933931828, -0.700244904, 0.369614154, -1.10790706, -0.675352216, -0.188850135, 1.08109188, 1.04684579, 0.308671802, -0.883098602, 1.05010533, -0.929381788, 0.879740238, -1.01128566, 1.10395002, -0.720393658, -0.740107059, -0.99103719, -0.831740022, 0.862007916, 0.894016087, 0.620524406, -0.769335091, 0.897905231, -0.941016138, -0.876742899, -0.708276153, -1.0367837, 0.912421107, -0.825091898, 0.808150589, -0.878788531, 0.916051567, 0.24332048, 1.05220306, -0.952991545, -0.748910844, -0.72116518, -0.374993294, -1.04492664, -0.917863369, -0.86367166, 1.08562934, -1.03882897, -0.218215466, -1.18063104, 1.1076721, 0.878296316, -0.0187482014, -0.528429568, 0.50169456, -0.147743478, -0.122764975, 0.250912666, 0.826420069, -0.730094612, 0.0589699149, -0.46761167, -1.05767417, -0.924309313, 0.804091275, -0.917768538, 0.983291626, -0.721830428, -1.09399235, -1.00202692, 0.562182307, -0.938353002, -0.593690991, -0.0125021413, 1.08856273, 0.906774461, 0.200605094, -1.08938837, 1.09823823, -0.911578178, 0.884976149, -0.867731512, 1.04740059, -0.83649385, -0.525554299, -0.861518741, -0.646086395, 0.715107501, 0.839924991, 0.465662718, -0.874607563, 0.756407976, -1.03819859, -0.815448523, -0.716991901, -0.929483712, 0.948846698, -0.929803491, 0.808668494, -0.6867944, 0.853445053, 0.421883553, 1.09852147, -0.981153369, -0.830782592, -0.503521681, -0.4611803, -1.19973147, -0.676306427, -1.06116807, 0.871525645, -0.893308938, -0.28923732, -1.20726645, 1.16319931, 0.773241103, -0.167875394, -0.538970232, 0.392856359, -0.0467808507, -0.323710591, 0.427655101, 0.908169866, -0.824398875, 0.0668496713, -0.599668503, -1.0336014, -0.750727057, 0.798111081, -0.88163656, 0.99468106, -0.953759074, -1.11895311, -0.975337088, 0.661303043, -1.18804455, -0.69579941, -0.169847563, 1.12572634, 1.17538476, 0.360282838, -0.972973466, 0.919509828, -1.08963072, 0.907667398, -1.18446136, 1.11237955, -0.756965399, -0.708337784, -0.773685694, -0.799184978, 0.745656848, 0.951413512, 0.638455451, -0.967878819, 0.724358022, -1.13330948, -0.790725529, -0.80226022, -1.08631873, 0.949474812, -1.05668902, 0.976779699, -0.861955762, 0.974520147, 0.512347758, 0.955908954, -0.892980337, -0.737581193, -0.617187142, -0.513221383, -1.12916565, -0.880242407, -1.06890917, 1.05162001, -0.815472901, -0.297819644, -1.18346536, 0.946695328, 0.716957748, 0.175897732, -0.667602539, 0.701610804, -0.0740017295, -0.369591564, 0.346157163, 1.05868769, -0.926508367, 0.179177567, -0.475888908, -1.04457426, -0.827824414, 0.98029995, -0.907244384, 0.943478882, -0.924352646, -0.773993492, -0.735044301, 0.0416651331, -0.907257199, -0.422367811, 0.440636724, 0.991895258, 0.759705484, -0.291431665, -0.956883132, 1.00003695, -0.956255972, 0.739793539, -0.74141562, 0.889753878, -0.670551538, -0.231987089, -0.823478103, -0.315503538, 0.595067739, 0.451488137, 0.0750449374, -0.821136713, 0.358170748, -0.763157308, -0.797085702, -0.222883433, -0.833063483, 0.897186339, -0.709599793, 0.797601998, -0.649135232, 0.575399876, 0.694169581, 0.94716084, -0.885367393, -0.612949193, -0.0731305555, -0.618689179, -0.870648324, -0.606274009, -0.917017341, 0.979093015, -0.664984584, 0.407488555, -0.880128086, 0.899560869, 0.68467778, -0.564382672, 0.114791416, -0.0359922089, 0.454897344, -0.658713877, 0.597083151, 0.692245722, -0.672556996, -0.559869766, 0.0941093266, -0.949851394, -0.656304598, 0.892188549, -0.610869884, 0.741495728, -0.754965186, -0.844388545, -0.663963437, 0.100156032, -0.714349389, -0.500820935, 0.0301809032, 0.93849498, 0.795188844, -0.0408474654, -0.778205931, 0.915193319, -0.715432703, 0.726488769, -0.624961197, 0.72919029, -0.444653422, -0.356808156, -0.66607815, -0.495592654, 0.736166477, 0.510713041, 0.304338694, -0.714937925, 0.685840368, -0.841898143, -0.785771668, -0.362618685, -0.843503535, 0.838873625, -0.642146051, 0.515100181, -0.688019276, 0.652499199, 0.163452625, 0.979091167, -0.728121579, -0.39419806, -0.316004902, -0.214974254, -1.02700996, -0.750581741, -0.716689885, 0.746017575, -0.68982774, -0.0666270852, -0.975651443, 0.74363929, 0.783233523, -0.12883997, -0.236293882, 0.151585028, 0.187489644, -0.403225034, 0.297997594, 0.644824266, -0.517803729, -0.261999905, -0.0935142711, -0.751379013, -0.799664259, 0.643151999, -0.769358695, 0.847976506, -0.443437487, -0.865745246, -0.858112276, -0.0854891911, -1.02697647, -0.563964605, 0.411286235, 0.842776775, 1.00849998, -0.220893413, -0.981626332, 0.841228247, -0.869051933, 0.73721987, -0.918379188, 1.00327122, -0.807156563, -0.193718016, -0.772623658, -0.298070163, 0.800232887, 0.408133507, 0.10237436, -0.81515944, 0.44498387, -0.992741346, -0.829405427, -0.15128015, -0.957665145, 0.855219305, -0.923042595, 0.91937834, -0.727190614, 0.777058065, 0.503481328, 0.972717345, -0.792999089, -0.822783053, -0.0296000838, -0.585992575, -1.12478924, -0.65349859, -0.874615133, 0.915536702, -0.865022838, 0.221339598, -0.970219016, 1.03011489, 0.84404099, -0.551715434, -0.000462494208, -0.0881480724, 0.490943015, -0.596435547, 0.544950843, 0.780327618, -0.848713815, -0.504931509, -0.0493441261, -0.965847492, -0.611734152, 0.833947718, -0.779928863, 0.84698987, -0.719679296, -0.888860345, -0.78719759, 0.376279891, -0.800401151, -0.6475631, 0.0540541522, 0.832768381, 0.9913221, 0.254653513, -0.795210302, 0.997577786, -0.926730752, 0.821435809, -0.942105949, 0.994723082, -0.72533679, -0.56359762, -0.830534875, -0.425396651, 0.696741581, 0.705276668, 0.492563456, -0.682713509, 0.685139418, -0.979230583, -0.730480373, -0.522351742, -0.871768355, 0.934757829, -0.723052382, 0.686145604, -0.776319683, 0.605920911, 0.436274976, 0.982208431, -0.929778159, -0.781040549, -0.443694592, -0.353642136, -1.03009582, -0.60700202, -0.745918989, 0.890347838, -0.80710572, -0.0572710522, -0.957512915, 1.00621009, 0.74390775, -0.0205915701, -0.513214886, 0.290729761, 0.10205552, -0.485159516, 0.324673235, 0.780689418, -0.763284326, -0.0712349787, -0.312666744, -0.757450044, -0.674579918, 0.928880155, -0.809836447, 0.961747348, -0.572299957, -0.987814963, -0.665709257, 0.023009887, -1.01407897, -0.491111904, 0.149622276, 1.08481824, 0.813495457, 0.00918790232, -0.988933444, 1.01304257, -0.736413836, 0.713366389, -0.77714926, 0.821009994, -0.718455791, -0.168555468, -0.701443851, -0.444518983, 0.824483514, 0.520365894, 0.331536323, -0.614189804, 0.710616112, -0.939932823, -0.83276999, -0.291009218, -0.740746975, 0.901486218, -0.695580423, 0.65776825, -0.584751487, 0.806130409, 0.480656713, 0.858114123, -0.722780287, -0.544448256, -0.233940363, -0.551465988, -1.09826517, -0.818630636, -0.807670295, 0.881042957, -0.746888697, 0.240349904, -1.04861701, 0.950304866, 0.81671983, -0.239935473, -0.28998813, 0.0921261236, 0.112538286, -0.583798945, 0.515947223, 0.817176998, -0.814985335, -0.317915797, -0.12826775, -0.930432558, -0.836291254, 0.694228888, -0.778837502, 0.935540259, -0.656916857, -0.988335431, -0.956956387, 0.0137774618, -1.12964177, -0.770840764, 0.454703301, 1.08889341, 1.10114956, -0.233997151, -0.9160344, 1.13169825, -0.838038266, 0.851185322, -0.777538717, 0.859436929, -0.862704158, -0.293443888, -0.956585228, -0.420471996, 0.920131326, 0.579383135, 0.173871115, -0.793714345, 0.735676169, -0.859370768, -1.05058193, -0.135776535, -1.05294931, 0.923585951, -0.962093055, 0.725955009, -0.728679836, 0.920734346, 0.429953694, 1.19835913, -0.917490304, -0.828156948, -0.125764608, -0.670550227, -1.15649199, -0.902004242, -0.842370331, 1.06699336, -0.965167105, 0.349797368, -0.910021544, 0.997987449, 0.791344106, -0.4023, -0.198947266, 0.0677236542, 0.388899982, -0.614362538, 0.507743657, 1.02602351, -0.830910623, -0.515007615, -0.0185752213, -0.92261529, -0.795056403, 0.738663793, -0.766319156, 0.822949409, -0.655317307, -0.93890965, -0.991864741, 0.326603681, -0.930119216, -0.815422237, -0.109608583, 0.934924841, 0.920461893, 0.35182032, -1.03809893, 1.10397971, -0.883284926, 0.994623005, -1.07502925, 1.05005991, -0.829090774, -0.672549129, -0.804675579, -0.568975568, 0.760407686, 0.737354517, 0.703553975, -0.8440485, 0.720817268, -0.91479063, -0.810900331, -0.507740676, -1.06939578, 0.840505183, -1.08498955, 0.917757034, -0.803289056, 0.911749065, 0.413806319, 0.992159247, -0.918016732, -0.710864782, -0.431193411, -0.444666862, -1.07377923, -0.78019011, -0.840355754, 0.860853255, -0.819990814, -0.260453254, -1.1637423, 0.952289402, 0.863986433, -0.0693490952, -0.43248719, 0.455752134, -0.168676227, -0.297006905, 0.378284246, 1.08168149, -0.759329259, -0.00800242741, -0.520838499, -1.0476948, -0.675572634, 0.885056794, -0.778042734, 0.970966935, -0.739053071, -1.18367076, -1.00170863, 0.515894175, -1.04622996, -0.734378457, -0.0634912625, 1.05683684, 1.13232851, 0.479658991, -1.14697683, 1.14479041, -1.14973688, 0.966424525, -1.11149096, 1.02778423, -0.863198936, -0.751709819, -0.888835311, -0.804755151, 0.858745933, 0.760714173, 0.756437302, -1.01159966, 0.79420507, -0.995307148, -0.96403861, -0.779833555, -1.0982914, 0.976376057, -0.940571666, 1.07449925, -0.787972987, 0.893660724, 0.253314584, 1.15125144, -0.931932032, -0.726671219, -0.747295558, -0.29423061, -1.28276575, -0.797924876, -0.918390751, 1.14562893, -0.875937521, -0.149294049, -1.15881169, 0.992793918, 0.796081841, 0.0344517604, -0.689107001, 0.556009471, -0.0333260484, -0.188356966, 0.273446709, 1.0719341, -0.849202156, -0.0576614663, -0.497593015, -0.946819425, -0.795422435, 1.04014468, -0.872544289, 1.03207433, -0.746326625, -1.02014303, -0.913138747, 0.174102426, -0.961304426, -0.703736424, 0.142996088, 0.887258172, 1.06656015, 0.0410478935, -0.815817237, 1.11459541, -0.986689091, 0.869543433, -0.807072699, 1.02771664, -0.741206229, -0.168933392, -0.840292573, -0.516178131, 0.788471043, 0.654079497, 0.241704389, -0.678604484, 0.690058768, -0.985296369, -0.889898062, -0.42652756, -0.942365468, 0.840480506, -0.84049958, 0.685397267, -0.654555202, 0.743690073, 0.498869985, 0.984338284, -0.931772113, -0.667692959, -0.149191111, -0.586353421, -1.2004689, -0.613616288, -0.750702798, 1.02661479, -0.968156934, 0.27459839, -1.09536994, 0.869792044, 0.795942605, -0.170552939, -0.119759001, 0.0561317392, 0.298612505, -0.487057149, 0.431264818, 0.776092827, -0.863675654, -0.31945172, -0.222689167, -0.939694643, -0.881493151, 0.77813375, -0.859104395, 0.980753601, -0.835472226, -0.780811608, -0.908254683, -0.0700671524, -0.95471555, -0.243140265, 0.656840563, 0.788265705, 0.808628798, -0.287140399, -0.73185581, 0.784762442, -0.899206996, 0.664094448, -0.895017982, 0.714929521, -0.709218681, -0.0350017548, -0.476985365, -0.132147655, 0.395060271, 0.278724641, 0.0243162718, -0.786040306, 0.254208386, -0.678958178, -0.484509289, -0.143013015, -0.938613236, 0.934693396, -0.907608032, 0.640249074, -0.42963931, 0.273129761, 0.511628985, 0.767143548, -0.835145712, -0.839953721, 0.0871558934, -0.592077434, -0.865831912, -0.400098443, -0.678308547, 0.920655668, -0.61952275, 0.457279861, -0.751586497, 0.815800011, 0.471407712, -0.510838628, -0.0146660823, 0.0550350286, 0.52525425, -0.518903434, 0.713679194, 0.761300564, -0.625218272, -0.626365364, -0.0270288847, -0.688027024, -0.415846318, 0.709429741, -0.505770206, 0.885988295, -0.633718252, -0.976370275, -0.805604398, 0.369813204, -1.09729612, -0.631916106, 0.0831616595, 0.925421715, 0.985631824, 0.132714882, -1.04596221, 0.945217013, -1.06315434, 0.974209487, -1.01574898, 1.08618009, -0.712410092, -0.450384706, -0.97908324, -0.498778701, 0.673285246, 0.646217763, 0.311322898, -0.774297357, 0.543726921, -0.994351029, -0.768154562, -0.448112994, -1.03144801, 1.08958042, -0.900835633, 0.93874824, -0.792783737, 0.862766981, 0.478894234, 0.927475333, -0.916345716, -0.760724545, -0.405634254, -0.749832273, -1.10986936, -0.626981199, -0.970400333, 0.897742629, -0.854419649, 0.0998076871, -0.885941565, 1.02640998, 0.810763836, -0.172908932, -0.219355851, 0.166053206, 0.361918479, -0.608354628, 0.483504057, 1.00468135, -0.954490066, -0.276456952, -0.409829766, -0.833084106, -0.650721133, 0.763146698, -0.666514695, 1.06439698, -0.975921452, -0.976468682, -0.791674674, -0.177903861, -0.843917489, -0.267525673, 0.634957194, 0.920786977, 0.971808851, -0.392000765, -0.850517333, 0.800255775, -0.802226901, 0.909082353, -0.877137661, 0.730122745, -0.851397216, -0.0722328052, -0.537836909, -0.187319443, 0.36514619, 0.253046304, 0.10816586, -0.727519393, 0.41508621, -0.938324273, -0.499514312, -0.12158455, -0.918444216, 0.761836886, -0.689384639, 0.710212231, -0.410224855, 0.548989832, 0.634191751, 0.939039767, -0.704807699, -0.801940441, 0.0953865424, -0.540097415, -1.03223205, -0.523439586, -0.819470525, 0.860700846, -0.656160235, 0.297524452, -0.947977126, 0.90694356, 0.621159196, -0.502045631, -0.0506013669, -0.123203866, 0.503702044, -0.652031302, 0.529158711, 0.842695534, -0.672055542, -0.543978214, 0.20170027, -0.951138258, -0.517390072, 0.885154307, -0.364636242, 0.83135426, -0.658487439, -0.968474865, -0.622928381, 0.308044612, -0.946219087, -0.729095697, -0.020170588, 0.929763079, 0.992177188, 0.0572009496, -0.789075613, 0.864978194, -0.953618169, 0.711665154, -0.742936492, 0.943210602, -0.633800924, -0.483225018, -0.829375863, -0.47125262, 0.61733675, 0.571785808, 0.56263268, -0.589145005, 0.645672798, -0.800022244, -0.656003237, -0.306997836, -0.753312528, 0.707771122, -0.822233975, 0.788333774, -0.610611498, 0.576294065, 0.368350208, 0.956656158, -0.788423836, -0.574761868, -0.428307831, -0.336391181, -0.882566571, -0.633512914, -0.797103524, 0.918003321, -0.843789279, -0.0639619157, -0.80085057, 0.995271385, 0.673964679, -0.0921275243, -0.465578198, 0.266843677, 0.156025752, -0.212184533, 0.420018256, 0.712551475, -0.611166835, 0.0293651894, -0.373225451, -0.869483173, -0.824524105, 0.650054216, -0.835338175, 0.69953686, -0.733144045, -0.94825989, -0.829286873, 0.498820007, -1.10125899, -0.934159279, -0.237553403, 1.17959416, 1.00506413, 0.241874829, -1.10324156, 1.08897948, -1.04178441, 0.961241484, -1.05229485, 1.16768396, -0.701199234, -0.684071183, -0.882459939, -0.842701197, 1.0047071, 0.993355274, 0.698987246, -0.736815214, 0.930523276, -1.00445724, -0.908867478, -0.62573576, -0.918404937, 0.990144253, -1.01239693, 0.988601685, -0.930237651, 0.933457732, 0.253664821, 1.04263794, -0.863427281, -0.590768814, -0.540168464, -0.446616054, -1.17079878, -0.859642208, -0.895760119, 0.942056179, -1.00492251, -0.170379594, -1.21758735, 1.19851482, 0.993596911, 0.113135502, -0.49006626, 0.397776872, -0.213488877, -0.203544989, 0.229960397, 1.05145907, -0.759326816, -0.055846002, -0.525532544, -0.943355918, -0.8732934, 1.04964459, -1.01602924, 0.884545803, -0.781898618, -0.723886073, -0.62977469, -0.204483747, -0.829271317, -0.245969415, 0.436119974, 0.811825335, 0.602030814, -0.28100431, -0.742344499, 0.827918768, -0.690657675, 0.799997211, -0.829492569, 0.817033291, -0.544541478, 0.0358796567, -0.484106064, -0.0552955978, 0.382008195, 0.129058108, 0.0748274773, -0.628724813, 0.250387967, -0.706169128, -0.34636569, -0.116365537, -0.719126046, 0.759861112, -0.715697706, 0.609559476, -0.281813145, 0.249621287, 0.675493002, 0.778470099, -0.730745196, -0.775118828, -0.0318290442, -0.635053277, -0.64971602, -0.264338791, -0.766497374, 0.836210966, -0.335421443, 0.336263001, -0.797662616, 0.600033104, 0.447682649, -0.477033317, -0.00602800678, -0.00347518804, 0.343229294, -0.595320761, 0.690001249, 0.743430614, -0.678604662, -0.573144078, -0.00853874814, -0.787870467, -0.398957372, 0.805735111, -0.208311886, 0.579948843, -0.63110131, -0.929738283, -0.772374809, 0.271806598, -1.01329947, -0.858100355, 0.452278465, 0.916744471, 1.14639127, -0.0263592731, -1.10906065, 1.10039926, -0.990095317, 0.872081578, -1.00980031, 1.0308758, -0.929622769, -0.465474278, -1.04688621, -0.639739394, 0.931501687, 0.756015897, 0.321964175, -0.837107778, 0.727318883, -0.864199638, -0.92858845, -0.460382283, -1.00176477, 1.08890307, -0.86653173, 0.931799054, -0.745827913, 0.919408202, 0.704915285, 0.975672781, -0.900074422, -0.817533493, -0.44180873, -0.754927456, -1.14283717, -0.874060333, -0.996847332, 0.962824225, -1.00731623, 0.143175423, -1.13962972, 0.926433623, 0.944086671, -0.256617039, -0.177992538, 0.234126672, 0.226686522, -0.728595674, 0.598063231, 1.08225262, -0.801509559, -0.299066722, -0.216455579, -1.04918098, -0.889964759, 0.808224797, -0.858967721, 1.00894785, -0.893621087, -1.11113048, -0.911374986, 0.0543966405, -1.00301683, -0.733756423, 0.162385717, 1.0429635, 0.924938262, 0.0733157992, -0.956732213, 1.098562, -0.887375534, 0.966252506, -0.887113035, 1.02406406, -0.76543504, -0.400138885, -0.833865285, -0.589645863, 0.911189914, 0.675319374, 0.241477102, -0.848621309, 0.712136924, -0.961093903, -0.76611954, -0.396515459, -0.87194252, 1.02525055, -0.935948014, 0.96596688, -0.670312822, 0.669189751, 0.521194339, 0.981858134, -0.923735201, -0.834396899, -0.380213201, -0.490119696, -1.01803303, -0.837935627, -1.01692939, 0.893213272, -0.890941322, 0.0512234196, -0.938236773, 1.12978613, 0.822078764, -0.381286681, -0.354263991, 0.140916765, 0.279109687, -0.467644393, 0.549917936, 0.861881733, -0.847081482, -0.202907324, -0.183476627, -0.885915756, -0.69544071, 0.890836477, -0.817651927, 0.933344722, -0.846282125, -1.03862607, -0.947054029, 0.0615682788, -1.11174715, -0.548233747, 0.256683737, 1.14824474, 1.03675997, -0.306727588, -0.964119434, 0.973472714, -0.999305964, 0.839141071, -0.847896695, 0.932551801, -0.85014081, -0.284629256, -0.997696638, -0.367976367, 0.86989969, 0.621583104, 0.341185182, -0.79054755, 0.637244344, -0.795998812, -1.03838813, -0.121878378, -1.02120984, 1.03450096, -0.847081721, 0.791102886, -0.929135621, 0.91503346, 0.493659556, 1.08521104, -0.794698179, -0.783615708, -0.149818674, -0.577271104, -1.22717381, -0.729105532, -0.907890081, 0.904237509, -0.840050995, 0.355233908, -1.16810739, 1.03836215, 0.833904982, -0.270463109, -0.190144002, 0.053217493, 0.424836487, -0.619497418, 0.575297952, 0.876965404, -0.721707761, -0.473643988, -0.0170233063, -0.972761631, -0.806016803, 0.886822879, -0.859126747, 0.807136118, -0.873356402, -0.532830179, -0.612299204, -0.122964926, -0.61621964, -0.069940798, 0.433616072, 0.501196623, 0.503526568, -0.233648106, -0.60350734, 0.448003024, -0.501408577, 0.619695842, -0.559005618, 0.637978077, -0.461325794, 0.105104662, -0.2573511, -0.186585173, 0.354441494, 0.0737063959, -0.0460065231, -0.527710378, 0.219412535, -0.493068904, -0.205879152, 0.105828926, -0.675325096, 0.475340486, -0.548010886, 0.423154175, -0.336760581, 0.255975366, 0.460904866, 0.59745276, -0.58728838, -0.609239519, -0.103507549, -0.399057329, -0.407381773, -0.241226628, -0.419427693, 0.671428859, -0.44988206, 0.220640793, -0.421603203, 0.538674831, 0.297478944, -0.44234702, 0.0603176206, 0.0442613475, 0.371121526, -0.471603364, 0.439350307, 0.667813361, -0.391252607, -0.265212685, 0.00789033435, -0.435489267, -0.239340037, 0.593510747, -0.247391731, 0.534566224, -0.603185236, -0.792371094, -0.739380062, 0.713901758, -0.817053378, -0.852856994, -0.179341659, 0.959845006, 0.770885408, 0.324391484, -0.854621291, 0.786259651, -0.661624253, 0.757754922, -0.741588593, 0.824353218, -0.569926322, -0.575232327, -0.886677504, -0.837767422, 0.783255398, 0.733940661, 0.607587218, -0.757613301, 0.867251217, -0.983041406, -0.95171237, -0.758144796, -0.83637464, 0.595348895, -0.936923146, 0.668096066, -0.798557997, 0.725486815, 0.424645394, 0.707889974, -0.665016055, -0.47084704, -0.67993921, -0.375449032, -0.918146729, -0.776643753, -0.827958047, 0.819822788, -0.888391256, -0.210734129, -0.90350759, 0.928226888, 0.923699737, 0.104914516, -0.624729991, 0.554213703, -0.303485304, -0.377347738, 0.128166661, 0.864066422, -0.585147917, 0.200534806, -0.728587449, -0.80727452, -0.68116796, 0.707198918, -0.795398533, 0.679158926, -0.710352719, -0.962701142, -0.812521577, 0.127895594, -0.848725259, -0.558891773, 0.243628547, 0.956765711, 0.816756129, 0.108055905, -0.944031239, 1.00386214, -0.892733634, 0.766236484, -0.806172073, 0.940659046, -0.641631424, -0.318218708, -0.931178689, -0.340961009, 0.828006566, 0.722664773, 0.248382315, -0.824228764, 0.508430898, -0.891737044, -0.878963828, -0.301210672, -0.746851981, 0.863421857, -0.857524335, 0.777775943, -0.735813081, 0.728388309, 0.34783417, 0.965335965, -0.786547422, -0.812392235, -0.321248323, -0.538291335, -1.09552181, -0.805899978, -0.891295195, 0.924740314, -0.796732783, 0.0918886662, -1.09573889, 0.823742509, 0.724403679, -0.32133618, -0.198802829, 0.122519381, 0.0665191114, -0.591669798, 0.354328364, 0.860146463, -0.769168377, -0.328037053, -0.152577445, -0.765176296, -0.798249722, 0.721755147, -0.802870333, 0.974007308, -0.765210569, -1.02971113, -0.863262057, 0.294929892, -0.873904765, -0.668876112, 0.224371701, 0.850640297, 1.01778233, -0.0772373825, -0.797427595, 1.05826008, -0.930305243, 0.792840004, -0.764625669, 0.843560815, -0.631143749, -0.3468557, -0.82498461, -0.365978032, 0.778761089, 0.538974524, 0.40057835, -0.742695212, 0.532127142, -0.897926211, -0.93071723, -0.499519289, -0.883000612, 0.792768776, -0.867752314, 0.751485407, -0.818368495, 0.623130143, 0.346275657, 1.03179812, -0.977597117, -0.863486946, -0.480615079, -0.519268036, -1.00494742, -0.667935312, -0.914928854, 0.873737097, -0.858839393, -0.0702849999, -1.06019449, 1.0806725, 0.772564471, -0.251107931, -0.252646863, 0.3580468, 0.136758775, -0.557268441, 0.447885424, 0.954984426, -0.92693764, -0.222680256, -0.201380536, -0.79762882, -0.641146898, 0.73164171, -0.804575026, 1.01352036, -0.876159906, -0.993184566, -0.791009843, 0.504641533, -0.921791077, -0.816360116, -0.196006298, 1.17310393, 1.05226195, 0.382271826, -0.894057274, 0.984008789, -1.09940231, 1.00387776, -1.00434065, 0.94280237, -0.691696286, -0.81867069, -0.82539314, -0.828855813, 0.80027622, 0.888840199, 0.800766945, -0.748210132, 0.834859431, -0.880362272, -1.03611803, -0.686120629, -1.06963181, 1.07744288, -1.03263533, 0.885977745, -0.782256365, 0.808066666, 0.316192836, 1.15501893, -0.884240448, -0.611134648, -0.812284827, -0.347036064, -1.00437868, -0.841145515, -0.869562924, 0.925918996, -1.00450277, -0.273400426, -1.16757858, 0.982424915, 0.847116649, -0.0370410681, -0.546299517, 0.568685651, -0.237957954, -0.110121593, 0.262624055, 1.06115329, -0.711271048, 0.201648265, -0.638166785, -0.890225887, -0.771624029, 0.82232964, -1.02269852, 0.905648887, -0.859919012, -1.01018035, -0.852937341, 0.199344724, -1.02075493, -0.557302475, 0.122542568, 1.04583883, 1.05831313, -0.131008953, -1.04885328, 1.13267505, -0.973243535, 0.892987728, -0.859983087, 1.00251496, -0.922155261, -0.49669224, -0.813681483, -0.459259152, 0.90394032, 0.520107567, 0.40480119, -0.884002805, 0.734116495, -0.846735358, -0.961679697, -0.353904635, -0.985855341, 0.886004329, -0.976658583, 0.887159467, -0.660021305, 0.760787725, 0.630375803, 1.00861239, -0.990624189, -0.776782095, -0.300165325, -0.613854587, -1.16555989, -0.739156306, -0.887333751, 1.07783723, -0.886344194, 0.183636725, -1.04426599, 0.903318882, 0.800231457, -0.209712222, -0.32627964, 0.352689356, 0.333587348, -0.646154046, 0.6284917, 1.00177336, -0.7466923, -0.262597769, -0.228939399, -0.921233594, -0.690168798, 0.961507738, -0.825392723, 0.950034082, -0.894637525, -1.07029724, -0.74155581, -0.110260643, -1.01186144, -0.467203647, 0.419715881, 1.02206957, 1.06065667, -0.193051681, -1.01871479, 1.04745793, -0.969526291, 0.882115364, -0.793250442, 1.00953889, -0.881716251, -0.285185963, -0.733971596, -0.430095583, 0.666744351, 0.537245572, 0.197210357, -0.820546985, 0.478942424, -0.867832482, -0.904418588, -0.306358516, -0.987072885, 0.923965573, -0.827970445, 0.942754388, -0.813830674, 0.810630918, 0.598882854, 0.965327322, -0.958405077, -0.789805353, -0.0247831345, -0.64611125, -1.0609479, -0.646289349, -0.943482101, 0.90460068, -0.898542881, 0.241582885, -1.05070531, 0.839297295, 0.659592569, -0.306077451, 0.0500512682, -0.0570018664, 0.510157228, -0.61130023, 0.708471656, 0.852460563, -0.701989949, -0.37463814, 0.00335903093, -1.03780794, -0.670634925, 0.787285209, -0.635788918, 0.847452581, -0.702324629, -1.005234, -0.968812108, 0.447139084, -1.17164814, -0.869274616, -0.0655961037, 0.966442049, 0.993079126, 0.415281653, -1.0261327, 1.03079224, -0.937661529, 0.961169541, -1.15573311, 1.12316489, -0.947063088, -0.609770119, -0.827906549, -0.691708922, 0.942700982, 0.827459455, 0.576645792, -0.842250884, 0.842586279, -1.15715313, -0.955552638, -0.59762311, -1.01382136, 1.08575153, -0.963505149, 1.00307536, -0.936788976, 0.826114357, 0.386973441, 0.980013311, -0.95651722, -0.925170422, -0.611601055, -0.611125529, -1.0324471, -0.726434052, -0.87263602, 1.10575986, -0.897451043, -0.208583012, -1.07795715, 1.14604986, 0.928188145, -0.0521513931, -0.618541777, 0.59916842, -0.193706781, -0.415743053, 0.440905035, 1.14346862, -0.926543593, -0.0363977067, -0.477990896, -0.982643366, -0.867311776, 0.935358524, -0.973981082, 0.931315124, -0.845630407, -0.861772954, -0.721524179, 0.0986454412, -1.03133488, -0.570533097, 0.261758417, 0.965813875, 0.982137144, -0.0293426253, -1.03436482, 1.06985724, -0.950913906, 0.922353983, -0.806497097, 0.783380806, -0.658890784, -0.449607164, -0.89537859, -0.385259211, 0.713460863, 0.729782641, 0.473796427, -0.924663186, 0.578554451, -0.803543389, -0.671633184, -0.382577837, -0.8009305, 1.00022399, -0.933638573, 0.836028934, -0.563164771, 0.629320562, 0.546176434, 0.915136099, -0.869614005, -0.753042638, -0.4967058, -0.524411798, -0.951225638, -0.611946225, -0.92792213, 1.05263615, -0.89749366, 0.0132358298, -1.11050832, 0.983382344, 0.854296625, -0.182954162, -0.181268334, 0.198000371, 0.302228659, -0.43596226, 0.403358847, 0.850450814, -0.853324413, -0.220359758, -0.166480929, -0.943998992, -0.767611206, 0.848755598, -0.657482505, 0.841426432, -0.721938431, -0.808539927, -0.923175871, 0.05690597, -0.875962317, -0.495678008, 0.557142079, 0.931773603, 0.924619436, -0.44155696, -0.836186647, 1.08503079, -0.938528895, 0.992791533, -0.907654107, 1.02695823, -0.728081107, -0.0550730638, -0.679002643, -0.221366316, 0.680275738, 0.391920954, 0.214570433, -0.699837446, 0.654629827, -0.907504678, -0.761733353, -0.138699621, -0.858287454, 0.829922318, -1.01176488, 0.793316185, -0.719401836, 0.715198278, 0.698503673, 1.03310657, -0.94738251, -0.69627142, 0.00782040507, -0.652584016, -1.15452898, -0.698288977, -0.787849724, 1.0273881, -0.834000468, 0.372734994, -1.11593997, 0.926637769, 0.772196352, -0.35649237, 0.12004476, 0.0972433984, 0.553599775, -0.4949072, 0.76016742, 0.810973287, -0.905270457, -0.523971677, 0.0969828069, -0.832741797, -0.768331468, 0.775760949, -0.682405889, 0.883137941, -0.85619998, -0.989380658, -1.03457499, -0.0517622754, -0.932550669, -0.694942057, 0.528805315, 0.975854874, 0.958423674, -0.140165061, -1.08478153, 1.1421417, -0.970185518, 0.968834043, -0.844599009, 1.11847758, -0.774316072, -0.211446851, -0.861546516, -0.456038833, 0.966504276, 0.710692942, 0.214514136, -0.992433667, 0.674419701, -0.838600397, -0.797830403, -0.452291369, -0.87957257, 0.952979147, -1.04137182, 0.756499469, -0.881576478, 0.697081447, 0.495766819, 1.02677464, -0.817020655, -0.823269069, -0.18381232, -0.535384774, -1.06303358, -0.883768439, -0.897187591, 1.11861014, -0.870897472, 0.187550664, -1.03782761, 1.17324579, 0.888868153, -0.341810137, -0.0556954741, -0.0158871058, 0.322948873, -0.588214874, 0.501251698, 1.04257047, -0.742597222, -0.393232524, -0.0918072313, -0.945177972, -0.824784875, 0.926980078, -0.747276783, 0.995664954, -0.691841543, -1.00853765, -0.713255107, 0.647285819, -0.852226436, -0.846004665, -0.168666676, 0.902311683, 0.944902182, 0.267628074, -0.958007157, 0.840322256, -0.887698829, 0.961279511, -0.776420653, 0.94608885, -0.862158537, -0.605205178, -0.915220797, -0.628228426, 0.848300576, 0.839160681, 0.57141012, -0.905398667, 0.858483016, -0.889531493, -0.82938236, -0.598610878, -0.968016028, 0.819422901, -0.985393584, 0.842359126, -0.748422325, 0.876093566, 0.386232138, 0.704279602, -0.881875217, -0.762673676, -0.629377842, -0.501640975, -0.807521403, -0.884190679, -0.717874348, 0.913320184, -0.892254114, -0.298563749, -0.930075765, 0.775691807, 0.863675773, 0.125792608, -0.618853033, 0.577705622, -0.0251189768, -0.432866186, 0.377281308, 0.980280399, -0.649286807, -0.0607887618, -0.45323652, -0.968550265, -0.698687017, 0.831464946, -0.749712884, 0.786249042, -0.669413984, -0.700759172, -0.690960705, 0.219630286, -0.874300182, -0.59967339, 0.000577162486, 0.755742371, 0.729254723, 0.199102446, -0.876938522, 0.794218957, -0.663940489, 0.733607531, -0.698495746, 0.885335922, -0.571763039, -0.293765396, -0.804308891, -0.550076067, 0.569750428, 0.615945041, 0.313869447, -0.587247789, 0.688019931, -0.895350873, -0.723046601, -0.452467203, -0.820372641, 0.6793347, -0.766393602, 0.565901518, -0.507283568, 0.568262339, 0.415052295, 0.915370524, -0.716443479, -0.424843311, -0.460298181, -0.361261994, -0.903628588, -0.648115396, -0.738555253, 0.800467253, -0.795145512, -0.0115165636, -0.944992721, 0.889130592, 0.767579377, -0.139246643, -0.375697315, 0.36367327, 0.143317923, -0.265599102, 0.306399882, 0.68444252, -0.647032976, -0.108279914, -0.276576221, -0.652727604, -0.799071014, 0.564529896, -0.729636312, 0.606915534, -0.580234945, -0.774507999, -0.857604742, 0.429399729, -0.930867374, -0.651145041, -0.0314018019, 0.9284513, 0.950723827, 0.181736708, -0.94284606, 0.777048528, -0.899705112, 0.752479076, -0.709820509, 0.953935325, -0.536857426, -0.453155041, -0.679491878, -0.604841769, 0.783517122, 0.599752367, 0.318136007, -0.594205081, 0.676581621, -0.877049088, -0.731319427, -0.511449099, -0.862341225, 0.892369747, -0.814184546, 0.754008353, -0.715054214, 0.698685884, 0.233145103, 1.01863647, -0.690535367, -0.589026153, -0.334243953, -0.220951915, -0.930629253, -0.559661031, -0.749486089, 0.953985274, -0.831374645, -0.0278570782, -0.82597959, 0.771127641, 0.682325423, 0.0170961022, -0.279765844, 0.382275105, -0.023843443, -0.234016284, 0.137231991, 0.922935069, -0.595442712, 0.0992795452, -0.49003467, -0.927733064, -0.688692808, 0.736590385, -0.632792711, 0.925248921, -0.613666236, -1.16928852, -0.854762793, 0.0468913354, -1.18165219, -0.781460166, 0.331295043, 1.18376422, 1.15690267, -0.241335928, -1.13221955, 1.17465961, -1.12600315, 0.85642612, -1.0159322, 1.13213372, -0.90468365, -0.414374441, -0.809111953, -0.528228104, 0.830214083, 0.714342952, 0.362617999, -0.976914048, 0.72939831, -1.04324293, -0.884737849, -0.339856893, -0.906443477, 0.955860972, -1.04917729, 0.858124316, -0.725417972, 0.743358731, 0.585490286, 1.20731747, -0.850624859, -0.874786615, -0.405697405, -0.565402925, -1.04332829, -0.759941936, -0.922682583, 1.02715707, -1.02701879, 0.190939397, -1.04053569, 1.0984509, 0.769177556, -0.344820887, -0.306929022, 0.040846061, 0.500335574, -0.723776221, 0.589993179, 0.981675565, -0.991475999, -0.425548941, -0.117642395, -0.915643394, -0.815215707, 0.916038752, -0.969600379, 1.12809849, -0.751632512, -0.862899303, -0.829141974, -0.0570159368, -0.737937391, -0.273056149, 0.489814162, 0.882974625, 0.689721644, -0.325598091, -0.854503095, 0.690012515, -0.717048287, 0.858363569, -0.755031466, 0.654838562, -0.727559149, 0.116936356, -0.403147727, -0.0911585465, 0.421337515, 0.204730436, -0.0789451748, -0.842997909, 0.138907969, -0.854771733, -0.345312566, 0.0786507577, -0.880420327, 0.7018255, -0.648191214, 0.608898759, -0.424877197, 0.386772513, 0.689378798, 0.812096119, -0.645421565, -0.738684177, 0.092786476, -0.520626843, -0.807718277, -0.174863353, -0.81000948, 0.828145087, -0.413771659, 0.345121145, -0.790848255, 0.682513893, 0.404779643, -0.457731128, 0.234948263, -0.0156717561, 0.387670338, -0.727176011, 0.640328646, 0.74883163, -0.835190475, -0.563892007, 0.0542730503, -0.864046574, -0.342467546, 0.816046357, -0.424440503, 0.70988059, -0.637702584, -0.937841892, -0.889083564, 0.268207818, -0.805704176, -0.721465349, -0.00490556099, 0.901388884, 0.80767101, 0.213178098, -0.751282811, 0.899395168, -0.725854814, 0.748562276, -0.986488461, 1.00970292, -0.628750443, -0.404512465, -0.834999561, -0.666034818, 0.780131698, 0.580195248, 0.443588674, -0.779767275, 0.75757575, -0.764169872, -0.708934724, -0.357157409, -0.990183473, 0.773827612, -0.729798257, 0.909026921, -0.786345541, 0.774623275, 0.468835086, 0.890515149, -0.753928065, -0.60978061, -0.565818489, -0.363415778, -0.886048853, -0.586931825, -0.881760061, 0.751504302, -0.743851066, -0.00649144407, -0.97195828, 0.961859286, 0.657981575, 0.0401829779, -0.278608352, 0.372902483, -0.131196737, -0.36559844, 0.192959338, 0.882446885, -0.665415108, -0.139419302, -0.510242403, -0.971634388, -0.814798832, 0.688571632, -0.67599684, 0.900357485, -0.822175205, -1.1110909, -0.866408885, 0.537440896, -0.982464671, -0.892360926, -0.0193753131, 1.1145103, 0.985346854, 0.177099958, -0.932675481, 1.0265522, -0.955097854, 0.866545022, -0.951171875, 0.936732709, -0.586589515, -0.753251791, -0.954349875, -0.913152814, 0.846741498, 0.921646535, 0.601255655, -0.841526389, 0.821996033, -1.10704231, -0.938263834, -0.786375642, -0.959054649, 1.06783462, -0.897728741, 0.715040922, -0.954261363, 0.90016979, 0.314348668, 1.08457112, -0.897332907, -0.586558402, -0.513837397, -0.468146712, -1.04694176, -0.997831762, -0.988519728, 1.08274424, -1.03911412, -0.0763379037, -1.19924867, 1.13884616, 0.861875355, -0.035394527, -0.645141602, 0.540617466, -0.00713570463, -0.398186237, 0.188419178, 0.941889644, -0.585887313, 0.0222373828, -0.59352988, -0.954482138, -0.827650249, 0.993924975, -1.01277149, 1.00802708, -0.588631153, -1.02202189, -0.747009635, 0.613322556, -0.897544682, -0.732982278, -0.456595093, 0.962276399, 0.795332074, 0.671077371, -0.967659414, 0.853868723, -0.770793259, 0.833329558, -0.97578615, 0.848643482, -0.857904911, -0.798365831, -0.795888245, -0.857467532, 0.966209948, 0.736484468, 0.695706427, -0.886226654, 0.788673043, -1.01052272, -1.0286032, -0.748519123, -1.0185672, 0.874143004, -1.06077802, 0.694009662, -0.843938947, 0.878933787, 0.349594027, 0.800177395, -0.717908025, -0.594196796, -0.656258881, -0.556953669, -0.846859157, -0.79142803, -0.845962942, 1.04326403, -0.868588626, -0.562533617, -0.85183394, 1.01098347, 0.952204704, 0.282487959, -0.872518361, 0.721074104, -0.31151703, -0.378997952, 0.282929897, 1.03048205, -0.549017072, 0.0635976419, -0.835636377, -0.912023246, -0.88585341, 0.776455045, -0.85138154, 0.971118808, -0.843461335, -0.921734393, -0.891871095, 0.215065777, -0.998061776, -0.627441168, -0.00694472902, 0.936757505, 0.960935533, 0.124367289, -0.888317347, 0.825734615, -0.937575281, 0.886772931, -0.929073453, 0.91916132, -0.616435409, -0.292480201, -0.790857792, -0.357805163, 0.654396594, 0.474305242, 0.45884648, -0.80382973, 0.717312634, -0.807204485, -0.658123434, -0.377325684, -0.822481692, 0.724415779, -0.953108728, 0.76014626, -0.693366945, 0.563358843, 0.411203325, 1.03892446, -0.712390542, -0.538339972, -0.27133134, -0.402222306, -0.99378258, -0.604566932, -0.665674448, 0.884491324, -0.862252116, -0.0283179767, -0.967720449, 1.02005899, 0.699623823, -0.192977205, -0.361554682, 0.226021931, 0.0313617177, -0.443519056, 0.394279808, 0.711178541, -0.585805237, -0.0763858184, -0.431294441, -0.882086337, -0.688799143, 0.765866399, -0.600738764, 0.872073233, -0.585193992, -1.14066052, -1.01628506, 0.468449682, -1.05726838, -0.758302093, -0.319746405, 1.06616163, 1.23968601, 0.471936852, -1.17176759, 1.14338076, -1.0373919, 1.01719534, -1.04405451, 1.15122747, -0.736556053, -0.817210734, -0.87207818, -0.880215645, 0.807342827, 0.825081289, 0.657493591, -0.826831758, 0.96656388, -1.18908823, -0.881948113, -0.884769559, -1.16256285, 1.16519034, -1.12716424, 1.03457212, -0.750531316, 0.834807634, 0.189688057, 1.15967309, -0.925843418, -0.622301936, -0.56216079, -0.412126422, -1.16535819, -0.798312604, -0.987665236, 1.16538191, -1.06542087, -0.114130765, -1.16750205, 1.01994395, 0.928645372, -0.0757360235, -0.509201884, 0.527584434, -0.276150465, -0.224989578, 0.251699209, 1.17536449, -0.669173241, -0.0418375544, -0.71047467, -1.13567662, -0.879538894, 0.937010527, -0.958074749, 1.07342601, -0.771591127, -0.898289621, -0.610124648, 0.23924163, -0.769600093, -0.548261344, 0.402057856, 0.92328161, 0.74641782, -0.33475405, -0.734599233, 0.875175834, -0.87895298, 0.725653946, -0.902100265, 0.764896214, -0.69176358, -0.284559339, -0.494734585, -0.365131497, 0.588428736, 0.344578713, 0.193848446, -0.673172235, 0.547721148, -0.726282358, -0.504092455, -0.417677313, -0.798350036, 0.632530272, -0.857168376, 0.615213275, -0.581914425, 0.578558266, 0.447241008, 0.771184087, -0.820596159, -0.715781569, -0.222367719, -0.712529957, -0.773471415, -0.446331292, -0.862668872, 0.708845675, -0.646493077, 0.343099028, -0.872348428, 0.842768073, 0.437714696, -0.387816608, -0.235918418, 0.238533229, 0.552209973, -0.447900772, 0.586615801, 0.89375782, -0.769779444, -0.455967426, -0.135496899, -0.746009052, -0.653398037, 0.863333583, -0.598646224, 0.710586071, -0.793436229, -0.794035196, -0.644094527, 0.158939242, -0.80322212, -0.477397323, -0.115651518, 0.893703222, 0.991062164, 0.223283187, -0.98810339, 0.848653674, -0.782176256, 0.809766829, -0.796902239, 0.859373271, -0.733840704, -0.315199107, -0.655109882, -0.388337314, 0.85081476, 0.512403607, 0.541898727, -0.789254367, 0.632047057, -0.869125187, -0.689603567, -0.417844146, -0.786599994, 0.844494522, -0.717500627, 0.836738884, -0.683015943, 0.688111186, 0.353871852, 0.881329238, -0.823342502, -0.67863524, -0.404293686, -0.423918992, -0.942907155, -0.587039173, -0.631044865, 0.86594981, -0.908970654, -0.0822079778, -0.929236293, 0.992730558, 0.59928304, -0.179815695, -0.406772912, 0.410552382, 0.0469524488, -0.216171399, 0.170646578, 0.789297104, -0.700347602, -0.127496094, -0.471921772, -0.927259624, -0.822308719, 0.793311954, -0.865695298, 0.687847137, -0.684672594];
    CONSTANT recurrent_3_i : ARRAY[0..4095] OF REAL := [-0.0771211386, -0.041904971, -0.0283814035, -0.0384180062, -0.037035238, 0.0755894855, 0.0912913829, 0.00833980925, -0.040718168, -0.0379342623, 0.0494960211, -0.0679311827, -0.0527894385, 0.0977362394, 0.0656317398, 0.0776981115, 0.06924472, 0.00551402941, -0.00546423346, 0.0256145597, 0.0663869157, 0.0448067561, -0.076562196, -0.0898107216, 0.0113763548, -0.153227463, -0.00167952105, -0.000464737415, 0.00439467467, -0.086409919, -0.0667009279, -0.0556129441, 0.0551343858, -0.120897166, -0.0255078562, -0.0891846493, -0.0639392585, 0.0117626972, -0.0803451017, -0.0123659503, 0.0534541979, 0.0729514435, -0.0211154483, 0.018317543, -4.61786985e-05, -0.0382464863, -0.0782647729, -0.015573822, -0.0043241363, -0.148820177, 0.0135069331, -0.0417309552, 0.0900624469, -0.0594736226, -0.0332042128, -0.0981074423, -0.0342614017, -0.0221951418, 0.0398744494, 0.0292471536, -0.0385849997, 0.00922256242, -0.102232851, 0.00561684091, 0.068692863, 0.0208462477, 0.00374138681, 0.0191529803, 0.000650386326, -0.0334673561, -0.0440338105, 0.0698852465, 0.041924905, -0.0118842367, 0.12935029, 0.125775233, -0.00667375699, -0.0881955922, 0.12345317, 0.0304863304, 0.0154025434, -0.00849951431, -0.0940478072, -0.0569340736, 0.0397216305, -0.0101688467, 0.0636173189, -0.0275668763, -0.0776927918, -0.00831863191, -0.0517599955, -0.00621921942, 0.0752723888, -0.0160099473, -0.0405343659, 0.139895663, -0.0825378597, -0.0492977053, 0.00898302533, -0.00459001446, -0.0101332637, 0.0280130263, -0.000348683447, -0.0557230823, 0.0340168104, 0.0289709847, 0.00258996524, -0.0492569655, 0.0154668484, -0.0495375916, -0.0926592499, -0.00718875788, 0.0474499613, 0.00148090534, 0.014299131, -0.0274025276, -0.0290415343, -0.030516278, -0.0101340506, 0.0522375405, 0.039179109, 0.068894051, 0.0322507881, -0.162401929, -0.0554244108, -0.0205325596, -0.0785830021, 0.0307614394, 0.0223672967, -0.0722827613, 0.0852478743, 0.0494147651, 0.0145334667, -0.0208612103, -0.0429588556, 0.0381661505, -0.0254635643, -0.0736351311, 0.0957547128, -0.0774454325, -0.0347611792, 0.0680866167, 0.016637262, 0.0466553494, 0.033682324, -0.0863118842, -0.0845884606, 0.0137423016, -0.016874576, -0.165303648, 0.0474241152, -0.0929194614, -0.0767099485, 0.0418002605, 0.0954845101, -0.00080230023, -0.0807549134, 0.0121842455, 0.0311720297, -0.0555889904, -0.0261414796, 0.0444951095, 0.0685377568, -0.0603509247, 0.0394478515, -0.0426621363, -0.028166268, -0.111334451, -0.00541599607, 0.0391055457, 0.0406126902, -0.0042554047, -0.0693275034, 0.027714774, 0.0115201902, 0.0424438566, -0.0750981644, -0.0402415507, 0.0593367405, 0.000854386715, -0.114437148, -0.0489385724, -0.0201637335, -0.00409932295, 0.0365078077, -0.0941109583, 0.0433239974, 0.0391140729, -0.0613765344, -0.000776667846, -0.0493680127, -0.0485325456, -0.0351513848, 0.0862187147, -0.00819134247, 0.0379211903, -0.000430813408, -0.0901147798, 0.0257685203, 0.108759008, -0.0223718863, -0.0338063687, 0.0156060597, -0.0172953494, 0.105790891, -0.0348870568, -0.0238552466, -0.00988221075, -0.0594870858, -0.0270350054, -0.0289226882, 0.056025885, -0.0559534319, 0.020340465, 0.0709189698, -0.00690495083, -0.0614235885, 0.0191929154, -0.0386514366, -0.018077353, 0.00255588954, -0.0549483672, -0.00174959237, 0.0446115658, 0.0373613685, -0.0370806232, 0.0284372792, 0.0797402859, -0.00256645121, 0.0148433009, -0.0631293207, 0.0278138295, 0.0731672049, -0.0447285399, 0.0508892573, -0.0192828514, 0.0280563608, -0.111958891, -0.0154376552, -0.0134562105, -0.0191528574, 0.0128744598, -0.0721960068, 0.0127519071, 0.0261764918, 0.00257971184, 0.0371103063, 0.220796183, -0.0201993361, 0.136452839, -0.0829204321, -0.00433726329, -0.0309275035, 0.0139829013, -0.051826857, -0.0566153042, -0.0116139706, 0.142482996, -0.0337721556, -0.0867007822, -0.0408329964, -0.0801567733, -0.0191535316, 0.0158957019, 0.0364312977, 0.0103620645, 0.0660757124, -0.100970119, 0.00712347124, -0.0876183659, -0.0854493976, 0.0477382392, -0.0373322181, -0.10326831, -0.0345545262, -0.0589192808, 0.0612725839, -0.0597315729, 0.0500357635, -0.04096343, -0.0692025051, -0.0106984116, 0.0438899919, 0.0404368266, 0.071749717, -0.0615543127, -0.0598752797, 0.0415351987, 0.02201939, 0.00219875015, -0.0673001781, 0.00924704876, 0.0722749159, -0.00525195571, 0.113458283, 0.0372568965, 0.0262363628, -0.0441234633, -0.157484531, -0.00621980149, 0.00702268817, 0.000515939551, 0.0563302599, 0.0814431012, -0.00974204205, 0.0340133868, 0.10453859, -0.0763610899, 0.181937218, 0.0482747033, -0.0712695792, 0.00854755938, 0.125115588, -0.0461000651, -0.0238136984, 0.053446807, 0.0636589676, -0.0651496276, 0.0328514501, -0.0157776587, -0.0405609868, 0.0313981287, -0.039560575, -0.0540332682, 0.0873858109, 0.0195426941, -0.0589045882, -0.0835158303, 0.00876367651, 0.0174001865, -0.0799380466, 0.0423592404, 0.0804384351, -0.0816923082, -0.0501725748, 0.0174710006, 0.00766914617, 0.0943023041, 0.0225947294, 0.0731049329, 0.0203260779, 0.0116448291, 0.0441071019, -0.0682512969, -0.029621724, -0.0456192233, 0.0643681064, -0.0228619743, -0.0348646864, 0.00293346378, -0.0453966931, -0.0378940366, 0.0893360525, -0.0297199413, 0.0621536076, 0.0571176335, -0.00713542569, 0.00198624004, -0.0263217017, -0.00695461687, -0.062595658, -0.0356898196, 0.0519921929, 0.0773653537, 0.0256005786, 0.0134280697, -0.181774542, 0.0606586337, -0.0386322141, 0.079398334, 0.0183406621, 0.0610715933, -0.0669881776, 0.0885097384, -0.0829677358, 0.0276328847, -0.126968756, 0.0522386208, 0.0957871079, -0.123197556, -0.0739446953, -0.0316405408, -0.0435967892, 0.0860320777, -0.0220160093, 0.0570985079, -0.0832202658, -0.0193082672, -0.0668374896, 0.0475501716, 0.0844978094, 0.000630278606, 0.0638538375, 0.0542233847, -0.0417887084, -0.00277152518, -0.0250559971, 0.0337195545, 0.0427481867, 0.015459504, -0.0582500286, 0.0722409189, -0.0537337177, -0.0623925738, -0.0234598946, -0.00134511478, -0.0242168568, -0.0526385382, 0.00195068866, 0.0186914504, -0.0119787138, 0.0187721029, -0.033073511, 0.0115096737, -0.0633152574, -0.00176272169, 0.030483298, 0.0767166764, -0.138829052, 0.0149489995, 0.0345533825, -0.102163568, -0.104449436, -0.0121117663, -0.0284647569, 0.185877964, 0.00462655164, 0.0652706698, 0.0703491792, -0.0313264355, -0.055347681, 0.0250781216, -0.0712601691, -0.0117419995, 0.0371713117, 0.0855040774, 0.00171021745, -0.079428114, 0.0225222223, 0.0360391289, 0.0283598211, 0.0123287961, 0.0588385053, -0.0281411186, -0.0607317239, 0.0662985221, 0.0331876278, -0.055067122, -0.0299345013, 0.000159702147, 0.0443185419, 0.0587667078, -0.0132936174, -0.00628238171, -0.0756097957, 0.000682532787, -0.050425522, -0.0115786884, -0.00569279492, -0.0613335297, 0.0146273952, -0.0631228238, -0.0581459589, -0.0151755679, 0.0857625604, 0.0821363926, 0.115290247, -0.0549297854, 0.0494527891, -0.0702691972, 0.143419236, -0.000891714124, -0.0305100456, -0.0913166925, 0.0610314682, -0.00264202012, 0.0289883371, 0.135914102, 0.0355210379, -0.00808628649, -0.0574536361, 0.00994824804, -0.0611675978, 0.0921703205, -0.0638784096, 0.020130869, -0.0362409279, -0.00529598212, 0.0173103288, -0.00330379046, 0.0372529067, -0.00947646052, 0.00849558599, -0.0442692153, 0.0606488958, 0.00228718901, 0.0758064687, -0.012268913, -0.094871521, 0.0871430188, 0.0136561962, -0.000904569402, 0.0177231189, -0.0620503128, -0.00116063561, 0.089274697, -0.0410311706, -0.0160198882, -0.0176485721, -0.0251905806, 0.0309642088, -0.0365208983, -0.0692796856, 0.050867036, 0.0156931747, 0.0287272036, 0.0371698886, 0.0470653847, 0.0171248168, -0.038513612, -0.0526604652, 0.0604412891, 0.0703500807, 0.0379981175, 0.129006818, 0.0396738537, -0.0257127378, 0.00598947424, 0.00387466792, -0.0582250282, 0.0306714829, -0.0903960094, -0.0177030656, -0.0494029149, -0.167852327, -0.00442219153, 0.0496009812, 0.013880033, -0.0902066082, -0.00579406694, -0.149498537, 0.0741799176, 0.0138978958, 0.0207201876, -0.029839877, -0.107697017, 0.0754648596, 0.0499061793, -0.0648064092, -0.0602546036, -0.0953533798, 0.00365704438, 0.0356753245, -0.0100625791, -0.0301756747, -0.0183225106, 0.0209142882, 0.000961192884, -0.00425785966, 0.0731755793, 0.0539571531, 0.0307768025, 0.0192657448, 0.121937618, -0.0402431674, 0.0851507634, -0.0264093336, 0.00447697798, 0.00402681436, -0.0473406613, -0.105135515, -0.0504542477, -0.0541321822, 0.00259122159, 0.0348727964, -0.0885458589, 0.0608932152, 0.0967864767, 0.119259723, -0.00126710534, 0.099387981, 0.0255985558, 0.00795432366, 0.0200677458, -0.0657623336, 0.190532804, -0.0352462381, 0.11204578, 0.0583575144, -0.0365644731, -0.0667472258, 0.0420552082, 0.104517318, -0.123279393, -0.025258502, 0.0455506109, 0.0645823553, -0.0150504466, -0.0935732126, -0.0465937927, -0.00506780948, 0.0766709894, 0.016313877, -0.0589278638, -0.0213123448, -0.00999987405, 0.0372834876, 0.0003843382, -0.0424535349, -0.0291266404, -0.0146436654, -0.00614433317, -0.115411565, -0.00276262173, 0.0107895397, -0.032524284, 0.0721799359, -0.115214683, -0.0201889109, 0.0353863686, -0.0889972821, -0.0150663191, 0.0311618596, 0.097947672, 0.0337602422, 0.0297635645, 0.131509572, 0.0590009764, -0.0416336432, 0.0261052232, -0.029010294, -0.0259194914, 0.0256441385, 0.04547894, 0.0276543871, -0.0115486104, -0.00763038546, 0.0314593501, -0.0427584499, 0.0405674614, 0.029487269, -0.0592614375, 0.0180521794, 0.0585754439, -0.0690455586, -0.0602442659, -0.0481735766, -0.0419904962, 0.0475285091, -0.0502720438, -0.0131537914, -0.0166091621, -0.000902149361, 0.0570480227, 0.0707662702, -0.0314460434, -0.0985292792, 0.0363963433, 0.0452788696, 0.0805958211, -0.0927961469, -0.0842332914, 0.0785057843, -0.0252397936, 0.063726902, -0.0157659501, 0.0154123157, -0.0701188073, -0.0163884759, 0.117669068, 0.0686297193, -0.0508072823, -0.00954249315, 0.0685154498, 0.00789694674, 0.0402810648, -0.0445739515, 0.0538645312, -0.0362013169, -0.0298318546, 0.00947535317, -0.022353489, -0.018312728, 0.129584163, 0.0519749038, -0.0102249188, 0.106327176, -0.00141187524, 0.104458824, 0.0900954306, 0.0631913096, 0.0487863906, 0.0143436007, -0.0466737151, -0.0175238848, -0.0134204691, 0.0936064124, 0.0213608462, -0.0548267998, 0.0156905074, -0.0593934953, -0.0977132469, 0.00202449691, 0.00566504337, 0.101919673, -0.0227482766, 0.0688653514, 0.0549680814, -0.0696360543, 0.111353241, -0.0198062696, -0.0470485538, 0.0482638553, 0.0627034158, 0.0686005205, -0.0104259253, 0.0585279539, -0.0265351944, -0.0823240802, 0.0223231334, 0.0155628044, 0.0399463028, -0.0703131333, 0.0192429498, 0.0842892677, -0.0436442904, 0.00773867406, -0.0787202716, 0.0446639024, 0.000940637663, 0.0502416268, -0.0171056073, 0.00118341111, -0.20054698, -0.000826745294, 0.0638445243, 0.115336217, 0.0489696115, 0.0723453835, -0.00212192163, -0.106923357, -0.0138108861, -0.00562525727, 0.10132996, -0.0545146763, -0.0471567214, -0.0582389571, 0.0267263185, -0.0706184208, -0.014614461, -0.0879550129, 0.0106655899, 0.00542923622, -0.0904930532, -0.00561792776, -0.0161186848, 0.106282473, -0.0461229794, 0.095484823, -0.102420568, -0.0115131736, -0.0411330983, -0.0572963804, 0.0411828123, 0.0175885111, -0.00862000976, -0.072997123, 0.0657924712, 0.039794296, -0.00335495267, -0.0449964553, 0.0481781289, 0.0714197829, 0.0511781946, -0.0879000053, 0.0544147305, -0.0406234711, -0.0558374897, 0.0643390119, 0.0160111859, 0.00428581238, -0.0187804457, 0.015720617, -0.0579953454, 0.0280058905, -0.00923684798, -0.0470739752, 0.0321382321, 0.0422517508, 0.0183307044, -0.00781843718, -0.0342937969, 0.0205556918, -0.0981495678, 0.0488321632, -0.011658892, 0.0305980891, 0.118306451, 0.0768781081, 0.024575863, -0.100505978, 0.04237964, -0.189520091, 0.105704762, 0.135003522, 0.010658402, -0.0483942032, -0.0704915226, 0.0844620317, 0.0273216274, -0.0259813722, -0.0111644482, 0.06088854, -0.0766476393, -0.00363370311, -0.0178547688, -0.0920214877, -0.00513554085, 0.0269423816, 0.0703381896, 0.118874483, -0.0575212762, 0.119425707, 0.0529291444, -0.0860894471, -0.0865111127, -0.0148848416, 0.19253251, 0.104712084, -0.0555614047, -0.0672845915, 0.0351972207, 0.00676282309, -0.0296126883, 0.0261259004, -0.00242765062, -0.0275501218, 0.0260865837, 0.10234154, -0.0501713939, 0.0731360838, -0.0291022677, -0.0139559144, 0.0922236666, -0.105612159, 0.0131138563, -0.0829087719, 0.00905138254, 0.0465265922, 0.0365543664, 0.0536549091, -0.0559660532, 0.115871899, -0.0190141965, 0.0573159829, -0.00187401986, -0.0605982132, 0.0414755642, -0.00944722258, 0.0610298775, -0.0544121191, -0.0403051525, -0.0444469973, -0.00737518445, -0.0570647344, 0.0424280278, 0.0314462781, -0.0356462114, -0.00442456827, 0.00501318881, 0.0772018582, 0.0401184224, -0.0479452647, -0.0308884569, -0.0212140195, 0.02648261, -0.0255462639, -0.0302096345, -0.0782852694, 0.0235898439, 0.0513489395, -0.0660517588, -0.00344516197, -0.110358223, -0.0641045943, -0.0483674482, -0.0172280818, 0.0570637062, -0.0584195331, 0.0135480603, -0.0512361005, -0.0377590358, -0.0496845767, 0.00837638974, -0.131501243, -0.0485012457, -0.0867616311, 0.00172824948, -0.0483968779, 0.00378531776, -0.0201999806, 0.0129637346, -0.107964613, -0.0680155903, -0.0121945422, 0.0332003571, -0.142481193, 0.0353830494, -0.0529950261, 0.0895682052, -0.113010526, -0.129145518, 0.0134146102, 0.0746574625, -0.0465294942, -0.0412936099, 0.017362833, 0.0181081146, -0.067679368, 0.0175119545, -0.123860918, -0.0328148454, -0.123511083, -0.0364386067, -0.0311892685, 0.0184607543, -0.0311089717, 0.000620753504, -0.0568052083, 0.011010047, 0.0740614906, 0.0737213343, 0.132467821, 0.0134541467, -0.0517201014, 0.0371107683, -0.0747232139, 0.0175857544, 0.0185665116, -0.085187152, 0.0808551088, -0.0630146116, 0.0255866461, 0.0362472124, 0.0900037512, 0.0042063524, -0.0614381544, 0.0115199219, -0.0224268176, -0.0755639523, -0.010225663, -0.0233745798, 0.08830823, 0.00794417504, 0.100218058, -0.0395819508, 0.00176830171, -0.0245204028, 0.0422842354, -0.0372996591, -0.00241308706, 0.0962401032, -0.113369778, 0.0433700494, -0.114136435, 0.0341613181, -0.130839184, -0.089457199, -0.0233602859, -0.0479965173, 0.0391149297, 0.0692763552, 0.194222391, 0.0147205666, 0.00688768551, -0.0260862112, -0.159773886, -0.00286880438, 0.120641142, 0.0765589625, 0.0160452854, 0.0994570404, 0.00954604149, -0.019290071, -0.0922267511, 0.0113348532, -0.0906397477, 0.046988558, 0.072404258, -0.14337185, -0.0172273871, -0.114456639, 0.0451756306, 0.0412931889, 0.0209460594, 0.0381604433, 0.048741173, 0.0535983518, -0.117481872, -0.0597166754, 0.0416786224, -0.109581009, 0.00134346401, -0.0438084416, 0.00310220965, 0.0906066746, 0.102428459, -0.0467643961, -0.0134145245, 0.00761311688, -0.0128192632, -0.0144976024, 0.0508668683, -0.0244545713, -0.163217515, 0.0707146078, -0.0414909683, -0.020475097, -0.0709300339, 0.110582337, 0.0458872691, 0.0147851352, 0.0236281417, 0.0267456733, 0.0351790637, -0.0111391153, -0.0429372862, -0.0653672218, -0.00234420202, -0.0397546403, 0.000486603472, 0.00611863658, 0.0549708642, 0.00347794965, -0.103336439, -0.0649053305, 0.0232978202, 0.092099525, -0.035087008, 0.0587510988, -0.0260108709, 0.0149294846, 0.149228558, 0.00796078984, -0.0348771624, -0.0376017764, -0.00330119394, 0.0105758226, -0.0476414561, 0.0779505596, 0.0283059888, 0.068600148, 0.00378933013, -0.0553796664, -0.0282109361, -0.00815444812, 0.0270443503, 0.0880057812, 0.0859450847, -0.036509417, 0.0516473651, -0.107805446, -0.00200375728, -0.0827743858, 0.0520797148, -0.0391699858, -0.0311506353, -0.0506948382, -0.031195391, 0.0115020834, -0.0476800315, -0.063335754, 0.132047504, 0.0484156534, -0.0179302748, 0.157283068, 0.0366875157, 0.0251473393, -0.0673718005, -0.0393670425, -0.03770978, -0.0478124507, -0.0309036858, 0.0446205698, 0.0311251916, 0.0245048814, -0.0259537641, 0.0997335464, -0.0605693161, 0.00225354522, 0.0080093611, -0.0326315872, 0.0134006618, -0.0756340176, 0.0391127281, -0.0530095957, -0.0592922792, -0.0589320287, -0.0158974119, 0.0390460417, -0.0620967709, -0.00484201685, -0.0339126587, -0.114744462, 0.0272865258, -0.0148388147, -0.0874240547, -0.130963251, -0.00731145218, 0.0346865393, 0.0248591453, 0.132716715, 0.0567845628, -0.0396426059, 0.0966895819, -0.0279246792, 0.0332853012, -0.0544270054, -0.0434819683, 0.0667337701, 0.0185598992, -0.0217630044, -0.0630863756, 0.0165286437, -0.0175159127, 0.0732632279, -0.0882861689, 0.00874199346, -0.0702120736, -0.00991208293, -0.107882038, -0.057309255, -0.0370102227, 0.0218572132, 0.0131309144, -0.0377560779, 0.00983685162, -0.010612092, 0.00618636748, 0.0234554112, -0.00349855889, 0.032401789, 0.00883803703, 0.0168552957, -0.0251002647, -0.147040695, -0.0349156298, -0.0705754906, -0.0755141303, -0.0358002782, -0.0804489627, -0.0872704983, -0.10116975, -0.0111940997, 0.185184717, -0.0291834772, -0.0106254304, 0.0199537389, -0.0575619712, 0.0327430181, -0.0982737988, 0.00400483515, 0.0415157862, 0.0418619663, -0.0547926277, 0.122650564, 0.0924820527, -0.0236307867, -0.025062155, -0.00689590909, 0.0673624277, -0.059796568, -0.0229343288, 0.1029379, -0.0339142159, -0.0528561883, -0.0526297614, 0.150432065, -0.00509574916, -0.0739349201, -0.084164843, -0.0795581341, -0.00410477351, 0.0224036723, 0.0124150803, 0.0239414368, -0.0398170687, 0.177057952, -0.0192521326, 0.103363805, 0.0614584386, 0.0694947913, -0.0193667188, -0.0576172173, 0.0620115176, -0.0870990381, 0.0496941507, -0.0259861536, 0.0403347239, 0.0496604256, -0.0786272138, -0.0154306944, -0.081339933, -0.0445302837, 0.102406658, -0.061163269, 0.0604605749, 0.057162337, 0.0785773769, 0.049725607, 0.0122487135, 0.0674273595, -0.0874722376, 0.0738762915, 0.0531259775, 0.080693908, 0.106209084, 0.0290892515, 0.0115198158, -0.0458286665, -0.0384727009, 0.0816580355, -0.0311149843, 0.0961059481, -0.035856396, -0.0599000305, -0.0631308854, -0.0129607571, 0.111237794, -0.0191058517, 0.0521618016, -0.00881535746, 0.125796705, -0.0308310576, 0.0099222362, 0.00214290619, 0.00591849908, 0.0316641741, 0.108231694, -0.0540060773, 0.159002408, -0.0459824465, -0.0337038673, 0.113687485, -0.100403123, -0.0782597214, 2.66171992e-06, -0.030309476, 0.0187225994, 0.070588693, -0.021095952, 0.0898897126, 0.0519983917, -0.00222996995, 0.0286504477, -0.0130401272, 0.0265140049, -0.0149852019, 0.034320049, 0.0317233875, 0.0892530233, 0.0787781104, -0.0337975733, -0.0102227032, 0.0430831984, 0.000701051205, 0.0882281661, 0.0165888332, 0.0865149796, -0.0396107659, -0.0339075737, -0.0606385767, -0.0798013657, -0.0987702385, 0.0128210438, 0.0787314102, 0.0952082276, 0.0263865329, -6.64079562e-05, -0.0520985238, 0.048642315, -0.0639183447, 0.120937899, -0.054034628, 0.0577845201, 0.164206862, 0.00996304303, 0.0452152342, 0.012397184, -0.00907938741, 8.59340653e-05, -0.0279395226, -0.064995572, -0.0103277853, 0.0347133391, 0.0380030274, -0.156820685, 0.0496531799, 0.0056411447, -0.0199967287, 0.0349395275, -0.0178748965, -0.0971291438, 0.0238538645, -0.0882459134, -0.0474008173, 0.0881513059, -0.0397922955, 0.0727870688, -0.131201446, -0.0279316753, 0.0408275947, 0.0168356095, 0.0744072869, 0.0187169667, -0.068779774, 0.0426025018, -0.0193063281, -0.0520456582, 0.0416068994, 0.0160504002, -0.0849148706, -0.0781304762, 0.168890104, 0.0400321707, -0.0366453379, 0.0254135281, -0.0447303839, 0.00366006792, 0.00179227069, -0.073159337, -0.0863961428, -0.0180702675, 0.0033401968, 0.0471517816, -0.0329570249, 0.0174799431, -0.0915972367, -0.00979953818, 0.0262655523, -0.00219394523, -0.0771069601, -0.00288106315, -0.0112265646, -0.0510940552, -0.036896605, -0.0146863656, 0.00246440712, -0.1058181, 0.053954836, -0.132233366, -0.0751370564, -0.0461335778, 0.0248641428, 0.0206944253, 0.044601813, 0.0917557999, 0.0854347199, 0.00680780411, 0.0388449728, -0.0178329702, -0.0440684296, -0.0474345945, 0.0536735989, 0.0156669542, -0.0179837942, 0.015049316, -0.0944499746, 0.0255464185, 0.0139696524, -0.0183444917, -0.00965639576, -0.0268477555, 0.135275558, 0.0509962142, -0.0986917242, -0.0227983035, 0.00305658765, -0.0856561884, 0.0290389154, -0.0660269186, -0.0633658916, 0.0124608278, -0.0484014228, 0.010453742, -0.0150720328, 0.0921224728, 0.0343518369, -0.0277125072, -0.0351466686, 0.0913387537, -0.0382746346, 0.0982387662, 0.0597138219, -0.0440888293, -0.0873766094, 0.134155929, -0.000342816114, -0.112505727, 0.0339261889, 0.00784657151, 0.0422569774, 0.0304149017, -0.0174519662, -0.100313917, -0.0682862401, -0.078867808, 0.0252579935, 0.0598724373, 0.0175824519, -0.0580917522, 0.0579990409, -0.00509794895, -0.013098672, 0.0134000657, 0.00295411795, -0.0628975779, -0.0807553232, 0.00282261497, 0.0151576092, 0.0765760168, 0.0573970042, 0.037956208, 0.076710701, -0.029479716, -0.0708900243, -0.0150526743, -0.122771248, -0.0357170552, 0.0486811101, 0.0018941164, 0.0022100471, -0.0338713638, 0.138970211, -0.0620444939, 0.0276888832, -0.0742791072, 0.0107768327, -0.013218767, -0.0233383588, -0.00579264993, -0.122329608, -0.0303021222, -0.105152994, -0.00944907404, -0.0473172814, 0.0247038007, -0.0754274428, -0.00730832759, 0.0661038682, -0.00139894523, 0.0394513085, 0.0232133511, -0.136513174, 0.0769726634, -0.0362442955, -0.0387526341, -0.215772748, 0.0400592461, 0.148775563, -0.0179366972, -0.0344711952, -0.105664037, 0.0565368906, 0.0767515525, -0.0210688021, -0.0248218253, 0.0139113367, -0.0503477789, -0.0919362679, 0.00241893739, -0.150888786, -0.0521079935, -0.0130923521, -0.102624953, 0.0652719885, 0.0720933452, -0.0342555232, 0.143231511, -0.0571466684, 0.0597913601, 0.0616353974, 0.0496004112, -0.00588138867, -0.124242619, 0.0982202068, 0.0385833755, -0.0267478451, 0.0698152184, -0.0226045679, 0.0295436215, 0.0269691981, -0.0145521704, -0.0704007372, 0.0563407354, -0.0541602373, 0.0702264085, -0.0287812315, 0.0237359479, 0.0170573685, -0.0314531364, -0.0559237301, -0.0229936354, -0.0873287767, 0.0505414829, 0.0730561092, -0.12192782, -0.104775615, 0.099988088, 0.0937188119, 0.0256949309, 0.00599367218, -0.0792903006, -0.0849900469, -0.0244031977, 0.0517280139, 0.00284449384, 0.0588323995, 0.0150726568, 0.0705374852, 0.0227077417, 0.0698392466, -0.0465410054, 0.0897336528, -0.140212193, -0.0762655437, -0.0484272018, 0.0781526566, 0.0329838879, -0.0322162881, 0.0493155643, -0.0422493964, -0.0149069745, -0.00729649886, 0.116023973, 0.0208215024, -0.0119661624, -0.0600190572, 0.0152146658, 0.0232678521, 0.031961374, -0.076048471, 0.0752262473, -0.0254874378, 0.0603693463, -0.0214568563, 0.0443627983, 0.0861600712, 0.110576168, -0.0153700281, -0.0522413626, -0.0181858595, -0.102767073, 0.0204370059, 0.00640147924, -0.0462402776, 0.0303416587, -0.014012333, -0.101610146, -0.0537055694, 0.0660692453, 0.0320705734, 0.0438896939, 0.0207390673, -0.0499086902, -0.025366487, 0.0747519806, -0.0316851549, -0.0759165585, 0.0436173193, -0.0106276162, 0.015699055, -0.0377657488, -0.0501587577, 0.106968641, -0.0271445233, 0.114476688, 0.00821631402, 0.0723700747, -0.00975259766, -0.144449532, 0.000877615996, -0.0187783428, 0.0982629582, -0.0616536327, 0.0501482002, -0.00122638233, 0.0282082222, 0.0182234906, -0.0169871524, -0.0162812453, -0.0360330716, -0.0333503634, 0.0434881076, 0.026132334, -0.0594973639, 0.0357384905, 0.10762547, 0.0930696428, -0.032664597, 0.0310225002, 0.0313590989, 0.0207410716, 0.00215228461, 0.0220122356, -0.0219471399, 0.0972534791, 0.0126505364, 0.0284033492, -0.0381177627, 0.0166915413, 0.0413518623, -0.0191520825, -0.000985896448, 0.00584470853, -0.011032097, -0.0880968124, -0.0672093704, -0.00587202143, 0.095265761, 0.126526862, -0.0436578542, -0.0140812155, 0.0604392216, 0.0731392428, -0.0256851912, -0.105274037, 0.106243387, 0.0340439156, 0.131831095, -0.0265626591, 0.0286284406, -0.0759204477, -0.0156980269, 0.00696976855, -0.00866186433, -0.00699613057, 0.0219969749, -0.0664360374, 0.0397608355, -0.113807514, 0.0428919867, 0.132699594, 0.0729412511, 0.0291228183, -0.0552000776, 0.0984611437, 0.0857509077, -0.176901773, 0.0790669769, -0.0925221816, -0.141180128, 0.0706448629, 0.050350558, -0.0397202708, -0.0755624548, 0.0277449936, 0.0465391055, 0.0242460705, -0.0519197322, -0.0352012888, -0.0360889398, -0.0180267282, 0.0771338642, -0.0200135168, -0.0418161638, -0.104534358, -0.0436706729, 0.0487912074, -0.0194058344, -0.110537097, -0.0642443299, 0.0491082668, -0.119076572, 0.108019292, -0.0060014613, 0.0306117442, -0.00466304319, -0.0232913699, -0.0511650331, 0.0275231972, 0.0840327442, -0.134391844, 0.0361698754, 0.0546769425, -0.00451168697, -0.124834865, 0.00793889817, -0.0194791071, -0.047546424, 0.00907409191, 0.0667063519, -0.0414150916, -0.00810996629, 0.0252991784, 0.00813391805, -0.101334795, -0.068073824, -0.00572252087, -0.0330414437, -0.00174164213, -9.43699852e-05, -0.003085576, 0.0486874282, -0.0364591666, -0.0317699015, -0.0173614342, -0.128078446, -0.00707710255, 0.0569778122, -0.00317369495, 0.0616593473, 0.105571508, -0.0600511916, -0.125462323, 0.0620394647, 0.0330251008, -0.0224925671, -0.06249341, 0.0392381921, 0.0241978578, 0.00201773271, 0.0761228129, -0.0289585106, 0.0902938694, 0.0738835782, -0.016410742, -0.117978804, -0.0864401907, 0.039015539, -0.0713666528, 0.0403234623, -0.0509619899, -0.194570005, -0.066731289, 0.0154067371, -0.0439324453, 0.0847003162, 0.107806429, -0.033445593, -0.0332155339, 0.0183431655, 0.0231716502, 0.0285760835, -0.0442197695, -0.089011088, -0.0314625204, 0.0825669691, 0.0989553183, 0.126024291, -0.0403006971, -0.0249300376, -0.00175470766, -0.0387068391, 0.103461869, 0.104851246, -0.078734979, -0.0869031996, -0.00940553006, 0.0473936833, -0.0492781959, 0.011214152, 0.0900023058, -0.139418155, -0.0459762774, -0.0767275542, 0.038480971, 0.0355797447, 0.0246626176, -0.067918703, 0.0173300691, -0.0111240037, 0.00440449361, -0.0675490722, -0.117332205, 0.0323232301, 0.0494250655, -0.039023485, -0.0351693928, -0.0558870584, 0.0212836526, -0.0763815865, 0.0145481098, 0.030264806, -0.0194271654, -0.0656424165, 0.0946357548, 0.0536819957, 0.0625644103, -0.100732088, -0.0241884068, 0.0235884488, -0.00379322818, 0.0470121168, -0.0830290541, -0.00274844444, 0.035193529, -0.00292130839, -0.0975778103, -0.146146074, 0.0253734533, 0.0170242153, -0.0313359797, 0.120178267, 0.0498198569, -0.142378464, 0.00051176548, 0.0584818572, 0.0537292473, -0.108122371, -0.0433480218, 0.0291369781, -0.0533202067, -0.0646765009, 0.00796661153, 0.0651323423, -0.0704324991, -0.0595270172, -0.0637600347, -0.0255695526, -0.0359119177, -0.0329027623, -0.0251953397, -0.00202006707, -0.0203789137, -0.0562391691, -0.080313772, 0.0577877834, 0.0348158069, 0.0304604135, -0.00427031424, 0.137653306, 0.0444946364, -0.135594085, 0.00807581842, 0.0390937254, -0.0484327748, -0.00712263305, -0.00467313454, 0.0213462058, -0.0569633618, 0.014585142, -0.00903347321, -0.0474929325, -0.0491582491, -0.0225354433, -0.060164921, 0.0331706293, 0.033714164, -0.0489883646, -0.000850817189, 0.0880154669, -0.0255647115, 0.0434250459, -0.120299645, 0.00521157775, -0.0519536845, 0.12155582, 0.0670317113, 0.0390714034, -0.0730279163, 0.108900294, 0.0190060548, -0.0151199531, 0.0411870778, 0.0563757047, -0.10859707, -0.0251432694, 0.127860352, 0.0683794245, 0.0160465818, -0.0222009514, 0.0233334191, 0.0192102417, 0.00722608529, 0.0708645135, 0.161178872, 0.0612367056, 0.00366378948, -0.0137775969, -0.0395795293, -0.0202920213, -0.078712672, 0.0827812701, 0.0557660833, 0.00758445263, 0.0559690334, -0.0459271818, 0.0884366781, 0.0462979972, -0.118541867, -0.0199150778, -0.0930863246, 0.0684344172, -0.0483856648, -0.0175752882, 0.00132881314, -0.0874542668, -0.00535436114, 0.0246759802, 0.0050930893, -0.104525492, 0.0308124907, -0.0427543446, 0.0113368044, 0.117691182, -0.00788058154, 0.0374500006, -0.0663976371, -0.0379608162, 0.0824671388, 0.040722385, 0.113066494, -0.0284847841, 0.0628969744, 0.0176786631, 0.106616139, 0.0364625454, -0.0395449772, 0.0711597875, -0.115894616, 0.0616638251, 0.033880759, 0.0842308551, -0.0200199522, 0.0854050592, 0.00240669074, -0.0221695919, -0.0171297081, -0.0368121415, 0.0901898295, 0.0558736101, 0.052049391, -0.044363752, -0.00578884175, -0.139492258, 0.0934761465, 0.0463176742, -0.0893110707, -0.0234638881, -0.0254841838, -0.0230731126, 0.023535518, 0.0606091544, 0.0712842196, 0.0151794199, 0.0228757747, -0.00670690928, 0.0243334826, 0.00760607189, 0.0909763575, -0.0020671133, 0.0380613878, 0.0523210615, -0.00226617698, -0.0527453385, 0.0873451531, 0.00789528619, -0.039309945, 0.0657774359, -0.0373396091, 0.0121234003, -0.0608648509, 0.0955511183, 0.106229104, -0.0227189902, 0.0181806684, 0.0313352682, 0.0983065665, -0.0655134469, -0.0100321807, -0.0214557108, -0.0323480032, 0.0399547108, 0.0510334969, 0.0764594153, 0.120244615, 0.100224771, 0.0613763817, 0.0966042578, 0.119996041, -0.0274828617, 0.0648390055, -0.0121074114, -0.0551745556, 0.0166523531, -0.0572726466, 0.011296981, 0.0738770068, -0.028714275, 0.0734295845, 0.0108936559, 0.0432941616, -0.00889409427, -0.008979748, -0.0243339837, -0.0185373686, 0.00247844215, -0.00585353561, 0.0613322258, -0.0551779605, -0.00296961702, 0.0106428079, -0.0408338606, -0.0757235661, -0.00855779834, -0.0684195235, -0.0265507028, 0.0798603669, -0.0745164007, 0.0298931263, 0.107402548, -0.0163386203, 0.0202664565, 0.0360967554, 0.0445154905, 0.0351002701, 0.0772979185, -0.0847752467, -0.0830296054, -0.0078751957, -0.0517528765, 0.0568756424, -0.0522266701, -0.0157700721, -0.0453625172, 0.121910952, 0.00520794094, 0.0594974682, -0.0149897374, 0.0535635464, 0.0229940414, 0.0360345319, 0.11592412, -0.0503912047, 0.00695486646, 0.0321925282, -0.00204658881, 0.0299749561, 0.0869947672, -0.131942108, 0.0256948676, -0.0761573315, -0.0721464306, 0.0488116369, -0.0233175065, 0.0251011774, -0.0364564434, 0.0703453049, -0.0303190667, 0.020260239, -0.0368825868, 0.0204307344, -0.138143018, 0.0240335371, -0.12227723, -0.000719763339, 0.0397568047, -0.0108157676, 0.0380594246, -0.0454414487, 0.00395573629, -0.079955548, -0.103262126, 0.0717545897, 0.0462553948, -0.0749582872, -0.0598753132, -0.0549320504, 0.167967528, -0.0342475176, -0.0678644106, 0.014138151, 0.0883469209, -0.0422446132, 0.00910017174, -0.0278913192, -0.0617286935, 0.0945532322, -0.0891489685, 0.00157077983, 0.0810243636, 0.036433693, -0.0354036316, 0.0656190589, 0.11084713, -0.0328651145, 0.0968796238, 0.0468874946, 0.0668853596, -0.0326856822, -0.0238782857, 0.0019241781, 0.0953875333, 0.111255117, -0.0768138543, 0.000530576333, 0.000880140811, 0.147702083, 0.0755548328, -0.0203691162, -0.0268486366, -0.044232972, 0.045487687, -0.103220411, 0.0775320604, 0.00794593431, -0.0394486375, -0.0247686394, 0.0284869447, -0.0534544103, 0.00503673032, -0.0112144612, -0.0468843877, 0.0273283813, 0.0793735757, 0.00207741046, 0.0429351106, -0.00290703773, 0.00570422132, -0.0043573156, 0.109113462, -0.0445359349, 0.0418569483, 0.0393498242, -0.0209372249, -0.00551870884, 0.107174665, 7.90264457e-05, -0.042608235, 0.0417940132, 0.0433975756, 0.0341972709, 0.0231017601, -0.0823120326, -0.0285989456, -0.0565683097, 0.00515736546, -0.0216090027, -0.055794172, -0.0425441638, 0.0674974695, -0.0372256935, -0.00943269115, 0.0081518339, 0.169903964, -0.0767062902, 0.0181438327, 0.0594843477, 0.0724104196, 0.0623655654, -0.0627258271, 0.108728275, 0.066685833, -0.00326387049, 0.0191066675, 0.0488062687, -0.0557465106, -0.0717181638, -0.120245077, -0.0263934378, -0.0217542164, -0.0377301425, 0.0505158901, -0.00943231955, -0.0811585411, -0.0633471459, -0.0922307, 0.00297417305, -0.0283020921, -0.00233821943, -0.0317868218, 0.022295991, -0.102933459, 0.0353327431, -0.0564441793, 0.0270108245, 0.111416861, 0.054940667, 0.045586627, -0.0325855613, -0.0276312456, 0.108739905, -0.13752073, -0.0148813566, -0.0878764614, -0.00616987422, -0.0113345832, 0.111377209, 0.0674577281, 0.0334462859, -0.0528105721, -0.0283257961, -0.0640272871, -0.104231998, -0.0182194225, 0.0253928099, -0.010000607, 0.0893871188, -0.0936637968, 0.0359381177, -0.0572381169, 0.0415782668, -0.0515473448, -0.0592029989, -0.0162340757, 0.0372194499, 0.000869643176, 0.0569775514, 0.12664406, -0.00410834746, -0.0598526485, -0.0145936832, 0.00541882915, -0.0387819409, -0.0705848932, 0.131225437, 0.0606011972, 0.0260585826, 0.0326864943, 0.0327170156, -0.0681137666, 0.0398291536, 0.0150668863, -0.0623713508, -0.0654203072, -0.0855273381, 0.0542779416, -0.0772915483, -0.00739911618, 0.111987807, -0.0434356108, -0.109296009, -0.000388567569, -0.0285733771, -0.126296833, 0.0530360192, -0.0114716245, 0.0218612682, 0.0229222216, 0.0851885229, -0.0389903337, 0.0584750213, 0.0194483101, 0.0111343805, 0.0142656472, -0.00225033797, 0.00987144839, 0.00450252695, -0.00685430365, -0.0110871671, -0.064477019, -0.108237572, 0.0994877592, 0.0447605662, 0.0851446614, -0.0512959659, -0.0695576966, -0.056695722, 0.0151356487, 0.0813366249, 0.0509820394, 0.130533665, -0.0970403776, -0.06133876, 0.062047407, 0.000485517085, 0.0295372587, -0.0825812668, 0.103946805, -0.0272734016, -0.0142017547, 0.0348625258, -0.0194650106, 0.054473225, 0.0277187414, 0.00521013513, -0.0750550181, -0.0112232966, 0.061832428, 0.0267357174, 0.0369789787, 0.0242078975, -0.0639228001, -0.076738812, -0.105967775, -0.00552886352, 0.0244175512, 0.0138396807, 0.0793611556, 0.0163184702, 0.017674122, 0.0549585409, -0.0119000934, 0.00208156183, -0.0401373133, -0.062261004, -0.0735801086, -0.0862724259, -0.0881317705, 0.030051088, -0.017848039, 0.0650936216, 0.0235368982, -0.0109532671, 0.0914635584, 0.0342697278, 0.0226438977, 0.1154567, 0.0288205035, -0.0857841223, -0.0564709753, -0.0212000832, 0.0331944302, -0.0697550699, 0.0471978039, -0.0747845024, -0.0133633576, 0.111894704, -0.0159318224, 0.0424069613, -0.0777497888, 0.0269897413, -0.0035970686, -0.0470015891, 0.0703898668, -0.0996557772, -0.0109145269, 0.0119720763, -0.0309154429, 0.0772444978, 0.0240636114, 0.0555266663, -0.0486289486, -0.0358316675, 0.0310520343, 0.0524581783, -0.02964909, -0.0225995835, 0.0202129167, 0.0492513031, 0.0024611596, 0.0920979604, -0.147307992, -0.057231009, 0.0140033029, 0.00698713493, 0.0638547167, -0.12043111, 0.0617109016, 0.0197395254, 0.0250540208, 0.0461532772, 0.0631778687, 0.0675501153, -0.0640308559, -0.0384968631, 0.124442965, -0.0169296619, -0.0591387115, 0.00277835689, 0.03010704, 0.0170286968, 0.0438472293, -0.0421725586, 0.0105780903, 0.0187833142, 0.0932823047, 0.0797822848, -0.0400023311, 0.0413492993, -0.00490421942, 0.0261564571, 0.0153271826, 0.0136942901, -0.0678173229, 0.069321245, -0.0221962631, -0.053999871, -0.0290583689, 0.0566808693, -0.068984136, -0.0322767571, -0.0840166956, 0.0840327293, -0.0266867373, 0.0181480683, 0.141900614, -0.0741518885, -0.0462956466, -0.113084376, -0.0761168301, -0.119766846, -0.0191113465, 0.0263688825, -0.0602698475, 0.0213941634, -0.00738273561, 0.066034399, -0.112135068, -0.0262510292, 0.0678964183, -0.0115228705, -0.0385066345, -0.00596521609, 0.00337880291, 0.0653976202, 0.101864547, -0.0145517476, 0.0115391631, -0.149418652, 0.0152731091, 0.0258516744, -0.141610175, 0.0650391579, -0.0218729898, -0.0738234967, 0.087863043, -0.109388128, -0.0587620288, 0.00153938029, -0.0472481102, 0.0655660331, 0.046287518, 0.00191088393, -0.0099407332, -0.0366902761, -0.0758936703, -0.00195228774, 0.132410303, -0.0897945017, -0.0828643367, -0.0931508541, -0.0858343989, 0.0220552962, -0.0318561718, 0.0606997572, -0.0955435112, 0.0174528975, -0.0370034575, 0.000795804895, 0.0466999449, -0.00521745998, 0.0106653189, -0.0342373848, -0.0102693718, -0.054669518, -0.0429277383, -0.0600964017, 0.0296549965, -0.0716629699, 0.0814423859, -0.0409946404, 0.0218861047, -0.0409745276, 0.0469141454, 3.98382545e-05, 0.0468013287, 0.0229902081, 0.0182137676, -0.0610425286, 0.0229899418, 0.142873287, 0.0214464925, 0.0217601303, 0.0480984598, 0.132810012, -0.0424922258, -0.0198705606, -0.0383956023, -0.0761293694, -0.0926634222, 0.135834634, -0.0136811342, 0.0532483645, -0.01176906, -0.0229151398, 0.0479301736, -0.062715888, -0.130381748, -0.0411189981, -0.0947250798, -0.068229951, -0.0499406345, 0.0430741422, 0.0469632521, 0.032190226, 0.0405618772, -0.0297602359, -0.0669889972, -0.0655034855, 0.078095153, 0.00653720647, 0.0422790386, 0.0746423826, -0.0137710692, 0.00105908152, 0.0166120734, -0.119933531, -0.0162646584, 0.0831588954, -0.0413135663, -0.0308480002, 0.0571599156, -0.0818429664, -0.0296073332, -0.0288697742, -0.0251193624, 0.00306123914, -0.0458743162, -0.121116683, 0.0111547802, -0.112941243, -0.0577419885, 0.0467755049, -0.0507814661, -0.051298175, -0.110015258, 0.00560337678, -0.183197498, -0.0217102468, -0.0208833274, -0.00695190392, -0.123197421, 0.032691773, 0.0942695662, 0.0321684778, -0.0735458806, 0.0188958589, -0.0569661036, -0.0828002393, 0.0375961661, 0.00283417851, -0.0231414177, -0.0458211303, 0.027478531, -0.0677815825, 0.0677349195, 0.0259536654, -0.069852069, 0.0958945453, -0.0408855304, 0.0159991458, -0.0688989162, 0.0626117587, 0.0124521516, -0.0413726643, -0.0320701264, 0.0376031771, -0.126749635, 0.00893450901, -0.0760586113, 0.00351698697, -0.0616703182, -0.0376914926, -0.089731127, -0.0248150546, -0.00226218812, -0.0297166444, 0.0724341646, 0.0295588318, 0.0506805852, 0.0683638975, 0.0346119218, 0.0146825043, -0.0300900675, 0.120438926, -0.00266315043, 0.0247528851, -0.0554317571, 0.0749954581, -0.0660863221, -0.0665542111, -0.0541550033, -0.0416485667, 0.0372959226, -0.127699882, -0.084750995, -0.0336081795, -0.0684883595, -0.0341891944, -0.0812875256, 0.0163575001, -0.0336027704, 0.0934475213, -0.0343994573, 0.0371381752, -0.07674779, -0.0452275723, 0.0257721879, -0.0229448806, 0.114483461, -0.0620328411, -0.0166221671, -9.28267837e-05, 0.00410251226, -0.043749325, 0.0121183004, -0.0199087746, 0.0343265273, -0.0519517921, 0.0498782434, -0.00514894351, 0.105170429, -0.0145044802, 0.0170543566, 0.0612747185, 0.0635284111, 0.0722448826, -0.0402126908, 0.0406716689, 0.180485785, 0.0420826823, 0.011254332, -0.07383883, 0.00756357796, -0.00653190818, -0.118777044, 0.0412342064, -0.00101301633, 0.00468574138, 0.0618331097, 0.129026562, 0.0577140562, -0.119758949, 0.0418074131, -0.10028886, 0.146321386, 0.00203114515, -0.0382076167, -0.0158315971, -0.0185160302, -0.0585700981, -0.0892127752, -0.0502712131, -0.00863518007, 0.00928955711, 0.0245242007, -0.0761695579, -0.016499823, -0.0851950496, 0.0302402433, -0.0451599397, -0.000235274434, 0.134561434, 0.0654707849, -0.039849773, 0.0276978035, 0.0976922065, 0.0597911887, 0.128048003, -0.0642070174, 0.0135878399, -0.014466498, 0.00938953552, -0.00197627768, -0.0473276153, 0.0124964295, -0.0482927561, -0.0500519387, -0.0224759765, -0.117781542, 0.0445974693, -0.00626224931, -0.0716539621, 0.0209659114, 0.0950907618, 0.055297289, 0.0339224786, -0.0361117683, 0.00555084739, -0.115107872, 0.000439941883, -0.0202993192, 0.0453407951, 0.0561007559, -0.11338371, -0.0781322941, -0.0260165855, 0.0112777418, 0.0960166007, 0.0797323436, -0.00932762027, 0.148689911, 0.0673603341, -0.00126363337, -0.0395420641, -0.0616854914, -0.0218652152, -0.0841251686, -0.0654635057, -0.13668707, -0.00122302305, -0.0790907443, 0.0650716498, -0.0057691643, -0.0128726279, -0.0956908092, -0.0315712467, 0.0279215723, -0.101440802, -0.0671161041, -0.0240076855, -0.0446522608, -0.0316099077, -0.00810685288, -0.108626872, -0.022286335, 0.0336487666, 0.0771654397, -0.0866703987, -0.109500088, -0.00691062957, 0.00515462086, -0.120609254, -0.0162109509, 0.0773937255, 0.0669814423, 0.0372542813, 0.0293540005, 0.0399727486, 0.0871676579, -0.0184890218, 0.0546814017, -0.0425825901, 0.067953147, -0.0311761238, 0.0312341489, 0.0876554847, -0.0146615878, 0.0407922156, 0.116035752, -0.0404246673, 0.0638451576, 0.101785071, 0.00436116382, 0.036284972, -0.0171610918, -0.0127823167, 0.123123139, 0.0832545161, -0.0702112019, -0.0220967159, -0.00930657797, 0.0471730381, -0.0502699539, 0.0598344095, 0.00845675543, -0.121706769, 0.147291899, 0.0185488053, 0.0772631615, -0.0692496821, 0.092323333, 0.0531550683, -0.091813907, 0.0341402963, 0.0104403701, 0.008129769, -0.0408172235, 0.0606573857, 0.00977760367, 0.0389199331, 0.0131801832, -0.0922353864, -0.098223269, -0.0419626646, -0.0593111143, 0.10533867, -0.0268028136, -0.00331548043, -0.163931951, -0.033068873, -0.00352114672, -0.0809657648, 0.0686088428, -0.00292867795, -0.0278624669, 0.00411469908, 0.0318309069, -0.0307580922, -0.0397743359, 0.00780036114, -0.0651816577, 0.0145179741, -0.023223361, -0.0542891026, -0.121250667, -0.0295627341, 0.02031634, -0.0493941419, -0.0111236311, -0.0228398573, -0.0352995545, -0.0289986897, 0.0391738042, 0.0846049562, -0.086711213, -0.0735283643, -0.0955764875, 0.00540071353, -0.0682940334, -0.0206642989, -0.0456988215, 0.151994646, 0.0301898979, 0.0369524732, 0.0502344705, 0.0833638757, 0.121431336, -0.0410372801, -0.0254659615, 0.0228950866, 0.0228525996, 0.0083724726, -0.0585110821, 0.0608403683, -0.0204683263, 0.00102710386, -0.0463586897, -0.00256409403, -0.0700236112, 0.0309709981, -0.0577077791, -0.00222884188, 0.0324225649, -0.0529456697, 0.0334489383, -0.0258610249, 0.140200675, 0.027081497, 0.0447089374, -0.0138469264, -0.044828862, -0.0518506318, -0.043909952, 0.0304525048, -0.0991320908, 0.0472474843, 0.0305546597, 0.030144278, 0.0851663947, -0.0152060036, -0.0141895618, 0.0190068781, -0.04600906, 0.137501746, 0.10347534, -0.0207075998, -0.0712871552, -0.0669450387, -0.0113951489, 0.00467752712, -0.040738754, -0.0361441448, -0.00970679428, 0.0331211239, -0.0323049687, 0.00529360026, 0.0707725734, 0.116111211, -0.0430333167, 0.0310098082, 0.00512955338, 0.0163368694, -0.0464587808, 0.0123096537, -0.0234641749, 0.000730314292, -0.112272233, 0.0216336772, 0.0133584049, -0.0161934346, 0.0556386374, 0.0335740149, -0.0173839238, 0.039414037, 0.0958736166, 0.033290185, 0.0287034474, 0.0432678051, 0.017504232, 0.108818457, -0.0528055504, 0.0226539914, -0.0613601804, 0.00927608088, -0.0999047384, -0.0737604499, -0.00714416057, 0.0170378312, 0.0955149829, 0.0398799814, 0.0177485012, 0.080797337, -0.0437004454, 0.00450856751, -0.0644934624, 0.0559109151, 0.0616841912, 0.0297846273, -0.0220688954, 0.0190214403, 0.1088126, -0.00498170266, -0.0906166136, 0.153623462, 0.048660934, 0.0527924597, 0.0132156964, -0.0345814601, -0.047118552, 0.0239117257, -0.0547183156, 0.0468712188, 0.0610508956, -0.00730768964, 0.0571509115, -0.0177728441, 0.108094901, 0.000422280282, 0.0676494464, 0.0548462979, 0.0319501087, 0.0757430568, -0.0270296652, 0.0219633151, -0.0551248714, 0.0401655883, 0.0186556727, 0.0519931801, 0.074958913, 0.0776639879, -0.00639817771, 0.0184700675, -0.0563476905, -0.0846942812, -0.0214337297, -0.0115232533, -0.0333131962, 0.16067192, 0.0255485959, 0.03676489, 0.094095245, -0.0732448176, -0.0146226548, -0.0105268834, -0.0823027566, 0.00527555775, 0.00325848535, 0.103646882, -0.0838223398, -0.0200149957, -0.0291824713, 0.0694787055, 0.0277231112, 0.0374957621, 0.0328506157, 0.0508431233, 0.00787144154, -0.0617377684, 0.00957613159, -0.133195773, 0.0383893773, -0.0733166188, -0.00745590124, -0.0818732083, 0.060960643, 0.0544005632, -0.140092775, -0.0229060613, -0.00408835337, -0.0823066682, 0.0300217345, 0.00907065999, 0.0392521843, -0.0700395405, 0.0079762768, -0.1493496, 0.0583605468, 0.0270410068, -0.0341156311, -0.0386294425, 0.0662309453, 0.0872389451, -0.0472744517, -0.0228074081, 0.0684124902, -0.0888471007, 0.0761127099, -0.0326396823, 0.0732444823, 0.0456608236, -0.0937242955, 0.0504064783, -0.141814753, 0.162431598, -0.102114215, -0.0397514515, 0.0473489277, 0.0336118191, 0.148338452, -0.0122316275, 0.0432145298, -0.109083384, -0.0186488908, 0.0720187798, -0.106312886, -0.0913583338, -0.0169402808, -0.0123407505, 0.00822057761, 0.0596636757, 0.0205631852, -0.0619561039, -0.0609639287, 0.0482201204, 0.0354727581, -0.0402187109, 0.0445601232, 0.0287282206, -0.0440565534, -0.0619057789, -0.0213008486, -0.0699777231, 0.0775571316, 0.0231237784, -0.00883588009, -0.113154605, -0.00541019021, -0.033951968, 0.0411423817, 0.053961359, -0.00288748881, 0.0706721246, -0.0491243415, 0.00054154871, 0.0138199497, 0.127938673, 0.0159905218, 0.0829677731, 0.108012542, -0.0567845702, -0.157686636, -0.0702316687, 0.00892338157, -0.165532067, 0.076706022, -0.057830967, 0.00497925933, -0.0186288226, -0.0808018744, -0.0206770748, -0.0118557923, -0.0637545362, 0.0900221914, -0.0139558092, -0.00739696994, 0.074806042, -0.119168133, 0.0166030899, -0.11083927, -0.0656669214, -0.0363056958, -0.00638495618, -0.0680301413, -0.0248918328, 0.00398088805, -0.0237197392, 0.00691889878, 0.0542797484, 0.0325936712, 0.00915190857, 0.00299844984, -0.0195343439, 0.131595939, 0.118413478, -0.0392579846, -0.0031316895, 0.00834177993, 0.0611352138, 0.00132380705, -0.00584108802, -0.0469935127, -0.0832609683, 0.0250498392, -0.116703823, -0.00103460811, 0.102866396, 0.0110065071, -0.0472957417, -0.0647558421, -0.1213881, 0.183602601, 0.0604174212, 0.0105359852, -0.0726647228, -0.08007323, 0.0142628476, -0.0803629532, -0.077605769, 0.093770422, 0.0476225019, 0.0822985619, -0.0843518898, 0.0317965075, 0.0298086535, -0.0405269526, -0.0544525683, -0.0352851711, -0.0550699346, 0.0060656406, 0.0519128218, -0.0409257188, -0.026854191, -0.0174814686, 0.0396045148, 0.00388014689, 0.0182089992, -0.109553322, -0.0415327437, -0.105616137, -0.00612959452, 0.00763020385, -0.0235190243, 0.0448918492, 0.0302004609, -0.0875566453, 0.00955081545, 0.0885803998, -0.0824447349, -0.0201507267, 0.0728382841, -0.0490038544, 0.0268885419, 0.0938861519, 0.0330029763, 0.00269161188, 0.0447449647, 0.0945401639, 0.119459607, 0.00680486578, -0.0233078562, 0.0511108488, 0.060301017, -0.00174694043, -0.0356153585, -0.0987226442, 0.014362609, 0.0541739948, 0.00264295842, -0.0994685963, 0.0274561457, 0.0371477269, 0.0386635065, -0.0900390595, 0.0335176848, -0.00698496494, -0.0795145631, -0.0263204202, -0.0387219936, 0.0372513533, 0.069616653, -0.016119089, -0.0331068784, 0.0249988548, -0.0215352178, 0.00688688643, 0.0810623392, -0.0860611647, -0.0309012495, 0.0779893696, -0.032125663, -0.0114999395, 0.0288507938, -0.0429686308, 0.0445714816, 0.0473432317, -0.0187126808, -0.129243702, -0.0237859432, -0.0638953745, 0.0924817994, 0.0782472268, -0.0220032651, -0.0668439865, -0.0025732331, 0.0527206101, 0.0441822261, -0.0282638352, -0.0422725491, 0.00705240667, -0.0633908585, 0.0137796365, -0.02615471, -0.00124217058, -0.0351347774, 0.0385856144, 0.030581506, -0.0795791894, -0.0542370453, -0.00510898372, 0.10081286, 0.0338734984, -0.101331621, -0.0985490754, -0.00705705443, 0.0109579377, -0.00333777769, 0.0622152798, 0.00363911875, 0.0481062233, 0.068813026, -0.0234865788, 0.0290710796, -0.082115069, 6.35739416e-05, -0.0284638852, 0.001483083, -0.0426237248, 0.00982693397, -0.082873404, 0.0160913952, 0.0433014482, -0.109392956, 0.00402180618, -0.0129479989, -0.121640407, -0.0853046253, -0.0276072361, 0.0528869592, -0.157933325, -0.041677475, -0.0513420925, -0.0716695487, 0.125380233, -0.0541120097, -0.0270892903, -0.0354004353, -0.00983749889, 0.0150565766, 0.0727557763, 0.0440372378, 0.042118784, -0.0513586737, 0.127804816, -0.08231204, -0.0144347623, 0.144508213, 0.0170834213, 0.018995095, 0.0261083096, -0.0523809604, -0.0183201581, -0.0198718794, -0.0594392829, -0.0548257902, -0.0362088345, 0.17197448, -0.016027078, -0.0518785976, 0.0124345161, -0.0428913534, -0.0327314138, 0.000454797671, -0.0294881854, 0.0233004484, -0.0170797016, 0.0684266165, -0.0772320628, -0.00519311149, 0.0680455938, -0.118872553, -0.0149460202, 0.0620664768, 0.0202575028, -0.0733660832, -0.0887743235, -0.0459058397, -0.0442075208, 0.0459926054, -0.0317461155, 0.0334063917, 0.122998029, -0.0343262479, 0.0153604876, 0.0213850737, 0.0250464212, -0.0142205656, -0.0834608525, -0.126580968, 0.0660800561, 0.0521790944, -0.126256555, 0.0789100155, 0.0505135357, 0.0294168368, 0.0424421951, 0.0443682894, 0.0175621547, 0.0369247049, -0.0763881132, 0.00241885148, 0.123601884, -0.0437575728, -0.0337525159, 0.0584881753, 0.072721459, 0.0268098582, -0.0642768964, 0.0777513832, -0.0668801144, 0.152455807, 0.0384080373, -0.0813715234, 0.123705864, 0.0704651251, -0.0142856771, 0.0225876421, -0.032844767, -0.0282874554, -0.0180452634, -0.0589442588, 0.0211542696, -0.0840755552, -0.0346978456, 0.0624949932, 0.0413371325, 0.0347261764, 0.0189449582, 0.104123369, 0.0629087538, 0.206078738, 0.0759140998, 0.00179275218, 0.0178793985, -0.0904001892, -0.0120746437, 0.125980869, -0.0509332716, -0.0251817312, -0.0342635326, 0.0150608607, -0.0486635156, -0.0707176998, -0.088892363, -0.013950143, -0.144070938, -0.0290455334, 0.103315793, 0.00691494159, 0.0516338274, 0.0357198566, -0.0407630056, -0.0704655498, -0.0061621801, -0.0163742173, -0.00286670402, 0.0717858896, -0.0403173119, -0.0242009424, -0.0255283937, -0.146040618, 0.00370218931, -0.0169456266, 0.0739331171, -0.00640878826, -0.0625880584, -0.0078162197, -0.109838225, 0.00966158137, -0.0124182813, 0.0556307025, -0.040832039, -0.0159406848, -0.0489371084, 0.0553769767, -0.0129255224, 0.00165747106, -0.0153565537, 0.0232416987, 0.0490295142, -0.0645253658, 0.057539735, -0.0697470456, 0.00253124698, -0.0123401824, 0.0267368481, 0.0345181003, 0.0153361401, -0.0566138327, -0.0957990736, -0.0121652279, -0.0328246318, -0.0706163049, 0.0241552666, 0.0602169149, 0.0483116619, -0.00645811856, 0.115425527, -0.0619513579, -0.00985607132, 0.00515981205, 0.121840969, -0.0654161051, 0.0609334558, -0.0703953058, -0.0466380939, 0.00197777338, 0.0263202935, -0.0276529472, -0.0145663982, 0.0825188756, -0.0154785737, -0.00760034472, -0.00398123916, -0.0517241657, -0.0116613209, -0.0224521235, 0.0680376142, -0.00622316822, 0.12626937, -0.042651087, -0.0322515182, 0.0697021931, 0.0727702975, 7.03553669e-05, -0.117054015, -0.0118676685, 0.130442441, -0.0633720309, -0.0175191481, 0.0502342433, -0.0153560489, -0.00189093128, -0.0899978802, -0.0814712644, 0.00397173129, -0.00799734332, 0.112588078, -0.0880026966, -0.0207088478, -0.0840146393, 0.104321539, 0.0305856038, -0.0066149896, 0.00385881821, 0.0438802727, 0.00694280025, 0.031775374, -0.029828202, -0.0140974158, 0.0417685509, 0.0469135605, 0.0260566361, 0.0252963938, 0.000886915484, -0.0506873876, 0.073806785, 0.0405627377, 0.0770382509, -0.0126297167, 0.0539279208, -0.0134933405, -0.0488830209, -0.0149195949, 0.0286664907, 0.0258389022, -0.0504526757, -0.0995170474, -0.0514720455, -0.0692799166, -0.0749276727, 0.163625076, -0.0215796567, 0.101433694, 0.0290257093, -0.0497782454, 0.078620024, -0.0765042529, 0.0157838799, -0.0605206639, -0.109294169, 0.0945193022, 0.070097968, 0.0111340079, 0.00806904491, -0.119950257, -0.117081717, -0.0467412733, 0.00635355525, -0.0328157395, -0.0779284537, -0.0535240695, 0.118558511, -0.0796102732, -0.025870543, -0.0800812095, 0.0445277505, -0.050483115, 0.0729925111, 0.0596612878, 0.0246837493, -0.00155314244, 0.031930197, -0.145665765, -0.0536895916, 0.00893774256, -0.0883497596, -0.0918533802, 0.0466198847, 0.0609964356, -0.0676815137, 0.0174437314, -0.0376639664, -0.0100301281, -0.00489459373, 0.108539455, -0.0867397934, 0.00289764069, -0.0308248531, 0.0253050923, -0.00659247162, -0.0553039759, 0.0530485287, 0.0618184507, 0.0723310336, -0.000700828619, 0.0406789705, -0.0380382352, 0.195782676, 0.0544773676, 0.0280783065, 0.12561442, 0.0357654579, -0.00801739655, 0.00788500346, -0.00631313305, 0.0241355672, 0.0768359303, -0.0964802206, -0.00253858231, -0.100009397, 0.0262479931, -0.0976248756, -0.111943744, 0.0919356421, 0.125938892, -0.0401543379, 0.117040925, 0.0532688424, -0.061242871, 0.0221033189, -0.0276570898, -0.0478152446, -0.0574466176, 0.00819699839, -0.0348973684, 0.0246670842, -0.00592264906, -0.0111077726, 0.0866995007, -0.0227352083, 0.00829381496, -0.103243813, -0.0592893697, 0.0485052206, -0.050603468, -0.0623348616, 0.0450620539, 0.101759166, -0.0575572327, 0.0495275408, 0.0339027867, 0.0608742572, 0.0387787558, 0.0444233604, -0.0218878668, -0.119515583, -0.0267581306, 0.0620956197, 0.0759401843, -0.10464073, 0.039943669, -0.120554805, 0.0142001938, 0.0104443245, -0.0431935564, 0.0729510784, 0.0970963985, -0.0129293296, -0.0586054623, 0.017743174, -0.031778641, -0.0015063294, 0.0412261188, 0.0484331958, -0.0161143709, -0.00549984351, -0.0493346676, -0.0827445388, -0.0279450174, 0.00426994078, -0.0378730223, 0.0813675001, -0.0221152548, 0.162851453, -0.0593155697, -0.113409579, 0.0896707177, -0.0561915897, 0.12033812, 0.0299672019, 0.0382056236, -0.148166642, 0.0616600066, -0.0390294828, 0.076734677, -0.0610635877, -0.0314789601, 0.0106446203, -0.152618423, 0.00824991614, 0.0208676532, -0.0452706739, 0.0296786539, -0.00171152223, 0.0278075878, -0.0647582039, -0.0934415385, -0.00471531227, -0.0295969844, 0.0392355211, -0.0213776827, -0.00345349312, 0.0103437174, 0.0793427601, 0.0244922396, 0.0769085586, -0.0180552974, -0.0139173642, 0.0365448445, 0.110751674, -0.079107523, -0.0148752257, 0.055928126, -0.0583166182, -0.0278848745, -0.0543133169, -0.0146240722, 0.0462388359, -0.0462089404, 0.100065276, -0.0377004668, -0.0627923459, 0.0160569306, 0.122475393, -0.0237609986, 0.0326469876, 0.0121175274, 0.00290823728, -0.0759213045, -0.0410238355, 0.0405264311, 0.0794125274, -0.027770102, -0.0214025844, -0.000634195749, 0.0711863413, -0.0176606383, 0.0656886324, 0.0760930926, -0.0337079838, 0.0103172548, -0.0442149788, 0.0296556819, 0.0896399617, 0.0926107764, -0.0657806844, -0.0730204955, 0.0364074558, 0.0463961698, 0.0280023143, 0.0347175673, -0.0382448807, -0.0151486043, -0.0351293534, -0.0893038735, -0.0119186798, 0.0224835817, 0.0259567983, -0.00618832652, -0.0423954725, 0.0166269671, 0.00578288734, 0.0424060039, 0.00587061886, -0.0524880104, 0.109365225, -0.0914567709, -0.0388044044, 0.0739863664, 0.00929750502, 0.0168155134, 0.0719892383, -0.0457954593, 0.0540598556, 0.0506090075, 0.0544214435, 0.0112028988, 0.000449611805, 0.0767428875, -0.0880494937, -0.00829705596, 0.00506457034, 0.0316372067, 0.037886627, -0.0634205043, -0.0767910033, 0.00139203761, -0.0141287921, 0.065350242, 0.00455083512, -0.0507521704, 0.0327888578, -0.0450044125, 0.0352456719, -0.0213064775, -0.0177522674, -0.00198644958, 0.0105824154, 0.0127733704, 0.0429498255, -0.0461088046, -0.0140869189, -0.032076247, 0.0223935302, -0.0219765306, 0.0266452357, 0.0498517863, -0.0713030845, -0.0465965495, 0.015960671, 0.0765702203, 0.0080312388, 0.0792805627, -0.0662729442, -0.0218281597, -0.0474443845, 0.0242550168, -0.0282644872, 0.033289507, 0.0334301293, 0.0314183831, 0.0155287907, -0.0582918338, 0.0822805017, -0.0742264017, 0.1563963, -0.0114020435, -0.01263176, -0.0115720499, 0.113865636, 0.0781941637, -0.0390629768, 0.0707460418, -0.0352013633, -0.0346395001, -0.0204303395, 0.0684736595, -0.0650949702, -0.10914959, -0.143572226, -0.0396091603, -0.031377703, -0.0407384969, 0.0292514525, -0.0254713856, 0.00264162617, 0.000173193286, -0.085854508, -0.126747891, 0.017126631, 0.134934887, -0.110217519, -0.0356670469, -0.0543404818, 0.0187333152, 0.107053265, -0.0248832926, 0.101865664, -0.0710972846, 0.0722196847, -0.0384056494, -0.0161709804, 0.013287331, 0.00541426614, 0.0130335232, 0.0400547385, 0.0100121098, 0.0154263554, -0.0629646033, 0.0193865523, 0.00167901674, -0.00236805435, 0.0101759396, -0.107627042, 0.00447156373, -0.0081684785, -0.0686657578, -0.105860122, -0.0145202372, 0.105648175, 0.0951744467, 0.0278701279, 0.058870703, 0.0614429303, 0.0409474671, -0.0196230002, -0.059842132, -0.072326608, 0.078839533, 0.0461710729, 0.0051418962, 0.00476863049, 0.0325647667, 0.0355884321, 0.0283987522, 0.0260669962, 0.00147352088, -0.00998620968, 0.014060949, 0.0530263782, 0.0267538447, -0.178208858, 0.0138209928, -0.166257203, 0.00249827933, 0.0588419065, 0.00965133496, 0.0388614498, -0.0354404189, 0.101525106, 0.0155021399, -0.0782295838, 0.00205751229, -0.0115062622, 0.0447000861, -0.0492403507, 0.0462464131, 0.0278545078, 0.0493896231, -0.00348212384, 0.0177688748, 0.0589764938, -0.0141374562, -0.153412342, -0.0877678543, -0.163386658, 0.0293954685, -0.108064502, 0.0414382406, -0.0368895829, -0.00636456022, 0.00416772999, 0.008211473, -0.0767143965, -0.0195856318, 0.0320273377, -0.0896992087, -0.0541382805, -0.114244811, -0.026452342, 0.0807037503, 0.0398947708, 0.00308981165, 0.0229013935, 0.0499595329, 0.126231, 0.105691493, 0.0247283503, -0.0480804071, -0.0219699144, 0.0844142735, 0.0152459517, -0.0940366089, 0.0213311259, 0.0797767118, -0.0654330328, 0.0303749572, 0.0221867338, -0.0245458521, -0.0113317519, 0.00932829455, 0.0289108455, -0.0212216694, 0.00822014734, 0.0457722098, 0.0130141452, -0.16610533, -0.0211480781, -0.0197458994, 0.0688880235, -0.00803674106, -0.0433641002, -0.075563252, 0.0635190159, -0.101971351, -0.164013535, 0.0825247914, 0.0201021656, -0.0529738441, -0.0211677011, -0.0466175154, 0.00472022966, 0.06616579, 0.129757211, -0.0536907986, -0.0515484139, 0.00854382385, 0.0687660128, -0.000543623697, -0.00421395339, -0.0509204641, 0.0787195489, -0.0955284685, 0.0278457161, 0.032738395, -0.0350810252, 0.021184016, -0.00620284677, -0.0157659762, -0.120136291, -0.0488379225, -0.0571413785, -0.00956039596, -0.130700439, -0.0297761634, 0.0620664358, -0.0984532908, 0.036326915, 0.0142956804, -0.0336640477, -0.00327738747, 0.052082818, -0.0302631166, -0.0566398501, 0.00357326865, 0.0498971753, 0.0090519404, 0.0498086736, -0.0356872156, -0.158793435, -0.0531598851, -0.0724413022, 0.0847426951, -0.0579689369, -0.0855806544, 0.0161144361, -0.0345754586, 0.0575088561, -0.0482305698, 0.0408530161, -0.0572958775, -0.0430949926, -0.0452227145, -0.0143297808, 0.136190906, 0.0158195812, -0.047018975, -0.00814411417, 0.029649578, -0.0406708904, 0.0951420739, -0.0738690346, 0.0941496119, 0.0681650266, -0.0519653335, 0.0357567519, 0.0538630001, -0.0222863052, 0.151022032, -0.0852258503, 0.000150131527, 0.0268831402, 0.0451235622, 0.019896077, -0.0390991308, 0.0395388827, 0.0464649163, -0.0528178029, -0.0634406283, 0.032435406, 0.0321994387, 0.0763059929, -0.0442365222, -0.0384837463, -0.0376992933, 0.0821993724, -0.0429838598, 0.0302058551, 0.039350383, -0.0757741854, 0.0359587148, -0.0675518662, -0.100005239, -0.0506118014, 0.0944177061, 0.0117894504, -0.0284820385, -0.0153114414, -0.0337097533, -0.121349752, -0.0296758302, 0.0677160621, -0.0469472483, -0.0317657143, 0.0904516056, 0.00663401838, -0.0561745241, -0.0492588803, 0.0282529946, -0.101061374, 0.0839226246, 0.0480642021, -0.0347557813, 0.0767452791, -0.0702294558, 0.0499737225, -0.0848984867, 0.0706430674, 0.0254755691, 0.0556517467, 0.00553852506, 0.0453726128, 0.0186469965, 0.0565884635, 0.0242560711, 0.0359231979, -0.0724069178, 0.0165634658, -0.135310367, -0.032013312, 0.00181994541, 0.0117271263, 0.121910825, -0.0625010505, 0.0669507533, -0.0225233231, 0.0245092064, -0.126561821, -0.0302848145, 0.035558477, -0.0703105628, 0.0638471842, 0.0306731332, -0.0481522381, -0.0406722277, -0.0409029052, 0.0873740166, 0.0292977374, -0.0487803295, -0.0623919293, -0.0670752674, -0.0582743771, -0.0369736739, 0.00244259834, 0.0422472432, 0.0661929622, 0.0405329838, 0.0844473615, -0.0196251534, 0.0165268667, -0.0535134524, 0.0382272936, -0.0927124992, -0.0902759209, 0.0418790802, 0.00131716207, -0.0810423568, 0.0556469485, 0.145353869, -0.0974263251, -0.0265319683, -0.00157782063, 0.0342672877, -0.0780519694, -0.100708544, 0.00392956845, 0.0333812498, 0.0530423149, 0.0157616548, 0.00743991509, 0.0668429434, 0.0836819857, 0.0426887535];
    CONSTANT bias_3_i : ARRAY[0..63] OF REAL := [0.64754945, 0.691847086, 0.64616853, 0.738801003, 0.681163371, 0.618074238, 0.642219305, 0.681924105, 0.725929916, 0.669821262, 0.642402828, 0.64420867, 0.699106872, 0.731772006, 0.736818969, 0.668383598, 0.68884635, 0.640938818, 0.655000389, 0.732870162, 0.669698298, 0.703552306, 0.687165737, 0.693419755, 0.586305499, 0.688813746, 0.689942062, 0.622232378, 0.665326953, 0.657587767, 0.708570719, 0.641408205, 0.706247687, 0.728076875, 0.694459498, 0.697739005, 0.68515265, 0.63921845, 0.67039603, 0.669698596, 0.672608674, 0.459624499, 0.698169529, 0.630342007, 0.631216407, 0.73681736, 0.703925788, 0.700100422, 0.725266874, 0.671362042, 0.728427231, 0.723560095, 0.694639802, 0.607155502, 0.655874491, 0.73296082, 0.65932858, 0.686508298, 0.673355281, 0.734046161, 0.674785137, 0.674265325, 0.703997612, 0.652445555];
    CONSTANT weights_3_f : ARRAY[0..4095] OF REAL := [-0.0521443337, -0.127342403, 0.0130717456, -0.0596655086, -0.0273111761, 0.0327247679, 0.0394109637, -0.0123401359, 0.0960776955, 0.0669516474, 0.000666379929, 0.111136854, -0.121887974, 0.0318512022, -0.092767477, -0.0571558774, 0.0440648943, 0.0670731962, 0.0755134374, -0.0248164758, -0.0245014653, 0.116271675, -0.0863337666, -0.110264994, 0.0281036198, -0.131201297, 0.121819913, -0.0493896604, -0.108632259, 0.0232308805, 0.11175859, 0.113334209, -0.0309745446, 0.00279828906, -0.0263097361, 0.116411507, 0.134985745, 0.00494657457, 0.00834363699, 0.0148295909, 0.123774081, 0.0418391377, 0.135640502, -0.111531332, 0.109959185, -0.135435939, 0.0361935198, 0.0986461937, 0.0639104098, 0.0740167797, 0.0907477438, -0.0655242056, -0.121550567, 0.0214169323, -0.037972711, -0.0314986184, 0.020315364, -0.0910601765, -0.0322241634, 0.037475571, 0.0928814858, -0.01218725, 0.102777243, -0.0764217377, 0.0783669055, 0.122343868, 0.0670614392, -0.122746259, 0.125813544, -0.136584193, -0.0129609108, 0.0863741189, -0.0260882974, 0.0346245915, 0.0256888568, 0.107945338, -0.101845935, 0.0761630833, -0.0844016373, 0.111051813, -0.009620592, -0.0630434677, 0.0688468665, 0.0351438075, 0.120586038, -0.0786037594, -0.10621427, 0.107332289, -0.1062335, -0.0398073941, 0.0100298226, -0.00765535235, 0.0600221753, -0.0497887656, 0.0726344436, 0.0244747847, -0.133941308, -0.0139969289, -0.0164956525, -0.032233499, -0.0143216625, -0.0229434296, -0.0581621826, 0.0872895122, 0.0427271277, 0.117294371, -0.0419999585, 0.00527742505, -0.0238697454, 0.0134884566, -0.0728438497, -0.0774436891, -0.078616783, -0.0915552676, 0.112122655, -0.104264475, -0.0764580816, 0.0231063664, 0.0415457487, 0.0922157466, 0.112544298, -0.0208588988, -0.00843825936, -0.125481308, -0.0991969109, 0.131200939, 0.0391524434, -0.047940731, 0.00629302859, -0.0649658442, 0.129364312, 0.0668620318, 0.0720915645, 0.117274612, -0.0617987812, 0.10781534, 0.118253678, -0.091769591, 0.0618039668, 0.0271771252, 0.129491687, 0.0751471817, 0.0123195052, 0.12247768, -0.100104749, -0.0376960635, -0.0299254358, 0.0191544443, -0.0680884495, -0.105288088, 0.0125788152, 0.0202235281, 0.0872109234, -0.0292338505, 0.105079204, 0.0722285211, 0.0492487848, -0.0207891911, 0.035598442, 0.0796257257, -0.0816210359, 0.0394578874, 0.10630095, -0.0223288164, -0.0539216921, -0.0801568329, -0.0579407737, -0.0488362312, 0.0901255012, -0.0542660505, 0.123969197, 0.0129767805, 0.0857983679, -0.0723153949, -0.116513394, -0.0345694795, -0.0708460286, -0.0530526638, 0.112991229, 0.110247165, 0.055062592, -0.0358034968, -0.0648803413, -0.00882329047, -0.0386624709, -0.0317198709, -0.0141925812, 0.133358002, -0.119553827, -0.0781110525, -0.0169827417, 0.0419830829, 0.0809727758, -0.0601022243, 0.0752082318, 0.0453452766, 0.0357860625, 0.0793421566, -0.125073418, 0.0902063996, 0.0117165446, -0.0659095347, 0.00580528378, 0.00889448822, -0.12447641, 0.0204410553, -0.0412814021, 0.0495228618, 0.0835448503, 0.116250575, -0.0654591396, 0.136590302, -0.0437139794, -0.130533695, -0.0867854059, 0.072424531, -0.0716329142, 0.099989742, -0.029022947, -0.118508801, -0.00216673315, -0.00964409113, 0.0275921971, -0.0702549517, 0.0168310702, 0.0938851982, 0.0028321445, -0.114841782, 0.0769343674, 0.00749561191, 0.00931432843, 0.129629493, -0.00428524613, -0.0622541383, 0.0181307346, 0.128360391, 0.00720927119, -0.00107601285, 0.135486186, 0.0301079601, -0.122348845, -0.106044114, 0.017554909, -0.0103668272, -0.0536207855, 0.0721321106, -0.11596261, 0.0342057943, 0.0130974054, -0.0751927495, -0.0975918621, 0.0968466997, 0.111900821, 0.0677128434, -0.0339190885, -0.0657791123, -0.0346289575, 0.132123798, -0.107705772, -0.00667120516, -0.0373312384, 0.0983017981, 0.0146001726, 0.0881693661, 0.0728048384, -0.0892456695, -0.0545547754, -0.0606427193, 0.127758384, -0.11426615, -0.0448431, 0.0735787302, 0.0686352849, 0.105652809, -0.0194403604, 0.0510896444, -0.0973827839, 0.0499836057, -0.0842511952, 0.0107224584, 0.0790108889, -0.0802243128, 0.00903344154, 0.133382469, -0.0144729838, 0.00228916109, 0.00299805403, 0.136510193, -0.0606871843, -0.0106766224, -0.0197322518, 0.101590022, 0.034936294, 0.127533883, 0.00446902215, 0.00279822946, 0.115145057, -0.065636538, -0.0213813409, 0.0332797915, 0.0421897322, -0.04739739, -0.03065712, 0.122296244, 0.0230481327, 0.0973794311, 0.0809123367, 0.109200478, -0.0475174636, -0.0738452896, -0.0478056669, -0.0509483814, -0.0712444782, 0.101722687, 0.120032609, 0.0380587727, 0.115555257, 0.0806039274, -0.0530673563, -0.130207911, 0.077729404, 0.0261965245, -0.0817069337, -0.0618148744, -0.00412149727, -0.014915511, -0.103205219, -0.134377867, -0.0374422371, 0.13429296, -0.0570919588, -0.0797002017, 0.0528538823, 0.0800858587, 0.0458294004, 0.0261586457, -0.0560341701, -0.133453399, -0.0814694911, 0.0389332771, -0.0216553807, -0.0522843227, 0.0104800165, 0.054231286, -0.0362112522, -0.121657453, -0.0945644826, -0.0313536674, 0.110182002, -0.0274486542, -0.0645038635, -0.0392875969, -0.054631725, 0.0906170607, 0.0446703285, 0.0665438026, 0.0628865361, 0.0406519026, 0.0847905278, 0.013615489, -0.0455756336, -0.0462128669, 0.0173976421, -0.121880502, 0.117248267, -0.106539533, -0.0776506662, 0.0470769554, 0.0631131977, 0.0956659615, 0.106449336, 0.0514396876, 0.0951529741, 0.0847110301, 0.0335356891, -0.128389612, -0.0655849278, 0.0276690274, -0.0208295137, 0.0726699382, 0.0539053679, 0.0205788165, -0.0640053451, 0.0256249309, 0.132323802, 0.0422382504, -0.00320878625, 0.0842960477, -0.121599346, -0.0290251002, 0.0178422928, 0.0335367322, -0.0237912312, -0.0647743717, -0.104194477, -0.047350511, 0.0779209435, 0.080603987, -0.0237182304, 0.0247604847, 0.0798442066, -0.113430329, 0.101311639, -0.0551978573, -0.0396380946, 0.133087188, -0.0148522779, -0.00979818404, -0.00603397191, -0.10580916, -0.133506253, -0.00967347622, -0.0730265379, -0.0310022905, -0.029996708, 0.129264534, 0.123995304, 0.136550188, -0.0245039761, 0.109209001, -0.0926341116, -0.0518179983, -0.033019796, -0.0177469328, 0.0844373554, -0.0381035581, 0.0177293122, 0.0150468796, 0.103413239, 0.0835546106, -0.0884617865, -0.00752341747, -0.0771219507, -0.110308968, -0.0577309504, 0.0467014909, 0.124507934, 0.100173935, -0.0943341628, 0.0161749572, -0.108874336, -0.0713768005, 0.135854423, 0.0966987014, -0.0205949098, -0.101613097, 0.104421154, -0.0497194603, 0.0223887563, 0.0740994364, 0.0744936168, 0.115517199, 0.0120522231, -0.0541860983, 0.020311147, -0.0562019721, 0.124659091, 0.0691441149, -0.053887479, 0.0724818856, -0.0313050598, -0.0811104104, 0.104190558, -0.0330485925, 0.111697629, 0.0963663608, -0.0238290727, 0.0223227441, 0.0528036952, -0.0996605903, -0.021703206, -0.0652093217, -0.0223025084, 0.0271105915, 0.0292074382, 0.00457368791, -0.068554908, -0.0547924116, 0.108942538, 0.0641764849, -0.0987549722, -0.119499959, 0.0951081514, -0.0419656485, 0.118541718, -0.0252901465, 0.121815503, 0.0855444968, 0.0422533005, 0.0254690796, -0.0655569509, 0.00358602405, -0.0913407132, 0.082400322, -0.0784052312, -0.0180871487, 0.124201268, -0.136227459, -0.0170292258, -0.0532112941, 0.131566346, 0.06952402, 0.0666095465, -0.110658646, 0.113614708, 0.0028873235, -0.109899834, -0.014672257, 0.0058144629, 0.132832855, 0.00573641062, -0.0126792714, 0.0756112784, -0.125071108, 0.0649617016, 0.0426058769, 0.131729156, -0.0732614994, 0.0341416746, -0.0541509688, -0.101108447, 0.0102382302, -0.124604024, 0.130719483, -0.0247230083, 0.00963482261, 0.0265038162, 0.0424721539, -0.123501085, 0.00206148624, 0.0938844234, -0.0733475909, 0.0948895514, -0.120868802, 0.120048553, -0.131673038, -0.0366031453, -0.0553891286, -0.0627916306, -0.0435904413, -0.057633467, -0.0436587781, 0.102742121, -0.0266828611, 0.131982088, -0.0139831528, 0.104467243, -0.0220600367, 0.101302817, 0.0486853719, -0.000630795956, 0.0732958168, 0.0789853334, 0.0535539538, -0.046998024, -0.00175790489, 0.043284148, 0.0617725253, 0.130353421, 0.0918721706, -0.00624765456, -0.131705746, -0.0312967971, 0.128403842, 0.0586179644, 0.0303991735, 0.00364759564, -0.0247948915, -0.0597023666, 0.0240047723, 0.085168764, -0.0661254898, 0.0477693081, 0.0469849259, -0.104816139, 0.0806702971, -0.0418047309, 0.115232438, -0.100655794, 0.125909954, 0.0046890974, 0.0220941156, -0.0794617161, -0.0660549402, -0.0322142392, 0.0484143049, -0.0505887121, 0.0484498292, 0.101025939, -0.0860916302, -0.0568180159, -0.0740828887, 0.132015139, 0.0850556791, 0.0805580616, -0.0910110474, -0.0797288641, 0.0998696536, 0.00483940542, -0.0404196531, -0.029866904, -0.0876832604, -0.0712021068, 0.0319518596, 0.056360662, -0.0139351264, 0.000249356031, 0.0315214694, -0.0407522917, -0.135266572, -0.128061816, 0.0832460374, 0.0479347855, -0.103647217, -0.115489721, -0.0657822117, 0.108107135, -0.089061439, -0.0267519727, -0.058967188, -0.0365279913, -0.0619976595, 0.121219993, -0.0310177654, -0.0474473089, -0.000912636518, -0.11945869, -0.00367443264, -0.0183600113, -0.0413725525, -0.107271016, 0.104627863, -0.100125641, -0.123059146, 0.0906228423, 0.0421913713, -0.0222766176, 0.12505427, -0.114441305, 0.0816470981, 0.0929709375, -0.119069442, -0.0779820979, 0.119288027, -0.110795863, -0.0563212335, 0.118073702, 0.0981317759, 0.0664688647, 0.0602101237, 0.0270466805, -0.10832414, 0.00654751062, -0.0517121553, 0.021417737, 0.095620811, 0.11452195, 0.0508430004, -0.0997347683, 0.0343427062, 0.0199356079, -0.0386759862, 0.0982036293, -0.0412252843, 0.112768382, -0.0958701, 0.0842528045, 0.0155244023, -0.098992601, -0.052829951, 0.104019761, 0.00673630834, -0.0389265865, -0.0390314832, 0.0433861464, -0.0208425373, -0.115250684, -0.00176331401, -0.0448659211, -0.0905172676, -0.0429517403, 0.096448794, 0.059812814, 0.0969527662, 0.120459139, 0.027512908, 0.0399251282, -0.00255598128, -0.135592774, 0.0619364232, 0.118778795, -0.128738359, -0.0909728482, 0.123057872, -0.000388264656, -0.134973079, -0.0446337387, -0.0617902279, 0.0797113329, 0.0840478092, -0.109512709, -0.0891110003, -0.123604089, 0.0288672596, 0.0394423455, -0.045054324, 0.0299270004, -0.0326793268, -0.0441791937, 0.0433877707, -0.0327894092, 0.0628817081, -0.120908603, -0.135370582, -0.129082546, -0.00913827121, -0.133775815, 0.0925979167, -0.0279047936, 0.0137742162, -0.0684487373, 0.0832460076, 0.0778043717, 0.0220358074, 0.116572708, 0.120394021, -0.126439199, -0.0440204367, 0.116596639, -0.00574839115, -0.121665649, -0.117598802, -0.133597374, -0.123539574, -0.0827658027, 0.0988901258, 0.0562292635, 0.0241476446, 0.0646850467, 0.0456878394, 0.114608794, 0.0522514731, -0.0722370073, 0.0649634004, -0.0653436705, 0.00828239322, 0.0441260487, -0.0794956684, -0.112388924, 0.047713086, 0.105907008, -0.0337683558, 0.112112969, 0.00168156624, 0.0221335292, 0.0984038562, -0.0405161902, 0.101812184, -0.0306580663, 0.00638313591, -0.00933606923, -0.0495209992, -0.0118647963, 0.133386314, 0.0972756445, 0.127949864, -0.0170405582, 0.030266434, 0.0644918531, -0.0410653427, 0.0243677348, -0.126150668, -0.0376376882, 0.0793990642, 0.115365475, 0.125485301, 0.132854491, -0.0173375756, 0.123990357, 0.126760542, 0.0199246109, 0.0463828295, 0.133341432, 0.0799899697, 0.0754961669, -0.0465824604, -0.0846978053, 0.0873944014, -0.00712434947, 0.0672320575, 0.0847331285, -0.031734623, -0.0822531432, 0.112729147, 0.091640383, -0.0295949876, -0.101722397, -0.0939373076, -0.0188322812, 0.136161178, -0.111046098, -0.0737150609, -0.00393897295, -0.0723129138, -0.00878252089, 0.0726039559, -0.0808813944, -0.104831845, 0.11933437, -0.0736284181, 0.117690653, 0.132863224, -0.106923886, -0.130747631, 0.0599240363, -0.0373848379, 0.0192611963, 0.00730569661, -0.105000041, -0.0734499022, -0.11048428, -0.134641781, 0.0674274415, -0.105549127, 0.0875730067, -0.0965825468, 0.0865682364, 0.0314493179, -0.0624415278, -0.0868700892, 0.132529616, -0.00267550349, 0.123484045, 0.0232645124, -0.0157514364, 0.100139067, -0.0107656717, -0.031046465, -0.125469819, -0.00878351927, -0.0412467942, 0.051600799, -0.0452794284, -0.0817394853, -0.111147568, -0.10428945, 0.0193194747, -0.0737061799, 0.0928273499, 0.0987958759, 0.0650438666, 0.0444750786, 0.0709429234, -0.0109952241, -0.0512328371, 0.0293803364, -0.0724560991, -0.0101262629, -0.0339284912, -0.102498278, -0.0825525522, -0.0278738439, -0.0327277705, -0.0812947005, 0.033122018, 0.00578024983, 0.0188989043, 0.116528481, -0.027826868, 0.000491172075, -0.106478974, -0.011813581, 0.010574013, -0.0519400612, 0.123747796, 0.0615936518, -0.119706713, 0.0965384394, -0.108477712, -0.0182201862, 0.0777682662, -0.0450730026, 0.0741986185, -0.0867925212, -0.0914172977, -0.0107384473, 0.131009102, 0.100436121, -0.00689902902, -0.0676930621, 0.133405417, 0.0340053141, -0.0278127939, 0.0735555142, -0.00789925456, 0.0237952769, 0.125645787, -0.00715275109, 0.0814768672, 0.0229864568, 0.039741382, 0.0535612106, -0.00911837816, -0.073020339, -0.136608064, -0.0868141353, 0.105997264, -0.108271837, -0.0134975314, 0.0235030651, -0.0706957877, 0.0434921086, -0.0152588561, -0.0328821242, 0.0723848939, -0.0791713893, -0.0699490532, -0.0299490392, -0.090794012, -0.0844306946, 0.133389503, 0.117837787, -0.115428381, -0.0866210312, 0.0410853177, -0.0918630287, 0.118478656, 0.0146174431, 0.0953406394, -0.0962813497, 0.0473799258, -0.0181181654, 0.131747723, -0.120570317, 0.136137247, 0.0953928381, 0.0457116365, -0.00359970331, 0.0654873103, 0.0974072814, -0.119495809, 0.0238964856, 0.0779941678, 0.12287885, -0.0259701163, -0.077402845, -0.0903707147, -0.0973898098, 0.0840773582, 0.084917292, -0.0957877338, 0.00296367705, 0.0508234501, -0.025126718, 0.0773919076, -0.0142726302, 0.0410522819, -0.0980267525, -0.0504460782, -0.117062584, -0.118355528, 0.110945344, -0.0739619359, -0.00828537345, 0.0250171572, -0.0373283327, 0.0482215881, 0.0739530623, -0.00570225716, -0.131928071, -0.0220187083, -0.0621101633, 0.073841244, 0.0657580495, -0.0160987303, -0.0192219168, -0.0456597954, 0.115348727, -0.105435088, -0.0813490897, -0.136476174, -0.0613244548, 0.012233153, -0.0721570551, -0.0675859153, -0.104073301, 0.0922733992, 0.0365638137, -0.0522537977, -0.13286984, -0.129645869, -0.0356296524, 0.108128846, 0.118089706, 0.134406865, 0.000925406814, 0.0339840204, 0.0268510282, 0.136217177, -0.0668128356, 0.0955496728, -0.0347480252, -0.0991844982, -0.0170325562, 0.0585017502, 3.32742929e-05, 0.104093537, 0.0859187245, -0.0749645233, -0.136781573, 0.0874286443, -0.0839600861, -0.0636291578, 0.0829299092, 0.00441795588, -0.0970190763, -0.13331753, -0.0837791264, 0.0838996172, -0.109015271, -0.133527741, 0.0867631137, 0.0342673063, -0.0698866695, 0.0552534908, 0.122101486, 0.097059682, -0.0596561059, -0.0732495785, -0.0900109708, 0.0287191421, 0.0704183877, -0.0147428438, -0.0729215443, -0.02997493, 0.0591437072, 0.0911006927, -0.0470742807, -0.0834658444, -0.128154859, -0.128171474, -0.0141603276, -0.0415874943, -0.0741763264, 0.0191976279, 0.00458350778, -0.0131755695, -0.0289093405, 0.108689323, 0.0278994441, 0.0151216388, 0.0795960575, 0.10847947, -0.0252841711, 0.121694714, -0.09039177, 0.121906906, -0.0624969006, -0.122551583, 0.0379208326, 0.0489537269, 0.0682066679, 0.0822287202, -0.0358567089, -0.105450898, -0.0416091457, -0.0385292098, -0.00931750238, 0.118311584, 0.0558300316, -0.104803734, 0.0148100257, 0.0676030517, 0.0233720094, 0.10112904, 0.0701182336, 0.000294700265, 0.0258774012, -0.0826673359, 0.136286765, 0.104154587, 0.120219171, 0.0439334363, -0.057297565, -0.0512804985, -0.128053397, -0.0474716276, 0.0476621836, 0.031222567, -0.0340055376, 0.050065577, 0.11938867, 0.13348335, 0.12134698, 0.107014388, -0.0903482512, -0.106243461, -0.028781265, 0.119756818, 0.0329640061, 0.053051725, 0.0452067256, 0.0849139988, 0.0232935995, -0.00309948623, 0.0251261592, -0.0166506246, 0.0362438411, 0.0985837728, -0.128518403, -0.0527147353, 0.0568866134, -0.0457645282, 0.0102809668, -0.00682477653, -0.111691199, -0.0985759348, -0.119488858, -0.0336322561, -0.00871042907, 0.0908353776, -0.102891028, 0.0237320364, 0.109722108, 0.0339153707, 0.0781892389, -0.0568968281, -0.070392102, 0.00909925997, -0.0573852882, -0.0305456594, 0.109213173, 0.119168997, -0.132001013, 0.0735763758, -0.04390046, 0.0619595945, -0.132424966, -0.117013089, -0.0970229208, -0.119751304, 0.0943338424, -0.00310666859, 0.0708045363, -0.0581020787, -0.128431141, -0.121518217, -0.0430620909, -0.119222105, -0.00157390535, 0.00488206744, 0.0923803449, -0.0263164267, 0.128791809, -0.091206111, -0.128529444, 0.0107199401, 0.0514403731, 0.00419060886, 0.0311676115, -0.0974185318, 0.105336308, -0.0783051699, 0.00641301274, 0.0655302703, 0.0650752187, -0.0335167795, -0.0150460303, -0.121415116, -0.00268605351, 0.0662408918, 0.0607724637, 0.0548945069, -0.0603127927, 0.132084787, -0.00612483919, -0.061769329, -0.0205898881, 0.0278406739, 0.0459839404, 0.109364167, 0.0521156639, -0.136487722, -0.0256103128, 0.132692397, -0.0793503895, -0.0167675614, -0.0664683804, -0.133050963, 0.0292422771, 0.0520415008, -0.036471352, -0.124928989, 0.0878525674, -0.0451673493, -0.0438311845, 0.0276689231, 0.110060781, 0.0252711177, 0.0686930269, -0.117099896, -0.0133249238, -0.0166052803, -0.120200396, 0.0487333685, 0.133657664, 0.100010395, -0.0016284585, -0.120911248, -0.0790074319, 0.0274080038, -0.11876113, 0.0467091352, -0.0860109925, 0.0293624401, -0.124765135, 0.0377427191, -0.00803343952, 0.128490061, -0.0583512112, -0.111046851, 0.0569658428, -0.105105519, 0.0783790797, 0.122847766, 0.0893425643, 0.0331273377, 0.0140959769, 0.120581686, -0.0513454303, -0.0712746456, -0.0107715577, -0.0754768774, 0.00752152503, 0.123520523, 0.0994419903, 0.042070508, 0.116076678, 0.108907014, -0.0100371242, -0.0502856821, -0.127781808, -0.0959718227, -0.00823584199, 0.103984758, 0.00784423947, 0.136094183, 0.13676849, -0.0667719617, -0.0593828186, -0.111090891, 0.110446766, -0.0694717243, 0.126528531, -0.131870806, -0.126988739, 0.0219853669, -0.0724558756, -0.0417747572, 0.0626463294, -0.0257236287, -0.092297107, -0.0480091572, 0.0706134886, 0.0550106615, 0.0181860328, 0.0275326818, -0.0548655391, -0.101263121, 0.0703497231, -0.0191987753, -0.106192559, 0.0636165142, 0.00324371457, -0.0499303266, -0.0433189198, 0.039193213, -0.0623440817, -0.082757771, -0.108307488, 0.077211827, -0.0241999403, 0.0282767415, 0.100406244, 0.069861725, -0.0870052502, -0.115959577, -0.136538222, -0.105175421, -0.136884451, 0.035523057, 0.0981892049, 0.11644423, -0.0965195149, 0.0948940217, 0.0897577703, -0.119575374, -0.068613112, -0.039985843, -0.0190420374, 0.0148238391, -0.095509544, -0.0392760411, -0.0559469983, -0.0620127767, -0.0302660093, 0.106922835, 0.132595956, -0.0433744565, 0.0305157602, 0.056451723, 0.0654757917, 0.103904799, 0.0396663249, 0.0550738573, 0.0720562786, 0.10757558, -0.026466243, -0.0444748476, -0.0581008419, -0.111512296, 0.0722546428, 0.123054862, -0.0892638266, 0.0384279788, 0.0987899601, -0.0856239945, -0.0184375793, 0.133606642, 0.0523470044, 0.126677632, -0.000685289502, 0.0932309926, 0.0348463953, 0.0536953509, 0.105479881, -0.0786405206, -0.00612908602, 0.0537355691, 0.116253257, -0.0880500823, -0.0127767548, -0.0298942924, -0.0561042279, 0.0919492245, 0.0362647623, 0.0261767954, 0.0154044032, -0.118463717, -0.0106966347, 0.0869911462, 0.0964087099, -0.116868556, -0.0612397343, -0.0924005955, -0.0270310044, 0.0967000425, 0.121895581, 0.130125463, -0.0907645673, -0.0897659287, 0.0844743699, -0.0405976772, -0.0880294144, -0.0699958727, -0.0804035068, -0.113904461, 0.00601027906, -0.0234429538, -0.0116924196, 0.126409292, -0.0303086415, 0.113090932, 0.0786094069, 0.114850223, -0.123965874, 0.04720366, -0.0705588013, -0.0382724777, -0.103151806, -0.0243912116, 0.122166961, 0.12630558, 0.111489579, 0.0731034577, -0.0456609353, 0.0503623039, 0.099888131, -0.063670747, 0.126902491, -0.0737484917, 0.0970897228, 0.00655455887, 0.0902363658, 0.0328852683, -0.120686963, 0.0849710852, -0.102837935, -0.0925061107, -0.0784913525, -0.0852063149, 0.00321094692, -0.0445294008, -0.133646205, 0.109196946, 0.116363645, -0.00162254274, 0.0841408223, 0.0649395585, 0.0306562632, 0.124539614, -0.0997705758, -0.0310134217, -0.102773756, 0.0394320637, 0.0774853081, 0.0297313184, -0.0408617556, -0.0799109042, 0.0766610801, -0.078001976, 0.0935018957, -0.0187650248, 0.0326421708, -0.113368921, -0.0512247086, 0.0387326032, -0.048958458, 0.0846625119, -0.0432993993, -0.113230005, 0.0856152177, -0.107339084, 0.0999075621, -0.0594706386, -0.0687982887, -0.0745980591, 0.0952702165, -0.0735825151, 0.103935629, 0.0240671337, -0.0319503248, -0.055029951, 0.126859069, 0.00795416534, 0.0563020408, -0.10236688, 0.13665995, 0.0107578039, -0.122057773, 0.132144094, -0.0724108815, -0.0900636017, 0.0899018645, -0.0209324136, -0.120483376, 0.0978723913, 0.0331790447, -0.0832656175, 0.0845608264, -0.125201523, -0.0578101203, 0.0134700686, 0.0208921582, 0.104788646, -0.127424389, 0.0944375247, 0.043242991, -0.107128546, 0.0195430666, -0.0772839487, 0.0700984448, 0.0560875088, -0.114404187, 0.0533519685, 0.0696230829, 0.0500552952, -0.0486046374, -0.100405201, 0.133118063, 0.0117811859, -0.0582463518, -0.0252300426, 0.0213049799, 0.118892163, 0.0619460791, 0.0371985584, -0.00492532551, 0.0355799645, 0.0832643807, 0.0933858752, -0.00250583887, -0.0811907873, -0.0571916625, 0.0886474848, -0.13435021, -0.0582796782, -0.0443269908, -0.0121342316, -0.0409444571, 0.0860714465, 0.00317509472, 0.0317439884, 0.0716000348, -0.0742574185, -0.0234479532, 0.0419644117, 0.0696455687, 0.117133528, 0.069949612, -0.054899171, 0.0629307032, -0.00542390347, -0.0756822601, 0.0755674988, -0.088504687, 0.0961316973, -0.120285079, 0.128451705, 0.0585775822, -0.124496162, -0.113663524, 0.0804674625, 0.0603919327, -0.015699625, -0.0458351076, -0.0837002173, -0.036410138, -0.0842880234, -0.0957390517, -0.126437411, 0.055495888, -0.0290719867, -0.115706533, 0.00690737367, -0.106253356, -0.00222922862, 0.00638636947, 0.136639714, -0.130089208, -0.0571671128, 0.0308016837, -0.127073139, -0.0840152949, 0.0520015359, -0.0486909226, -0.0650354177, -0.125432044, -0.0534592792, 0.0923637003, 0.0989185274, -0.120891556, -0.000621885061, 0.13054949, -0.0274071917, -0.113035627, 0.0832538009, 0.113880157, -0.113907561, -0.00255301595, -0.000591561198, 0.130752295, -0.045228824, -0.0526037365, 0.123807877, 0.0970283747, -0.102338865, 0.069728002, -0.104946956, 0.102437556, 0.0581571907, -0.0741001293, 0.0444572121, -0.0030233264, -0.0282619521, -0.0256473646, 0.0676550567, -0.13509123, 0.0396783501, -0.0301795602, -0.0897156149, -0.0638799146, 0.0823161602, -0.0953015238, -0.0743213445, 0.0201806277, -0.0811779946, 0.107954443, -0.00337570906, -0.00971934199, 0.0885137022, 0.0604767799, -0.119999848, 0.0861417353, -0.119649321, -0.0760148987, 0.089216575, 0.0480475128, -0.00522832572, 0.106205195, 0.126377225, 0.13524431, -0.0834581703, -0.000878751278, 0.0671182126, -0.0438458398, -0.0107437074, -0.0491714478, 0.0218756795, 0.0627507269, -0.037882641, -0.0736816302, -0.0426758751, 0.0872242749, 0.128437817, -0.100631341, -0.0738518834, -0.107284829, 0.0454461575, -0.0564804524, 0.0316800028, -0.0166500658, 0.0586845726, 0.0480518341, -0.0206569433, 0.0516817868, -0.00426511467, -0.0620380118, 0.0527656078, -0.0513607785, 0.0292428583, -0.0290877521, -0.0475891903, 0.0364919454, 0.0036188066, 0.0160036981, 0.0517819226, 0.131391287, -0.121882394, -0.0802767724, -0.0106136799, 0.13031289, -0.0857627764, -0.135954931, 0.0724732429, 0.0937915444, -0.00633455813, 0.0220428705, 0.131122321, 0.0100516528, -0.0629529431, 0.0558041036, -0.0757858455, -0.0485834777, 0.0231841058, -0.0111280531, 0.127422839, 0.0986086726, 0.0358464271, -0.0342786312, -0.0679353029, 0.123054206, 0.0904192179, -0.109934345, 0.0577495992, 0.114916652, -0.135566831, -0.0446366146, -0.0408690721, -0.0263216868, 0.12370643, -0.0191679224, 0.124116838, -0.0694237649, 0.130773544, 0.0519571751, -0.0522508249, -0.106997699, 0.0546361357, 0.0576944202, -0.0237817988, 0.059796229, -0.129319265, 0.0842217803, 0.131958067, 0.128440678, -0.00129529834, 0.0223187655, 0.133176416, 0.055896014, 0.0757275373, 0.0713572055, -0.0836920589, -0.103879668, 0.132169753, -0.102196105, 0.0688092262, -0.109179191, 0.13486439, -0.0893321186, -0.0739976838, -0.0681645125, -0.0610896572, 0.0293230712, 0.00956080854, -0.00190111995, 0.0921217203, -0.127043292, -0.0280772373, 0.0288666636, 0.0143638104, 0.0984716862, -0.0585380793, -0.0271505862, 0.03382653, -0.0623259246, -0.00730890036, 2.32756138e-05, -0.0943615884, -0.0858648643, -0.0644539446, -0.0675351471, -0.111309886, 0.019990921, 0.0293648541, -0.047796987, -0.0938501433, 0.0293900222, -0.046621345, 0.113267362, -0.109652013, -0.0356403291, 0.122125745, 0.108362004, -0.0301989838, 0.0521476269, -0.0828424543, -0.103570864, 0.0743227452, -0.0115605295, 0.0945950449, 0.136096179, 0.00197905302, -0.116294429, -0.00212404132, 0.0813746601, -0.0810060352, -0.0970925912, -0.0726671964, 0.12972039, 0.0690163672, 0.124263674, 0.0461698622, 0.1159949, 0.0975343734, -0.0393245518, -0.127924308, 0.0933650732, -0.0110772252, 0.0892811865, -0.0825201645, 0.103403583, 0.0490089357, -0.0741517469, 0.106485367, 0.118132323, 0.0707530826, 0.0261539072, -0.0248588473, 0.0466733426, 0.0414143354, 0.0181136876, 0.115674973, 0.011881277, -0.0440483466, 0.0855888724, 0.00350424647, 0.120592654, 0.0910972953, 0.0350409895, -0.0663104057, 0.084793359, 0.0223444551, -0.0145348832, 0.0328541547, -0.05145026, -0.0464102477, -0.0853003338, -0.114435062, 0.104983583, -0.0497277826, -0.0830415636, -0.0658770204, 0.102298945, 0.00115860999, 0.076831758, -0.0143973753, 0.0154636204, 0.12856555, -0.118063398, 0.0759682059, -0.0122529045, -0.0851866603, 0.118180871, 0.0136093795, -0.136744693, -0.072859779, 0.0305171311, 0.0487162173, -0.0113377422, 0.126042128, 0.091231674, 0.0114648342, -0.0360141322, -0.037275672, 0.0722761154, 0.113058642, -0.00639308989, -0.132716686, -0.0679949448, 0.100947499, 0.104375213, -0.0530837476, -0.0409268215, 0.0480398834, -0.0657091513, -0.00375974178, -0.0540021956, -0.0989605784, 0.0222224593, -0.10744907, -0.0570113212, 0.108316958, 0.0982603282, -0.036241062, 0.0474478602, -0.0650933981, -0.0180442855, 0.028708294, -0.127319127, -0.100772992, 0.126135617, 0.113112897, 0.0675831437, 0.0374301821, 0.0869508535, -0.0204449371, -0.134612367, 0.0226760209, -0.0383700877, -0.0839552879, -0.023379229, 0.0797197223, -0.116203152, -0.0964124948, 0.0375358015, 0.128981233, -0.0111501515, 0.109349832, 0.0896549672, 0.0227474123, 0.0783401728, -0.095428586, -0.114835836, -0.0875191092, -0.0574464351, -0.0511667877, 0.0159212649, -0.0904242545, 0.128912687, -0.100479662, 0.0770364553, -0.0549969152, -0.0592422411, -0.0238574073, 0.13500914, 0.0938336849, 0.0219465941, -0.0315933973, -0.0424854159, -0.0863585472, -0.0336530134, 0.0599575639, -0.0114217103, 0.0038972497, 0.103980511, 0.0115303993, -0.133669689, 0.0990677625, 0.0294876099, -0.091690585, 0.113523692, -0.0224685147, -0.0752440095, -0.129941583, -0.0415092409, 0.0575455874, 0.0270656347, -0.0653796792, -0.117771082, -0.0929383188, -0.111615658, 0.0808861554, -0.0996594802, 0.124172539, 0.0921595991, -0.135693133, -0.0708992705, 0.0151500106, -0.101841167, -0.0409430191, -0.108884647, 0.0614504069, 0.1250543, 0.0496179909, -0.0460122526, 0.0921798944, -0.0285486206, -0.0166778192, 0.00766223669, -0.132137239, -0.0908356681, -0.109672323, -0.0587465316, -0.0917949229, -0.0321453214, 0.0525925756, 0.132113189, -0.0612824336, -0.124468543, 0.00918523967, 0.0290578753, -0.0458133966, 0.0937909931, 0.115016282, 0.0108943731, 0.0714527071, -0.109289736, 0.0439956188, 0.0853204131, -0.0383676067, -0.0620002076, 0.115915984, 0.0567686558, 0.0642954111, -0.0811725408, -0.0673033893, 0.122292489, 0.0605366826, 0.0960350931, 0.0956777781, 0.00737962127, -0.0711956695, 0.0689126849, -0.0438272357, 0.0890601724, 0.00938785076, 0.126547694, -0.0471894965, -0.128692806, 0.00478981435, 0.00796082616, 0.130308151, 0.0800433755, -0.0513560101, -0.110880062, -0.0965960622, -0.131567493, 0.0993641615, -0.0600399971, 0.124575794, -0.0420187265, -0.07880757, -0.00749345124, -0.0227379128, -0.125631228, 0.0740180612, -0.075208813, 0.0675159842, 0.0104151517, -0.026500918, -0.0756703466, 0.0744711608, 0.13343218, 0.12198481, 0.0918223858, 0.0317174792, 0.0774797201, 0.00680048764, 0.0539913327, 0.116550624, 0.0325739086, -0.00708575547, -0.0607766733, 0.051164642, -0.0221630409, 0.018378526, -0.0512623787, 0.0383725315, -0.0461483896, -0.0641455278, -0.0965751708, 0.0970107168, 0.105739132, -0.122537419, 0.0178013295, 0.107133016, 0.0125948191, -0.0135797337, 0.0797807425, 0.0611358136, 0.0529499948, -0.135286316, -0.0640067458, -0.120747462, 0.0661098212, -0.105924435, 0.0982864797, 0.0967068374, -0.0613402873, 0.0689376295, -0.0656040907, 0.0363693982, 0.111808658, -0.0275689587, 0.00758306682, 0.0290805399, -0.131993115, 0.0235240757, 0.0112666488, 0.0848694593, -0.0882292092, -0.120486349, 0.0718367547, 0.0624758005, -0.0758686066, -0.0128832832, -0.136147812, -0.0521976128, 0.113158196, 0.103650421, 0.121767521, 0.0231329054, 0.0155290365, -0.0927346349, -0.0189576074, 0.0683096647, -0.130036056, 0.124609053, -0.0170007572, -0.0893515423, 0.060974285, -0.0451976135, 0.0573027879, 0.0536007732, -0.104038201, -0.123042397, -0.015266858, -0.00371608138, -0.0795646831, -0.0452143624, 0.136367708, 0.118662477, 0.0296504796, 0.135353684, 0.0211382806, 0.0997147113, -0.0202512741, 0.122795224, 0.133774847, 0.0252506733, -0.0868833512, -0.0196186081, 0.11263822, 0.110760838, 0.00225409865, 0.129932493, -0.0822386518, -0.0750381649, 0.112813398, -0.0326290801, 0.0869027376, 0.122541666, -0.117104858, -0.0811770707, -0.00336121023, 0.0891758353, 0.120802879, 0.0851752311, -0.127724662, 0.075992927, 0.00552037358, 0.00993840396, 0.0839840174, 0.000344485044, 0.0288314372, 0.130288333, -0.131219804, 0.0781232864, -0.114732742, 0.00839407742, 0.0153136402, 0.0134378225, 0.0699736327, -0.0791138634, 0.0551245958, -0.0434599221, 0.0988393575, -0.0179145783, -0.106059656, -0.115503855, 0.0305479467, -0.0638865456, 0.101052254, -0.0421021432, -0.0806993544, -0.0345053896, -0.100246072, -0.0207606927, 0.0162339211, -0.0814323127, 0.110953644, 0.00843192637, -0.107001454, -0.0608810782, -0.133155733, -0.0369181558, -0.0392057523, -0.0369349718, 0.0566265434, -0.0147343874, 0.0925732255, -0.00758492947, 0.135466546, -0.0622921661, 0.0643838197, 0.110984847, 0.0497137159, -0.129211992, -0.0791157559, -0.129735216, -0.0425587744, 0.0275189131, -0.00198623538, 0.010402903, -0.0209983289, 0.0361455083, -0.0859315246, 0.0176406354, -0.0969529599, -0.0926274881, -0.0650475249, 0.0944561064, 0.0582294315, 0.0810323507, -0.0295920148, -0.00400814414, 0.0725500286, -0.0864371955, 0.0339131206, 0.0362699181, 0.0280079544, -0.130080238, -0.0683498159, -0.123454332, 0.104002938, -0.0686788633, 0.0247931331, -0.124924809, -0.0422899947, -0.00432136655, 0.0393503457, -0.104298234, -0.0987556875, 0.10403429, -0.0171738565, -0.0580046326, -0.000511705875, 0.0794814676, 0.106441498, 0.125230491, 0.031059593, -0.0224574804, 0.0882577747, 0.112146825, 0.125952125, 0.124437779, 0.0567529202, -0.0847644657, -0.0479874462, 0.00017952919, 0.0494967401, -0.0327971131, -0.101243794, 0.0755880326, -0.0679002032, 0.13497588, 0.135284036, -0.00892116129, 0.0503858775, -0.0320283473, 0.101213798, 0.0958126336, -0.0420148149, -0.0682129934, 0.0186359435, 0.0203741491, -0.110912152, 0.0118872523, 0.0944701731, -0.0212488323, -0.055293642, 0.0734030604, -0.122572541, 0.0197974145, -0.131350681, 0.0986521244, -0.0759862661, -0.111149952, 0.054469347, -0.100436568, 0.00284297764, -0.131670073, -0.0733880699, 0.0850994289, 0.0944229364, -0.105013229, -0.0282981545, 0.062829569, 0.064699024, 0.0377689004, 0.0846547186,